# B&R Automation Studio project TD52 (part 39)

### module_CU.typ - Predefined package data types
```iecst
TYPE
	IN_Cust_Struct : 	STRUCT
		bEO_FreshOilPump_Dem : BOOL; (*Status: fresh oil pump (OUT_AG.tEO_FreshOilPump_Dem)*) (*OldName:new V4.14; Cycle:5*)
		bEO_WasteOilPump_Dem : BOOL; (*Status:waste oil pump(OUT_AG:tEO_WasteOilPump_Dem)*) (*OldName:new V4.14; Cycle:5*)
		bAux_OilValve_IsOpen : BOOL; (*valve status for fresh/waste oil in oil pan (without TOF), to be used for release of customized oil pump controls*) (*OldName:new V4.14; Cycle:5*)
		bFreshOilPump_RTC : BOOL; (*Status:fresh oil pump run time exceeded signal (OUT_AG.tFreshOilPump_RTC)*) (*OldName:new V4.14; Cycle:5*)
		tL_FreshOilTank : HALioAi_Type; (*Tank Level measurement input*) (*OldName: NewPv V4.14*)
		tL_WasteOilTank : HALioAi_Type; (*Tank Level measurement input*) (*OldName: NewPv V4.14*)
		tL_DayOilTank : HALioAi_Type; (*Tank Level measurement input*) (*OldName: NewPv V4.14*)
		bBlocDelay_ManStart : BOOL; (* = 		-	blocking of next manual start by delay	*) (*OldName: T26	; Cycle: 5;*)
		bCnt_Gas_NormM3 : BOOL; (*Normal cubic meter - Impulse*) (* OldName: NORM_M3; Cyclic: ; *)
		bCnt_Gas_OpM3 : BOOL; (*Operation cubic meter - Impulse*) (* OldName: BTRB_M3; Cyclic: ; *) (* Gridcode interfaces added *)
		bEG_BoVaOpened : BOOL; (* exhaust gas boiler valve opened *) (*OldName:M_KKAUF; Cycle:5*)
		bEG_ByVaOpened : BOOL; (* exhaust gas bypass valve opened *) (*OldName:M_BKAUF; Cycle:5*)
		bEng_Aux_Dem : BOOL; (* = 		-	demand auxiliaries	*) (*OldName: M_ANFHBT	; Cycle: 5;*)
		bEng_Aux_Dem_CDR : BOOL; (* SS445 Anforderung Hilfsbetriebe  *) (*OldName: ANFHBT	; Cycle: 5;*)
		bEng_Aux_Dem_TOF : BOOL; (* = Auxiliarys demand with TOF -  replacement for old T12 bReq_AuxMod_OfC - request auxiliary mode with off-carriage (Nachlauf)	*) (*OldName: T12	; Cycle: 5;*)
		bEng_Bloc : BOOL; (* = 		-	blocking engine	*) (*OldName: M_BLOCK	; Cycle: 5;*)
		bEng_CDR : BOOL; (* = 		-	manual stop	*) (*OldName: M_STOP	; Cycle: 5;*)
		bEng_Dem : BOOL; (* SS448 Modul ANGEFORDERT  *) (*OldName: M_AGFD	; Cycle: 5;*)
		bEng_Dem_Aut : BOOL; (* = 		-	demand automatic mode	*) (*OldName: M_ANF_A	; Cycle: 5;*)
		bEng_Dem_Bloc : BOOL; (* blocking release of engine	*) (*OldName: ANFBLO	; Cycle: 5;*)
		bEng_Dem_EPS : BOOL; (* = 		-	engine demand for emergency operation	*) (*OldName: M_NANF	; Cycle: 5;*)
		bEng_Dem_Man : BOOL; (* = 		-	demand manual mode	*) (*OldName: M_ANF_H	; Cycle: 5;*)
		bEng_Rdy_Aut : BOOL; (* ready for automatic mode	*) (*OldName: M_BERAUT	; Cycle: 5;*)
		bEng_Rdy_Aut_Exc : BOOL; (*engine ready for automatic operation information for the excitation system	*) (*OldName: BERAUT	; Cycle: 5;*)
		bEng_Rdy_Man : BOOL; (* = 		-	ready for manual mode	*) (*OldName: M_STBT_H	; Cycle: 5;*)
		bEng_Rel : BOOL; (* = 		-	release engine	*) (*OldName: M_FG_MOT	; Cycle: 5;*)
		bEng_Rel_SU : BOOL; (* = 		-	engine starting	*) (*OldName: M_MOST	; Cycle: 5;*)
		bEng_RPSDem : BOOL; (* = 		-	demand RPS	*) (*OldName: M_AGRPS	; Cycle: 5;*)
		bEng_RSBoc : BOOL; (* = 		-	cool down run	*) (*OldName: T10	; Cycle: 5;*)
		bEng_Start : BOOL; (* = 		-	engine start command	*) (*OldName: unkM_STRTnown	; Cycle: 5;*)
		bEng_Stop_Man : BOOL; (* = 		-	demand automatic for start up failure	*) (*OldName: BRI	; Cycle: 5;*)
		bEng_SU_Man : BOOL; (* = 		-	manual start	*) (*OldName: M_HSTART	; Cycle: 5;*)
		bFC_SOf_Bus : BOOL; (*Bus feedback signal: FC switched off*)
		bFC_SOn_Bus : BOOL; (*Bus feedback signal: FC switched on*)
		bILF_SOf_Bus : BOOL; (*Bus feedback signal: ILF switched off*)
		bILF_SOn_Bus : BOOL; (*Bus feedback signal: ILF switched on*)
		bGasTyp1_Act : BOOL; (* gas type 1 active	*) (*OldName: AN_GAS1	; Cycle: 5;*)
		bGasTyp2_Act : BOOL; (* = 		-	gas type 2 active	*) (*OldName: AN_GAS2	; Cycle: 5;*)
		bGasTyp3_Act : BOOL; (* = 		-	gas type 3 active	*) (*OldName: AN_GAS3	; Cycle: 5;*)
		bGasTyp4_Act : BOOL; (* = 		-	gas type 4 active	*) (*OldName: AN_GAS4	; Cycle: 5;*)
		bGasTypMix1_2_Act : BOOL; (* gas type mix 1-2 active	*) (*OldName: AN_GAS1_2 unknown	; Cycle: 5;*)
		bGCB_DemSy : BOOL; (*Demand synchronization generator circuit breaker *) (*OldName:ASYANW,gcb[1].dmnd_sy; Cycle:5;*)
		bGCB_On : BOOL; (* SS446 Generatorschalter EIN  *) (*OldName: MCB_ON	; Cycle: 5;*)
		bGV_Open_Opstate : BOOL; (* = 		-	gas valve open - from opstate module	*) (*OldName: ZM_GASV	; Cycle: 5;*)
		bGV_Rel : BOOL; (* = 		-	release gas valves - freigabe gasventile	*) (*OldName: ZUEND_WEG	; Cycle: 5;*)
		bIgn_Dem : BOOL; (* = 		-	demand ignition	*) (*OldName: ZUEND	; Cycle: 5;*)
		bImp_Start : BOOL; (*start counter impulse *) (*OldName: new PV; Cycle: 5;*)
		bLR_GasStop : BOOL; (*V04.02.00.00*)
		bMCB_DemSy : BOOL; (*Demand synchronization mains circuit breaker *) (*OldName:ARSYANW,mcb[1].dmnd_sy; Cycle:5;*)
		bMCB_On : BOOL; (* SS447 Netzschalter EIN  *) (*OldName: MCB_ON	; Cycle: 5;*)
		bMsg : ARRAY[0..9999]OF BOOL; (*V4.13 simplification: this array replaces all single boolean vars in IN_CU*)
		bOMSS_Aut : BOOL; (*SS427 Betriebswahlschalter AUTOMATIK *) (*OldName: AUTO	; Cycle: 5;*)
		bOMSS_Man : BOOL; (*SS426 Betriebswahlschalter HAND *) (*OldName: HAND; Cycle: 5;*)
		bOpAlm_Res01 : BOOL; (* Alarm Reserve failure 1 trip *) (*OldName: ;Cycle:5;*)
		bOpAlm_Res03 : BOOL; (* Alarm  Reserve failure 3 trip *) (*OldName: ;Cycle:5;*)
		bParaSetupOk : BOOL; (* 	parameter setup ok	*) (*OldName: FGDRPS	; Cycle: 5;*)
		bPr_ECW_Lo1 : BOOL; (*Limit reached pressure engine cooling water limit low 1*) (*OldName:AN_KDGW1; Cycle:5;*)
		bP_Red_Active : BOOL; (* = 		-	 power reduction active - any kind - Module Output and Visu	*) (*OldName: PredAkt	; Cycle: 5;*)
		bP_Rmp_Frz : BOOL; (* = 		-	freeze raising power ramp if control deviation of power exceeds 5% of nominal power	*) (*OldName: bPowerRampFreeze	; Cycle: 5;*)
		bP_Set_FC_Enable : BOOL; (*frequency control active *)
		bRel_Sync_Load : BOOL; (* = 		-	release engine load	*) (*OldName: SY_LFG	; Cycle: 5;*)
		bRPM_Count1_Act : BOOL; (* 	Handle for other modules to activate daily operation hour counter	*) (*OldName: RPMZ1	; Cycle: 5;*)
		bRPM_Count2_Act : BOOL; (* Handle for other modules to activate daily operation hour counter	*) (*OldName: RPMZ2	; Cycle: 5;*)
		bRPM_Count3_Act : BOOL; (* 	Handle for other modules to activate daily operation hour counter	*) (*OldName: RPMZ3	; Cycle: 5;*)
		bRPM_Count4_Act : BOOL; (* 	Handle for other modules to activate daily operation hour counter	*) (*OldName: RPMZ4	; Cycle: 5;*)
		bRPM_Count5_Act : BOOL; (* 	Handle for other modules to activate daily operation hour counter	*) (*OldName: RPMZ5	; Cycle: 5;*)
		bRPM_Count6_Act : BOOL; (* 	Handle for other modules to activate daily operation hour counter	*) (*OldName: RPMZ6	; Cycle: 5;*)
		bRPM_Count7_Act : BOOL; (* 	Handle for other modules to activate daily operation hour counter	*) (*OldName: RPMZ7	; Cycle: 5;*)
		bRPM_Count8_Act : BOOL; (*	Handle for other modules to activate daily operation hour counter	*) (*OldName: RPMZ8	; Cycle: 5;*)
		bRPM_Count9_Act : BOOL; (* 	Handle for other modules to activate daily operation hour counter	*) (*OldName: RPMZ9	; Cycle: 5;*)
		bRPM_Count10_Act : BOOL; (* Handle for other modules to activate daily operation hour counter	*) (*OldName: RPMZ10	; Cycle: 5;*)
		bRPM_Count11_Act : BOOL; (* Handle for other modules to activate daily operation hour counter	*) (*OldName: RPMZ11	; Cycle: 5;*)
		bRPM_Count12_Act : BOOL; (* Handle for other modules to activate daily operation hour counter	*) (*OldName: RPMZ12	; Cycle: 5;*)
		bRPM_Count13_Act : BOOL; (* Handle for other modules to activate daily operation hour counter	*) (*OldName: RPMZ13	; Cycle: 5;*)
		bRPM_Count14_Act : BOOL; (* Handle for other modules to activate daily operation hour counter	*) (*OldName: RPMZ14	; Cycle: 5;*)
		bRPM_Count15_Act : BOOL; (* Handle for other modules to activate daily operation hour counter	*) (*OldName: RPMZ15	; Cycle: 5;*)
		bRPM_Count16_Act : BOOL; (* 	Handle for other modules to activate daily operation hour counter	*) (*OldName: RPMZ16	; Cycle: 5;*)
		bScavFanCoOn : BOOL; (* Scavenging fan on *) (*OldName: unknown	; Cycle: 5;*)
		bSelGasTyp0 : BOOL; (* = 		-	Selection of gas type 0	*) (*OldName: GAS1_2_MAN	; Cycle: 5;*)
		bSelGasTyp1 : BOOL; (* = 		-	Selection of gas type 1	*) (*OldName: GAS1	; Cycle: 5;*)
		bSelGasTyp2 : BOOL; (* = 		-	Selection of gas type 2	*) (*OldName: GAS2	; Cycle: 5;*)
		bSelGasTyp3 : BOOL; (* = 		-	Selection of gas type 3	*) (*OldName: GAS3	; Cycle: 5;*)
		bSelGasTyp4 : BOOL; (* = 		-	Selection of gas type 4	*) (*OldName: GAS4	; Cycle: 5;*)
		bSelGasTypAut : BOOL; (* = 		-	Selection of automatic gas type switching	*) (*OldName: AUTGAS	; Cycle: 5;*)
		bSelGasTypMix : BOOL; (* = 		-	Selection of mixed gas 	*) (*OldName: GAS1_3_MAN	; Cycle: 5;*)
		bTC_CoolDownRun : BOOL; (* = Turbo charger CoolDownRun (from V4.2.x on)*)
		bUniDigSet : ARRAY[0..250]OF BOOL; (* *) (*OldName: bUniDigSet	; Cycle: 5;*)
		bWarn_AmbPress : BOOL; (* ?OLD-HANG LU? Warn: W1197 reserve, Ambient pressure deviation P2 to P2s *) (*OldName:new PV;Cycle:2;*)
		bWarn_TC_Speed_PRed : BOOL; (* ?OLD-HANG LU? Warn: W1198 reserve, Power reduction due to TC Speed *) (*OldName:new PV;Cycle:2;*)
		iCnt_OpHours : DINT; (*IF541 oper.hours count.high word	*) (* OldName:  	BTRB_high	; Cycle: 5;*)
		iCnt_Starts : DINT; (*IF543 start counter    high word	*) (* OldName:  	STRT_high	; Cycle: 5;*)
		iGM1_MStepActPos : DINT; (*gasmixer 1 - Actual position from SM1426-Module [Microsteps]*) (*OldName: slGM1_MStepActPos_TC1; Cycle: 5;*)
		iGM1_Status : UINT; (*gasmixer 1 - Status Word from SM1426-Module*) (*OldName: usGM1_Status_TC1; Cycle: 5;*)
		iGM2_MStepActPos : DINT; (*gasmixer 2 - Actual position from SM1426-Module [Microsteps]*) (*OldName: slGM2_MStepActPos_TC1; Cycle: 5;*)
		iGM2_Status : UINT; (*gasmixer 2 - Status Word from SM1426-Module*) (*OldName: usGM2_Status_TC1; Cycle: 5;*)
		iHeatPowerCount : DINT; (*Retired, not used anymore! old: STM - FXXX counter heating power engine heat water circuit*) (*OldName: Retired; Cycle: 5;*) (*STM*)
		iIdx_OMSS : INT; (* SS425 Betriebswahlschalter AUS *) (*OldName: BWS_HA; Cycle: 5;*)
		iIdx_ProcessStep : DINT; (*Optional step information to display on VIS*)
		iIdx_ProcessStep_AG : DINT; (*Optional step information to display on VIS from module AG*)
		iIdx_RSS : INT; (* = 		-	index of request selector switch	*) (*OldName: AWS_A	; Cycle: 5;*)
		iMsg : ARRAY[0..9999]OF USINT; (*provides data from all alarms - Version 2018, from CBM Version*) (*OldName:newPv; Cycle:2;*)
		InData1 : ARRAY[0..MAX_IN_DATA_ARRAY]OF INT; (*input data from master coupling 1*)
		InData2 : ARRAY[0..MAX_IN_DATA_ARRAY]OF INT; (*input data from master coupling 2*)
		iProcessStepTime : DINT; (*Optional step time  info to display on VIS*)
		iProcessStepTime_AG : DINT; (*Optional step time  info to display on VIS from module AG*)
		iSt_OpMode : UDINT; (* = 		-	engine operation mode	*) (*OldName: A_BWS_HA	; Cycle: 5;*)
		iSt_OpMode_Main : INT; (* = 		-	GeneratorControl.(iSt_OpMode / 65535) = 60	*) (*OldName: InselM	; Cycle: 5;*)
		rCA_IgnP_Set : REAL; (*Global ignition timing point*) (*OldName: ZZP_SOLL	; Cycle: 5;*)
		rScalBlock_X : ARRAY[0..30]OF REAL;
		rCustAnaIn : ARRAY[0..120]OF REAL; (*OLD_ DO NOT USE ANYMORE!  Prepared spare analog input = measured and scaled signal from hardcoded reserve channel			*) (*OldName: ANA_RAN; Cycle: ;*)
		rCustAnaIn_ErrMax : ARRAY[0..120]OF REAL;
		rCustAnaIn_ErrMin : ARRAY[0..120]OF REAL;
		rCustomizedAG : ARRAY[0..99]OF REAL; (*optional prepared customizable interface V4.5 - BETA PHASE, use only in coordination with TPSS*)
		rCustomizedCH : ARRAY[0..99]OF REAL; (*optional prepared customizable interface V4.5 - BETA PHASE, use only in coordination with TPSS*)
		rCustomizedCP : ARRAY[0..99]OF REAL; (*optional prepared customizable interface V4.5 - BETA PHASE, use only in coordination with TPSS*)
		rCustomizedEC : ARRAY[0..99]OF REAL; (*optional prepared customizable interface V4.5 - BETA PHASE, use only in coordination with TPSS*)
		rCustomizedHA : ARRAY[0..300]OF REAL; (*optional prepared customizable interface for HAL, V4.5 - BETA PHASE, use only in coordination with TPSS*)
		rCustomizedHC : ARRAY[0..99]OF REAL; (*optional prepared customizable interface V4.5 - BETA PHASE, use only in coordination with TPSS*)
		rCustomizedOP : ARRAY[0..99]OF REAL; (*optional prepared customizable interface V4.5 - BETA PHASE, use only in coordination with TPSS*)
		rEO_Level : REAL; (*IF630 oil level	*) (* OldName:  	ANA.OELST	; Cycle: 5;*)
		rF_MMD : ARRAY[0..2]OF REAL; (* frequency multi measure device *) (* OldName:ssFreq; Cycle: *)
		rGT_CH4 : REAL; (*CH4 content, 1.0 = 100% *) (* OldName: 	ANA_CH4	; Cyclic: ; *)
		rGT_CV : REAL; (*Calorific value *) (* OldName: 	ANA_CV	; Cyclic: ; *)
		rGT_O2 : REAL; (*O2 content *) (* OldName: 	ANA_O2	; Cyclic: ; *)
		rI_Avg : ARRAY[0..2]OF REAL; (* current average *) (* OldName:ssIAvg; Cycle: *)
		rI_L1 : ARRAY[0..2]OF REAL; (* current 1 *) (* OldName:ssIL1; Cycle: *)
		rI_L2 : ARRAY[0..2]OF REAL; (* current 2 *) (* OldName:ssIL2; Cycle: *)
		rI_L3 : ARRAY[0..2]OF REAL; (* current 3 *) (* OldName:ssIL3; Cycle: *)
		rI_N : ARRAY[0..2]OF REAL; (* current neutral *) (* OldName:ssIN; Cycle: *)
		rLam_Eng_LL_Set : REAL; (* Leanox Lambda set point *) (* OldName: ssPosGasmixerNominal; Cycle:2; *)
		rN_EngAct : REAL; (*IF611 speed	*) (* OldName:  	ANA.DREHZ	; Cycle: 5;*)
		rN_Set_Norm : REAL; (* = 		-	speed setpoint speed controller 	*) (*OldName: n_soll	; Cycle: 5;*)
		rPF_Act : ARRAY[0..2]OF REAL; (* power factor *) (* OldName:ssCosPhi; Cycle: *)
		rPos_Act_GM1_Norm : REAL; (*gasmixer 1 - normed actual position [%]*) (*OldName: bp_y; ANA.LLPOS; ANA.TJ_y; S_K_W[137]; S_K_W[142]; Cycle: 5;*)
		rPos_CBV : REAL; (* compressor bypass valve position *) (*OldName: rPos_CBV; Cycle: 2 *)
		rPos_ChC_Valve : REAL; (*IFXXX position control valve charge cooler circuit temperature*) (*OldName: newPV; Cycle: 5;*) (*STM*)
		rPos_CircLou1 : REAL; (*IFxxx position air circulation louver 1*) (*OldName: newPV; Cycle: 5;*) (*STM*)
		rPos_CircLou2 : REAL; (*IFxxx position air circulation louver 2*) (*OldName: newPV; Cycle: 5;*) (*STM*)
		rPos_GM_Set_Norm : REAL; (* set point for the gasmixer *) (*OldName: ssPosGasmixerNominal; Cycle:2; *)
		rPos_HW_EC_ReValve : REAL; (*IFXXX position control valve heat water return temperature after cooler*) (*OldName: newPV; Cycle: 5;*) (*STM*)
		rPos_HW_ReValve : REAL; (*IFXXX position control valve heat water return temperature*) (*OldName: newPV; Cycle: 5;*) (*STM*)
		rPos_InlLou1 : REAL; (*IFxxx position air inlet louver 1*) (*OldName: newPV; Cycle: 5;*) (*STM*)
		rPos_InlLou2 : REAL; (*IFxxx position air inlet louver 2*) (*OldName: newPV; Cycle: 5;*) (*STM*)
		rPos_OutlLou1 : REAL; (*IFxxx position air outlet louver 1*) (*OldName: newPV; Cycle: 5;*) (*STM*)
		rPos_OutlLou2 : REAL; (*IFxxx position air outlet louver 2*) (*OldName: newPV; Cycle: 5;*) (*STM*)
		rPos_TV : REAL; (* throttle valve position *) (*OldName: drkl_y; Cycle:2; *)
		rPrDiff_ER : REAL; (*IFxxx engine room difference pressure*) (*OldName: newPV; Cycle: 5;*) (*STM 2*)
		rPr_Baro_Internal : REAL; (*V04.02.00.00*)
		rPr_Ch_P2s_A : REAL; (*V04.02.00.00*)
		rPr_Ch_P2s_Avg : REAL; (*average charge pressure p2' (after throttle valve) [bar]*)
		rPr_Ch_P2s_B : REAL; (*V04.02.00.00*)
		rPr_ECW : REAL; (*IF502 jacket water pressure *) (* OldName:  	ANA.KWD		; Cycle: 5;*)
		rPr_EngLubOil : REAL; (*IF504 oil pressure *) (* OldName:  	ANA.ODR		; Cycle: 5;*)
		rPr_GT_Gas : REAL; (*Gas pressure *) (* OldName: 	ANA_GD	; Cyclic: ; *)
		rPr_GT_Suct : REAL; (*Gas suction pressure *) (* OldName: 	ANA_SD	; Cyclic: ; *)
		rPr_PCG : REAL; (*Pressure pre chamber gas compressor  *) (* OldName: 	ANA_VKGD	; Cyclic: ; *)
		rPr_PC_Diff : REAL; (*Prechamber differential pressure*) (* OldName: 	ANA_PDIFF	; Cyclic: ; *)
		rP_Act : ARRAY[0..2]OF REAL; (* IF500 active power (IF LIST FROM TASK snd_cst) ??normiert 0-1?? 	*) (*OldName: ANA.P_IST	; Cycle: 5;*)
		rP_Act_Norm_Filt : REAL; (* = 		-	actual power related to rP_Nom filtered T=1s	*) (*OldName: P_IST	; Cycle: 5;*)
		rP_FC_ContOutput : REAL; (*controller output FC*)
		rP_Heat : REAL; (*IFXXX heating power engine heat water circuit *) (*OldName: newPV; Cycle: 5;*) (*STM 2*)
		rP_Nom : REAL; (* = 		-	nominal power	*) (*OldName: PN_GASART	; Cycle: 5;*)
		rP_Red_Norm : REAL; (* = 		-	power reduction related to rP_Nom	*) (*OldName: RedPowerProm	; Cycle: 5;*)
		rP_Set : REAL; (*IF540 setpoint power control	*) (* OldName:  	ANA.SOLL_PREG ; Cycle: 5;*)
		rP_Set_ExtBus_Norm : REAL; (*external power setpoint via bus related to rP_Nom*)
		rP_Set_FC_Norm : REAL; (*generator power setpoint by frequency control*)
		rP_Set_Min : REAL; (*minimal power setpoint related to rP_nom*) (*OldName:p_min;Cycle:5;*)
		rP_Set_Min_Norm : REAL := 0.51; (*Fehlt Noch*)
		rP_Set_Norm : REAL; (* = 		-	power setpoint related to rP_Nom	*) (*OldName: p_soll	; Cycle: 5;*)
		rP_WorkAct : ARRAY[0..2]OF REAL; (*IF536 total act.  outp.high word OldName > iP_WorkAct?	*) (* OldName:  	ANA.WARBH	; Cycle: 5;*)
		rQ_Act : ARRAY[0..2]OF REAL; (* power reactive *) (* OldName:ssPReac; Cycle: *)
		rQ_WorkReac : ARRAY[0..2]OF REAL; (*IF538 total react.outp.high word  OldName > iQ_WorkReac?*) (* OldName:  	ANA.BARBH	; Cycle: 5;*)
		rQ_WorkReacRet : ARRAY[0..2]OF REAL; (* counter last received reactive engine work  *) (* OldName:slWorkReacRet; Cycle: *)
		rS_Act : ARRAY[0..2]OF REAL; (* power apperent *) (* OldName:ssPApper; Cycle: *)
		rT_AirER : REAL; (*vis air engine room temperature [degC]*) (*OldName:ANA_RTM; Cycle:5;*)
		rT_AirOutdoor : REAL; (*temperature air outdoor *) (*OldName:ANA_ULT; Cycle:5;*)
		rT_Cat : REAL; (*AI exhaust gas temperature catalyst general (before)*) (*OldName:ANA.KATP;Cycle:;*)
		rT_Ch_T1LP_Avg : REAL; (*average charge temperature before low-pressure turbocharger (= engine intake air) [degC]*) (*OldName:ssIATemp,ANA_ZLTP,rT_InAirER; Cycle:5;*) (* V04.04.00.00 *)
		rT_Ch_T2s_Avg : REAL; (*average charge temperature t2' (after throttle valve) [degC]*)
		rT_ECW : REAL; (*IF501 jacket water temperature	*) (* OldName:  	ANA.KWT		; Cycle: 5;*)
		rT_EGaCat : REAL; (*exhaust gas temperature after catalyst*) (*OldName:ANA.NKAT;Cycle:;*)
		rT_EGaHE : REAL; (*AI exhaust gas temperature after heat exchanger [degC]*) (*OldName:ANA.NABK;Cycle:5*)
		rT_EGaHE1 : REAL; (*exhaust gas temperature after heat exchanger 1*) (*OldName:NWTT1_WE;Cycle:5*)
		rT_EGaHE2 : REAL; (*exhaust gas temperature after heat exchanger 2*) (*OldName:NWTT2_WE;Cycle:5*)
		rT_EGaTC : REAL; (*AI exhaust gas temperature after turbo charger [degC]*) (*OldName:ANA.VABK;Cycle:5*)
		rT_EGbCat : REAL; (*exhaust gas temperature before catalyst*) (*OldName:ANA.VKAT;Cycle:;*)
		rT_EGbTC : REAL; (*AI exhaust gas temperature before turbo charger*) (*OldName:ANA.T3;Cycle:5*)
		rT_EG_Avg : REAL; (* cylinder temperature average [degC] *) (* OldName: t_zyl_mw; Cycle:5; *)
		rT_EO : REAL; (*IF503 oil temperature	*) (* OldName:  	ANA.OTP		; Cycle: 5;*)
		rT_EPU_EG : ARRAY[0..24]OF REAL; (*EngineController::  engine power unit exhaust gas temperatures *) (* OldName:  T_ZYL ; Cycle: 5;*)
		rT_Gen_Bear_A_Act : REAL; (*IF609 gen.bearing temp.(A)	*) (* OldName:  	ANA.LAG1	; Cycle: 5;*)
		rT_Gen_Bear_B_Act : REAL; (*IF610 gen.bearing temp.(B)	*) (* OldName:  	ANA.LAG2	; Cycle: 5;*)
		rT_Gen_Wind_Act : REAL; (* generator winding temperature signal *) (*OldName:ANA.WICK;Cycle:;*)
		rT_Gen_Wind_Act_L1 : REAL; (*IF606 gen.winding temp.L1	*) (* OldName:  	ANA.WICK1	; Cycle: 5;*)
		rT_Gen_Wind_Act_L2 : REAL; (*IF607 gen.winding temp.L2	*) (* OldName:  	ANA.WICK2	; Cycle: 5;*)
		rT_Gen_Wind_Act_L3 : REAL; (*IF608 gen.winding temp.L3	*) (* OldName:  	ANA.WICK3	; Cycle: 5;*)
		rT_GT : REAL; (*Gas temperature *) (* OldName: 	ANA_GT	; Cyclic: ; *)
		rT_HW_Re : REAL; (*IF509 return water temperature	*) (* OldName:  	ANA.RLTP	; Cycle: 5;*)
		rT_HW_ReAfEC : REAL; (*temperature heat water return after emergency cooler [degC]*) (*OldName:ANA.RLT_NK; Cycle:5;*)
		rT_HW_Su : REAL; (*IF510 supply water temperature	*) (* OldName:  	ANA.VLTP	; Cycle: 5;*)
		rT_PlateHE : REAL; (*AI exhaust gas temperature before heat exchanger*) (*OldName:ANA.ROHR;Cycle:5*)
		rT_PlateHE_Vis : REAL; (*IF507 plate temp.exh.gas heat exc.	*) (* OldName:  	ANA.ROHR	; Cycle: 5;*)
		rT_Re_PriCirc : REAL; (*IFXXX return water temperature high primary circuit*) (*OldName: newPV; Cycle: 5;*) (*STM*)
		rT_Re_SecCirc : REAL; (*IFXXX return water temperature high secondary circuit*) (*OldName: newPV; Cycle: 5;*) (*STM*)
		rT_Su_PriCirc : REAL; (*IFXXX supply water temperature high primary circui*) (*OldName: newPV; Cycle: 5;*) (*STM*)
		rT_Su_SecCirc : REAL; (*IFXXX supply water temperature high secondary circuit*) (*OldName: newPV; Cycle: 5;*) (*STM*)
		rUniAnaSet : ARRAY[0..151]OF REAL; (* *) (*OldName: rUniAnaSet	; Cycle: 5;*)
		rU_Avg : ARRAY[0..2]OF REAL; (* voltage average *) (* OldName:ssUAvg; Cycle: *)
		rU_Gen_Exc : REAL; (*IF605 gen.excitation voltage*) (*OldName: ANA.ERREG; Cycle:;*)
		rU_L1L2 : ARRAY[0..2]OF REAL; (* voltage 12 *) (* OldName:ssUL1L2; Cycle: *)
		rU_L1N : ARRAY[0..2]OF REAL; (* voltage 1 *) (* OldName:ssUL1N; Cycle: *)
		rU_L2L3 : ARRAY[0..2]OF REAL; (* voltage 23 *) (* OldName:ssUL2L3; Cycle: *)
		rU_L2N : ARRAY[0..2]OF REAL; (* voltage 2 *) (* OldName:ssUL2N; Cycle: *)
		rU_L3L1 : ARRAY[0..2]OF REAL; (* voltage 31 *) (* OldName:ssUL3L1; Cycle: *)
		rU_L3N : ARRAY[0..2]OF REAL; (* voltage 3 *) (* OldName:ssUL3N; Cycle: *)
		rVol_GT : REAL; (*Gas volume *) (* OldName: 	ANA_GM	; Cyclic: ; *)
		tAB2CU : AmmBase2MM; (* Caution: use apropriate structure member of local AMM- interfacestructure	*) (*OldName: QUITT_AB; Cycle: 5;*)
		tActFiltAlarm : HALioDi_Type; (*DIactivfilteralarm*)
		tActFiltWarn : HALioDi_Type; (*DIactivfilterwarning*)
		tActuator_Ok : HALioDi_Type; (*DI:Actuatorokay*)
		tActuator_Ok_CBV1 : HALioDi_Type; (*DI:Actuatorokaycompressorbypassvalve1*)
		tActuator_Ok_CBV2 : HALioDi_Type; (*DI:Actuatorokaycompressorbypassvalve2*)
		tActuator_Ok_CBV_A : HALioDi_Type; (* DI: Actuator okay compressor by pass valve 1A *) (* OldName: DI_F_ACT_TBV_A; Cycle:2; *)
		tActuator_Ok_CBV_B : HALioDi_Type; (* DI: Actuator okay compressor by pass valve 1B *) (* OldName: DI_F_ACT_TBV_B; Cycle:2; *)
		tActuator_Ok_TV1A : HALioDi_Type; (*DI:Actuatorokaythrottlevalve1A*)
		tActuator_Ok_TV1B : HALioDi_Type; (*DI:Actuatorokaythrottlevalve1B*)
		tActuator_Ok_TV2A : HALioDi_Type; (*DI:Actuatorokaythrottlevalve2A*)
		tActuator_Ok_TV2B : HALioDi_Type; (*DI:Actuatorokaythrottlevalve2B*)
		tAirER_FS : HALioDi_Type; (*DIengineroomVEflowswitch*)
		tAuxErrWarn : HALioDi_Type; (*DIauxiliarieserror*)
		tAuxFail : HALioDi_Type; (*DIauxilariesfailure*)
		tAuxOverVoltProt_Ok : HALioDi_Type; (*failureovervoltageprotectionauxiliariespowersupply*)
		tAuxV_Aux_ok : HALioDi_Type; (*DI: Auxiliaries voltage auxiliaries panel OK*)
		tAuxV_Eng_ok : HALioDi_Type; (*DIauxiliariesvoltageengineok*)
		tAuxV_ModIf_ok : HALioDi_Type; (*DI: Auxiliaries voltage module interface OK*)
		tAuxV_Supply_Ok : HALioDi_Type; (*DIauxiliaryvoltagesupplyok*)
		tBbBlower_FC_Rdy : HALioDi_Type; (*DI Blow-by Blower FC ready *)
		tBB_Alive : HALioDi_Type; (*DIbusbaralive*)
		tBB_Dead_MMD : ARRAY[0..2]OF HALioDi_Type; (*DIbusbardeadfromMMD*)
		tBHV_Op : HALioDi_Type; (*DI: Failure boiler house ventilation*)
		tCCWP_Op : HALioDi_Type; (*DIchargecoolingwaterpumpoperating*)
		tCDP_Op : HALioDi_Type; (*DI: Failure condensor pump*)
		tChC_Failure : HALioDi_Type; (*DIchargecoolerfailure*)
		tChC_FanRdy : HALioDi_Type; (*DIchargecoolerfanready*)
		tChUnit1_CB_On : HALioDi_Type; (*Circuit breaker tripped Charging unit 1*)
		tChUnit2_CB_On : HALioDi_Type; (*Circuit breaker tripped Charging unit 2*)
		tChUnit3_CB_On : HALioDi_Type; (*Circuit breaker tripped +ENGIA Charging unit 1*)
		tChUnit4_CB_On : HALioDi_Type; (*Circuit breaker tripped +ENGIA Charging unit 2*)
		tCnt_GasImp : HALioDi_Type; (*DIImpulsegascounter*)
		tCnt_N_AirStarter : HALioAi_INT_Type; (*AI air starter speed [rpm]*)
		tCnt_OilPulse : HALioDi_Type; (*DIoilcounter*)
		tCnt_Oil_DC2395 : HALioAi_INT_Type; (*AIoilcountercircularbuffer*)
		tCnt_Oil_NC150 : HALioAi_Type; (*AIoilcounter*)
		tCO2_Demand : HALioDi_Type; (*DICO2demand*)
		tCO2_DevFailure : HALioDi_Type; (*DICO2devicefailure*)
		tCO2_FanFailure : HALioDi_Type; (*DICO2fanfailure*)
		tCO2_VaClosed : HALioDi_Type; (*DICO2valveclosed*)
		tCO2_VaFailure : HALioDi_Type; (*DICO2valvefailure*)
		tCO2_VaLockout : HALioDi_Type; (*DIlockoutCO2valve*)
		tCO2_VaOpened : HALioDi_Type; (*DICO2valveopened*)
		tCodinox_Rdy : HALioDi_Type; (*DICODINOXreadyforoperation*)
		tCO_Alarm : HALioDi_Type; (*DICOalarm*)
		tCO_PreAlarm : HALioDi_Type; (*DICOprealarm*)
		tCP_CBTrip : HALioDi_Type; (*DImoduleand/orinterfacecontrolpanel-circuitbreakertripped*)
		tCtr_Mns_Anain_Setp_W_ext : HALioAi_Type; (*(Interace) Mains Ctrl*)
		tCustAnaIn : ARRAY[0..120]OF HALioAi_Type; (*Replacement for RAN_KANAL...*) (*OldName: ANA_RAN	; Cycle: 5;*)
		tCustDigIn : ARRAY[0..200]OF HALioDi_Type; (*Prepared Spare Inputs, reserved for project specific use*) (*OldName: new PV	; Cycle: 5;*)
		tCustDigIn_TC2 : ARRAY[0..200]OF HALioDi_Type; (*Prepared Spare Inputs, reserved for project specific use for fastc counter inputs in task class2  (V4.07)*) (*OldName: new PV	; Cycle: 5;*)
		tCV_Eng_Low : HALioDi_Type; (*Control voltage min*)
		tCV_MCP_Low : HALioDi_Type; (*control voltage low - module control panel*) (*OldName:DI_CV_MCP_low; Cycle:5;*)
		tCV_TCA_Low : HALioDi_Type; (*Control voltage min*)
		tC_CB_EDC : HALioDi_Type; (*DIcustomercircuitbreaker(engine*)
		tC_CB_ESL : HALioDi_Type; (*DIcustomercircuitbreaker(engine*)
		tC_CB_Off : HALioDi_Type; (*DIcustomercircuitbreakeropened*)
		tC_CB_On : HALioDi_Type; (*DIcustomercircuitbreakerclosed*)
		tDayOilTank_Leck : HALioDi_Type; (*DI: Leck day oil tank*)
		tDemEngOpExt : HALioDi_Type; (*externaldemandofengineoperation*)
		tDemFlair : HALioDi_Type; (*DIDemandgascompressorforflairoperationmode*)
		tDemnd_BHV : HALioDi_Type; (*DI: Demand boiler house ventilation*)
		tDem_Ctr_Mns : HALioDi_Type; (*Activation Customer Interface*)
		tDiffPrct : HALioDi_Type; (*DI:Differentialprotection*)
		tDI_Dem_EU_Block : HALioDi_Type; (*externalrequestfromutility(evu*)
		tDI_Dem_P_Red_EVU_Stage1 : HALioDi_Type; (*external request from utility (evu) ==>> lpower reduction stage 1*) (*OldName: DI_EVU_1; Cycle: 5;*)
		tDI_Dem_P_Red_EVU_Stage2 : HALioDi_Type; (*external request from utility (evu) ==>> power reduction stage 2*) (*OldName: DI_EVU_2; Cycle: 5;*)
		tDI_Dem_P_Red_EVU_Stage3 : HALioDi_Type; (*external request from utility (evu) ==>> power reduction stage 3*) (*OldName: DI_EVU_3; Cycle: 5;*)
		tDI_Dem_P_Red_EVU_Stage4 : HALioDi_Type; (*external request from utility (external, vintagestyled utilisation) ==>> power reduction stage 4*) (*OldName: DI_EVU_4; Cycle: 5;*)
		tDI_Dem_P_Red_EVU_Stage5 : HALioDi_Type; (*external request from utility (external, vintagestyled utilisation) ==>> power reduction stage 5*) (*OldName: DI_EVU_5; Cycle: 5;*)
		tDPr_AirFilt : HALioAi_Type; (*engineairinletfilterdifferencepressure[bar]*)
		tDPr_AirFilt_A : HALioAi_Type; (*engineairinletfilterdifferencepressureA[bar]*)
		tDPr_AirFilt_B : HALioAi_Type; (*engineairinletfilterdifferencepressureB[bar]*)
		tDPr_AirFilt_Hi : HALioDi_Type; (*engineairinletfilterdifferencepressureHIGH*)
		tDPr_OilSkid_FiltHP_DE_Hi : HALioDi_Type; (*DI OilSkid difference pressure - oil high pressure filter to DE bearing*)
		tDPr_OilSkid_FiltHP_NDE_Hi : HALioDi_Type; (*DI OilSkid fan - circuit breaker*)
		tDPr_OilSkid_FiltLP_Hi : HALioDi_Type; (*DI OilSkid difference pressure - oil low pressure filter*)
		tEarthCB_Off : HALioDi_Type; (*DIearthcircuitbreakeropened,francecountryspecific*)
		tECWPrehV_Opened : HALioDi_Type; (*DIenginecoolingwaterpreheatingvalveopened*)
		tECWP_FC_Rdy : HALioDi_Type; (*DIenginecoolingwaterpumpfrequencyconverterreadyforoperation*)
		tECWP_Op : HALioDi_Type; (*DIenginecoolingwaterpumpoperating*)
		tECWP_PreH_CB_On : HALioDi_Type; (*Failure Engine jacket water Preheating pump*)
		tECWP_PreH_Dem : HALioDo_Type; (*VORW  DO engine cooling water preheating pump demand*) (*OldName:A_VORW;Cycle:5*)
		tECWP_Service_CB_On : HALioDi_Type; (*Failure Service Pump Engine jacket water*)
		tECWP_Service_COn : HALioDi_Type; (*Demand Service Pump Engine jacket water*)
		tECWV_Fail : HALioDi_Type; (*Failure Flap Preheating Engine jacket water*)
		tECW_PreHV_Closed : HALioDi_Type; (*DIenginecoolingwaterpreheatingvalvestatusclosed*)
		tECW_PreHV_Opened : HALioDi_Type; (*DIenginecoolingwaterpreheatingvalvestatusopened*)
		tEC_Failure : HALioDi_Type; (*DIemergencycoolerfailure*)
		tEGScavStart_Ext : HALioDi_Type; (*DIexhaustgasscavengingstartfromexternal*)
		tEG_BoVaClosed : HALioDi_Type; (*DIexhaustgasboilervalveclosed*)
		tEG_BoVaClosedTo : HALioDi_Type; (*DIexhaustgasboilervalveclosedtorch*)
		tEG_BoVaFailure : HALioDi_Type; (*DIexhaustgasboilervalvefailure*)
		tEG_BoVaOpened : HALioDi_Type; (*DIexhaustgasboilervalveopened*)
		tEG_BypassDemand : HALioDi_Type; (*DIdemandexhaustgasbypass*)
		tEG_ByVaClosed : HALioDi_Type; (*DIexhaustgasbypassvalveclosed*)
		tEG_ByVaClosedTo : HALioDi_Type; (*DIexhaustgasbypassvalveclosedtorch*)
		tEG_ByVaFailure : HALioDi_Type; (*DIexhaustgasbypassvalvefailure*)
		tEG_ByVaOpened : HALioDi_Type; (*DIexhaustgasbypassvalveopened*)
		tEleStarter_Dem : HALioDo_Type; (*DO electric starter demand*) (*OldName:A_STRT;Cycle:5;*)
		tEmStop_CoolRun : HALioDi_Type; (*DI: Emergency stop with cool down run*)
		tEngDemIsland : HALioDi_Type; (*DIenginedemandforislandoperation*)
		tENGIA_CB_On : HALioDi_Type; (*power supply engine interface panel circuit breaker on*) (*OldName:DI_ENGIA_CB_On; Cycle:5;*)
		tENGIA_UPS_CB_On : HALioDi_Type; (*Circuit breaker tripped supply UPS +TCAI --> +ENGIA*)
		tEngStartFailure : HALioDi_Type; (*DIenginestartfailure*)
		tEngTurn : HALioDi_Type; (*DIengineturnequipmentactive*)
		tEngTurn2 : HALioDi_Type; (*Failure engine turning device*)
		tEng_Dem_EPS_Ext : HALioDi_Type; (*enginedemandemergencypowersupplyfromexternal*)
		tEng_Rdy_Rem : HALioDo_Type; (* Ready for Remote Operation *) (*OldName:BERZLT;Cycle:2;*)
		tEng_Run : HALioDo_Type; (* SS449 Betrieb EIN  *) (*OldName: M_BTRB	; Cycle: 5;*)
		tEng_SUExc_Rel : HALioDi_Type; (*start-upexcitationrelease*)
		tEOF_DiffMax : HALioDi_Type; (*DI:Oildifferencepressuremaximum*)
		tEOP1AC_CB_trip : HALioDi_Type; (*DIengineoilpump1ACcircuitbreakertrip*)
		tEOP_DemExt : HALioDi_Type; (*DIengineoilpumpdemandfromexternal*)
		tEOP_FC_Rdy : HALioDi_Type; (*DI:engineoilpumpfreq.converteroperation/ready*)
		tEOP_Op : HALioDi_Type; (*DIengineoilpumpoperating*)
		tEO_Level : HALioAi_Type; (*Engine Oil Pan Level*) (*OldName: unknown	; Cycle: 5;*)
		tEO_Level_Hi : HALioDi_Type; (*DIengineoillevelhighfromlevelswitch*)
		tEO_Level_Lo : HALioDi_Type; (*DIengineoillevellowfromlevelswitch*)
		tEO_Quality : HALioAi_Type; (*AI:Oilqualitysensor,QTOil1/AI_*)
		tEO_Refill : HALioDi_Type; (*DIengineoilrefillONfromlevelswitch*)
		tEO_Supply_Fail : HALioDi_Type; (*DI:Oilsupplyfailure*)
		tERV_InlAir_Op : HALioDi_Type; (*DIengineroomventilationinletairnoperating/airflowok*)
		tERV_Op : HALioDi_Type; (*DIengineroomventilationoperating/airflowok*)
		tERV_OutlAir_Op : HALioDi_Type; (*DIengineroomventilationoutletairnoperating/airflowok*)
		tER_DoorClosed : HALioDi_Type; (*DI engine room doors closed*)
		tER_Ext_Err : HALioDi_Type; (*DIengineroomVEfailure*)
		tER_InlAir_Ext_Err : HALioDi_Type; (*DIengineroomInlVEfailure*)
		tER_OutlAir_Ext_Err : HALioDi_Type; (*DIengineroomOutlVEfailure*)
		tEU_RM_BLOCK : HALioDo_Type;
		tEVU_PowerSet3Dem : HALioDi_Type; (*demandmoduleblockedbyutility*)
		tFastStartReq : HALioDi_Type; (* DI: Fast Start Required *) (* OldName: DI_FastStartReq; Cycle:2; *)
		tILF_SOf : HALioDo_Type; (*DO: feedback signal: ILF switched off*)
		tILF_SOn : HALioDo_Type; (*DO: feedback signal: ILF switched on*)
		tFC_SOf : HALioDo_Type; (*DO: feedback signal: FC switched off*)
		tFC_SOn : HALioDo_Type; (*DO: feedback signal: FC switched on*)
		tFireAlarm : HALioDi_Type; (*DIfirealarm*)
		tFlairRdy : HALioDi_Type; (*DIFlairready*)
		tFlow_Gen_Lube : HALioDi_Type; (*generatorlubricationfailure*)
		tFlow_HW_Lo : HALioDi_Type; (*DIheatwaterflowlow*)
		tFlow_OilSkid_DE : HALioAi_Type; (*AI OilSkid oil flow to DE bearing *)
		tFlow_OilSkid_NDE : HALioAi_Type; (*AI OilSkid oil flow to NDE bearing (G.03-FI-003)*)
		tFOP_Op : HALioDi_Type; (*DI: Fresh oil pump operation*)
		tFS_ECW : HALioDi_Type; (*DIflowswitchenginecoolingwater*)
		tF_GenBear_DE1 : HALioAi_Type; (*vibration generator bearing drive end 1*) (*Oldname:AI_v_GenBearDE1;Cycle:5;*)
		tF_GenBear_DE2 : HALioAi_Type; (*vibration generator bearing drive end 2*) (*Oldname:AI_v_GenBearDE2;Cycle:5;*)
		tF_GenBear_NDE1 : HALioAi_Type; (*vibration generator bearing non drive end 1*) (*Oldname:AI_v_GenBearNDE1;Cycle:5;*)
		tF_GenBear_NDE2 : HALioAi_Type; (*vibration generator bearing non drive end 2*) (*Oldname:AI_v_GenBearNDE2;Cycle:5;*)
		tF_MMD : ARRAY[0..2]OF HALioAi_Type; (*IF512 generator frequency	*) (* OldName:  	ANA.FREQ	; Cycle: 5;*)
		tF_MMD_BusBar : ARRAY[0..2]OF HALioAi_Type; (*Bus bar frequency*) (* OldName:  	ANA.FREQ	; Cycle: 5;*)
		tF_MMD_LimHi : ARRAY[0..2]OF HALioDi_Type; (*generatorfrequencytoohigh*)
		tF_MMD_LimLo : ARRAY[0..2]OF HALioDi_Type; (*generatorfrequencytoolow*)
		tF_MMD_Synch1 : ARRAY[0..2]OF HALioAi_Type; (* Frequency Sync-network 1 *)
		tF_MMD_Synch2 : ARRAY[0..2]OF HALioAi_Type; (* Frequency Sync-network 2 *)
		tF_N_DI_Dec : HALioDi_Type; (*synch.digitalindecreasespeed*)
		tF_N_DI_Inc : HALioDi_Type; (*synch.digitalinincreasespeed*)
		tGasAlarm : HALioDi_Type; (*DIgasalarm*)
		tGasPreAlarm : HALioDi_Type; (*DIgasprealarm*)
		tGCB_AGO : HALioDi_Type; (*DIallothergeneratorcircuitbreakeroff*)
		tGCB_DRM : HALioDi_Type; (*DIgeneratorcircuitbreakerdemandMCBclosingreturntomains*)
		tGCB_DSY : HALioDi_Type; (*DIgeneratorcircuitbreakerdemandsynchronization(synchline*)
		tGCB_DVM : HALioDi_Type; (*voltagematchingforsynchronization*)
		tGCB_Earth : HALioDi_Type; (*DIgeneratorcircuitbreakerpositionearth*)
		tGCB_MDL : HALioDi_Type; (*DIgeneratorcircuitbreakermasterdemandlock(forclosingotherGCBtodeadBB*)
		tGCB_MRC : HALioDi_Type; (*DIgeneratorcircuitbreakermasterreleaseclose(todeadbusbar*)
		tGCB_Off : HALioDi_Type; (*DIgeneratorcircuitbreakeropened*)
		tGCB_OGP : HALioDi_Type; (*DIgeneratorcircuitbreakerothergeneratorparallel*)
		tGCB_On : HALioDi_Type; (*DI generator circuit breaker closed*) (*OldName:GCB_ON;Cycle:5*)
		tGCB_OpF_Ext : HALioDi_Type; (*generator circuit breaker opening failure*) (*OldName:newPV; Cycle:5*)
		tGCB_Rac : HALioDi_Type; (*DIgeneratorcircuitbreakerrackedin*)
		tGCB_Rdy : HALioDi_Type; (*DIgeneratorcircuitbreakerready(forclose*)
		tGCB_RI : HALioDi_Type; (*DIgeneratorcircuitbreakerreelaseisland*)
		tGCB_SM1 : HALioDi_Type; (*DIgeneratorcircuitbreakeroutputsignalmonitoring1*)
		tGCB_SM2 : HALioDi_Type; (*DIgeneratorcircuitbreakercontactsignalmonitoring2*)
		tGenCtr_CktBkr_Trip : HALioDi_Type; (*generatorcicuitbreakeroff*)
		tGenHeat_CB_On : HALioDi_Type; (*Generator heater circuit breaker tripped*) (*Oldname:newPv;Cycle:5;*)
		tGenIF_CB_On : HALioDi_Type; (*Circuit breaker tripped supply +TCAI --> +GENI*)
		tGenLossExc_Ext : HALioDi_Type; (*Generator loss of excitation*) (* OldName: newPV; Cycle:2; *)
		tGenOverExc : HALioDi_Type; (*generator overexcitation*) (*OldName:newPV; Cycle:5*)
		tGenPrctTrip : HALioDi_Type; (*DI:Generatorprotectiontrip*)
		tGenRotorEarthFault : HALioDi_Type; (*rotor earth fault*) (*OldName:newPV; Cycle:5*)
		tGen_Exc_Off : HALioDi_Type; (*de-excitation*)
		tGen_LO_CoolingSys_Fail : HALioDi_Type; (*generatorlubeoilcoolingsystemfailure*)
		tGen_RVM : HALioDi_Type; (*DIgeneratorreleasevoltagematching(leroysomer*)
		tGen_T_In : HALioAi_Type; (*actualvaluegeneratorinlettemperature*)
		tGF_OilSystem : HALioDi_Type; (*DI general failure oil system*) (*OldName:newPV; Cycle:5*) (*STM*)
		tGndFailure : HALioDi_Type; (*DI:earthfailure*)
		tGT1_1_BackFireDev : HALioDi_Type; (*DIAntibackfiredevice1line1*)
		tGT1_1_SafeDevOK : HALioDi_Type; (*DIGassafetydevice1line1*)
		tGT1_2_BackFireDev : HALioDi_Type; (*DIAntibackfiredevice1line2*)
		tGT1_2_SafeDevOK : HALioDi_Type; (*DIGassafetydevice2line2*)
		tGT1_3_BackFireDev : HALioDi_Type; (*DIAntibackfiredevice1line3*)
		tGT1_3_SafeDevOK : HALioDi_Type; (*DIGassafetydevice3line3*)
		tGT1_4_BackFireDev : HALioDi_Type; (*DIAntibackfiredevice1line4*)
		tGT1_4_SafeDevOK : HALioDi_Type; (*DIGassafetydevice4line4*)
		tGT1_SafeDevOK : HALioDi_Type; (*DIGassafetydevice1*)
		tGT2_SafeDevOK : HALioDi_Type; (*DIGassafetydevice2*)
		tGT_AirSupply_LoLo : HALioDi_Type; (*DI FALSE = compressed air supply pressure for gas train too low - error*) (*Oldname : DI_GT_AirSupply_LoLo Cyclic: 2; *)
		tGT_BackFireDev : HALioDi_Type; (*DIAntibackfiredevice*)
		tGT_CalibrateActive : HALioDi_Type; (*DICalibrationGasanalysis*)
		tGT_CH4 : HALioAi_Type; (*IF653 CH4 content	*) (* OldName:  	ANA_CH4		; Cycle: 5;*)
		tGT_CV : HALioAi_Type; (*AICalorificvalue*)
		tGT_FlairFail : HALioDi_Type; (*DIFlarefailure*)
		tGT_Flap1_Closed : HALioDi_Type; (*DIGasflap1closed(Feedback*)
		tGT_Flap1_Opened : HALioDi_Type; (*DIGasflap1opened(Feedback*)
		tGT_Flap2_Closed : HALioDi_Type; (*DIGasflap2closed(Feedback*)
		tGT_Flap2_Opened : HALioDi_Type; (*DIGasflap2opened(Feedback*)
		tGT_FlareOpMod : HALioDi_Type; (*DIFlareinoperationalmode*)
		tGT_GC_Fail : HALioDi_Type; (*DIGascompressorfailure*)
		tGT_O2 : HALioAi_Type; (*IF656 O2 content	*) (* OldName:  	ANA_O2		; Cycle: 5;*)
		tGT_SelectRatioMix : HALioDi_Type; (*DI: Digital input to select gas mixing (1-3 or 1_2-3)*)
		tGT_TypSwitch : HALioDi_Type; (*DIGastypeswitchtosecondgas*)
		tHumidity_AirIn : HALioAi_Type;
		tHWF_Fail : HALioDi_Type; (*DI: Failure heat water flap*)
		tHWP_Op : HALioDi_Type; (*DIheatingwaterpumpoperating*)
		tIFCP_CBTrip : HALioDi_Type; (*DIinterfacecontrolpanel-circuitbreakertripped*)
		tIgn2_Run_Hal : HALioDi_Type; (*DI:Ignitionsystemdoublerunning*)
		tIgn_OverspeedRelay : HALioDi_Type; (*DI:Overspeedrelay*)
		tIgn_Run_Hal : HALioDi_Type; (*DI:Ignitionsystemrunning*)
		tImp_OpHour : HALioDo_Type; (*Operating hour impulse from Digital Output *) (*OldName: new PV; Cycle: 5;*)
		tInAirER_Lou1Opened : HALioDi_Type; (*DIintakeairengineroomlouver1open*)
		tInAirER_Lou2Opened : HALioDi_Type; (*DIintakeairengineroomlouver2open*)
		tIsoCB_Off : HALioDi_Type; (*DIdisconnectingcircuitbreakeropened,francecountryspecific*)
		tI_Avg : ARRAY[0..2]OF HALioAi_Type; (*IF513 gen.current average v.	*) (* OldName:  	ANA.IDURCH	; Cycle: 5;*)
		tI_Diff : HALioDi_Type; (*generatordifferentialprotectiontrip*)
		tI_GenAsy_Ext : HALioDi_Type; (*Current negative sequence*) (* OldName: newPV; Cycle:2; *)
		tI_L1 : ARRAY[0..2]OF HALioAi_Type; (*PhasecurrentgeneratorI1*)
		tI_L2 : ARRAY[0..2]OF HALioAi_Type; (*PhasecurrentgeneratorI2*)
		tI_L3 : ARRAY[0..2]OF HALioAi_Type; (*PhasecurrentgeneratorI3*)
		tI_MMD_Asy : ARRAY[0..2]OF HALioDi_Type; (*generatorcurrentnegativesequencetoohigh*)
		tI_MMD_LimHi : HALioDi_Type; (*MMD:overloadshortcircuit*)
		tI_MMD_Neutr_LimHi : ARRAY[0..2]OF HALioDi_Type; (*generatorneutralcurrenttoohigh*)
		tKLS90_1 : HALioAi_Type; (*AI:KLS90sensor1signal*)
		tKLS90_2 : HALioAi_Type; (*AI:KLS90sensor1signal*)
		tLam_Act : HALioAi_Type; (*actualLambdavalue*)
		tLeak_FreshOilPump : HALioDi_Type; (*DI leakage fresh oil pump*) (*OldName:newPV; Cycle:5*) (*STM*)
		tLeak_FreshOilTank : HALioDi_Type; (*DI leakage fresh oil tank*) (*OldName:newPV; Cycle:5*) (*STM*)
		tLeak_WasteOilPump : HALioDi_Type; (*DI leakage waste oil pump*) (*OldName:newPV; Cycle:5*) (*STM*)
		tLeak_WasteOilTank : HALioDi_Type; (*DI leakage waste oil tank*) (*OldName:newPV; Cycle:5*) (*STM*)
		tLev_OilSkid_Sump_Hi : HALioDi_Type; (*DI OilSkid oil in safety sump *)
		tLev_OilSkid_Tank : HALioAi_Type; (*AI OilSkid tank level*)
		tLineCB_On : HALioDi_Type; (*DIlinecircuitbreakerclosed*)
		tLSL_In : HALioAi_Type; (*AIloadsharingline*)
		tLSL_Out : HALioAo_Type; (* = 		-	AO load sharing line	*) (*OldName: LasttOut	; Cycle: 5;*)
		tL_DayOilSump_Hi : HALioDi_Type; (*DI: Day tank oil collector pan high*)
		tL_DayOilTank_Hi : HALioDi_Type; (*DI: Day oil tank high*)
		tL_DayOilTank_Lo : HALioDi_Type; (*DI Fresh oil day tank level low*)
		tL_DayOilTank_LoLo : HALioDi_Type; (*DI Fresh oil day tank level low (2nd level switch)*)
		tL_ECW_Lo : HALioDi_Type; (*DIenginecoolingwaterlevellow*)
		tL_ECW_LoLo : HALioDi_Type; (*DIenginecoolingwaterlevellowlow*)
		tL_FreshOilTank_Hi : HALioDi_Type; (*DI fresh oil tank level high*) (*OldName:newPV; Cycle:5*) (*STM*)
		tL_FreshOilTank_Lo : HALioDi_Type; (*DIfreshoiltanklevellow*)
		tL_FreshOilTank_LoLo : HALioDi_Type; (*DI Fresh oil tank level low (2nd level switch)*)
		tL_InMa_Hi : HALioDi_Type; (*DIwateringressintoinletmanifold*)
		tL_InMa_NotHi : HALioDi_Type; (*DIwateringressintoinletmanifoldnegated*)
		tL_OilSump2Hi : HALioDi_Type; (*DIleveloilsump2high*)
		tL_OilSump3Hi : HALioDi_Type; (*DIleveloilsump3high*)
		tL_OilSumpHi : HALioDi_Type; (*DIleveloilsumphigh*)
		tL_WasteOilDayTank_Hi : HALioDi_Type; (*DI Waste oil day tank level high*)
		tL_WasteOilTank_Hi : HALioDi_Type; (*DIwasteoiltanklevelhigh*)
		tMainsStartDevFail : HALioDi_Type; (*DImainsstartdevicefailure*)
		tMainsStartDevOk : HALioDi_Type; (*DImainsstartingdeviceOK*)
		tManAuxCtr : tManAuxCtr_typ; (*Manual operating auxiliaries control - Handbedienebene*) (*OldName: new PV; Cycle: 5;*)
		tMCB_DcpQu_SetEUCOf : HALioDi_Type; (* DI: reset decoupling quickly from EU (ERDF) *) (*OldName:DI_RFDemMCBoff PV;Cycle:2;*)
		tMCB_DcpQu_SetEUCOn : HALioDi_Type; (* DI: set decoupling quickly from EU (ERDF) *) (*OldName:DI_SFDemMCBoff PV;Cycle:2;*)
		tMCB_Dcp_SetEUCOf : HALioDi_Type; (* DI: rest requirement decoupling from EU(ERDF),DIs *) (*OldName:DI_RDemandMCBoff PV;Cycle:2;*)
		tMCB_Dcp_SetEUCOn : HALioDi_Type; (* DI: set requirement  decoupling from EU(ERDF),DIs *) (*OldName:DI_SDemandMCBoff PV;Cycle:2;*)
		tMCB_Off : HALioDi_Type; (*DImainscircuitbreakeropened*)
		tMCB_OL : HALioDi_Type; (*DImainscircuitbreakeroverload*)
		tMCB_On : HALioDi_Type; (*DI mains circuit breaker closed*) (*OldName:MCB_ON;Cycle:5*)
		tMCB_OpF_Ext : HALioDi_Type; (*generator circuit breaker opening failure*) (*OldName:newPV; Cycle:5*)
		tMCB_Rac : HALioDi_Type; (*DImainscircuitbreakerrackedin*)
		tMCB_Rdy : HALioDi_Type; (*DImainscircuitbreakerready(forclose*)
		tMCB_Rel_Sync : HALioDi_Type; (* DI: release synchronization from EU(ERDF) *) (*OldName:DI_ReleaseMCBon PV;Cycle:2;*)
		tMCB_Rem : HALioDi_Type; (*DImainscircuitbreakerremote(operatingmode*)
		tMCB_SM : HALioDi_Type; (*DImainscircuitbreakersignalmonitoring*)
		tMCP_CBTrip : HALioDi_Type; (*DImodulecontrolpanel-circuitbreakertripped*)
		tMMD_FW_Version : ARRAY[0..2]OF HALioAi_INT_Type; (* program version MMD firmware *)
		tMnsOk : HALioDi_Type; (*DImainsok*)
		tMnsOk_C13100 : HALioDi_Type; (*DImainsokC13.100monitoringdevice,francecountryspecific*)
		tMnsOk_ClosCond_Ok : HALioDi_Type; (*closing condition from external facility*) (* OldName: newPV; Cycle:2; *)
		tMnsOk_GTE : HALioDi_Type; (*DImainsokGTEmonitoringdevice,francecountryspecific*)
		tMnsOk_TGS : HALioDi_Type; (*DImainsokTGSmonitoringdevice,francecountryspecific*)
		tMns_MDF : HALioDi_Type; (*DImainsmonitoringdevicefailure*)
		tMO_PowerOverload : HALioDi_Type; (*DI:SAFIignitionpowermoduleoverload*)
		tMO_PwrReply : HALioDi_Type; (*DI:MORISIgnitionPowerModuleOn*)
		tMO_SaftyLoop : HALioDi_Type; (*DI:MORISSavetyloopclosed*)
		tN2_GV1_Closed : HALioDi_Type; (*DIN2gasvalve1closedstatus*)
		tN2_GV2_Closed : HALioDi_Type; (*DIN2gasvalve2closedstatus*)
		tN_Set_ExtAI_Norm : HALioAi_Type; (*External speed setpoint*) (*OldName: ; Cycle: 5;*)
		tN_TCHP : HALioAi_Type; (*highpressureturbochargerspeed[rpm]*)
		tN_TCHP_A : HALioAi_Type; (*highpressureturbochargerspeedA[rpm]*)
		tN_TCHP_B : HALioAi_Type; (*highpressureturbochargerspeedB[rpm]*)
		tN_TCLP : HALioAi_Type; (*lowpressureturbochargerspeed[rpm]*)
		tN_TCLP_A : HALioAi_Type; (*lowpressureturbochargerspeedA[rpm]*)
		tN_TCLP_B : HALioAi_Type; (*lowpressureturbochargerspeedB[rpm]*)
		tOF_DayOilTank : HALioDi_Type; (*DI Overfill prevention device fresh oil day tank*)
		tOF_FreshOilTank : HALioDi_Type; (*DI overfill prevention device fresh oil tank*) (*OldName:newPV; Cycle:5*) (*STM*)
		tOF_WasteOilDayTank : HALioDi_Type; (*DI Overfill prevention device waste oil day tank*)
		tOF_WasteOilTank : HALioDi_Type; (*DI overfill prevention device waste oil tank*) (*OldName:newPV; Cycle:5*) (*STM*)
		tOilSkid_AuxV_Ok : HALioDi_Type; (*DI OilSkid auxiliaries voltage not available*)
		tOilSkid_AuxV_Ok_UPS : HALioDi_Type; (*DI OilSkid auxiliaries voltage not available - UPS*)
		tOilSkid_Fan_CBOk : HALioDi_Type; (*DI OilSkid fan - circuit breaker*)
		tOilSkid_Heater_CBOk : HALioDi_Type; (*DI OilSkid heater - circuit breaker*)
		tOilSkid_MCB : HALioDi_Type; (*DI OilSkid main switch auxiliaries opened*)
		tOilSkid_PumpC_CBOk : HALioDi_Type; (*DI OilSkid circulation pump - circuit breaker*)
		tOilSkid_PumpHP_CBOk : HALioDi_Type; (*DI OilSkid high pressure pump - circuit breaker*)
		tOilSkid_PumpHP_CBOk_UPS : HALioDi_Type; (*DI OilSkid high pressure pump - circuit breaker UPS*)
		tOilSkid_PumpHP_DemOff : HALioDi_Type; (*DI OilSkid high pressure pump - demand OFF*)
		tOilSkid_PumpHP_DemOn : HALioDi_Type; (*DI OilSkid high pressure pump - demand ON*)
		tOilSkid_PumpLP_CBOk : HALioDi_Type; (*DI OilSkid low pressure pump - circuit breaker*)
		tOlShortCirc : HALioDi_Type; (*DI:Overload/shortcircuit*)
		tOnly_Island : HALioDi_Type; (*DIonlyislandoperation*)
		tOutAirER_LouOpened : HALioDi_Type; (*DIoutletairengineroomlouveropen*)
		tP0_BLOCK_DEIE : HALioDi_Type; (* DI : Installed 1/0 switch *) (*OldName:Cust_switch_erdf PV;Cycle:2;*)
		tPB2MM : ParaBase2MM_type; (*Data exchange structure to ParaBase*) (*OldName: new PV; Cycle: 5;*)
		tPCaComp_BackFireDev : HALioDi_Type; (*DIAntibackfire device prechamper after compressor*)
		tPCbComp_BackFireDev : HALioDi_Type; (*DIAntibackfire device prechamper before compressor*)
		tPCG_GC_Fail : HALioDi_Type; (*DIFailureprechambergascompressor*)
		tPCG_GC_Oil_Min : HALioDi_Type; (*DIprechambergascompressoroillevel*)
		tPFC_SetCOf : HALioDi_Type; (* DI:primary frequency control - off (deactivate) *) (* OldName: DI_GCP_PFC_R; Cycle:HALioDi_Type; *)
		tPFC_SetCOn : HALioDi_Type; (* DI:primary frequency control - on (activate) *) (* OldName: DI_GCP_PFC_S; Cycle:HALioDi_Type; *)
		tPFC_SOf : HALioDo_Type;
		tPFC_SOn : HALioDo_Type;
		tPFUC_GenC_SetEUCOf : HALioDi_Type; (* DI: setpoint reactive power characteristics COS(phi)=f(U) von EU -off (deactive) *) (* OldName: DI_GCQ_PFU_R; Cycle:HALioDi_Type; *)
		tPFUC_GenC_SetEUCOn : HALioDi_Type; (* DI: setpoint reactive power characteristics COS(phi)=f(U) von EU -on (active) *) (* OldName: DI_GCQ_PFU_S; Cycle:HALioDi_Type; *)
		tQP_GenC_SetEUCOf : HALioDi_Type; (* DI: setpoint reactive power characteristics Q=f(P) von EU -off (deactive) *) (* OldName: DI_GCQ_PFU_R; Cycle:HALioDi_Type; *)
		tQP_GenC_SetEUCOn : HALioDi_Type; (* DI: setpoint reactive power characteristics Q=f(P) von EU -on (active) *) (* OldName: DI_GCQ_PFU_S; Cycle:HALioDi_Type; *)
		tPFUC_GenC_SOf : HALioDo_Type;
		tPFUC_GenC_SOn : HALioDo_Type;
		tQP_GenC_SOn : HALioDo_Type; (*  reactive power characteristics Q=f(P) from EU is on  *)
		tQP_GenC_SOf : HALioDo_Type; (*  reactive power characteristics Q=f(P) from EU is off *)
		tPF_Act : ARRAY[0..2]OF HALioAi_Type; (*IF511 generator power factor	*) (* OldName:  	ANA.COSPHI	; Cycle: 5;*)
		tPF_GenC_Fix1SOn : HALioDo_Type;
		tPF_GenC_Fix2SOn : HALioDo_Type;
		tPF_GenC_Fix3SOn : HALioDo_Type;
		tPF_GenC_Fix4SOn : HALioDo_Type;
		tPF_GenC_Fix5SOn : HALioDo_Type;
		tPF_GenC_SetEU : HALioAi_Type; (* AI: setpoint  genetaror power factor (COS PHI) from EU *) (* OldName: AI_GCQ_PF; Cycle:HALioAi_Type; *)
		tPF_GenC_SetEUCOf : HALioDi_Type; (* DI: setpoint  genetaror power factor (COS PHI) from EVA - off (deactivate)  *) (* OldName: DI_GCQ_PF_R; Cycle:HALioDi_Type; *)
		tPF_GenC_SetEUCOn : HALioDi_Type; (* DI: setpoint  genetaror power factor (COS PHI) from EU - on (activate)  *) (* OldName: DI_GCQ_PF_S; Cycle:HALioDi_Type; *)
		tPF_GenC_SetFix1EU : HALioDi_Type; (* DI: setpoint  genetaror power factor (COS PHI) - Q-fixvalue 1 from EU *) (* OldName: DI_GCB_PF_FIX1; Cycle:HALioDi_Type; *)
		tPF_GenC_SetFix2EU : HALioDi_Type; (* DI: setpoint  genetaror power factor (COS PHI) - Q-fixvalue 2 from EU *) (* OldName: DI_GCB_PF_FIX2; Cycle:HALioDi_Type; *)
		tPF_GenC_SetFix3EU : HALioDi_Type; (* DI: setpoint  genetaror power factor (COS PHI) - Q-fixvalue 3 from EU *) (* OldName: DI_GCB_PF_FIX3; Cycle:HALioDi_Type; *)
		tPF_GenC_SetFix4EU : HALioDi_Type; (* DI: setpoint  genetaror power factor (COS PHI) - Q-fixvalue 4 from EU *) (* OldName: DI_GCB_PF_FIX4; Cycle:HALioDi_Type; *)
		tPF_GenC_SetFix5EU : HALioDi_Type; (* DI: setpoint  genetaror power factor (COS PHI) - Q-fixvalue 5 from EU *) (* OldName: DI_GCB_PF_FIX5; Cycle:HALioDi_Type; *)
		tPF_GenC_SOf : HALioDo_Type;
		tPF_GenC_SOn : HALioDo_Type;
		tPLim_GenC_Act : HALioDo_Type;
		tPLim_GenC_SetEU : HALioAi_Type; (*AI:setpointpowerlimitation(Plim*)
		tPLim_GenC_SetEUCOf : HALioDi_Type; (* DI: setpoint power limitation (Plim) from EU - off (deactivate) *) (* OldName: DI_GCP_Plim_R; Cycle:HALioDi_Type; *)
		tPLim_GenC_SetEUCOn : HALioDi_Type; (* DI: setpoint power limitation (Plim) from EU - on (activate) *) (* OldName: DI_GCP_Plim_S; Cycle:HALioDi_Type; *)
		tPLim_GenC_SetEUPFix1 : HALioDi_Type; (*DI:powerlimitationfixvalue1*)
		tPLim_GenC_SetEUPFix2 : HALioDi_Type; (*DI:powerlimitationfixvalue2*)
		tPLim_GenC_SetEUPFix3 : HALioDi_Type; (*DI:powerlimitationfixvalue3*)
		tPLim_GenC_SetEUPFix4 : HALioDi_Type; (*DI:powerlimitationfixvalue4*)
		tPLim_GenC_SetEUPFix5 : HALioDi_Type; (*DI:powerlimitationfixvalue5*)
		tPLim_GenC_SOf : HALioDo_Type;
		tPLim_GenC_SOn : HALioDo_Type;
		tPos_Act_CBV_A1 : HALioAi_Type; (*AI: compressor bypass valve position A1*)
		tPos_Act_CBV_A2 : HALioAi_Type; (*AI: compressor bypass valve position A2*)
		tPos_Act_CBV_B1 : HALioAi_Type; (*AI: compressor bypass valve position B1*)
		tPos_Act_CBV_B2 : HALioAi_Type; (*AI: compressor bypass valve position B2*)
		tPos_Act_GM1_Norm : HALioAi_Type; (*gasmixer1-normedactualpositionfrompotentiometer[%]*)
		tPos_Act_GM2_Norm : HALioAi_Type; (*gasmixer2-normedactualpositionfrompotentiometer[%]*)
		tPos_Act_TV : HALioAi_Type; (*AI: throttle valve bypass valve position*)
		tPos_Act_TV_A1 : HALioAi_Type; (*AI: throttle valve bypass valve position A1*)
		tPos_Act_TV_A2 : HALioAi_Type; (*AI: throttle valve bypass valve position A2*)
		tPos_Act_TV_B1 : HALioAi_Type; (*AI: throttle valve bypass valve position B1*)
		tPos_Act_TV_B2 : HALioAi_Type; (*AI: throttle valve bypass valve position B2*)
		tPos_Act_WG_A : HALioAi_Type; (*wastegatevalvepositionA*)
		tPos_Act_WG_B : HALioAi_Type; (*wastegatevalvepositionB*)
		tPos_ChC_Valve : HALioAi_Type; (*AI: position charge temperature regulation valve*) (*STM*)
		tPos_CircLou1 : HALioAi_Type; (*AI: position air circulation louver 1) (*STM*)
		tPos_CircLou2 : HALioAi_Type; (*AI: position air circulation louver 2 (*STM*)
		tPos_HW_EC_ReValve : HALioAi_Type; (*AI: position heating water return temperature after cooler regulation valve*) (*STM*)
		tPos_HW_ReValve : HALioAi_Type; (*AI: position heating water return temperature regulation valve*) (*STM*)
		tPos_InlLou1 : HALioAi_Type; (*AI: position air inlet louver 1*) (*STM*)
		tPos_InlLou2 : HALioAi_Type; (*AI: position air inlet louver 2*) (*STM*)
		tPos_OutlLou1 : HALioAi_Type; (*AI: position air outlet louver 1*) (*STM*)
		tPos_OutlLou2 : HALioAi_Type; (*AI: position air outlet louver 2*) (*STM*)
		tPos_SGM_Enc1 : HALioAi_INT_Type; (*SGM encoder position stepper 1 [1]*)
		tPos_SGM_Enc2 : HALioAi_INT_Type; (*SGM encoder position stepper 2 [1]*)
		tPos_SGM_Enc3 : HALioAi_INT_Type; (*SGM encoder position stepper 3 [1]*)
		tPos_ThR_Val_In1 : HALioDi_Type; (*DI1thermalreactorflapinpositionmovedin*)
		tPos_ThR_Val_In2 : HALioDi_Type; (*DI2thermalreactorflapinpositionmovedin*)
		tPos_ThR_Val_Mid : HALioDi_Type; (*DIthermalreactorflapinmiddleposition*)
		tPos_ThR_Val_Out1 : HALioDi_Type; (*DI1thermalreactorflapinpositionmovedout*)
		tPos_ThR_Val_Out2 : HALioDi_Type; (*DI2thermalreactorflapinpositionmovedout*)
		tPow_Heat : HALioAi_Type; (*IFXXX heating power engine heat water circuit*) (*OldName: newPV; Cycle: 5;*) (*STM*)
		tPrDiff_ER : HALioAi_Type; (*AI: engine room difference pressure*) (*STM 2*)
		tPr_AirStarter_Supply : HALioAi_Type; (*AI Air starter supply pressure [bar]*)
		tPr_AirStarter_Tank : HALioAi_Type; (*AI air starter tank pressure [bar]*)
		tPr_a_BbFilt : HALioAi_Type; (*AI Pressure after Blow-by filter *)
		tPr_a_BbFilt_A : HALioAi_Type; (*AI Pressure after Blow-by filter A*)
		tPr_a_BbFilt_B : HALioAi_Type; (*AI Pressure after Blow-by filter B*)
		tPr_Baro : HALioAi_Type; (*AIBarometricpressure*)
		tPr_CC : HALioAi_Type; (* AI pressure crank case [bar] *) (*OldName:AI_KGD; Cycle:5*)
		tPr_CCircuit_Lo : HALioDi_Type; (*DIwaterpressurecoolercircuitlow*)
		tPr_ChC_Lo : HALioDi_Type; (*DIchargecoolerwaterpressurelow*)
		tPr_Ch_P1HP : HALioAi_Type; (*chargepressurep1beforehighpressureTC[bar]*)
		tPr_Ch_P1HP_A : HALioAi_Type; (*chargepressurep1beforehighpressureTCA[bar]*)
		tPr_Ch_P1HP_B : HALioAi_Type; (*chargepressurep1beforehighpressureTCB[bar]*)
		tPr_Ch_P1LP_A : HALioAi_Type; (*Air pressure before low-pressure compressor A in exhaust gas turobcharger (P1 A)*)
		tPr_Ch_P1LP_B : HALioAi_Type; (*Air pressure before low-pressure compressor B in exhaust gas turobcharger (P1 B)*)
		tPr_Ch_P2 : HALioAi_Type; (*actualchargepressurebeforethrottlevalve*)
		tPr_Ch_P2s : HALioAi_Type; (*actualchargepressure  fuel mixture  - Input from HAL - !CONSIDER ALSO USING IN_CU.rPr_Ch_P2s_Avg! *)
		tPr_Ch_P2s_A : HALioAi_Type; (*chargepressurep2'afterthrottlevalveA[bar]*)
		tPr_Ch_P2s_B : HALioAi_Type; (*chargepressurep2'afterthrottlevalveB[bar]*)
		tPr_Ch_P2_A : HALioAi_Type; (*chargepressurep2beforethrottlevalveA[bar]*)
		tPr_Ch_P2_B : HALioAi_Type; (*chargepressurep2beforethrottlevalveB[bar]*)
		tPr_Diff_ExGCooler : HALioAi_Type; (*AI: Differential pressure exhaust gas cooler*)
		tPr_Diff_ExGFilter : HALioAi_Type; (*AI: Differential pressure exhaust gas filter*)
		tPr_ECW : HALioAi_Type; (*AIpressureenginecoolingwater*)
		tPr_ECWaEng : HALioAi_Type; (*Cooling water pressure downstream of the engine*)
		tPr_EGaHPTC_A : HALioAi_Type; (* AI: Exhaust gas pressure after high-pressure turbocharger A  (M.02-PI-153) *) (* OldName: AI_M_02_PI_153; Cyclic: 5; *)
		tPr_EGaHPTC_B : HALioAi_Type; (* AI: Exhaust gas pressure after high-pressure turbocharger B  (M.02-PI-253) *) (* OldName: AI_M_02_PI_253; Cyclic: 5; *)
		tPr_EGaLPTC_A : HALioAi_Type; (* AI: Exhaust gas pressure after low-pressure turbocharger A  (M.02-PI-154) *) (* OldName: AI_M_02_PI_154; Cyclic: 5; *)
		tPr_EGaLPTC_B : HALioAi_Type; (* AI: Exhaust gas pressure after low-pressure turbocharger B  (M.02-PI-254) *) (* OldName: AI_M_02_PI_254; Cyclic: 5; *)
		tPr_EGbHPTC_A : HALioAi_Type; (* AI: Exhaust gas pressure before high-pressure turbocharger A (M.02-PI-152) *) (* OldName: AI_M_02_PI_152; Cyclic: 5; *)
		tPr_EGbHPTC_B : HALioAi_Type; (* AI: Exhaust gas pressure before high-pressure turbocharger B (M.02-PI-252) *) (* OldName: AI_M_02_PI_252; Cyclic: 5; *)
		tPr_EG_Hi : HALioDi_Type; (*DIexhaustgasbackpressurehigh*)
		tPr_EngLubOil : HALioAi_Type; (*AIenginelubricatingoilpressure*)
		tPr_EOF_After : HALioAi_Type; (*AI:Engineoilpressureafteroilfilter,NUP57/AI_M_03_PI_057*)
		tPr_EOF_DiffMon : HALioAi_Type; (*AI:Oilpressurebeforeoilfilter*)
		tPr_EO_Gear_Min : HALioDi_Type; (*DI:Oilpressurelowtransmission*)
		tPr_EO_Mod_Out : HALioAi_Type; (*pressure engine oil module outlet M.03-PI-006*) (*V04.03.00.00*)
		tPr_f_BbFilt : HALioAi_Type; (*AI Pressure before Blow-by filter *)
		tPr_f_BbFilt_A : HALioAi_Type; (*AI Pressure before Blow-by filter A*)
		tPr_f_BbFilt_B : HALioAi_Type; (*AI Pressure before Blow-by filter B*)
		tPr_GR_I : HALioAi_Type; (*AI Gas Pressure in Gas Rail number 1 *) (* OldName: AIPressGasRail; Cyclic: 2; *)
		tPr_GR_II : HALioAi_Type; (*AI Gas Pressure in Gas Rail number 2*) (* OldName: AIPressGasRail_II; Cyclic: 2; *)
		tPr_GT1 : HALioAi_Type; (*AIGaspressuregastrain1afterfilter*)
		tPr_GT1_1_Max : HALioDi_Type; (*DIGaspressuremaximumgastrain1-line1*)
		tPr_GT1_1_Min : HALioDi_Type; (*DIGaspressurelowgastrain1-line1*)
		tPr_GT1_2_Max : HALioDi_Type; (*DIGaspressuremaximumgastrain1-line2*)
		tPr_GT1_2_Min : HALioDi_Type; (*DIGaspressurelowgastrain1-line2*)
		tPr_GT1_3_Max : HALioDi_Type; (*DIGaspressuremaximumgastrain1-line3*)
		tPr_GT1_3_Min : HALioDi_Type; (*DIGaspressurelowgastrain1-line3*)
		tPr_GT1_4_Max : HALioDi_Type; (*DIGaspressuremaximumgastrain1-line4*)
		tPr_GT1_4_Min : HALioDi_Type; (*DIGaspressurelowgastrain1-line4*)
		tPr_GT1_Max : HALioDi_Type; (*DIGaspressuremaximumgastrain1*)
		tPr_GT1_Min : HALioDi_Type; (*DIGaspressurelowgastrain1*)
		tPr_GT2_Max : HALioDi_Type; (*DIGaspressuremaximumgastrain2*)
		tPr_GT2_Min : HALioDi_Type; (*DIGaspressurelowgastrain2*)
		tPr_GT_Gas : HALioAi_Type; (*IF654 gas pressure	*) (* OldName:  	ANA_GD		; Cycle: 5;*)
		tPr_GT_MinBefCompr : HALioDi_Type; (*DIGaspressurelowbeforegascompressor*)
		tPr_GT_Suct : HALioAi_Type; (*IF655 suction pressure	*) (* OldName:  	ANA_SD		; Cycle: 5;*)
		tPr_HW_Hi : HALioDi_Type; (*DIheatwaterpressurehigh*)
		tPr_HW_Hi1 : HALioDi_Type; (*DIheatwaterpressurehigh*)
		tPr_HW_Lo : HALioDi_Type; (*DIheatwaterpressurelow*)
		tPr_HW_Re_HT : HALioAi_Type; (*pressure heat water return high temp.circuit M.06-PI-002*) (*V04.03.00.00*)
		tPr_HW_Re_LT : HALioAi_Type; (*pressure heat water return low temp.circuit M.07-PI-002*) (*V04.03.00.00*)
		tPr_HW_Re_PreH_ECW : HALioAi_Type; (*pressure heat water return preheating engine cooling water M.04-PI-005*) (*V04.03.00.00*)
		tPr_HW_Re_PreH_EO : HALioAi_Type; (*pressure heat water return preheating engine oil M.03-PI-005*) (*V04.03.00.00*)
		tPr_HW_Su_HT : HALioAi_Type; (*supply water pressure HT circuit*) (*OldName:AI_p_VL_HT; Cycle:5;*)
		tPr_HW_Su_LT : HALioAi_Type; (*supply water pressure LT circuit*) (*OldName:AI_p_VL_NT; Cycle:5;*)
		tPr_MGT_a_Filt : HALioAi_Type; (*AI main gas train pressure after filter [bar]*) (* OldName: AI_p_GT1; Cyclic: 2; *)
		tPr_N2_Hi : HALioDi_Type; (*DIpressureN2high*)
		tPr_N2_Lo : HALioDi_Type; (*DIpressureN2low*)
		tPr_OilSkid_HP_DE : HALioAi_Type; (*AI OilSkid oil pressure in high pressure circuit to DE bearing*)
		tPr_OilSkid_HP_NDE : HALioAi_Type; (*AI OilSkid oil pressure in high pressure circuit to NDE bearing *)
		tPr_Oil_LPTC_In_A : HALioAi_Type; (*oil pressure LP turbo charger A inlet*) (*OldName:P_OEL_ND_EintrittA; Cycle:5;*)
		tPr_Oil_LPTC_In_B : HALioAi_Type; (*oil pressure LP turbo charger B inlet*) (*OldName:P_OEL_ND_EintrittB; Cycle:5;*)
		tPr_PC : HALioAi_Type; (*AIPressureprechamber*)
		tPr_PCG : HALioAi_Type; (*IF650 pre chamber gas pressure	*) (* OldName:  	ANA_VKGD	; Cycle: 5;*)
		tPr_PCGBefComp_Lo : HALioDi_Type; (*DIsuctionpressureprechambergascompressorhigh*)
		tPr_PCGT : HALioAi_Type; (*AIGaspressureprechambergastrainafterfilter*)
		tPr_PCGT_a_Filt : HALioAi_Type; (*V04.02.00.00*)
		tPr_PCGT_Out : HALioAi_Type; (*AI Warning measuring signal failure - gas pressure after pre chamber gas pressure regulator*) (* OldName: AI_p_PCGT_Out; Cyclic: 2; *)
		tPr_PCG_Min : HALioDi_Type; (*DIPrechambergascompressorpressureminimum*)
		tPr_PC_Diff : HALioAi_Type; (*IFF	-	IF652 pre chamber diff.pressure	*) (* OldName:  	ANA_; Cycle: 5;*)
		tPr_TCOF_EOF_DiffMax : HALioDi_Type; (*DI:Differencepressureturbochargeroilfilterhigh*)
		tPr_TC_EOF_After : HALioAi_Type; (*AIoilpressureafterturbochargeroilfilter,NUP62/AI_M_03_PI_062*)
		tPr_TC_EOF_Before : HALioAi_Type; (*AI:Oilpressureinfrontofturbochargeroilfilter,NUP61/AI_M_03_PI_061*)
		tPr_ThR_AirLo : HALioDi_Type; (*DIthermalreactorcompressedairpressurelow*)
		tPS400V_ENGIA_CB_On : HALioDi_Type; (*Supply disconnecting device 400VAC +ENGIA on*)
		tPS_EI_CB_On : HALioDi_Type; (*power supply engine interface panel circuit breaker on*) (*OldName:PS_EI_CB_trip; Cycle:5;*)
		tPS_FreshOilPump_Hi : HALioDi_Type; (*DI Fresh oil pump oil pressure maximum*)
		tP_Act : ARRAY[0..2]OF HALioAi_Type; (*actualelectricpower[kW]*)
		tP_FC_RMC_neg : HALioAi_Type; (*AI: negative reserve power for FC [%/P_nom] *)
		tP_FC_RMC_pos : HALioAi_Type; (*AI: positive reserve power for FC [%/P_nom] *)
		tP_GenC_Fix0SOn : HALioDo_Type;
		tP_GenC_Fix1SOn : HALioDo_Type;
		tP_GenC_Fix2SOn : HALioDo_Type;
		tP_GenC_Fix3SOn : HALioDo_Type;
		tP_GenC_Fix4SOn : HALioDo_Type;
		tP_GenC_Fix5SOn : HALioDo_Type;
		tP_GenC_SetEU : HALioAi_Type; (*AI:requestpowervaluefromEU*)
		tP_GenC_SetEUCOf : HALioDi_Type; (* DI: request power value from EU - off (deactivate) *) (* OldName: DI_GCP_P_R; Cycle:HALioDi_Type; *)
		tP_GenC_SetEUCOn : HALioDi_Type; (* DI: request power value from EU - on (activate) *) (* OldName: DI_GCP_P_S; Cycle:HALioDi_Type; *)
		tP_GenC_SetFix1EU : HALioDi_Type; (*V04.03.00.00*)
		tP_GenC_SetFix2EU : HALioDi_Type; (*V04.03.00.00*)
		tP_GenC_SetFix3EU : HALioDi_Type; (*V04.03.00.00*)
		tP_GenC_SetFix4EU : HALioDi_Type; (*V04.03.00.00*)
		tP_GenC_SetFix5EU : HALioDi_Type; (*V04.03.00.00*)
		tP_GenC_SOf : HALioDo_Type;
		tP_GenC_SOn : HALioDo_Type;
		tP_GenRev_Ext : HALioDi_Type; (*Generator reverse power*) (* OldName: newPV; Cycle:2; *)
		tP_GT_Max_Backfire : HALioDi_Type; (*DIgaspressurehigh-backfire*)
		tP_Heat : HALioAi_Type; (*AI heating power engine heat water circuit [kW]*) (*STM 2*)
		tP_Heat_Imp : HALioDi_Type; (*heating power engine heat water circuit impulse (STM 2)*) (*STM*)
		tP_Mns_AnaIn : HALioAi_Type; (*(Interace) Mains Ctrl*)
		tP_Red_Active : HALioDo_Type; (* = 		-	power reduction active - any kind - HALIO DigitalOutput	*) (*OldName: PredAkt	; Cycle: 5;*)
		tP_Red_AI_Norm : HALioAi_Type; (*External power reduction	*) (*OldName: ; Cycle: 5;*)
		tP_Red_CH4Active : HALioDi_Type; (* Power limitation because of CH4 content active *) (*OldName: CH4RED_0; Cyclic:5*)
		tP_Red_GasPrActive : HALioDi_Type; (* Power limitation because OF gas pressure active*) (*OldName: GD_RED_0; Cyclic:5;*)
		tP_Red_Norm : HALioAo_Type; (* = 		-	power reduction	*) (*OldName: P_RED_WE	; Cycle: 5;*)
		tP_Red_SuctPrActive : HALioDi_Type; (* Power limitation because OF suction pressure active*) (*OldName: SD_RED_0; Cyclic:5;*)
		tP_Set_ExtAI_Norm : HALioAi_Type; (*External power setpoint	*) (*OldName:ssPowerSetAnalogWE; Cycle: 5;*)
		tP_Set_FC : HALioAi_Type; (*AI: generator power setpoint [%/P_nom]*)
		tQLim_GenC_Act : HALioDo_Type; (* DO: reactive power limitation (Plim) from EU is aktiv *) (* OldName: DO_GCQ_Qlim_ACT; Cycle: 5 *)
		tQLim_GenC_SetEU : HALioAi_Type; (*AI:setpointreactivepowerlimitation(Qlim*)
		tQLim_GenC_SetEUCOf : HALioDi_Type; (* DI: setpoint reactive power limitation (Qlim) from EU - off (deactivate) *) (* OldName: DI_GCQ_Qlim_R; Cycle:HALioDi_Type; *)
		tQLim_GenC_SetEUCOn : HALioDi_Type; (* DI: setpoint reactive power limitation (Qlim) from EU - on (activate) *) (* OldName: DI_GCQ_Qlim_S; Cycle:HALioDi_Type; *)
		tQLim_GenC_SOf : HALioDo_Type; (* DO: reactive power limiting (QLim)  is off *) (* OldName: DO_GCQ_Qlim_OFF; Cycle: 5 *)
		tQLim_GenC_SOn : HALioDo_Type; (* DO: reactive power limiting (QLim)  is on *) (* OldName: DO_GCQ_Qlim_ON; Cycle: 5 *)
		tQPC_GenC_SetEUCOf : HALioDi_Type; (* DI: setpoint reactive power characteristics COS(phi)=f(P) from EU - off (deactivate) *) (* OldName: DI_GCQ_PFP_R; Cycle:HALioDi_Type; *)
		tQPC_GenC_SetEUCOn : HALioDi_Type; (* DI: setpoint reactive power characteristics COS(phi)=f(P) from EU - on (activate) *) (* OldName: DI_GCQ_PFP_S; Cycle:HALioDi_Type; *)
		tQPC_GenC_SOf : HALioDo_Type;
		tQPC_GenC_SOn : HALioDo_Type;
		tQUC_GenC_SetEUCOf : HALioDi_Type; (* DI: setpoint reactive power characteristics Q=f(U) from EU -off (deactivate) *) (* OldName: DI_GCQ_QU_R; Cycle:HALioDi_Type; *)
		tQUC_GenC_SetEUCOn : HALioDi_Type; (* DI: setpoint reactive power characteristics Q=f(U) from EU -on (activate) *) (* OldName: DI_GCQ_QU_S; Cycle:HALioDi_Type; *)
		tQUC_GenC_SOf : HALioDo_Type;
		tQUC_GenC_SOn : HALioDo_Type;
		tQU_GenC_Set : HALioAi_Type; (*AI:setpointgeneratorvoltageforrectivepowercontrol[%]vorEU*)
		tQ_Act : ARRAY[0..2]OF HALioAi_Type; (*actualreactivepower[kVar]*)
		tQ_GenC_Fix1SOn : HALioDo_Type;
		tQ_GenC_Fix2SOn : HALioDo_Type;
		tQ_GenC_Fix3SOn : HALioDo_Type;
		tQ_GenC_Fix4SOn : HALioDo_Type;
		tQ_GenC_Fix5SOn : HALioDo_Type;
		tQ_GenC_SetEU : HALioAi_Type; (*AI:setpointreactivepowercharacteristic(Q*)
		tQ_GenC_SetEUCOf : HALioDi_Type; (* DI: setpoint reactive power characteristic (Q) from EU - off (deactivate) *) (* OldName: DI_GCQ_Q_R; Cycle:HALioDi_Type; *)
		tQ_GenC_SetEUCOn : HALioDi_Type; (* DI: setpoint reactive power characteristic (Q) from EU - on (activate) *) (* OldName: DI_GCQ_Q_S; Cycle:HALioDi_Type; *)
		tQ_GenC_SetFix1EU : HALioDi_Type; (*DI:reactivepower(Q*)
		tQ_GenC_SetFix2EU : HALioDi_Type; (*DI:reactivepower(Q*)
		tQ_GenC_SetFix3EU : HALioDi_Type; (*DI:reactivepower(Q*)
		tQ_GenC_SetFix4EU : HALioDi_Type; (*DI:reactivepower(Q*)
		tQ_GenC_SetFix5EU : HALioDi_Type; (*DI:reactivepower(Q*)
		tQ_GenC_SOf : HALioDo_Type;
		tQ_GenC_SOn : HALioDo_Type;
		tQ_GenUnderVoltProt : HALioDi_Type; (*reactive power/undervoltage protection (Q-U-protection)*) (*OldName:newPV; Cycle:5*)
		tRelAux : HALioDi_Type; (*DIreleaseengineoperationfromauxiliarieswithmonitoring*)
		tRelAuxNoMon : HALioDi_Type; (*DIreleaseengineoperationfromauxiliarieswithnomonitoring*)
		tRelEngOpFromGSy : HALioDi_Type; (*DIreleaseengineoperationfrom'gemeinsame'synchronization*)
		tRelGasPlant : HALioDi_Type; (*DIReleasefromgasplantmissing.FALSE=Missing*)
		tRelMainGVext : HALioDi_Type; (*DIreleasemaingasvalvefromexternal*)
		tRel_BS : HALioDi_Type; (*DIreleaseblackstart*)
		tRel_ER_PurgeCycle : HALioDi_Type; (*DIreleasepurgecycle*)
		tRel_I : HALioDi_Type; (*DIreleaseislandoperation*)
		tRel_LS : HALioDi_Type; (*DIreleaseloadshedding*)
		tRel_MasCtr : HALioDi_Type; (*releasefrommastercontrol*)
		tRel_U_Sel_LS_Gen : HALioDi_Type; (*ReleasevoltageselectionLS-Generator*)
		tReq_PeakLoad : HALioDi_Type; (*requestpeakload*)
		tReq_PowMod : HALioDi_Type; (*DIrequestpoweroperationmode*)
		tReq_Test : HALioDi_Type; (*requesttestmode*)
		tResetRemExt : HALioDi_Type; (*resetremoteexternal*)
		tResetRemoteExt : HALioDi_Type; (*resetremoteexternal*)
		tRMC_SetCOf : HALioDi_Type; (* DI:regulation margin control -off (deactivate) *) (* OldName: DI_GCP_RMC_R; Cycle:HALioDi_Type; *)
		tRMC_SetCOn : HALioDi_Type; (* DI:regulation margin control -on (activate) *) (* OldName: DI_GCP_RMC_S; Cycle:HALioDi_Type; *)
		tRMC_SOf : HALioDo_Type;
		tRMC_SOn : HALioDo_Type;
		tRSE_SetEUCOf : HALioDi_Type; (* DI: reset decoupling RSE from EU (ERDF) *) (*OldName:DI_RDEmRSE PV;Cycle:2;*)
		tRSE_SetEUCOn : HALioDi_Type; (* DI: set decoupling RSE from EU (ERDF) *) (*OldName:DI_SDEmRSE PV;Cycle:2;*)
		tSafetyLoop_EmStop : HALioDi_Type; (*safety loop emergency stop ok*) (*OldName:DI_SIS; Cycle:5*)
		tSafetyLoop_Eng : HALioDi_Type; (*safetyloopengine*)
		tSafetyLoop_Gas : HALioDi_Type; (*DIsafetyloopgasok*)
		tSafetyLoop_HWC : HALioDi_Type; (*safetyloopheatwatercircuitok*)
		tScavFanCB_trip : HALioDi_Type; (*DIexhaustgasscavengingfancircuitbreakertripped*)
		tScavFanFC_P_Lo : HALioDi_Type; (*DIexhaustgasscavengingfanfrequencyconverterpowerlow*)
		tScavFanFC_Rdy : HALioDi_Type; (*DIexhaustgasscavengingfanfrequencyconverterreadyforoperation*)
		tScavFanOp : HALioDi_Type; (*DIexhaustgasscavengingfanoperating*)
		tScavVaClosed : HALioDi_Type; (*DIscavengingvalveclosed*)
		tScavVaFailure : HALioDi_Type; (*DIscavengingvalvefailure*)
		tScavVaOpened : HALioDi_Type; (*DIscavengingvalveopened*)
		tSelGasTyp : HALioDi_Type; (*DI:Selectiongastype-general*)
		tSelGasTyp2 : HALioDi_Type; (*DI:Selectiongastype2*)
		tSelGasTyp3 : HALioDi_Type; (*DI:Selectiongastype3*)
		tSelGasTyp4 : HALioDi_Type; (*DI:Selectiongastype4*)
		tSet_ILF_COf : HALioDi_Type; (*DI: de-activation of local frequency integrator *)
		tSet_ILF_COn : HALioDi_Type; (*DI: activation of local frequency integrator *)
		tSet_FC_COf : HALioDi_Type; (*DI: de-activation of frequency control*)
		tSet_FC_COn : HALioDi_Type; (*DI: activation of frequency control*)
		tSTT_CB_On : HALioDi_Type; (*control voltage transformer circuit breaker on*) (*OldName:STT_CB_trip; Cycle:5;*)
		tSy_N_Down : HALioDi_Type; (*DIexternalspeedmatchingDOWN*)
		tSy_N_Up : HALioDi_Type; (*DIexternalspeedmatchingUP*)
		tS_Act : ARRAY[0..2]OF HALioAi_Type; (* appearent power [kV] *)
		tTBMode : HALioDi_Type; (*DItestbenchmode*)
		tTCOP_CB_On : HALioDi_Type; (*Failure Pump Turbocharger pressure*)
		tTCOP_Grid : HALioDi_Type; (*turbo charger oil pump mains voltage ok*)
		tTCOP_Op : HALioDi_Type; (*DIturbochargeroilpumpoperating*)
		tTCOP_UPS_CB_On : HALioDi_Type; (*Circuit breaker tripped Prelubrication oil pump / Cool down oilpump*)
		tTempMax_GenCB : HALioDi_Type; (*DI: Temperatur max Generatorschalter*)
		tThR_LampTest : HALioDi_Type; (*DIthermalreactorlamptest*)
		tThR_SL : HALioDi_Type; (*DIthermalreactorsafetyloop*)
		tThR_Swth_On : HALioDi_Type; (*DIthermalreactoroperationswitchon*)
		tTransformerTrip : HALioDi_Type; (*DItransformerfailure*)
		tTransformerWarning : HALioDi_Type; (*DItransformerfailure*)
		tT_AirER : HALioAi_Type; (*IF649 room temperature	*) (* OldName:  	ANA_RTM		; Cycle: 5;*)
		tT_AirER_Ext_Hi : HALioDi_Type; (*DIairengineroomtemperatureexternalhigh*)
		tT_AirER_Ext_Hi1 : HALioDi_Type; (*DIroomtemperaturelimit*)
		tT_AirER_Ext_Hi2 : HALioDi_Type; (*DIroomtemperaturelimit*)
		tT_AirER_Ext_Hi3 : HALioDi_Type; (*DIroomtemperaturelimit*)
		tT_AirIFCP_Hi : HALioDi_Type; (*DIairtemperatureinterfacecontrolpanelhigh*)
		tT_AirIn : HALioAi_Type;
		tT_AirOutdoor : HALioAi_Type; (*IF662 outdoor temperature	*) (* OldName:  	ANA_ULT		; Cycle: 5;*)
		tT_Cat : HALioAi_Type; (*AIcatalysttemperature*)
		tT_CBearing_Hi : HALioDi_Type; (*Warning Temperature conrod bearing*)
		tT_CBearing_HiHi : HALioDi_Type; (*Shut down Temperature conrod bearing*)
		tT_CD_Re : HALioAi_Type; (*AI: Return temperature condensor circuit*)
		tT_CD_Su : HALioAi_Type; (*AI: Supply temperature condensor circuit*)
		tT_ChCW_Hi : HALioDi_Type; (*DIchargecoolingwatertemperaturehigh*)
		tT_Ch_T1HP : HALioAi_Type; (*chargetemperaturebeforehighpressureTC[degC]*)
		tT_Ch_T1HP_A : HALioAi_Type; (*chargetemperaturebeforehighpressureTCA[degC]*)
		tT_Ch_T1HP_B : HALioAi_Type; (*chargetemperaturebeforehighpressureTCB[degC]*)
		tT_Ch_T2s : HALioAi_Type; (*AItemperaturechargeafterthrottlevalve IF601 fuel mixture temperature	- Input from HAL - !CONSIDER ALSO USING IN_CU.rT_Ch_T2s_Avg! 	(replaces old IN_CU.rT_Ch)*)
		tT_Ch_T2s_A : HALioAi_Type; (*chargetemperaturet2'afterthrottlevalveA[degC]*)
		tT_Ch_T2s_B : HALioAi_Type; (*chargetemperaturet2'afterthrottlevalveB[degC]*)
		tT_CO2_Hi : HALioDi_Type; (*DICO2temperaturereactorchamberhigh*)
		tT_ECW : HALioAi_Type; (*AItemperatureenginecoolingwater*)
		tT_ECWbEng : HALioAi_Type; (*Engine jacket water temperature befor Engine*)
		tT_ECW_AfEng : HALioAi_Type; (*AItemperatureenginecoolingwaterafterengine[degC]*)
		tT_ECW_Ext_Hi : HALioDi_Type; (*DItemperatureenginecoolingwaterhighexternal*)
		tT_ECW_Mod_In : HALioAi_Type; (*temperature engine cooling water, engine cooling water module inlet M.04-TI-003*) (*V04.03.00.00*)
		tT_ECW_Mod_Out : HALioAi_Type; (*temperature engine cooling water, engine cooling water module outlet M.04-TI-004*) (*V04.03.00.00*)
		tT_ECW_PreH_Hi : HALioDi_Type; (*DItemperatureenginecoolingwaterpreheatinghigh*)
		tT_ECW_PreH_HiHi : HALioDi_Type; (*DItemperatureenginecoolingwaterpreheatinghighhigh*)
		tT_EGaCat : HALioAi_Type; (*AIexhaustgastemperatureaftercatalyst*)
		tT_EGafHeEx1 : HALioAi_Type; (*IF660exh.gastemp.aft.heatexch.1*)
		tT_EGafHeEx2 : HALioAi_Type; (*IF661exh.gastemp.aft.heatexch.2*)
		tT_EGaHE : HALioAi_Type; (*AIexhaustgastemperatureafterheatexchanger*)
		tT_EGaHE1 : HALioAi_Type; (*AIexhaustgastemperatureafterheatexchanger1*)
		tT_EGaHE2 : HALioAi_Type; (*AIexhaustgastemperatureafterheatexchanger2*)
		tT_EGaHPTC_A : HALioAi_Type; (* AI: Exhaust gas temperatur after high-pressure turbocharger A  (M.02-TI-167) *) (* OldName: AI_M_02_TI_167; Cyclic: 5; *)
		tT_EGaHPTC_B : HALioAi_Type; (* AI: Exhaust gas temperatur after high-pressure turbocharger A  (M.02-TI-267) *) (* OldName: AI_M_02_TI_267; Cyclic: 5; *)
		tT_EGaLPTC_A : HALioAi_Type; (*AIexhaustgastemperatureafterlowpressureturbochargerA*)
		tT_EGaLPTC_B : HALioAi_Type; (*AIexhaustgastemperatureafterlowpressureturbochargerB*)
		tT_EGaTC : HALioAi_Type; (*AIexhaustgastemperatureafterturbocharger*)
		tT_EGbCat : HALioAi_Type; (*AIexhaustgastemperaturebeforecatalyst*)
		tT_EGbHPTC_A : HALioAi_Type; (* AI: Exhaust gas temperature before high-pressure turbocharger A  (M.02-TI-166) *) (* OldName: AI_M_02_TI_166; Cyclic: 5; *)
		tT_EGbHPTC_B : HALioAi_Type; (* AI: Exhaust gas temperature before high-pressure turbocharger B  (M.02-TI-266) *) (* OldName: AI_M_02_TI_266; Cyclic: 5; *)
		tT_EGbTC : HALioAi_Type; (*AIexhaustgastemperaturebeforeturbocharger*)
		tT_EG_Cyl : ARRAY[0..24]OF HALioAi_Type; (*AI cylinder exhaust gas temperatures*) (* OldName: t_zyl; Cycle:2*)
		tT_EO : HALioAi_Type; (*AItemperatureengineoil*)
		tT_EOP_After : HALioAi_Type; (*AI:Oiltemperatureafteroilpump,NUT71/AI_M_03_TI_071*)
		tT_EO_Gear_Max : HALioDi_Type; (*DI:Oiltemperaturehightransmission*)
		tT_EO_Mod_In : HALioAi_Type; (*temperature engine oil, oil module inlet M.03-TI-004*) (*V04.03.00.00*)
		tT_EO_Mod_Out : HALioAi_Type; (*temperature engine oil, oil module outlet M.03-TI-003*) (*V04.03.00.00*)
		tT_EO_Pan : HALioAi_Type; (*engine oil temperature oil pan, M.03-TI-002*) (*OldName:AI_t_OilPan; Cycle:5*)
		tT_EO_Preheating : HALioAi_Type; (*AI:Oiltemperaturepreheating,NUT78/AI_M_03_TI_078*)
		tT_EO_PreH_Hi : HALioDi_Type; (*Temperatur limit preheating EO warn*)
		tT_EO_PreH_HiHi : HALioDi_Type; (*Temperatur limit preheating EO alarm*)
		tT_GenAirOut : HALioAi_Type; (*Exhaust air Temperature*)
		tT_Gen_Bear_A_Act : HALioAi_Type; (*generatorbearingAtemperaturesignal*)
		tT_Gen_Bear_B_Act : HALioAi_Type; (*generatorbearingBtemperaturesignal*)
		tT_Gen_Wind : HALioAi_Type; (*actualgeneratorwindingtemperaturesignal*)
		tT_Gen_Wind_Act_L1 : HALioAi_Type; (*generatorwindingtemperaturesignal,windingphase1*)
		tT_Gen_Wind_Act_L2 : HALioAi_Type; (*generatorwindingtemperaturesignal,windingphase2*)
		tT_Gen_Wind_Act_L3 : HALioAi_Type; (*generatorwindingtemperaturesignal,windingphase3*)
		tT_GR : HALioAi_Type; (*AI Gas rail temperature*) (*OldName: AI_GRTP; Cyclic: 2; *)
		tT_GT : HALioAi_Type; (*IF657 gas temperature	*) (* OldName:  	ANA_GT		; Cycle: 5;*)
		tT_GT_Ok : HALioDi_Type; (*DIGastemperatureOK*)
		tT_HW_HC_Re : HALioAi_Type; (*AI: Heating circuit return temperature*)
		tT_HW_Hi : HALioDi_Type; (*DIheatwatertemperaturehigh*)
		tT_HW_Hi1 : HALioDi_Type; (*DIheatwatertemperaturehigh*)
		tT_HW_Re : HALioAi_Type; (*AItemperatureheatwaterreturn*)
		tT_HW_ReAfEC : HALioAi_Type; (*IF659 ret.wat.temp.after cooler	*) (* OldName:  	ANA.RLT_NK	; Cycle: 5;*)
		tT_HW_ReBeEng : HALioAi_Type; (*AItemperatureheatwaterreturnbeforeengine*)
		tT_HW_Re_LT : HALioAi_Type; (*AItemperatureheatwaterreturnlowtemp.circuit[degC]*)
		tT_HW_Re_PreH_ECW : HALioAi_Type; (*temperature heat water return preheating engine cooling water M.04-TI-006*) (*V04.03.00.00*)
		tT_HW_Re_PreH_EO : HALioAi_Type; (*temperature heat water return preheating engine oil M.03-TI-006*) (*V04.03.00.00*)
		tT_HW_Su : HALioAi_Type; (*AItemperatureheatwatersupply*)
		tT_HW_Su_LT : HALioAi_Type; (*AItemperatureheatwatersupplylowtemp.circuit[degC]*)
		tT_HW_Su_PreH_ECW : HALioAi_Type; (*temperature heat water supply preheating engine cooling water M.04-TI-005*) (*V04.03.00.00*)
		tT_HW_Su_PreH_EO : HALioAi_Type; (*temperature heat water supply preheating engine oil M.03-TI-005*) (*V04.03.00.00*)
		tT_OilSkid_Supply : HALioAi_Type; (*AI OilSkid supply temperature*)
		tT_OilSkid_Tank : HALioAi_Type; (*AI OilSkid tank temperature*)
		tT_PCGAfCo : HALioAi_Type; (*AItemperatureprechambergasaftercooler*)
		tT_PCGAfComp_Hi : HALioDi_Type; (*DItemperatureprechambergascompressoroutlethigh*)
		tT_PCGT : HALioAi_Type; (*AIPrechambergastemperature*)
		tT_PlateHE : HALioAi_Type; (*AIplatetemperatureheatexchanger*)
		tT_Re_PriCirc : HALioAi_Type; (*IFXXX return water temperature high primary circuit*) (*OldName: newPV; Cycle: 5;*) (*STM*)
		tT_Re_SecCirc : HALioAi_Type; (*IFXXX return water temperature high secondary circuit*) (*OldName: newPV; Cycle: 5;*) (*STM*)
		tT_Su_PriCirc : HALioAi_Type; (*IFXXX supply water temperature high primary circuit*) (*OldName: newPV; Cycle: 5;*) (*STM*)
		tT_Su_SecCirc : HALioAi_Type; (*IFXXX supply water temperature high secondary circuit*) (*OldName: newPV; Cycle: 5;*) (*STM*)
		tT_ThR_Chamber1_1 : HALioAi_Type; (*thermalreactorchambertemperature1_1*)
		tT_ThR_Chamber1_2 : HALioAi_Type; (*thermalreactorchambertemperature1_2*)
		tT_ThR_Chamber2_1 : HALioAi_Type; (*thermalreactorchambertemperature2_1*)
		tT_ThR_Chamber2_2 : HALioAi_Type; (*thermalreactorchambertemperature2_2*)
		tT_ThR_ChamberLo : HALioDi_Type; (*DIthermalreactorchambertemperaturelow*)
		tT_ThR_Comp : HALioAi_Type; (*thermalreactorcompensationtemperature*)
		tT_ThR_In : HALioAi_Type; (*thermalreactorinlettemperature*)
		tT_ThR_Out : HALioAi_Type; (*thermalreactoroutlettemperature*)
		tT_ThR_Swg_Hi : HALioDi_Type; (*DIthermalreactorswitchgeartemperaturehigh*)
		tUPS_CB_On : HALioDi_Type; (*Circuit breaker tripped supply UPS*)
		tUPS_Ok : HALioDi_Type; (*failureuninterruptedpowersupply*)
		tU_Adj_Minus : HALioDi_Type; (*VoltageadjustmentMinus*)
		tU_Adj_Plus : HALioDi_Type; (*VoltageadjustmentPlus*)
		tU_Avg : ARRAY[0..2]OF HALioAi_Type; (*IF514 gen.voltage average value	*) (* OldName:  	ANA.UDURCH	; Cycle: 5;*)
		tU_GenAsy_Ext : HALioDi_Type; (*Voltage negative sequence*) (* OldName: newPV; Cycle:2; *)
		tU_GenC_SetCUST : HALioAi_Type; (*costumiz:scalingvalueforgeneratorvoltageforreactivepowerfromEU*)
		tU_GenDiode_Fail : HALioDi_Type; (*generatordiodealarm*)
		tU_GenDiode_Trip : HALioDi_Type; (*generator diode trip*) (*OldName:DI_GEN_D_Tr ;Cycle:5*)
		tU_GenOverVolt : HALioDi_Type; (*failuregeneratorovervoltageprotection*)
		tU_Gen_Contr_Fail : HALioDi_Type; (*generatorvoltageregulatorfailure*)
		tU_Gen_Dec : HALioDi_Type; (*digitalinputforvoltageadjustmentbyMMU(decreasing*)
		tU_Gen_Exc : HALioAi_Type; (*actualexcitationvoltagesignal,filteredandscaled*)
		tU_Gen_Inc : HALioDi_Type; (*digitalinputforvoltageadjustmentbyMMU(increasing*)
		tU_Gen_LimHi : ARRAY[0..2]OF HALioDi_Type; (*generatorvoltagetoohigh*)
		tU_Gen_LimLo : ARRAY[0..2]OF HALioDi_Type; (*generatorvoltagetoolow*)
		tU_Gen_LimLo2 : ARRAY[0..2]OF HALioDi_Type; (*generatorvoltagetoolow2*)
		tU_L1L2 : ARRAY[0..2]OF HALioAi_Type; (* generator voltage phase 1_2 [V] *)
		tU_L1N : ARRAY[0..2]OF HALioAi_Type; (* generator voltage phase 1_N [V] *)
		tU_L2L3 : ARRAY[0..2]OF HALioAi_Type; (* generator voltage phase 2_3 [V] *)
		tU_L2N : ARRAY[0..2]OF HALioAi_Type; (* generator voltage phase 2_N [V] *)
		tU_L3L1 : ARRAY[0..2]OF HALioAi_Type; (* generator voltage phase 3_1 [V] *)
		tU_L3N : ARRAY[0..2]OF HALioAi_Type; (* generator voltage phase 3_N [V] *)
		tU_MMD_Asy : ARRAY[0..2]OF HALioDi_Type; (*generatorvoltagenegativesequencetoohigh*)
		tU_MMD_Synch1 : ARRAY[0..2]OF HALioAi_Type; (*synchronization voltage 1*)
		tU_MMD_Synch2 : ARRAY[0..2]OF HALioAi_Type; (*synchronization voltage 2*)
		tU_StarterBat_Lo : HALioDi_Type; (*DIvoltagestarterbatterylow*)
		tVol_GT : HALioAi_Type; (*IF658 gas quantity	*) (* OldName:  	ANA_GM		; Cycle: 5;*) (* ------------------ implemented for Coupling Module ---------------------------- -->> *)
		tSet_PU_COn : HALioDi_Type; (*DI: activation of P(U) on*)
		tSet_PU_COf : HALioDi_Type; (*DI: de-activation of P(U) off*)
		tPU_SOn : HALioDo_Type; (*DO: feedback signal: PU switched on*)
		tPU_SOf : HALioDo_Type; (*DO: feedback signal: PU switched off*)
		bReady4VeryFastStart : BOOL; (* Ready for very fast start *)
		bReady4FastStart : BOOL; (* Ready for fast start *)
		bVeryFastStart_Prep : BOOL; (* very fast start preperation running *)
		bFastStart_Prep : BOOL; (* fast start preperation running *)
		tU_SetExtAI_Norm : HALioAi_Type; (* External voltage set point [%Unom] *) (*OldName:tU_SetExt_Norm;Cycle:5*)
		tGR2CU : GRID2CUSTOM_Struct; (* Data exchange structure to Custom *)
		tHA2CU : HALIO2CUSTOM_Struct; (* Data exchange structure to HALIO *)
		rP_set_vis_Norm : REAL; (* setpoint value for power from visu [%Pnom] *)
		rDPr_OFU_Filt : REAL; (* Oilfilter difference pressure (oil filter unit) [bar] *)
		rGMU_Pr_DiffGas : ARRAY[0..4]OF REAL; (*Differential Pressure over device [mbar*10]*)
		rGMU_Pos_Valve_Prom : ARRAY[0..4]OF REAL; (*Valve Position [%o]*)
		rGMU_Pr_FuelGas : ARRAY[0..4]OF REAL; (*Fuel Gas Pressure at device inlet [mbar*10]*)
		rGMU_T_FuelGas : ARRAY[0..4]OF REAL; (*Fuel Gas Temperature at device inlet [degC *10]*)
		rGMU_Q_FuelGas : ARRAY[0..4]OF REAL; (*Fuel Gas Amount denormalized [l/s*1000]*)
		rCtr_Q_Set : REAL; (* Generator Q controller output *)
		rI_Dyn : ARRAY[0..2]OF REAL; (* current dynamic *) (* OldName:usIDyn; Cycle: *)
		rI_GenUnbalanced : ARRAY[0..2]OF REAL; (* unbalanced generator current [1/10 %]  *) (* OldName:ssIGenUnbalanced; Cycle: *)
		rU_MMD_Diff : ARRAY[0..2]OF REAL; (* votage deviation synchronization *) (* OldName:ssSynchVoltDeviation; Cycle: *)
		iIdx_MMD_SynchMode : ARRAY[0..2]OF INT; (* synchronization mode *) (* OldName:usVisSynchMode; Cycle: *)
		rU_Ign_Avg : REAL; (* *) (*OldName:AvgVolt; Cycle:;*)
		rU_Ign_Max : REAL; (* *) (*OldName:MaxVolt; Cycle:;*)
		rU_Ign_Min : REAL; (* *) (*OldName:MinVolt; Cycle:;*)
		rCA_Ign_Min : REAL; (*Actual min. cylinder ignition point*) (*OldName:ZZPMin; Cycle:;*)
		rCA_Ign_Max : REAL; (*Actual max. cylinder ignition point*) (*OldName:ZZPMax; Cycle:;*)
		iIdx_IgnSelfTest : INT; (*Number of shown picture regarding step of execution. 0 - 50 in steps of 10. Detailded description in every step where used.*) (*OldName:usP5xSelftestStep; Cycle:;*)
		bGen_DeExc_Rdy : BOOL; (* Generator Deexitation ready *)
		tCtrTR_Heater_Out : _tGeACtrOut; (* Heater Controller *) (*OldName: newPV; Cycle:5;*)
		rP_ThR_EH : REAL; (* thermal reactor electrical heating power *) (*OldName:y_HE_Prom; Cycle:5;*)
		tThR_Val_Air : HALioDo_Type; (* DO thermal reactor purge air valve *) (*OldName:DO_SPLU_STOP; Cycle:5;*)
		tThR_GT_COn1 : HALioDo_Type; (* DO1 thermal reactor gas injection command on *) (*OldName:DO_EIND_EIN1; Cycle:5;*)
		tThR_GT_COn2 : HALioDo_Type; (* DO2 thermal reactor gas injection command on *) (*OldName:DO_EIND_EIN2; Cycle:5;*)
		iSA_ERZuV : ARRAY[0..24]OF INT; (* Error Rate for spark delay  *) (* OldName:ucERZuV; Cycle: *)
		iSA_ERDurTol : ARRAY[0..24]OF INT; (* Error Rate for Duration Tolerance  *) (* OldName:ucERDurTol; Cycle: *)
		rPr_Leanox_Dev : REAL; (* leanox controller deviation [bar] *) (* OldName: ssPressLeanoxError; Cycle: 2 *)
		rMisf_Intgr : REAL; (* integrator electrical misfires [0..1] *) (* OldName: ssMisfInt; Cycle: 2 *)
		rP_Power_Dev : REAL; (* power controller deviation [kW] *) (* OldName: new PV; Cycle: 2 *)
		rN_Speed_Dev : REAL; (* speed controller deviation [rpm] *) (* OldName: new PV; Cycle: 2 *)
		tLL : _tLL_Struct; (* Leanox line for all gas types, including interpolation *)
		iPassLevel : INT; (*pass level actual*) (*OldName:ucPassLevel; Cycle:2;*)
		tExtCtrOk : HALioDi_Type; (* DI: External speed / voltage controller okay *) (*OldName: newPV; Cycle:5;*)
		iPanelSelection : INT; (*Controls lock of local operation for additional touch panels*)
		bMsg1041Set : BOOL; (*power signal missing*)
		bMsg1042Set : BOOL; (*power signal overload*)
		bMsg2801Set : BOOL; (*module blocked by grid connection conditions*)
		bMsg2934Set : BOOL; (*module blocked by grid connection conditions after mains failure*)
		bMsg1038Set : BOOL; (*Generator reverse power, Trip*)
		bMsg1109Set : BOOL; (*loss of excitation (trip)*)
		bMsg1110Set : BOOL; (*Generator frequency low, Trip*)
		bMsg1111Set : BOOL; (*Generator frequency high, Trip*)
		bMsg1112Set : BOOL; (*Neutral current high, Trip*)
		bMsg1126Set : BOOL; (*generator voltage low, Trip*)
		bMsg1127Set : BOOL; (*generator voltage high, Trip*)
		bMsg1143Set : BOOL; (*Voltage negative sequence (Voltage asymmetry), Trip*)
		bMsg1144Set : BOOL; (*Current negative sequnece (Current asymmetrt), Trip*)
		bMsg2277Set : BOOL; (*Generator voltage too low 2*)
		bMsg2316Set : BOOL; (*generator voltage high 2 (one phase)*)
		bMMD_BB_AlarmTestOn : BOOL; (*MMD_BB  alarm test On*)
		rP_Red_T_Oil_Norm : REAL; (*power reduction by oil temp. max related to rP_Nom*) (*OldName:RED_OLT; Cycle:5;*)
		tEOVal_DemOpen : HALioDo_Type; (*DO engine oil refill valve demand open *) (*OldName:OELV_AUF; Cycle:5*)
		rP_Red_Ch_T2HP_Norm : REAL; (*power reduction by charge temperatur T2 after high-pressure TC related to rP_Nom*) (*OldName:new PV;Cycle:5;*)
		rP_Red_Ch_T2LP_Norm : REAL; (*power reduction by charge temperatur T2 after low-pressure TC related to rP_Nom*) (*OldName:new PV;Cycle:5;*)
		rP_Red_Ch_T2s : REAL; (*	power reduction by mixture temperatiure [KW]	*) (*OldName:ssPowerRedGemisch;Cycle:5;*)
		rP_Red_Ch_T2s_Norm : REAL; (*power reduction by charge temperature T2'[%Pnom]*) (*OldName: ssPowerRedGemisch; Cycle: 5;*)
		rP_Red_TC_Norm : REAL; (*power reduction by turbo charger speed related to rP_Nom*) (*OldName:new PV;Cycle:5;*)
		bBus_Dem : BOOL; (*demand fieldbus*) (*OldName:BUS_ANF;Cycle:5;*)
		bBusPulse : BOOL; (*bus pulse signal from customer*) (*OldName:newPV; Cycle:5;*)
		bFastStartReq_Bus : BOOL; (* TRUE = Command: get ready for fast start *) (*OldName:newPV; Cycle:5;*)
		bVeryFastStartReq_Bus : BOOL; (* TRUE = Command: get ready for very fast start *) (*OldName:newPV; Cycle:5;*)
		rP_Red_ExtBus_Norm : REAL; (*power reduction by primary control related to rP_Nom [%]*) (*OldName: ssPowerRedZLT; Cyclic:5;*)
		rCA_Ign_Act : ARRAY[0..24]OF REAL; (*  actual cylinder ignition point  *) (* OldName: ActTiming / ZZPCyl; Cycle:5; *)
		rP_Red_EGT_Norm : REAL; (* power reduction by exhaust gas temp. *) (* OldName: abgas_dp; Cycle:5; *)
		rP_Red_Leanox_Norm : REAL; (*power reduction by leanox related to rP_Nom*) (*OldName:new PV;Cycle:5;*)
		rP_Red_Misf_Norm : REAL; (*power reduction by misfire related to rP_Nom*) (*OldName:new PV;Cycle:5;*)
		iIdx_Gtyp_Dem : INT; (* actual gassort 1..4 *) (*OldName:gasart;Cycle:5;*)
		rGT_QualMix_1_2 : REAL; (*Mixture ratio bet. gas 1 and 2 [%], e.g. value 0.75 =75%*) (* OldName: 	ssMisch1_2	; Cyclic:5; *)
		rGT_RatioMix : REAL; (*Gas mixture rate after ramp fub [%], e.g. 0.5 = 50%*) (* OldName: 	ssRatioMix	; Cyclic:5; *)
		rP_Red_Pr_PCGT_Norm : REAL; (*power redutcion by pre chamber gas pressure related to rP_Nom*) (*OldName:new PV;Cycle:5;*)
		tGV1_Open : HALioDo_Type; (*DO: open gas valve 1*) (*OldName: GASV1; Cycle: 5*)
		tGV2_Open : HALioDo_Type; (*DO: open gas valve 2*) (*OldName: GASV2; Cycle: 5*)
		bGCB_Off_CNS : BOOL; (* generator circuit breaker opened by curent negative sequence *) (*OldName:gcb_off_iasy; Cycle:5;*)
		bGCB_Off_RP : BOOL; (* generator circuit breaker opened by reverse power *) (*OldName:gcb_off_rlsg; Cycle:5;*)
		rP_Red_CosPCtr_F_Norm : REAL; (*Generator power reduction due to Frequency*) (*OldName:ssPowerRedGenFrq;Cycle:5;*)
		rP_Red_CosPCtr_T_Norm : REAL; (*Generator power reduction due to Temperature*) (*OldName:ssPowerRedGenTemp;Cycle:5;*)
		rP_Red_CosPCtr_U_Norm : REAL; (*Generator power reduction due to Voltage*) (*OldName:ssPowerRedGenSpg;Cycle:5;*)
		rP_Red_T_ECW_Norm : REAL; (*power reduction engine cooling water temperature high [% Pnom]*) (*OldName:ssPowerRedKWT; Cycle:5;*)
		rCA_Ign_Avg : REAL; (*Actual ignition point average*) (*OldName:ZZPAvg; Cycle:5;*)
		rU_Ign_Cyl : ARRAY[0..24]OF REAL; (*Ignition voltage for each cylinder *) (*OldName:V_Zyl; Cycle:5;*)
		iKls98_KnckValue_Avg : UINT; (* knocking value average *) (* OldName: Fenst1Avg ; Cycle: 5 *)
		iKls98_KnckValue_Max : UINT; (* maximum knocking value *) (* OldName: Fenst1Max ; Cycle: 5 *)
		iKls98_KnckValue_Min : UINT; (* minimum knocking value *) (* OldName: Fenst1Min ; Cycle: 5 *)
		iKls98_VNValue_Avg : UINT; (* valve noise average *) (* OldName: Fenst2Avg ; Cycle: 5 *)
		iKls98_VNValue_Max : UINT; (* maximum valve noise *) (* OldName: Fenst2Max ; Cycle: 5 *)
		iKls98_VNValue_Min : UINT; (* minimum valve noise *) (* OldName: Fenst2Min ; Cycle: 5 *)
		rKnck_Intgr : ARRAY[0..24]OF REAL; (* integrated cylinder knock values *) (* OldName: IntKlopf ; Cycle: 5 *)
		rKnck_Intgr_Avg : REAL; (* integrated knock value average  *) (* OldName: IntKlopfAv ; Cycle: 5 *)
		rKnck_Intgr_Max : REAL; (* maximum integrated knock value *) (* OldName: IntKlopfMx ; Cycle: 5 *)
		rKnck_Intgr_Min : REAL; (* minimum integrated knock value *) (* OldName: IntKlopfMn ; Cycle: 5 *)
		rKnck_Noise : ARRAY[0..24]OF REAL; (* cylinder value for knocking noise *) (* OldName: Fenst1; Cycle: 5 *)
		rKno_IP_Red : REAL; (* timing reduction by knocking *) (* OldName: klreg_dz ; Cycle: 5 *)
		rKno_T2s_Red : REAL; (* mixture temp. red. by knocking *) (* OldName: klreg_dt2 ; Cycle: 5 *)
		rP_Red_Knck_Norm : REAL; (* power reduction by knocking *) (* OldName: ssPowerRedKlopf ; Cycle: 5 *)
		rVNValue : ARRAY[0..24]OF REAL; (* cylinder values for valve noise *) (* OldName: Fenst2; Cycle: 5 *)
		bSel_DeExc : BOOL; (* DeExcitation selected *) (*OldName:newPV; Cycle:5;*)
		tGCB_RUC : HALioDo_Type; (* generator circuit breaker release undervoltage coil *) (*OldName:A_USP; Cycle:5;*)
		tN_EngStart : HALioDo_Type; (* DO engine startup speed exceeded*) (*OldName:A_DREHZ; Cycle:5;*)
		tP_Lo : HALioDo_Type; (* DO power low (for opening GCB) *) (*OldName:P_MIN; Cycle:5;*)
		rAng_MMD_Diff : ARRAY[0..2]OF REAL; (* angle deviation synchronization *) (* OldName:ssSynchAngleDeviation; Cycle: 5*)
		rT_ThR_Chamber : REAL; (* thermal reactor chamber temperature *) (*OldName:TK; Cycle:5;*)
		rT_ThR_Chamber1_1 : REAL; (* thermal reactor chamber temperature 1_1 *) (*OldName:TK1_1; Cycle:5;*)
		rT_ThR_Chamber1_2 : REAL; (* thermal reactor chamber temperature 1_2 *) (*OldName:TK1_2; Cycle:5;*)
		rT_ThR_Chamber2_1 : REAL; (* thermal reactor chamber temperature 2_1 *) (*OldName:TK2_1; Cycle:5;*)
		rT_ThR_Chamber2_2 : REAL; (* thermal reactor chamber temperature 2_2 *) (*OldName:TK2_2; Cycle:5;*)
		rT_ThR_Comp : REAL; (* thermal reactor compensation temperature *) (*OldName:Tvgl; Cycle:5;*)
		tPr_TCO : HALioAi_Type; (*pressure oil before turbo charger M.03-PI-063*) (*OldName: ; Cycle: 5;*)
		tPr_OFUbFilt : HALioAi_Type; (*pressure oil filter unit before filter M.03-PI-011*) (*Oldname:newPV;Cycle:5*)
		tPr_OFUaFilt : HALioAi_Type; (*pressure oil filter unit after filter M.03-PI-012*) (*Oldname:newPV;Cycle:5*)
		tECW_PreH_Dem : HALioDo_Type; (*DO engine cooling water preheating demand *) (*OldName:A_VORWH; Cycle:5*)
		tCtr_Q_Out : _tGeACtrOut; (* Controller to visulization out structure *) (*OldName:new pv;Cycle:5*)
		tP_Droop_Set : HALioAi_Type; (*Active power setpoint in frequency droop*)
		tQ_Droop_Set : HALioAi_Type; (* Reactive power Droop Offset Setpoint via AI *)
		tU_Bus_L3_1 : ARRAY[0..2]OF HALioAi_Type; (*Line voltage bus bar 3 1 [V] *) (*OldName:ssBusVoltPh3_1; Cycle:5*)
		tU_Bus_L2_3 : ARRAY[0..2]OF HALioAi_Type; (*Line voltage bus bar 2 3 [V] *) (*OldName:ssBusVoltPh2_3; Cycle:5*)
		tU_Bus_L1_2 : ARRAY[0..2]OF HALioAi_Type; (*Line voltage bus bar 1 2 [V] *) (*OldName:ssBusVoltPh1_2; Cycle:5*)
		tU_Bus_L1N : ARRAY[0..2]OF HALioAi_Type; (*bus bar voltage phase 1 [V] *) (*OldName:ssBusVoltPh1_2; Cycle:5*)
		tU_Bus_L2N : ARRAY[0..2]OF HALioAi_Type; (*bus bar voltage phase 2 [V] *) (*OldName:ssBusVoltPh1_2; Cycle:5*)
		tU_Bus_L3N : ARRAY[0..2]OF HALioAi_Type; (*bus bar voltage phase 3 [V] *) (*OldName:ssBusVoltPh1_2; Cycle:5*)
		tGT_RatioMix_Set : HALioAi_Type; (*AI Gas mixing ratio in percent. 1.0 = 100% *)
		bCust_EO_Level_Hi : BOOL; (*Bus signal for customer: Oil level max signal - oil overfill protection*) (*OldName:newPv; Cycle:5;*) (*V04.13.00.00*)
		bPFC_SOf_Bus : BOOL; (*Bus feedback signal: LFSM switched off*)
		bPFC_SOn_Bus : BOOL; (*Bus feedback signal: LFSM switched on*)
		rP_Set_PFC_Norm : REAL; (* Power Setpoint FSM/LFSM *)
		iIdx_Pset_Type : INT; (*power setpoint type*)
		tQ_GenC_CUST : HALioAi_Type; (*costumized scaling value for reactive power (Q) from EU *)
		bBus_failure : BOOL; (*Bus failure new w/v4.13*)
		rHum_Mixture_Abs : REAL; (* absolute humidity mixture [g/kg] *)
		tPlantCom_M2E_In_Cust100ms : ARRAY[0..4]OF tPlantComData_Cust100ms; (*PlantCom Customized Data M2E_In_100ms*)
		tPlantCom_E2E_In_Cust100ms : ARRAY[0..32]OF tPlantComData_Cust100ms; (*PlantCom Customized Data E2E_In_100ms*)
		tPlantCom_E2E_In_Cust10ms : ARRAY[0..32]OF tPlantComData_Cust10ms; (*PlantCom Customized Data E2E_In_10ms*)
		tPlantCom_M2E_In_Cust10ms : ARRAY[0..4]OF tPlantComData_Cust10ms; (*PlantCom Customized Data M2E_In_10ms*)
		bPlantComCfgOk : BOOL; (*PlantCom Config Status*)
	END_STRUCT;
	OUT_Cust_Struct : 	STRUCT
		bCust_Dem_FreshOilPump : BOOL; (*Customized demand for fresh oil pump*) (*OldName:new V4.14; Cycle:5*)
		bCust_Dem_WasteOilPump : BOOL; (*Customized demand for waste oil pump*) (*OldName:new V4.14; Cycle:5*)
		bCust_Dem_OilFillValve : BOOL; (*Customized demand for (fresh) oil valve*) (*OldName:new V4.14; Cycle:5*)
		bPr_GT1_Min_Cust : BOOL; (*Customized set for  1028*) (*OldName: bGasPressureLOW; Cycle: 5;*)
		bPr_GT1_Max_Cust : BOOL; (*Customized set for  1056*) (*OldName: bGasPressureHIGH; Cycle: 5;*)
		bAuxCust_Dem : ARRAY[0..70]OF BOOL; (* Demand reserve auxiliary #21	 * watch for HMI Extension*) (*OldName: B_SV[44] to B_SV[53]	; Cycle: 5;*)
		bBus_Dem : BOOL; (* demand over bus and no bus failure *)
		bChC_Rel : BOOL; (*release charge cooler from monitoring*) (*OldName:GK_frg; Cycle:5;*) (* Gridcode interfaces added  *)
		bCustAlarm_Tripped : ARRAY[0..116]OF BOOL; (* M_A1 to M_A16	-	stored state of reserve alarm	*) (*OldName: bCustAlarm_Tripped	; Cycle: 5;*)
		bCustDigIn : ARRAY[0..200]OF BOOL; (* *) (*OldName: bCustDigIn; Cycle: 5;*)
		bCustDigOut : ARRAY[0..150]OF BOOL; (* *) (*OldName: bCustDigOut; Cycle: 5;*)
		bCustWarn_Tripped : ARRAY[0..60]OF BOOL; (* M_W1 to M_W16	-	stored state of reserve warning	[0..60]*) (*OldName: bCustWarn_Tripped	; Cycle: 5;*)
		bECW_PreH_Dem_Customized : BOOL; (*Engine preheating demand from customer*) (*OldName: new PV; Cycle: 5;*)
		bEC_Rel : BOOL; (*release emergency cooler from monitoring*) (*OldName:K_frg; Cycle:5;*)
		bEGValCtr_HeatOutputDown : BOOL; (*  Interface to connect customized exhaust flap control 	*) (*OldName: unknown	; Cycle: 5;*)
		bEGValCtr_HeatOutputUp : BOOL; (*  Interface to connect customized exhaust flap control 	*) (*OldName: unknown	; Cycle: 5;*)
		bEngDemIsland_Customized : BOOL; (*Engine demind in island mode Customized*) (*OldName: new PV; Cycle: 5;*)
		bEngDSS_Mains : BOOL; (* activate task for engine demand from mains power control  	*) (*OldName: ANF_NB	; Cycle: 5;*)
		bEngDSS_Mains_Block : BOOL; (* Engine shutdown by exceeding allowed grid power	*) (*OldName: BLOCK_NB	; Cycle: 5;*)
		bEngDSS_Mains_Rel : BOOL; (* activate controller demand from mains power control  	*) (*OldName: FG_NB_REG	; Cycle: 5;*)
		bEng_Block_Customized : BOOL; (* = 	BLOCK_NB	-	Engine shutdown by customized module*) (*OldName: unknown	; Cycle: 5;*)
		bEng_Block_EVU : BOOL; (* = 	BLOCK_EVU Engine shutdown by external utility(evu)demand*) (*OldName: BLOCK_EVU; Cycle: 5;*)
		bERDF_Activ : BOOL; (*OLD!- just for compatibility*)
		bILF_SetCOf : BOOL; (* local frequency integrator set command off *)
		bILF_SetCOn : BOOL; (* local frequency integrator set command on *)
		bFC_SetCOf : BOOL; (* frequency control set command off *)
		bFC_SetCOn : BOOL; (* frequency control set command on *)
		bGenC_PBC_SetCOf : BOOL; (* bus: setpoint power P from EU -off (deactivate) *) (* OldName: BUS_GCP_P_R; Cycle:5; *)
		bGenC_PBC_SetCOn : BOOL; (* bus: setpoint power P from EU -on (activate) *) (* OldName: BUS_GCP_P_S; Cycle:5; *)
		bGenC_PFBC_Set : BOOL; (* bus: setpoint  genetaror power factor (COS PHI) from EU *) (* OldName: BUS_GCQ_PF; Cycle:5; *)
		bGenC_PFBC_SetCOf : BOOL; (* bus: setpoint  genetaror power factor (COS PHI) from EU - off (deactivate) *) (* OldName: BUS_GCQ_PF_R; Cycle:5; *)
		bGenC_PFBC_SetCOn : BOOL; (* bus: setpoint  genetaror power factor (COS PHI) from EU - on (activate) *) (* OldName: BUS_GCQ_PF_S; Cycle:5; *)
		bGenC_PFCBC_SetCOf : BOOL; (* bus: primary frequency control - off (deactivate) *) (* OldName: BUS_GCP_PFC_R; Cycle:5; *)
		bGenC_PFCBC_SetCOn : BOOL; (* bus: primary frequency control - on (activate) *) (* OldName: BUS_GCP_PFC_S; Cycle:5; *)
		bGenC_PFUCBC_SetCOf : BOOL; (* bus: setpoint reactive power characteristics COS(phi)=f(U) from EU -off (deactive) *) (* OldName: BUS_GCQ_PFU_R; Cycle:5; *)
		bGenC_PFUCBC_SetCOn : BOOL; (* bus: setpoint reactive power characteristics COS(phi)=f(U) from EU -on (active) *) (* OldName: BUS_GCQ_PFU_S; Cycle:5; *)
		bGenC_PLimBC_SetCOf : BOOL; (* bus: power limition from  EU - off (deactivate) *) (* OldName: BUS_GCP_Plim_R; Cycle:5; *)
		bGenC_PLimBC_SetCOn : BOOL; (* bus: power limition from  EU - on (activate) *) (* OldName: BUS_GCP_Plim_S; Cycle:5; *)
		bGenC_PUBC_SetCOf : BOOL; (*demand off P(U) over Bus*)
		bGenC_PUBC_SetCOn : BOOL; (*demand on P(U) over Bus*)
		bGenC_QBC_SetCOf : BOOL; (* bus: setpoint reactive power (Q) from EU - off (deactivate) *) (* OldName: BUS_GCQ_Q_R; Cycle:5; *)
		bGenC_QBC_SetCOn : BOOL; (* bus: setpoint reactive power (Q) from EU - on (activate) *) (* OldName: BUS_GCQ_Q_S; Cycle:5; *)
		bGenC_QCustBC_SetCOf : BOOL; (*bus: Customized Q setpoint - off (deactivate)*)
		bGenC_QCustBC_SetCOn : BOOL; (*bus: Customized Q setpoint - on (activate)*)
		bGenC_QLimBC_SetCOf : BOOL; (* bus: setpoint reactive power limitation (Qlim) from EU - off (deactivate) *) (* OldName: BUS_GCQ_Qlim_R; Cycle:5; *)
		bGenC_QLimBC_SetCOn : BOOL; (* bus: setpoint reactive power limitation (Qlim) from EU - on (activate) *) (* OldName: BUS_GCQ_Qlim_S; Cycle:5; *)
		bGenC_QLimSetErrBC : BOOL; (* bus: setpoint reactive power limitation from EU error - use backupvalue *)
		bGenC_QPBC_SetCOf : BOOL; (* Bus setpoint reactive power characteristics Q=f(P) from EU - off (deactivate) *)
		bGenC_QPBC_SetCOn : BOOL; (* Bus setpoint reactive power characteristics Q=f(P) from EU - on (activate) *)
		bGenC_QPCBC_SetCOf : BOOL; (* bus: setpoint reactive power characteristics COS(phi)=f(P) from - off (deactivate) *) (* OldName: BUS_GCQ_PFP_R; Cycle:5; *)
		bGenC_QPCBC_SetCOn : BOOL; (* bus: setpoint reactive power characteristics COS(phi)=f(P) from EU - on (activate) *) (* OldName: BUS_GCQ_PFP_S; Cycle:5; *)
		bGenC_QUCBC_SetCOf : BOOL; (* bus: setpoint reactive power characteristics Q=f(U) from EU -off (deactivate) *) (* OldName: BUS_GCQ_QU_R; Cycle:5; *)
		bGenC_QUCBC_SetCOn : BOOL; (* bus: setpoint reactive power characteristics Q=f(U) from EU -on (activate) *) (* OldName: BUS_GCQ_QU_S; Cycle:5; *)
		bGenC_RMCBC_SetCOf : BOOL; (* bus: regulation margin control -off (deactivate) *) (* OldName: BUS_GCP_RMC_R; Cycle:5; *)
		bGenC_RMCBC_SetCOn : BOOL; (* bus: regulation margin control -on (activate) *) (* OldName: BUS_GCP_RMC_S; Cycle:5; *)
		bGenC_UBC_SetCOf : BOOL; (*Bus: Voltage control for reactive power - off (deactivated)*)
		bGenC_UBC_SetCOn : BOOL; (*Bus: Voltage control for reactive power - on (activated)*)
		bGenC_UQBC_SetCOf : BOOL; (* bus: setpoint generator voltage for rective power - off (deactivate) *) (* OldName: BUS_GCQ_Uset_R; Cycle:5; *)
		bGenC_UQBC_SetCOn : BOOL; (* bus: setpoint generator voltage for rective power - on (activate) *) (* OldName: BUS_GCQ_Uset_S; Cycle:5; *)
		bMsg1001 : BOOL; (*reserve alarm message 1*)
		bMsg1002 : BOOL; (*reserve alarm message 2*)
		bMsg1003 : BOOL; (*reserve alarm message 3*)
		bMsg1004 : BOOL; (*reserve alarm message 4*)
		bMsg1005 : BOOL; (*reserve alarm message 5*)
		bMsg1006 : BOOL; (*reserve alarm message 6*)
		bMsg1007 : BOOL; (*reserve alarm message 7*)
		bMsg1008 : BOOL; (*reserve alarm message 8*)
		bMsg1009 : BOOL; (*reserve alarm message 9*)
		bMsg1010 : BOOL; (*reserve alarm message 10*)
		bMsg1011 : BOOL; (*reserve alarm message 11*)
		bMsg1012 : BOOL; (*reserve alarm message 12*)
		bMsg1013 : BOOL; (*reserve alarm message 13*)
		bMsg1014 : BOOL; (*reserve alarm message 14*)
		bMsg1015 : BOOL; (*reserve alarm message 15*)
		bMsg1016 : BOOL; (*reserve alarm message 16*)
		bMsg1177 : BOOL; (*Signal error Reserve Analog Input 1*)
		bMsg1178 : BOOL; (*Signal error Reserve Analog Input 2*)
		bMsg1179 : BOOL; (*Signal error Reserve Analog Input 3*)
		bMsg1180 : BOOL; (*Signal error Reserve Analog Input 4*)
		bMsg1181 : BOOL; (*Signal error Reserve Analog Input 5*)
		bMsg1182 : BOOL; (*Signal error Reserve Analog Input 6*)
		bMsg1183 : BOOL; (*Signal error Reserve Analog Input 7*)
		bMsg1184 : BOOL; (*Signal error Reserve Analog Input 8*)
		bMsg1193 : BOOL; (*reserve warning message 1*)
		bMsg1194 : BOOL; (*reserve warning message 2*)
		bMsg1195 : BOOL; (*reserve warning message 3*)
		bMsg1196 : BOOL; (*reserve warning message 4*)
		bMsg1197 : BOOL; (*reserve warning message 5*)
		bMsg1198 : BOOL; (*reserve warning message 6*)
		bMsg1199 : BOOL; (*reserve warning message 7*)
		bMsg1200 : BOOL; (*reserve warning message 8*)
		bMsg1201 : BOOL; (*reserve warning message 9*)
		bMsg1202 : BOOL; (*reserve warning message 10*)
		bMsg1203 : BOOL; (*reserve warning message 11*)
		bMsg1204 : BOOL; (*reserve warning message 12*)
		bMsg1205 : BOOL; (*reserve warning message 13*)
		bMsg1206 : BOOL; (*reserve warning message 14*)
		bMsg1207 : BOOL; (*reserve warning message 15*)
		bMsg1208 : BOOL; (*reserve warning message 16*)
		bMsg1601 : BOOL; (*reserve alarm message 17*)
		bMsg1602 : BOOL; (*reserve alarm message 18*)
		bMsg1603 : BOOL; (*reserve alarm message 19*)
		bMsg1604 : BOOL; (*reserve alarm message 20*)
		bMsg1605 : BOOL; (*reserve alarm message*)
		bMsg1606 : BOOL; (*reserve alarm message*)
		bMsg1607 : BOOL; (*reserve alarm message*)
		bMsg1608 : BOOL; (*reserve alarm message*)
		bMsg1609 : BOOL; (*reserve alarm message*)
		bMsg1610 : BOOL; (*reserve alarm message*)
		bMsg1611 : BOOL; (*reserve alarm message*)
		bMsg1612 : BOOL; (*reserve alarm message*)
		bMsg1613 : BOOL; (*reserve alarm message*)
		bMsg1614 : BOOL; (*reserve alarm message 30*)
		bMsg1615 : BOOL; (*reserve alarm message*)
		bMsg1616 : BOOL; (*reserve alarm message*)
		bMsg1617 : BOOL; (*reserve alarm message*)
		bMsg1618 : BOOL; (*reserve alarm message*)
		bMsg1619 : BOOL; (*reserve alarm message*)
		bMsg1620 : BOOL; (*reserve alarm message*)
		bMsg1621 : BOOL; (*reserve alarm message*)
		bMsg1622 : BOOL; (*reserve alarm message*)
		bMsg1623 : BOOL; (*reserve alarm message*)
		bMsg1624 : BOOL; (*reserve alarm message 40*)
		bMsg1625 : BOOL; (*reserve alarm message*)
		bMsg1626 : BOOL; (*reserve alarm message*)
		bMsg1627 : BOOL; (*reserve alarm message*)
		bMsg1628 : BOOL; (*reserve alarm message*)
		bMsg1629 : BOOL; (*reserve alarm message*)
		bMsg1630 : BOOL; (*reserve alarm message*)
		bMsg1631 : BOOL; (*reserve alarm message*)
		bMsg1632 : BOOL; (*reserve alarm message*)
		bMsg1633 : BOOL; (*reserve alarm message*)
		bMsg1634 : BOOL; (*reserve alarm message 50*)
		bMsg1635 : BOOL; (*reserve alarm message*)
		bMsg1636 : BOOL; (*reserve alarm message*)
		bMsg1637 : BOOL; (*reserve alarm message*)
		bMsg1638 : BOOL; (*reserve alarm message*)
		bMsg1639 : BOOL; (*reserve alarm message*)
		bMsg1640 : BOOL; (*reserve alarm message*)
		bMsg1641 : BOOL; (*reserve alarm message*)
		bMsg1642 : BOOL; (*reserve alarm message*)
		bMsg1643 : BOOL; (*reserve alarm message*)
		bMsg1644 : BOOL; (*reserve alarm message 60*)
		bMsg1645 : BOOL; (*reserve alarm message*)
		bMsg1646 : BOOL; (*reserve alarm message*)
		bMsg1647 : BOOL; (*reserve alarm message*)
		bMsg1648 : BOOL; (*reserve alarm message*)
		bMsg1649 : BOOL; (*reserve alarm message*)
		bMsg1650 : BOOL; (*reserve alarm message*)
		bMsg1651 : BOOL; (*reserve alarm message*)
		bMsg1652 : BOOL; (*reserve alarm message*)
		bMsg1653 : BOOL; (*reserve alarm message*)
		bMsg1654 : BOOL; (*reserve alarm message 70*)
		bMsg1655 : BOOL; (*reserve alarm message*)
		bMsg1656 : BOOL; (*reserve alarm message*)
		bMsg1657 : BOOL; (*reserve alarm message*)
		bMsg1658 : BOOL; (*reserve alarm message*)
		bMsg1659 : BOOL; (*reserve alarm message*)
		bMsg1660 : BOOL; (*reserve alarm message*)
		bMsg1661 : BOOL; (*reserve alarm message*)
		bMsg1662 : BOOL; (*reserve alarm message*)
		bMsg1663 : BOOL; (*reserve alarm message*)
		bMsg1664 : BOOL; (*reserve alarm message 80*)
		bMsg1665 : BOOL; (*reserve alarm message*)
		bMsg1666 : BOOL; (*reserve alarm message*)
		bMsg1667 : BOOL; (*reserve alarm message*)
		bMsg1668 : BOOL; (*reserve alarm message*)
		bMsg1669 : BOOL; (*reserve alarm message*)
		bMsg1670 : BOOL; (*reserve alarm message*)
		bMsg1671 : BOOL; (*reserve alarm message*)
		bMsg1672 : BOOL; (*reserve alarm message*)
		bMsg1673 : BOOL; (*reserve alarm message*)
		bMsg1674 : BOOL; (*reserve alarm message 90*)
		bMsg1675 : BOOL; (*reserve alarm message*)
		bMsg1676 : BOOL; (*reserve alarm message*)
		bMsg1677 : BOOL; (*reserve alarm message*)
		bMsg1678 : BOOL; (*reserve alarm message*)
		bMsg1679 : BOOL; (*reserve alarm message*)
		bMsg1680 : BOOL; (*reserve alarm message*)
		bMsg1681 : BOOL; (*reserve alarm message*)
		bMsg1682 : BOOL; (*reserve alarm message*)
		bMsg1683 : BOOL; (*reserve alarm message*)
		bMsg1684 : BOOL; (*reserve alarm message 100*)
		bMsg1685 : BOOL; (*reserve alarm message*)
		bMsg1686 : BOOL; (*reserve alarm message*)
		bMsg1687 : BOOL; (*reserve alarm message*)
		bMsg1688 : BOOL; (*reserve alarm message*)
		bMsg1689 : BOOL; (*reserve alarm message*)
		bMsg1690 : BOOL; (*reserve alarm message*)
		bMsg1691 : BOOL; (*reserve alarm message*)
		bMsg1692 : BOOL; (*reserve alarm message*)
		bMsg1693 : BOOL; (*reserve alarm message*)
		bMsg1694 : BOOL; (*reserve alarm message 110*)
		bMsg1695 : BOOL; (*reserve alarm message*)
		bMsg1696 : BOOL; (*reserve alarm message*)
		bMsg1697 : BOOL; (*reserve alarm message*)
		bMsg1698 : BOOL; (*reserve alarm message*)
		bMsg1699 : BOOL; (*reserve alarm message 115*)
		bMsg1700 : BOOL; (*reserve alarm message 116*)
		bMsg1701 : BOOL; (*reserve warning message 27*)
		bMsg1702 : BOOL; (*reserve warning message 28*)
		bMsg1703 : BOOL; (*reserve warning message 29*)
		bMsg1704 : BOOL; (*reserve warning message 30*)
		bMsg1705 : BOOL; (*reserve warning message 31*)
		bMsg1706 : BOOL; (*reserve warning message*)
		bMsg1707 : BOOL; (*reserve warning message*)
		bMsg1708 : BOOL; (*reserve warning message*)
		bMsg1709 : BOOL; (*reserve warning message*)
		bMsg1710 : BOOL; (*reserve warning message*)
		bMsg1711 : BOOL; (*reserve warning message*)
		bMsg1712 : BOOL; (*reserve warning message*)
		bMsg1713 : BOOL; (*reserve warning message*)
		bMsg1714 : BOOL; (*reserve warning message 40*)
		bMsg1715 : BOOL; (*reserve warning message 41*)
		bMsg1716 : BOOL; (*reserve warning message*)
		bMsg1717 : BOOL; (*reserve warning message*)
		bMsg1718 : BOOL; (*reserve warning message*)
		bMsg1719 : BOOL; (*reserve warning message*)
		bMsg1720 : BOOL; (*reserve warning message*)
		bMsg1721 : BOOL; (*reserve warning message*)
		bMsg1722 : BOOL; (*reserve warning message*)
		bMsg1723 : BOOL; (*reserve warning message*)
		bMsg1724 : BOOL; (*reserve warning message 50*)
		bMsg1725 : BOOL; (*reserve warning message*)
		bMsg1726 : BOOL; (*reserve warning message*)
		bMsg1727 : BOOL; (*reserve warning message*)
		bMsg1728 : BOOL; (*reserve warning message*)
		bMsg1729 : BOOL; (*reserve warning message*)
		bMsg1730 : BOOL; (*reserve warning message*)
		bMsg1731 : BOOL; (*reserve warning message*)
		bMsg1732 : BOOL; (*reserve warning message*)
		bMsg1733 : BOOL; (*reserve warning message*)
		bMsg1734 : BOOL; (*reserve warning message 60*)
		bMsg1735 : BOOL; (*reserve warning message*)
		bMsg1736 : BOOL; (*reserve warning message*)
		bMsg1737 : BOOL; (*reserve warning message*)
		bMsg1738 : BOOL; (*reserve warning message*)
		bMsg1739 : BOOL; (*reserve warning message*)
		bMsg1740 : BOOL; (*reserve warning message*)
		bMsg1741 : BOOL; (*reserve warning message*)
		bMsg1742 : BOOL; (*reserve warning message*)
		bMsg1743 : BOOL; (*reserve warning message*)
		bMsg1744 : BOOL; (*reserve warning message 70*)
		bMsg1745 : BOOL; (*reserve warning message*)
		bMsg1746 : BOOL; (*reserve warning message*)
		bMsg1747 : BOOL; (*reserve warning message*)
		bMsg1748 : BOOL; (*reserve warning message*)
		bMsg1749 : BOOL; (*reserve warning message*)
		bMsg1750 : BOOL; (*reserve warning message*)
		bMsg1751 : BOOL; (*reserve warning message*)
		bMsg1752 : BOOL; (*reserve warning message*)
		bMsg1753 : BOOL; (*reserve warning message*)
		bMsg1754 : BOOL; (*reserve warning message 80*)
		bMsg1755 : BOOL; (*reserve warning message*)
		bMsg1756 : BOOL; (*reserve warning message*)
		bMsg1757 : BOOL; (*reserve warning message*)
		bMsg1758 : BOOL; (*reserve warning message*)
		bMsg1759 : BOOL; (*reserve warning message*)
		bMsg1760 : BOOL; (*reserve warning message*)
		bMsg1761 : BOOL; (*reserve warning message*)
		bMsg1762 : BOOL; (*reserve warning message*)
		bMsg1763 : BOOL; (*reserve warning message*)
		bMsg1764 : BOOL; (*reserve warning message 90*)
		bMsg1765 : BOOL; (*reserve warning message*)
		bMsg1766 : BOOL; (*reserve warning message*)
		bMsg1767 : BOOL; (*reserve warning message*)
		bMsg1768 : BOOL; (*reserve warning message*)
		bMsg1769 : BOOL; (*reserve warning message*)
		bMsg1770 : BOOL; (*reserve warning message*)
		bMsg1771 : BOOL; (*reserve warning message*)
		bMsg1772 : BOOL; (*reserve warning message*)
		bMsg1773 : BOOL; (*reserve warning message*)
		bMsg1774 : BOOL; (*reserve warning message 100*)
		bMsg1775 : BOOL; (*reserve warning message*)
		bMsg1776 : BOOL; (*reserve warning message*)
		bMsg1777 : BOOL; (*reserve warning message*)
		bMsg1778 : BOOL; (*reserve warning message*)
		bMsg1779 : BOOL; (*reserve warning message*)
		bMsg1780 : BOOL; (*reserve warning message*)
		bMsg1781 : BOOL; (*reserve warning message*)
		bMsg1782 : BOOL; (*reserve warning message*)
		bMsg1783 : BOOL; (*reserve warning message*)
		bMsg1784 : BOOL; (*reserve warning message 110*)
		bMsg1785 : BOOL; (*reserve warning message*)
		bMsg1786 : BOOL; (*reserve warning message*)
		bMsg1787 : BOOL; (*reserve warning message*)
		bMsg1788 : BOOL; (*reserve warning message*)
		bMsg1789 : BOOL; (*reserve warning message*)
		bMsg1790 : BOOL; (*reserve warning message*)
		bMsg1791 : BOOL; (*reserve warning message*)
		bMsg1792 : BOOL; (*reserve warning message*)
		bMsg1793 : BOOL; (*reserve warning message*)
		bMsg1794 : BOOL; (*reserve warning message 120*)
		bMsg1795 : BOOL; (*reserve warning message 121*)
		bMsg1796 : BOOL; (*reserve warning message 122*)
		bMsg1797 : BOOL; (*reserve warning message 123*)
		bMsg1798 : BOOL; (*reserve warning message 124*)
		bMsg1799 : BOOL; (*reserve warning message 125*)
		bMsg1800 : BOOL; (*reserve warning message 126*)
		bMsg2032 : BOOL;
		bMsg2033 : BOOL;
		bMsg2034 : BOOL;
		bMsg2035 : BOOL;
		bMsg2036 : BOOL;
		bMsg2037 : BOOL;
		bMsg2050 : BOOL;
		bMsg2051 : BOOL;
		bMsg2087 : BOOL; (*reserve warning message 17*)
		bMsg2088 : BOOL; (*reserve warning message 18*)
		bMsg2089 : BOOL; (*reserve warning message 19*)
		bMsg2090 : BOOL; (*reserve warning message 20*)
		bMsg2091 : BOOL; (*reserve warning message 21*)
		bMsg2092 : BOOL; (*reserve warning message 22*)
		bMsg2093 : BOOL; (*reserve warning message 23*)
		bMsg2094 : BOOL; (*reserve warning message 24*)
		bMsg2095 : BOOL; (*reserve warning message 25*)
		bMsg2096 : BOOL; (*reserve warning message 26*)
		bMsg2302 : BOOL; (*alarm message mns import ctr*)
		bMsg2303 : BOOL; (*alarm message mns import ctr*)
		bMsg2415 : BOOL; (*warning message mns import ctr*)
		bMsg2416 : BOOL; (*warning message mns import ctr*)
		bMsg2417 : BOOL; (*warning message mns import ctr*)
		bMsg2418 : BOOL; (*warning message mns import ctr*)
		bMsg2419 : BOOL; (*operating message mns import ctr*)
		bMsg2420 : BOOL; (*operating message mns import ctr*)
		bMsg3232 : BOOL; (*reserve operating message 1*)
		bMsg3233 : BOOL; (*reserve operating message 2*)
		bMsg3234 : BOOL; (*reserve operating message 3*)
		bMsg3235 : BOOL; (*reserve operating message 4*)
		bMsg3236 : BOOL; (*reserve operating message 5*)
		bMsg3237 : BOOL; (*reserve operating message 6*)
		bMsg3250 : BOOL; (*reserve operating message 7*)
		bMsg3251 : BOOL; (*reserve operating message 8*)
		bMsg3565 : BOOL; (*Messignalstoerung Generator Leistungssollwert*)
		bMsg3566 : BOOL; (*Messignalstoerung Generator Leistungsfaktorsollwert*)
		bMsg3601 : BOOL; (*reserve operating message 9*)
		bMsg3602 : BOOL; (*reserve operating message 10*)
		bMsg3603 : BOOL; (*reserve operating message 11*)
		bMsg3604 : BOOL; (*reserve operating message 12*)
		bMsg3605 : BOOL; (*reserve operating message 13*)
		bMsg3606 : BOOL; (*reserve operating message 14*)
		bMsg3607 : BOOL; (*reserve operating message 15*)
		bMsg3608 : BOOL; (*reserve operating message 16*)
		bMsg3609 : BOOL; (*reserve operating message 17*)
		bMsg3610 : BOOL; (*reserve operating message 18*)
		bMsg3611 : BOOL; (*reserve operating message 19*)
		bMsg3612 : BOOL; (*reserve operating message 20*)
		bMsg3613 : BOOL; (*reserve operating message *)
		bMsg3614 : BOOL; (*reserve operating message *)
		bMsg3615 : BOOL; (*reserve operating message *)
		bMsg3616 : BOOL; (*reserve operating message *)
		bMsg3617 : BOOL; (*reserve operating message *)
		bMsg3618 : BOOL; (*reserve operating message *)
		bMsg3619 : BOOL; (*reserve operating message *)
		bMsg3620 : BOOL; (*reserve operating message *)
		bMsg3621 : BOOL; (*reserve operating message *)
		bMsg3622 : BOOL; (*reserve operating message 30*)
		bMsg3623 : BOOL; (*reserve operating message *)
		bMsg3624 : BOOL; (*reserve operating message *)
		bMsg3625 : BOOL; (*reserve operating message *)
		bMsg3626 : BOOL; (*reserve operating message *)
		bMsg3627 : BOOL; (*reserve operating message *)
		bMsg3628 : BOOL; (*reserve operating message *)
		bMsg3629 : BOOL; (*reserve operating message *)
		bMsg3630 : BOOL; (*reserve operating message *)
		bMsg3631 : BOOL; (*reserve operating message *)
		bMsg3632 : BOOL; (*reserve operating message 40*)
		bMsg3633 : BOOL; (*reserve operating message *)
		bMsg3634 : BOOL; (*reserve operating message *)
		bMsg3635 : BOOL; (*reserve operating message *)
		bMsg3636 : BOOL; (*reserve operating message *)
		bMsg3637 : BOOL; (*reserve operating message *)
		bMsg3638 : BOOL; (*reserve operating message *)
		bMsg3639 : BOOL; (*reserve operating message *)
		bMsg3640 : BOOL; (*reserve operating message *)
		bMsg3641 : BOOL; (*reserve operating message *)
		bMsg3642 : BOOL; (*reserve operating message 50*)
		bMsg3643 : BOOL; (*reserve operating message *)
		bMsg3644 : BOOL; (*reserve operating message *)
		bMsg3645 : BOOL; (*reserve operating message *)
		bMsg3646 : BOOL; (*reserve operating message *)
		bMsg3647 : BOOL; (*reserve operating message *)
		bMsg3648 : BOOL; (*reserve operating message *)
		bMsg3649 : BOOL; (*reserve operating message *)
		bMsg3650 : BOOL; (*reserve operating message *)
		bMsg3651 : BOOL; (*reserve operating message *)
		bMsg3652 : BOOL; (*reserve operating message 60*)
		bMsg3653 : BOOL; (*reserve operating message *)
		bMsg3654 : BOOL; (*reserve operating message *)
		bMsg3655 : BOOL; (*reserve operating message *)
		bMsg3656 : BOOL; (*reserve operating message *)
		bMsg3657 : BOOL; (*reserve operating message *)
		bMsg3658 : BOOL; (*reserve operating message *)
		bMsg3659 : BOOL; (*reserve operating message *)
		bMsg3660 : BOOL; (*reserve operating message *)
		bMsg3661 : BOOL; (*reserve operating message *)
		bMsg3662 : BOOL; (*reserve operating message 70*)
		bMsg3663 : BOOL; (*reserve operating message *)
		bMsg3664 : BOOL; (*reserve operating message *)
		bMsg3665 : BOOL; (*reserve operating message *)
		bMsg3666 : BOOL; (*reserve operating message *)
		bMsg3667 : BOOL; (*reserve operating message *)
		bMsg3668 : BOOL; (*reserve operating message *)
		bMsg3669 : BOOL; (*reserve operating message *)
		bMsg3670 : BOOL; (*reserve operating message *)
		bMsg3671 : BOOL; (*reserve operating message *)
		bMsg3672 : BOOL; (*reserve operating message 80*)
		bMsg3673 : BOOL; (*reserve operating message *)
		bMsg3674 : BOOL; (*reserve operating message *)
		bMsg3675 : BOOL; (*reserve operating message *)
		bMsg3676 : BOOL; (*reserve operating message *)
		bMsg3677 : BOOL; (*reserve operating message *)
		bMsg3678 : BOOL; (*reserve operating message *)
		bMsg3679 : BOOL; (*reserve operating message *)
		bMsg3680 : BOOL; (*reserve operating message *)
		bMsg3681 : BOOL; (*reserve operating message *)
		bMsg3682 : BOOL; (*reserve operating message 90*)
		bMsg3683 : BOOL; (*reserve operating message *)
		bMsg3684 : BOOL; (*reserve operating message *)
		bMsg3685 : BOOL; (*reserve operating message *)
		bMsg3686 : BOOL; (*reserve operating message *)
		bMsg3687 : BOOL; (*reserve operating message *)
		bMsg3688 : BOOL; (*reserve operating message *)
		bMsg3689 : BOOL; (*reserve operating message *)
		bMsg3690 : BOOL; (*reserve operating message *)
		bMsg3691 : BOOL; (*reserve operating message *)
		bMsg3692 : BOOL; (*reserve operating message 100*)
		bMsg3693 : BOOL; (*reserve operating message 101*)
		bMsg3694 : BOOL; (*reserve operating message 102*)
		bMsg3695 : BOOL; (*reserve operating message 103*)
		bMsg3696 : BOOL; (*reserve operating message 104*)
		bMsg3697 : BOOL; (*reserve operating message 105*)
		bMsg3698 : BOOL; (*reserve operating message 106*)
		bMsg3699 : BOOL; (*reserve operating message 107*)
		bMsg3700 : BOOL; (*reserve operating message 108*)
		bMsg3701 : BOOL; (*alarm message reserve analog input*)
		bMsg3702 : BOOL; (*alarm message reserve analog input*)
		bMsg3703 : BOOL; (*alarm message reserve analog input*)
		bMsg3704 : BOOL; (*alarm message reserve analog input*)
		bMsg3705 : BOOL; (*alarm message reserve analog input*)
		bMsg3706 : BOOL; (*alarm message reserve analog input*)
		bMsg3707 : BOOL; (*alarm message reserve analog input*)
		bMsg3708 : BOOL; (*alarm message reserve analog input*)
		bMsg3709 : BOOL; (*alarm message reserve analog input*)
		bMsg3710 : BOOL; (*alarm message reserve analog input*)
		bMsg3711 : BOOL; (*alarm message reserve analog input*)
		bMsg3712 : BOOL; (*alarm message reserve analog input*)
		bMsg3713 : BOOL; (*alarm message reserve analog input*)
		bMsg3714 : BOOL; (*alarm message reserve analog input*)
		bMsg3715 : BOOL; (*alarm message reserve analog input*)
		bMsg3716 : BOOL; (*alarm message reserve analog input*)
		bMsg3717 : BOOL; (*alarm message reserve analog input*)
		bMsg3718 : BOOL; (*alarm message reserve analog input*)
		bMsg3719 : BOOL; (*alarm message reserve analog input*)
		bMsg3720 : BOOL; (*alarm message reserve analog input*)
		bMsg3721 : BOOL; (*alarm message reserve analog input*)
		bMsg3722 : BOOL; (*alarm message reserve analog input*)
		bMsg3723 : BOOL; (*alarm message reserve analog input*)
		bMsg3724 : BOOL; (*alarm message reserve analog input*)
		bMsg3725 : BOOL; (*alarm message reserve analog input*)
		bMsg3726 : BOOL; (*alarm message reserve analog input*)
		bMsg3727 : BOOL; (*alarm message reserve analog input*)
		bMsg3728 : BOOL; (*alarm message reserve analog input*)
		bMsg3729 : BOOL; (*alarm message reserve analog input*)
		bMsg3730 : BOOL; (*alarm message reserve analog input*)
		bMsg3731 : BOOL; (*alarm message reserve analog input*)
		bMsg3732 : BOOL; (*alarm message reserve analog input*)
		bMsg3733 : BOOL; (*alarm message reserve analog input*)
		bMsg3734 : BOOL; (*alarm message reserve analog input*)
		bMsg3735 : BOOL; (*alarm message reserve analog input*)
		bMsg3736 : BOOL; (*alarm message reserve analog input*)
		bMsg3737 : BOOL; (*alarm message reserve analog input*)
		bMsg3738 : BOOL; (*alarm message reserve analog input*)
		bMsg3739 : BOOL; (*alarm message reserve analog input*)
		bMsg3740 : BOOL; (*alarm message reserve analog input*)
		bMsg3741 : BOOL; (*alarm message reserve analog input*)
		bMsg3742 : BOOL; (*alarm message reserve analog input*)
		bMsg3743 : BOOL; (*alarm message reserve analog input*)
		bMsg3744 : BOOL; (*alarm message reserve analog input*)
		bMsg3745 : BOOL; (*alarm message reserve analog input*)
		bMsg3746 : BOOL; (*alarm message reserve analog input*)
		bMsg3747 : BOOL; (*alarm message reserve analog input*)
		bMsg3748 : BOOL; (*alarm message reserve analog input*)
		bMsg3749 : BOOL; (*alarm message reserve analog input*)
		bMsg3750 : BOOL; (*alarm message reserve analog input*)
		bMsg3751 : BOOL; (*alarm message reserve analog input*)
		bMsg3752 : BOOL; (*alarm message reserve analog input*)
		bMsg3753 : BOOL; (*alarm message reserve analog input*)
		bMsg3754 : BOOL; (*alarm message reserve analog input*)
		bMsg3755 : BOOL; (*alarm message reserve analog input*)
		bMsg3756 : BOOL; (*alarm message reserve analog input*)
		bMsg3757 : BOOL; (*alarm message reserve analog input*)
		bMsg3758 : BOOL; (*alarm message reserve analog input*)
		bMsg3759 : BOOL; (*alarm message reserve analog input*)
		bMsg3760 : BOOL; (*alarm message reserve analog input*)
		bMsg3761 : BOOL; (*alarm message reserve analog input*)
		bMsg3762 : BOOL; (*alarm message reserve analog input*)
		bMsg3763 : BOOL; (*alarm message reserve analog input*)
		bMsg3764 : BOOL; (*alarm message reserve analog input*)
		bMsg3765 : BOOL; (*alarm message reserve analog input*)
		bMsg3766 : BOOL; (*alarm message reserve analog input*)
		bMsg3767 : BOOL; (*alarm message reserve analog input*)
		bMsg3768 : BOOL; (*alarm message reserve analog input*)
		bMsg3769 : BOOL; (*alarm message reserve analog input*)
		bMsg3770 : BOOL; (*alarm message reserve analog input*)
		bMsg3771 : BOOL; (*alarm message reserve analog input*)
		bMsg3772 : BOOL; (*alarm message reserve analog input*)
		bMsg3773 : BOOL; (*alarm message reserve analog input*)
		bMsg3774 : BOOL; (*alarm message reserve analog input*)
		bMsg3775 : BOOL; (*alarm message reserve analog input*)
		bMsg3776 : BOOL; (*alarm message reserve analog input*)
		bMsg3777 : BOOL; (*alarm message reserve analog input*)
		bMsg3778 : BOOL; (*alarm message reserve analog input*)
		bMsg3779 : BOOL; (*alarm message reserve analog input*)
		bMsg3780 : BOOL; (*alarm message reserve analog input*)
		bMsg3781 : BOOL; (*alarm message reserve analog input*)
		bMsg3782 : BOOL; (*alarm message reserve analog input*)
		bMsg3783 : BOOL; (*alarm message reserve analog input*)
		bMsg3784 : BOOL; (*alarm message reserve analog input*)
		bMsg3785 : BOOL; (*alarm message reserve analog input*)
		bMsg3786 : BOOL; (*alarm message reserve analog input*)
		bMsg3787 : BOOL; (*alarm message reserve analog input*)
		bMsg3788 : BOOL; (*alarm message reserve analog input*)
		bMsg3789 : BOOL; (*alarm message reserve analog input*)
		bMsg3790 : BOOL; (*alarm message reserve analog input*)
		bMsg6701 : BOOL; (*reserve operating message 109*) (*import HMI Extension*)
		bMsg6702 : BOOL; (*reserve operating message 110*) (*import HMI Extension*)
		bMsg6703 : BOOL; (*reserve operating message 111*) (*import HMI Extension*)
		bMsg6704 : BOOL; (*reserve operating message 112*) (*import HMI Extension*)
		bMsg6705 : BOOL; (*reserve operating message 113*) (*import HMI Extension*)
		bMsg6706 : BOOL; (*reserve operating message 114*) (*import HMI Extension*)
		bMsg6707 : BOOL; (*reserve operating message 115*) (*import HMI Extension*)
		bMsg6708 : BOOL; (*reserve operating message 116*) (*import HMI Extension*)
		bMsg6709 : BOOL; (*reserve operating message 117*) (*import HMI Extension*)
		bMsg6710 : BOOL; (*reserve operating message 118*) (*import HMI Extension*)
		bMsg6711 : BOOL; (*reserve operating message 119*) (*import HMI Extension*)
		bMsg6712 : BOOL; (*reserve operating message 120*) (*import HMI Extension*)
		bMsg6713 : BOOL; (*reserve operating message 121*) (*import HMI Extension*)
		bMsg6714 : BOOL; (*reserve operating message 122*) (*import HMI Extension*)
		bMsg6715 : BOOL; (*reserve operating message 123*) (*import HMI Extension*)
		bMsg6716 : BOOL; (*reserve operating message 124*) (*import HMI Extension*)
		bMsg6717 : BOOL; (*reserve operating message 125*) (*import HMI Extension*)
		bMsg6718 : BOOL; (*reserve operating message 126*) (*import HMI Extension*)
		bMsg6719 : BOOL; (*reserve operating message 127*) (*import HMI Extension*)
		bMsg6720 : BOOL; (*reserve operating message 128*) (*import HMI Extension*)
		bMsg6721 : BOOL; (*reserve operating message 129*) (*import HMI Extension*)
		bMsg6722 : BOOL; (*reserve operating message 130*) (*import HMI Extension*)
		bMsg6723 : BOOL; (*reserve operating message 131*) (*import HMI Extension*)
		bMsg6724 : BOOL; (*reserve operating message 132*) (*import HMI Extension*)
		bMsg6725 : BOOL; (*reserve operating message 133*) (*import HMI Extension*)
		bMsg6726 : BOOL; (*reserve operating message 134*) (*import HMI Extension*)
		bMsg6727 : BOOL; (*reserve operating message 135*) (*import HMI Extension*)
		bMsg6728 : BOOL; (*reserve operating message 136*) (*import HMI Extension*)
		bMsg6729 : BOOL; (*reserve operating message 137*) (*import HMI Extension*)
		bMsg6730 : BOOL; (*reserve operating message 138*) (*import HMI Extension*)
		bMsg6731 : BOOL; (*reserve operating message 139*) (*import HMI Extension*)
		bMsg6732 : BOOL; (*reserve operating message 140*) (*import HMI Extension*)
		bMsg6733 : BOOL; (*reserve operating message 141*) (*import HMI Extension*)
		bMsg6734 : BOOL; (*reserve operating message 142*) (*import HMI Extension*)
		bMsg6735 : BOOL; (*reserve operating message 143*) (*import HMI Extension*)
		bMsg6736 : BOOL; (*reserve operating message 144*) (*import HMI Extension*)
		bMsg6737 : BOOL; (*reserve operating message 145*) (*import HMI Extension*)
		bMsg6738 : BOOL; (*reserve operating message 146*) (*import HMI Extension*)
		bMsg6739 : BOOL; (*reserve operating message 147*) (*import HMI Extension*)
		bMsg6740 : BOOL; (*reserve operating message 148*) (*import HMI Extension*)
		bMsg6741 : BOOL; (*reserve operating message 149*) (*import HMI Extension*)
		bMsg6742 : BOOL; (*reserve operating message 150*) (*import HMI Extension*)
		bMsg6743 : BOOL; (*reserve operating message 151*) (*import HMI Extension*)
		bMsg6744 : BOOL; (*reserve operating message 152*) (*import HMI Extension*)
		bMsg6745 : BOOL; (*reserve operating message 153*) (*import HMI Extension*)
		bMsg6746 : BOOL; (*reserve operating message 154*) (*import HMI Extension*)
		bMsg6747 : BOOL; (*reserve operating message 155*) (*import HMI Extension*)
		bMsg6748 : BOOL; (*reserve operating message 156*) (*import HMI Extension*)
		bMsg6749 : BOOL; (*reserve operating message 157*) (*import HMI Extension*)
		bMsg6750 : BOOL; (*reserve operating message 158*) (*import HMI Extension*)
		bMsg6751 : BOOL; (*reserve operating message 159*) (*import HMI Extension*)
		bMsg6752 : BOOL; (*reserve operating message 160*) (*import HMI Extension*)
		bMsg6753 : BOOL; (*reserve operating message 161*) (*import HMI Extension*)
		bMsg6754 : BOOL; (*reserve operating message 162*) (*import HMI Extension*)
		bMsg6755 : BOOL; (*reserve operating message 163*) (*import HMI Extension*)
		bMsg6756 : BOOL; (*reserve operating message 164*) (*import HMI Extension*)
		bMsg6757 : BOOL; (*reserve operating message 165*) (*import HMI Extension*)
		bMsg6758 : BOOL; (*reserve operating message 166*) (*import HMI Extension*)
		bMsg6759 : BOOL; (*reserve operating message 167*) (*import HMI Extension*)
		bMsg6760 : BOOL; (*reserve operating message 168*) (*import HMI Extension*)
		bMsg6761 : BOOL; (*reserve operating message 169*) (*import HMI Extension*)
		bMsg6762 : BOOL; (*reserve operating message 170*) (*import HMI Extension*)
		bMsg6763 : BOOL; (*reserve operating message 171*) (*import HMI Extension*)
		bMsg6764 : BOOL; (*reserve operating message 172*) (*import HMI Extension*)
		bMsg6765 : BOOL; (*reserve operating message 173*) (*import HMI Extension*)
		bMsg6766 : BOOL; (*reserve operating message 174*) (*import HMI Extension*)
		bMsg6767 : BOOL; (*reserve operating message 175*) (*import HMI Extension*)
		bMsg6768 : BOOL; (*reserve operating message 176*) (*import HMI Extension*)
		bMsg6769 : BOOL; (*reserve operating message 177*) (*import HMI Extension*)
		bMsg6770 : BOOL; (*reserve operating message 178*) (*import HMI Extension*)
		bMsg6771 : BOOL; (*reserve operating message 179*) (*import HMI Extension*)
		bMsg6772 : BOOL; (*reserve operating message 180*) (*import HMI Extension*)
		bMsg6773 : BOOL; (*reserve operating message 181*) (*import HMI Extension*)
		bMsg6774 : BOOL; (*reserve operating message 182*) (*import HMI Extension*)
		bMsg6775 : BOOL; (*reserve operating message 183*) (*import HMI Extension*)
		bMsg6776 : BOOL; (*reserve operating message 184*) (*import HMI Extension*)
		bMsg6777 : BOOL; (*reserve operating message 185*) (*import HMI Extension*)
		bMsg6778 : BOOL; (*reserve operating message 186*) (*import HMI Extension*)
		bMsg6779 : BOOL; (*reserve operating message 187*) (*import HMI Extension*)
		bMsg6780 : BOOL; (*reserve operating message 188*) (*import HMI Extension*)
		bMsg6781 : BOOL; (*reserve operating message 189*) (*import HMI Extension*)
		bMsg6782 : BOOL; (*reserve operating message 190*) (*import HMI Extension*)
		bMsg6783 : BOOL; (*reserve operating message 191*) (*import HMI Extension*)
		bMsg6784 : BOOL; (*reserve operating message 192*) (*import HMI Extension*)
		bMsg6785 : BOOL; (*reserve operating message 193*) (*import HMI Extension*)
		bMsg6786 : BOOL; (*reserve operating message 194*) (*import HMI Extension*)
		bMsg6787 : BOOL; (*reserve operating message 195*) (*import HMI Extension*)
		bMsg6788 : BOOL; (*reserve operating message 196*) (*import HMI Extension*)
		bMsg6789 : BOOL; (*reserve operating message 197*) (*import HMI Extension*)
		bMsg6790 : BOOL; (*reserve operating message 198*) (*import HMI Extension*)
		bMsg6791 : BOOL; (*reserve operating message 199*) (*import HMI Extension*)
		bMsg6792 : BOOL; (*reserve operating message 200*) (*import HMI Extension*)
		bMsg6793 : BOOL; (*reserve operating message 201*) (*import HMI Extension*)
		bMsg6794 : BOOL; (*reserve operating message 202*) (*import HMI Extension*)
		bMsg6795 : BOOL; (*reserve operating message 203*) (*import HMI Extension*)
		bMsg6796 : BOOL; (*reserve operating message 204*) (*import HMI Extension*)
		bMsg6797 : BOOL; (*reserve operating message 205*) (*import HMI Extension*)
		bMsg6798 : BOOL; (*reserve operating message 206*) (*import HMI Extension*)
		bMsg6799 : BOOL; (*reserve operating message 207*) (*import HMI Extension*)
		bMsg6800 : BOOL; (*reserve operating message 208*) (*import HMI Extension*)
		bMsg6801 : BOOL; (*reserve operating message 209*) (*import HMI Extension*)
		bMsg6802 : BOOL; (*reserve operating message 210*) (*import HMI Extension*)
		bMsg6803 : BOOL; (*reserve operating message 211*) (*import HMI Extension*)
		bMsg6804 : BOOL; (*reserve operating message 212*) (*import HMI Extension*)
		bMsg6805 : BOOL; (*reserve operating message 213*) (*import HMI Extension*)
		bMsg6806 : BOOL; (*reserve operating message 214*) (*import HMI Extension*)
		bMsg6807 : BOOL; (*reserve operating message 215*) (*import HMI Extension*)
		bMsg6808 : BOOL; (*reserve operating message 216*) (*import HMI Extension*)
		bMsg6809 : BOOL; (*reserve operating message 217*) (*import HMI Extension*)
		bMsg6810 : BOOL; (*reserve operating message 218*) (*import HMI Extension*)
		bMsg6811 : BOOL; (*reserve operating message 219*) (*import HMI Extension*)
		bMsg6812 : BOOL; (*reserve operating message 220*) (*import HMI Extension*)
		bMsg6813 : BOOL; (*reserve operating message 221*) (*import HMI Extension*)
		bMsg6814 : BOOL; (*reserve operating message 222*) (*import HMI Extension*)
		bMsg6815 : BOOL; (*reserve operating message 223*) (*import HMI Extension*)
		bMsg6816 : BOOL; (*reserve operating message 224*) (*import HMI Extension*)
		bMsg6817 : BOOL; (*reserve operating message 225*) (*import HMI Extension*)
		bMsg6818 : BOOL; (*reserve operating message 226*) (*import HMI Extension*)
		bMsg6819 : BOOL; (*reserve operating message 227*) (*import HMI Extension*)
		bMsg6820 : BOOL; (*reserve operating message 228*) (*import HMI Extension*)
		bMsg6821 : BOOL; (*reserve operating message 229*) (*import HMI Extension*)
		bMsg6822 : BOOL; (*reserve operating message 230*) (*import HMI Extension*)
		bMsg6823 : BOOL; (*reserve operating message 231*) (*import HMI Extension*)
		bMsg6824 : BOOL; (*reserve operating message 232*) (*import HMI Extension*)
		bMsg6825 : BOOL; (*reserve operating message 233*) (*import HMI Extension*)
		bMsg6826 : BOOL; (*reserve operating message 234*) (*import HMI Extension*)
		bMsg6827 : BOOL; (*reserve operating message 235*) (*import HMI Extension*)
		bMsg6828 : BOOL; (*reserve operating message 236*) (*import HMI Extension*)
		bMsg6829 : BOOL; (*reserve operating message 237*) (*import HMI Extension*)
		bMsg6830 : BOOL; (*reserve operating message 238*) (*import HMI Extension*)
		bMsg6831 : BOOL; (*reserve operating message 239*) (*import HMI Extension*)
		bMsg6832 : BOOL; (*reserve operating message 240*) (*import HMI Extension*)
		bMsg6833 : BOOL; (*reserve operating message 241*) (*import HMI Extension*)
		bMsg6834 : BOOL; (*reserve operating message 242*) (*import HMI Extension*)
		bMsg6835 : BOOL; (*reserve operating message 243*) (*import HMI Extension*)
		bMsg6836 : BOOL; (*reserve operating message 244*) (*import HMI Extension*)
		bMsg6837 : BOOL; (*reserve operating message 245*) (*import HMI Extension*)
		bMsg6838 : BOOL; (*reserve operating message 246*) (*import HMI Extension*)
		bMsg6839 : BOOL; (*reserve operating message 247*) (*import HMI Extension*)
		bMsg6840 : BOOL; (*reserve operating message 248*) (*import HMI Extension*)
		bMsg6841 : BOOL; (*reserve operating message 249*) (*import HMI Extension*)
		bMsg6842 : BOOL; (*reserve operating message 250*) (*import HMI Extension*)
		bMsg6843 : BOOL; (*reserve operating message 251*) (*import HMI Extension*)
		bMsg6844 : BOOL; (*reserve operating message 252*) (*import HMI Extension*)
		bMsg6845 : BOOL; (*reserve operating message 253*) (*import HMI Extension*)
		bMsg6846 : BOOL; (*reserve operating message 254*) (*import HMI Extension*)
		bMsg6847 : BOOL; (*reserve operating message 255*) (*import HMI Extension*)
		bMsg6848 : BOOL; (*reserve operating message 256*) (*import HMI Extension*)
		bMsg6849 : BOOL; (*reserve operating message 257*) (*import HMI Extension*)
		bMsg6850 : BOOL; (*reserve operating message 258*) (*import HMI Extension*)
		bMsg6851 : BOOL; (*reserve operating message 259*) (*import HMI Extension*)
		bMsg6852 : BOOL; (*reserve operating message 260*) (*import HMI Extension*)
		bMsg6853 : BOOL; (*reserve operating message 261*) (*import HMI Extension*)
		bMsg6854 : BOOL; (*reserve operating message 262*) (*import HMI Extension*)
		bMsg6855 : BOOL; (*reserve operating message 263*) (*import HMI Extension*)
		bMsg6856 : BOOL; (*reserve operating message 264*) (*import HMI Extension*)
		bMsg6857 : BOOL; (*reserve operating message 265*) (*import HMI Extension*)
		bMsg6858 : BOOL; (*reserve operating message 266*) (*import HMI Extension*)
		bMsg6859 : BOOL; (*reserve operating message 267*) (*import HMI Extension*)
		bMsg6860 : BOOL; (*reserve operating message 268*) (*import HMI Extension*)
		bMsg6861 : BOOL; (*reserve operating message 269*) (*import HMI Extension*)
		bMsg6862 : BOOL; (*reserve operating message 270*) (*import HMI Extension*)
		bMsg6863 : BOOL; (*reserve operating message 271*) (*import HMI Extension*)
		bMsg6864 : BOOL; (*reserve operating message 272*) (*import HMI Extension*)
		bMsg6865 : BOOL; (*reserve operating message 273*) (*import HMI Extension*)
		bMsg6866 : BOOL; (*reserve operating message 274*) (*import HMI Extension*)
		bMsg6867 : BOOL; (*reserve operating message 275*) (*import HMI Extension*)
		bMsg6868 : BOOL; (*reserve operating message 276*) (*import HMI Extension*)
		bMsg6869 : BOOL; (*reserve operating message 277*) (*import HMI Extension*)
		bMsg6870 : BOOL; (*reserve operating message 278*) (*import HMI Extension*)
		bMsg6871 : BOOL; (*reserve operating message 279*) (*import HMI Extension*)
		bMsg6872 : BOOL; (*reserve operating message 280*) (*import HMI Extension*)
		bMsg6873 : BOOL; (*reserve operating message 281*) (*import HMI Extension*)
		bMsg6874 : BOOL; (*reserve operating message 282*) (*import HMI Extension*)
		bMsg6875 : BOOL; (*reserve operating message 283*) (*import HMI Extension*)
		bMsg6876 : BOOL; (*reserve operating message 284*) (*import HMI Extension*)
		bMsg6877 : BOOL; (*reserve operating message 285*) (*import HMI Extension*)
		bMsg6878 : BOOL; (*reserve operating message 286*) (*import HMI Extension*)
		bMsg6879 : BOOL; (*reserve operating message 287*) (*import HMI Extension*)
		bMsg6880 : BOOL; (*reserve operating message 288*) (*import HMI Extension*)
		bMsg6881 : BOOL; (*reserve operating message 289*) (*import HMI Extension*)
		bMsg6882 : BOOL; (*reserve operating message 290*) (*import HMI Extension*)
		bMsg6883 : BOOL; (*reserve operating message 291*) (*import HMI Extension*)
		bMsg6884 : BOOL; (*reserve operating message 292*) (*import HMI Extension*)
		bMsg6885 : BOOL; (*reserve operating message 293*) (*import HMI Extension*)
		bMsg6886 : BOOL; (*reserve operating message 294*) (*import HMI Extension*)
		bMsg6887 : BOOL; (*reserve operating message 295*) (*import HMI Extension*)
		bMsg6888 : BOOL; (*reserve operating message 296*) (*import HMI Extension*)
		bMsg6889 : BOOL; (*reserve operating message 297*) (*import HMI Extension*)
		bMsg6890 : BOOL; (*reserve operating message 298*) (*import HMI Extension*)
		bMsg6891 : BOOL; (*reserve operating message 299*) (*import HMI Extension*)
		bMsg6892 : BOOL; (*reserve operating message 300*) (*import HMI Extension*)
		bMsg6893 : BOOL; (*reserve operating message 301*) (*import HMI Extension*)
		bMsg6894 : BOOL; (*reserve operating message 302*) (*import HMI Extension*)
		bMsg6895 : BOOL; (*reserve operating message 303*) (*import HMI Extension*)
		bMsg6896 : BOOL; (*reserve operating message 304*) (*import HMI Extension*)
		bMsg6897 : BOOL; (*reserve operating message 305*) (*import HMI Extension*)
		bMsg6898 : BOOL; (*reserve operating message 306*) (*import HMI Extension*)
		bMsg6899 : BOOL; (*reserve operating message 307*) (*import HMI Extension*)
		bMsg6700 : BOOL; (* DO NOT USE 308! reserve operating message 308 DO NOT USE LINE!*) (*import HMI Extension*)
		bMsg8701 : BOOL; (*reserve warning message 127*) (*import HMI Extension*)
		bMsg8702 : BOOL; (*reserve warning message 128*) (*import HMI Extension*)
		bMsg8703 : BOOL; (*reserve warning message 129*) (*import HMI Extension*)
		bMsg8704 : BOOL; (*reserve warning message 130*) (*import HMI Extension*)
		bMsg8705 : BOOL; (*reserve warning message 131*) (*import HMI Extension*)
		bMsg8706 : BOOL; (*reserve warning message 132*) (*import HMI Extension*)
		bMsg8707 : BOOL; (*reserve warning message 133*) (*import HMI Extension*)
		bMsg8708 : BOOL; (*reserve warning message 134*) (*import HMI Extension*)
		bMsg8709 : BOOL; (*reserve warning message 135*) (*import HMI Extension*)
		bMsg8710 : BOOL; (*reserve warning message 136*) (*import HMI Extension*)
		bMsg8711 : BOOL; (*reserve warning message 137*) (*import HMI Extension*)
		bMsg8712 : BOOL; (*reserve warning message 138*) (*import HMI Extension*)
		bMsg8713 : BOOL; (*reserve warning message 139*) (*import HMI Extension*)
		bMsg8714 : BOOL; (*reserve warning message 140*) (*import HMI Extension*)
		bMsg8715 : BOOL; (*reserve warning message 141*) (*import HMI Extension*)
		bMsg8716 : BOOL; (*reserve warning message 142*) (*import HMI Extension*)
		bMsg8717 : BOOL; (*reserve warning message 143*) (*import HMI Extension*)
		bMsg8718 : BOOL; (*reserve warning message 144*) (*import HMI Extension*)
		bMsg8719 : BOOL; (*reserve warning message 145*) (*import HMI Extension*)
		bMsg8720 : BOOL; (*reserve warning message 146*) (*import HMI Extension*)
		bMsg8721 : BOOL; (*reserve warning message 147*) (*import HMI Extension*)
		bMsg8722 : BOOL; (*reserve warning message 148*) (*import HMI Extension*)
		bMsg8723 : BOOL; (*reserve warning message 149*) (*import HMI Extension*)
		bMsg8724 : BOOL; (*reserve warning message 150*) (*import HMI Extension*)
		bMsg8725 : BOOL; (*reserve warning message 151*) (*import HMI Extension*)
		bMsg8726 : BOOL; (*reserve warning message 152*) (*import HMI Extension*)
		bMsg8727 : BOOL; (*reserve warning message 153*) (*import HMI Extension*)
		bMsg8728 : BOOL; (*reserve warning message 154*) (*import HMI Extension*)
		bMsg8729 : BOOL; (*reserve warning message 155*) (*import HMI Extension*)
		bMsg8730 : BOOL; (*reserve warning message 156*) (*import HMI Extension*)
		bMsg8731 : BOOL; (*reserve warning message 157*) (*import HMI Extension*)
		bMsg8732 : BOOL; (*reserve warning message 158*) (*import HMI Extension*)
		bMsg8733 : BOOL; (*reserve warning message 159*) (*import HMI Extension*)
		bMsg8734 : BOOL; (*reserve warning message 160*) (*import HMI Extension*)
		bMsg8735 : BOOL; (*reserve warning message 161*) (*import HMI Extension*)
		bMsg8736 : BOOL; (*reserve warning message 162*) (*import HMI Extension*)
		bMsg8737 : BOOL; (*reserve warning message 163*) (*import HMI Extension*)
		bMsg8738 : BOOL; (*reserve warning message 164*) (*import HMI Extension*)
		bMsg8739 : BOOL; (*reserve warning message 165*) (*import HMI Extension*)
		bMsg8740 : BOOL; (*reserve warning message 166*) (*import HMI Extension*)
		bMsg8741 : BOOL; (*reserve warning message 167*) (*import HMI Extension*)
		bMsg8742 : BOOL; (*reserve warning message 168*) (*import HMI Extension*)
		bMsg8743 : BOOL; (*reserve warning message 169*) (*import HMI Extension*)
		bMsg8744 : BOOL; (*reserve warning message 170*) (*import HMI Extension*)
		bMsg8745 : BOOL; (*reserve warning message 171*) (*import HMI Extension*)
		bMsg8746 : BOOL; (*reserve warning message 172*) (*import HMI Extension*)
		bMsg8747 : BOOL; (*reserve warning message 173*) (*import HMI Extension*)
		bMsg8748 : BOOL; (*reserve warning message 174*) (*import HMI Extension*)
		bMsg8749 : BOOL; (*reserve warning message 175*) (*import HMI Extension*)
		bMsg8750 : BOOL; (*reserve warning message 176*) (*import HMI Extension*)
		bMsg8751 : BOOL; (*reserve warning message 177*) (*import HMI Extension*)
		bMsg8752 : BOOL; (*reserve warning message 178*) (*import HMI Extension*)
		bMsg8753 : BOOL; (*reserve warning message 179*) (*import HMI Extension*)
		bMsg8754 : BOOL; (*reserve warning message 180*) (*import HMI Extension*)
		bMsg8755 : BOOL; (*reserve warning message 181*) (*import HMI Extension*)
		bMsg8756 : BOOL; (*reserve warning message 182*) (*import HMI Extension*)
		bMsg8757 : BOOL; (*reserve warning message 183*) (*import HMI Extension*)
		bMsg8758 : BOOL; (*reserve warning message 184*) (*import HMI Extension*)
		bMsg8759 : BOOL; (*reserve warning message 185*) (*import HMI Extension*)
		bMsg8760 : BOOL; (*reserve warning message 186*) (*import HMI Extension*)
		bMsg8761 : BOOL; (*reserve warning message 187*) (*import HMI Extension*)
		bMsg8762 : BOOL; (*reserve warning message 188*) (*import HMI Extension*)
		bMsg8763 : BOOL; (*reserve warning message 189*) (*import HMI Extension*)
		bMsg8764 : BOOL; (*reserve warning message 190*) (*import HMI Extension*)
		bMsg8765 : BOOL; (*reserve warning message 191*) (*import HMI Extension*)
		bMsg8766 : BOOL; (*reserve warning message 192*) (*import HMI Extension*)
		bMsg8767 : BOOL; (*reserve warning message 193*) (*import HMI Extension*)
		bMsg8768 : BOOL; (*reserve warning message 194*) (*import HMI Extension*)
		bMsg8769 : BOOL; (*reserve warning message 195*) (*import HMI Extension*)
		bMsg8770 : BOOL; (*reserve warning message 196*) (*import HMI Extension*)
		bMsg8771 : BOOL; (*reserve warning message 197*) (*import HMI Extension*)
		bMsg8772 : BOOL; (*reserve warning message 198*) (*import HMI Extension*)
		bMsg8773 : BOOL; (*reserve warning message 199*) (*import HMI Extension*)
		bMsg8774 : BOOL; (*reserve warning message 200*) (*import HMI Extension*)
		bMsg8775 : BOOL; (*reserve warning message 201*) (*import HMI Extension*)
		bMsg8776 : BOOL; (*reserve warning message 202*) (*import HMI Extension*)
		bMsg8777 : BOOL; (*reserve warning message 203*) (*import HMI Extension*)
		bMsg8778 : BOOL; (*reserve warning message 204*) (*import HMI Extension*)
		bMsg8779 : BOOL; (*reserve warning message 205*) (*import HMI Extension*)
		bMsg8780 : BOOL; (*reserve warning message 206*) (*import HMI Extension*)
		bMsg8781 : BOOL; (*reserve warning message 207*) (*import HMI Extension*)
		bMsg8782 : BOOL; (*reserve warning message 208*) (*import HMI Extension*)
		bMsg8783 : BOOL; (*reserve warning message 209*) (*import HMI Extension*)
		bMsg8784 : BOOL; (*reserve warning message 210*) (*import HMI Extension*)
		bMsg8785 : BOOL; (*reserve warning message 211*) (*import HMI Extension*)
		bMsg8786 : BOOL; (*reserve warning message 212*) (*import HMI Extension*)
		bMsg8787 : BOOL; (*reserve warning message 213*) (*import HMI Extension*)
		bMsg8788 : BOOL; (*reserve warning message 214*) (*import HMI Extension*)
		bMsg8789 : BOOL; (*reserve warning message 215*) (*import HMI Extension*)
		bMsg8790 : BOOL; (*reserve warning message 216*) (*import HMI Extension*)
		bMsg8791 : BOOL; (*reserve warning message 217*) (*import HMI Extension*)
		bMsg8792 : BOOL; (*reserve warning message 218*) (*import HMI Extension*)
		bMsg8793 : BOOL; (*reserve warning message 219*) (*import HMI Extension*)
		bMsg8794 : BOOL; (*reserve warning message 220*) (*import HMI Extension*)
		bMsg8795 : BOOL; (*reserve warning message 221*) (*import HMI Extension*)
		bMsg8796 : BOOL; (*reserve warning message 222*) (*import HMI Extension*)
		bMsg8797 : BOOL; (*reserve warning message 223*) (*import HMI Extension*)
		bMsg8798 : BOOL; (*reserve warning message 224*) (*import HMI Extension*)
		bMsg8799 : BOOL; (*reserve warning message 225*) (*import HMI Extension*) (*		bMsg4300 : BOOL; (xxx do not use this 226 *reserve warning message 226*)
		bMsg7966 : BOOL; (*reserve analog in 1 limit warning message*)
		bMsg7967 : BOOL; (*reserve analog in 2 limit warning message*)
		bMsg7968 : BOOL; (*reserve analog in 3 limit warning message*)
		bMsg7969 : BOOL; (*reserve analog in 4 limit warning message*)
		bMsg7970 : BOOL; (*reserve analog in 5 limit warning message*)
		bMsg7971 : BOOL; (*reserve analog in 6 limit warning message*)
		bMsg7972 : BOOL; (*reserve analog in 7 limit warning message*)
		bMsg7973 : BOOL; (*reserve analog in 8 limit warning message*)
		bMsg7974 : BOOL; (*reserve analog in 9 limit warning message*)
		bMsg7975 : BOOL; (*reserve analog in 10 limit warning message*)
		bMsg7976 : BOOL; (*reserve analog in 11 limit warning message*)
		bMsg7977 : BOOL; (*reserve analog in 12 limit warning message*)
		bMsg7978 : BOOL; (*reserve analog in 13 limit warning message*)
		bMsg7979 : BOOL; (*reserve analog in 14 limit warning message*)
		bMsg7980 : BOOL; (*reserve analog in 15 limit warning message*)
		bMsg7981 : BOOL; (*reserve analog in 16 limit warning message*)
		bMsg7982 : BOOL; (*reserve analog in 17 limit warning message*)
		bMsg7983 : BOOL; (*reserve analog in 18 limit warning message*)
		bMsg7984 : BOOL; (*reserve analog in 19 limit warning message*)
		bMsg7985 : BOOL; (*reserve analog in 20 limit warning message*)
		bMsg7986 : BOOL; (*reserve analog in 21 limit warning message*)
		bMsg7987 : BOOL; (*reserve analog in 22 limit warning message*)
		bMsg7988 : BOOL; (*reserve analog in 23 limit warning message*)
		bMsg7989 : BOOL; (*reserve analog in 24 limit warning message*)
		bMsg7990 : BOOL; (*reserve analog in 25 limit warning message*)
		bMsg7991 : BOOL; (*reserve analog in 26 limit warning message*)
		bMsg7992 : BOOL; (*reserve analog in 27 limit warning message*)
		bMsg7993 : BOOL; (*reserve analog in 28 limit warning message*)
		bMsg7994 : BOOL; (*reserve analog in 29 limit warning message*)
		bMsg7995 : BOOL; (*reserve analog in 30 limit warning message*)
		bMsg7996 : BOOL; (*reserve analog in 31 limit warning message*)
		bMsg7997 : BOOL; (*reserve analog in 32 limit warning message*)
		bMsg8966 : BOOL; (*reserve analog in 1 limit alarm message*)
		bMsg8967 : BOOL; (*reserve analog in 2 limit alarm message*)
		bMsg8968 : BOOL; (*reserve analog in 3 limit alarm message*)
		bMsg8969 : BOOL; (*reserve analog in 4 limit alarm message*)
		bMsg8970 : BOOL; (*reserve analog in 5 limit alarm message*)
		bMsg8971 : BOOL; (*reserve analog in 6 limit alarm message*)
		bMsg8972 : BOOL; (*reserve analog in 7 limit alarm message*)
		bMsg8973 : BOOL; (*reserve analog in 8 limit alarm message*)
		bMsg8974 : BOOL; (*reserve analog in 9 limit alarm message*)
		bMsg8975 : BOOL; (*reserve analog in 10 limit alarm message*)
		bMsg8976 : BOOL; (*reserve analog in 11 limit alarm message*)
		bMsg8977 : BOOL; (*reserve analog in 12 limit alarm message*)
		bMsg8978 : BOOL; (*reserve analog in 13 limit alarm message*)
		bMsg8979 : BOOL; (*reserve analog in 14 limit alarm message*)
		bMsg8980 : BOOL; (*reserve analog in 15 limit alarm message*)
		bMsg8981 : BOOL; (*reserve analog in 16 limit alarm message*)
		bMsg8982 : BOOL; (*reserve analog in 17 limit alarm message*)
		bMsg8983 : BOOL; (*reserve analog in 18 limit alarm message*)
		bMsg8984 : BOOL; (*reserve analog in 19 limit alarm message*)
		bMsg8985 : BOOL; (*reserve analog in 20 limit alarm message*)
		bMsg8986 : BOOL; (*reserve analog in 21 limit alarm message*)
		bMsg8987 : BOOL; (*reserve analog in 22 limit alarm message*)
		bMsg8988 : BOOL; (*reserve analog in 23 limit alarm message*)
		bMsg8989 : BOOL; (*reserve analog in 24 limit alarm message*)
		bMsg8990 : BOOL; (*reserve analog in 25 limit alarm message*)
		bMsg8991 : BOOL; (*reserve analog in 26 limit alarm message*)
		bMsg8992 : BOOL; (*reserve analog in 27 limit alarm message*)
		bMsg8993 : BOOL; (*reserve analog in 28 limit alarm message*)
		bMsg8994 : BOOL; (*reserve analog in 29 limit alarm message*)
		bMsg8995 : BOOL; (*reserve analog in 30 limit alarm message*)
		bMsg8996 : BOOL; (*reserve analog in 31 limit alarm message*)
		bMsg8997 : BOOL; (*reserve analog in 32 limit alarm message*)
		bMsg8998 : BOOL; (*reserve analog in 32 limit alarm message*)
		bMsg8999 : BOOL; (*reserve analog in 32 limit alarm message*)
		bN_Set_ExtAI_Enable : BOOL; (* *) (*OldName: AW_EXDSH; Cycle: 5;*)
		bOptGT_RatioMix_Set : BOOL; (*activation bit for custom gasmixing ratio setpoint - new V4.5*)
		bParaSetupOk : BOOL; (* = 	FGDRPS	-	parameter setup ok - release RPS operation (bAllModulesOk)	*) (*OldName: unknown	; Cycle: 5;*)
		bPFBC_GenC_SetErrBC : BOOL; (* bus: setpoint generator power factor (COS PHI) from EU error - use backupvalue *) (* OldName: bMSST_BUS_GCQ_PF; Cycle:5; *)
		bPFC_SetCOf : BOOL; (* primary frequency control - off (deactivate) *) (* OldName: DI_GCP_PFC_R; Cycle:HALioDi_Type; *)
		bPFC_SetCOn : BOOL; (* primary frequency control - on (activate) *) (* OldName: DI_GCP_PFC_S; Cycle:HALioDi_Type; *)
		bPFUC_GenC_SetEUCOf : BOOL; (* setpoint reactive power characteristics COS(phi)=f(U) von EU -off (deactive) *) (* OldName: DI_GCQ_PFU_R; Cycle:HALioDi_Type; *)
		bPFUC_GenC_SetEUCOn : BOOL; (* setpoint reactive power characteristics COS(phi)=f(U) von EU -on (active) *) (* OldName: DI_GCQ_PFU_S; Cycle:HALioDi_Type; *)
		bPF_GenC_SetEUCOf : BOOL; (* setpoint  genetaror power factor (COS PHI) from EVA - off (deactivate)  *) (* OldName: DI_GCQ_PF_R; Cycle:HALioDi_Type; *)
		bPF_GenC_SetEUCOn : BOOL; (* setpoint  genetaror power factor (COS PHI) from EU - on (activate)  *) (* OldName: DI_GCQ_PF_S; Cycle:HALioDi_Type; *)
		bPLim_GenC_SetEUCOf : BOOL; (* setpoint power limitation (Plim) from EU - off (deactivate) *) (* OldName: DI_GCP_Plim_R; Cycle:HALioDi_Type; *)
		bPLim_GenC_SetEUCOn : BOOL; (* setpoint power limitation (Plim) from EU - on (activate) *) (* OldName: DI_GCP_Plim_S; Cycle:HALioDi_Type; *)
		bPU_SetCOf : BOOL; (*demand off  P(U) over DIs*)
		bPU_SetCOn : BOOL; (*demand on P(U) over DIs*)
		bP_GenC_SetErr : BOOL; (* Generator power setpoint measuring signal failure *) (* OldName: bMSST_BUS_GCP_P; Cycle:5; *)
		bP_GenC_SetErrPlim : BOOL; (* Leistungslimitierung BUS EU gestoert - Backupwert verwenden *) (* OldName: bMSST_BUS_GCP_Plim; Cycle:5; *)
		bP_GenC_SetEUCOf : BOOL; (* request power value from EU - off (deactivate) *) (* OldName: DI_GCP_P_R; Cycle:HALioDi_Type; *)
		bP_GenC_SetEUCOn : BOOL; (* request power value from EU - on (activate) *) (* OldName: DI_GCP_P_S; Cycle:HALioDi_Type; *)
		bP_Red_AI_Enable : BOOL; (* *) (*OldName: RED_EVU_Aktiv; Cycle: 5;*)
		bP_Red_EVU_Enable : BOOL; (* *) (*OldName: RED_EVU_Aktiv; Cycle: 5;*)
		bP_Red_Sp_Lim1Act : BOOL; (* power setpoint limit 1 activ *) (*OldName: bPowerSetpointLimit1; Cycle: 5;*)
		bP_Red_Sp_Lim2Act : BOOL; (* power setpoint limit 2 activ *) (*OldName: bPowerSetpointLimit2; Cycle: 5;*)
		bP_Red_Sp_Lim3Act : BOOL; (* power setpoint limit 3 activ *) (*OldName: bPowerSetpointLimit3; Cycle: 5;*)
		bP_Set_Ctr_Mns_Enable : BOOL; (*! new V4.5 2017 !  (Mains Power Controller)*)
		bP_Set_ExtAI_Enable : BOOL; (* *) (*OldName: ssNominalPowerAnalog		; Cycle: 5;*)
		bP_Set_ExtDI_Enable : BOOL; (* *) (*OldName: AW_EXPSH_DI; Cycle: 5;*)
		bQLim_GenC_SetEUCOf : BOOL; (* setpoint reactive power limitation (Qlim) from EU - off (deactivate) *) (* OldName: DI_GCQ_Qlim_R; Cycle:HALioDi_Type; *)
		bQLim_GenC_SetEUCOn : BOOL; (* setpoint reactive power limitation (Qlim) from EU - on (activate) *) (* OldName: DI_GCQ_Qlim_S; Cycle:HALioDi_Type; *)
		bQPC_GenC_SetEUCOf : BOOL; (* setpoint reactive power characteristics COS(phi)=f(P) from EU - off (deactivate) *) (* OldName: DI_GCQ_PFP_R; Cycle:HALioDi_Type; *)
		bQPC_GenC_SetEUCOn : BOOL; (* setpoint reactive power characteristics COS(phi)=f(P) from EU - on (activate) *) (* OldName: DI_GCQ_PFP_S; Cycle:HALioDi_Type; *)
		bQP_GenC_SetEUCOf : BOOL; (* DI setpoint reactive power characteristics Q=f(P) from EU - off (deactivate) *)
		bQP_GenC_SetEUCOn : BOOL; (* DI setpoint reactive power characteristics Q=f(P) from EU - on (activate) *)
		bQUC_GenC_SetEUCOf : BOOL; (* setpoint reactive power characteristics Q=f(U) from EU -off (deactivate) *) (* OldName: DI_GCQ_QU_R; Cycle:HALioDi_Type; *)
		bQUC_GenC_SetEUCOn : BOOL; (* setpoint reactive power characteristics Q=f(U) from EU -on (activate) *) (* OldName: DI_GCQ_QU_S; Cycle:HALioDi_Type; *)
		bQ_GenC_SetErrBC : BOOL; (* W3594 - Q setpoint BUS EU error - use Backupvalue *) (* OldName: bMSST_BUS_GCQ_Q; Cycle:5; *)
		bQ_GenC_SetErrQlim : BOOL; (* W3595 - reactive power limitation meassur signal error *) (* OldName: bMSST_BUS_GCQ_Qlim; Cycle:5; *)
		bQ_GenC_SetEUCOf : BOOL; (* setpoint reactive power characteristic (Q) from EU - off (deactivate) *) (* OldName: DI_GCQ_Q_R; Cycle:HALioDi_Type; *)
		bQ_GenC_SetEUCOn : BOOL; (* setpoint reactive power characteristic (Q) from EU - on (activate) *) (* OldName: DI_GCQ_Q_S; Cycle:HALioDi_Type; *)
		bRelSy_Customized : BOOL; (*Freigabe Syncronisierungl vo Customized Modul*)
		bReqMaintenance : BOOL; (* =    maintenance counter has run out *) (*OldName: WART; Cycle: 5;*)
		bResetRemBus : BOOL; (* remote reset from fieldbus *)
		bRMC_SetCOf : BOOL; (* regulation margin control -off (deactivate) *) (* OldName: DI_GCP_RMC_R; Cycle:HALioDi_Type; *)
		bRMC_SetCOn : BOOL; (* regulation margin control -on (activate) *) (* OldName: DI_GCP_RMC_S; Cycle:HALioDi_Type; *)
		bRPM_Count1 : BOOL; (* = 		-	Report of daily operation hour counter	*) (*OldName: RPMZ1; Cycle: 5;*)
		bRPM_Count2 : BOOL; (* = 		-	Report of daily operation hour counter	*) (*OldName: RPMZ2; Cycle: 5;*)
		bRPM_Count3 : BOOL; (* = 		-	Report of daily operation hour counter	*) (*OldName: RPMZ3; Cycle: 5;*)
		bRPM_Count4 : BOOL; (* = 		-	Report of daily operation hour counter	*) (*OldName: RPMZ4; Cycle: 5;*)
		bRPM_Count5 : BOOL; (* = 		-	Report of daily operation hour counter	*) (*OldName: RPMZ5; Cycle: 5;*)
		bRPM_Count6 : BOOL; (* = 		-	Report of daily operation hour counter	*) (*OldName: RPMZ6; Cycle: 5;*)
		bRPM_Count7 : BOOL; (* = 		-	Report of daily operation hour counter	*) (*OldName: RPMZ7; Cycle: 5;*)
		bRPM_Count8 : BOOL; (* = 		-	Report of daily operation hour counter	*) (*OldName: RPMZ8; Cycle: 5;*)
		bRPM_Count9 : BOOL; (* = 		-	Report of daily operation hour counter	*) (*OldName: RPMZ9; Cycle: 5;*)
		bRPM_Count10 : BOOL; (* = 		-	Report of daily operation hour counter	*) (*OldName: RPMZ10; Cycle: 5;*)
		bRPM_Count11 : BOOL; (* = 		-	Report of daily operation hour counter	*) (*OldName: RPMZ11; Cycle: 5;*)
		bRPM_Count12 : BOOL; (* = 		-	Report of daily operation hour counter	*) (*OldName: RPMZ12; Cycle: 5;*)
		bRPM_Count13 : BOOL; (* = 		-	Report of daily operation hour counter	*) (*OldName: RPMZ13; Cycle: 5;*)
		bRPM_Count14 : BOOL; (* = 		-	Report of daily operation hour counter	*) (*OldName: RPMZ14; Cycle: 5;*)
		bRPM_Count15 : BOOL; (* = 		-	Report of daily operation hour counter	*) (*OldName: RPMZ15; Cycle: 5;*)
		bRPM_Count16 : BOOL; (* = 		-	Report of daily operation hour counter	*) (*OldName: RPMZ16; Cycle: 5;*)
		bSet_ILF_COf_Bus : BOOL; (* Bus: local frequency integrator set command off *)
		bSet_ILF_COn_Bus : BOOL; (* Bus: local frequency integrator set command on*)
		bSet_FC_COf_Bus : BOOL; (* Bus: frequency control set command off *)
		bSet_FC_COn_Bus : BOOL; (* Bus: frequency control set command on*)
		bT_ChC_Ctr_Wex_Enable_Cust : BOOL;
		bUist_max : BOOL; (*TRUE = Uist for Q(U) & cosphi(U) max. generator voltage Ph-Ph, FALSE = average generator voltage Ph-Ph*)
		bUniDig : ARRAY[0..125]OF BOOL; (* ARRAY of processed digita channel  values from UniversalIO system bUniDig[1]  to bUniDig[255]*) (*OldName: bUniDig; Cycle: 5;*)
		bUseCtrCust2_4HumidityCtr : BOOL; (*! new V4.5 2017 !  Option to use CtrCust2 as LLTP controller with humidity function *)
		bU_GenC_SetErrBC : BOOL; (* bus: setpoint voltage from EU error - use backupvalue *)
		bU_GenC_SetEUCOf : BOOL; (*DI: Voltage control for reactive power - off (deactivated)*)
		bU_GenC_SetEUCOn : BOOL; (*DI: Voltage control for reactive power - on (activated)*)
		iCount1 : DINT; (* = OutDisplay Customized Counter*) (*OldName: ZAEHL_1; Cycle: 5;*)
		iCount2 : DINT; (* = OutDisplay Customized Counter*) (*OldName: ZAEHL_2; Cycle: 5;*)
		iCount3 : DINT; (* = OutDisplay Customized Counter*) (*OldName: ZAEHL_3; Cycle: 5;*)
		iCount4 : DINT; (* = OutDisplay Customized Counter*) (*OldName: ZAEHL_4; Cycle: 5;*)
		iCount5 : DINT; (* = OutDisplay Customized Counter*) (*OldName: new PV; Cycle: 5;*)
		iCount6 : DINT; (* = OutDisplay Customized Counter*) (*OldName: new PV; Cycle: 5;*)
		iCount7 : DINT; (* = OutDisplay Customized Counter*) (*OldName: new PV; Cycle: 5;*)
		iCount8 : DINT; (* = OutDisplay Customized Counter*) (*OldName: new PV; Cycle: 5;*)
		iCount9 : DINT; (* = OutDisplay Customized Counter*) (*OldName: new PV; Cycle: 5;*)
		iCount10 : DINT; (* = OutDisplay Customized Counter*) (*OldName: new PV; Cycle: 5;*)
		iCount11 : DINT; (* = OutDisplay Customized Counter*) (*OldName: new PV; Cycle: 5;*)
		iCount12 : DINT; (* = OutDisplay Customized Counter*) (*OldName: new PV; Cycle: 5;*)
		iCount13 : DINT; (* = OutDisplay Customized Counter*) (*OldName: new PV; Cycle: 5;*)
		iCount14 : DINT; (* = OutDisplay Customized Counter*) (*OldName: new PV; Cycle: 5;*)
		iCount15 : DINT; (* = OutDisplay Customized Counter*) (*OldName: new PV; Cycle: 5;*)
		iCount16 : DINT; (* = OutDisplay Customized Counter*) (*OldName: new PV; Cycle: 5;*)
		iCount17 : DINT; (* = OutDisplay Customized Counter*) (*OldName: new PV; Cycle: 5;*)
		iCount18 : DINT; (* = OutDisplay Customized Counter*) (*OldName: new PV; Cycle: 5;*)
		iCount19 : DINT; (* = OutDisplay Customized Counter*) (*OldName: new PV; Cycle: 5;*)
		iCount20 : DINT; (* = OutDisplay Customized Counter*) (*OldName: new PV; Cycle: 5;*)
		iGenC_PLimBC : INT; (* bus: setpoint power limitation (Plim) from EU - on (activate) *) (* OldName: BUS_GCP_Plim; Cycle:5; *)
		iGenC_PrioPF : USINT; (* Prioritet  genetaror power factor (COS(phi)) - fixvalue *) (* OldName: usPrio_PFset; Cycle:5; *)
		iGenC_PrioPFPC : USINT; (* Prioritet  reactive power characteristic COS(phi)=f(P) *) (* OldName: usPrio_PF_P; Cycle:5; *)
		iGenC_PrioPFUC : USINT; (* Prioritet  reactive power characteristic COS(phi)=f(U) *) (* OldName: usPrio_PF_U; Cycle:5; *)
		iGenC_PrioQ : USINT; (* Prioritet  reactive power (Q) - fixvalue *) (* OldName: usPrio_Qset; Cycle:5; *)
		iGenC_PrioQCustSet : USINT; (* Prioritet  reactive power Q customized 	*)
		iGenC_PrioQP : USINT; (* Prioritet  reactive power characteristic Q=f(P)  *)
		iGenC_PrioQUC : USINT; (* Prioritet  reactive power characteristic Q=f(U) *) (* OldName: usPrio_Q_U; Cycle:5; *)
		iGenC_PrioQUset : USINT; (* Prioritet  reactive power U control(Q) -    *)
		iIdx_ProcessStep_CU : DINT; (*Step Time Display*) (*new with V4.4, 2016*)
		iMaintenanceCount1 : DINT; (* = OutDisplay Maintenance Counter*) (*OldName: wart_z1; Cycle: 5;*)
		iMaintenanceCount2 : DINT; (* = OutDisplay Maintenance Counter*) (*OldName: wart_z2; Cycle: 5;*)
		iMaintenanceCount3 : DINT; (* = OutDisplay Maintenance Counter*) (*OldName: wart_z3; Cycle: 5;*)
		iMaintenanceCount4 : DINT; (* = OutDisplay Maintenance Counter*) (*OldName: wart_z4; Cycle: 5;*)
		iMaintenanceCount5 : DINT; (* = OutDisplay Maintenance Counter*) (*OldName: new PV; Cycle: 5;*)
		iMaintenanceCount6 : DINT; (* = OutDisplay Maintenance Counter*) (*OldName: new PV; Cycle: 5;*)
		iMaintenanceCount7 : DINT; (* = OutDisplay Maintenance Counter*) (*OldName: new PV; Cycle: 5;*)
		iMaintenanceCount8 : DINT; (* = OutDisplay Maintenance Counter*) (*OldName: new PV; Cycle: 5;*)
		iMsg69xxErrInfo : ARRAY[0..100]OF INT;
		iMsg79xxErrInfo : ARRAY[0..100]OF INT;
		iMsg89xxErrInfo : ARRAY[0..100]OF INT;
		iProcessStepTime_CU : DINT; (*Step Time Display*) (*new with V4.4, 2016*)
		iP_FC_RMC_neg : INT; (* Bus: negative reserve power for frequency control [kW]*)
		iP_FC_RMC_pos : INT; (* Bus: positive reserve power for frequency control [kW]*)
		iRPS_Day : DINT; (* = 	Time			*)
		iRPS_h : DINT; (* = 	Time			*)
		iRPS_m : DINT; (* = 	Time			*)
		iRPS_Month : DINT; (* = 	Time			*)
		iRPS_s : DINT; (* = 	Time			*)
		PF_GenC_SetFix1 : BOOL; (* setpoint  genetaror power factor (COS PHI) - Fixvalue 1 from EU *)
		PF_GenC_SetFix2 : BOOL; (* setpoint  genetaror power factor (COS PHI) - Fixvalue 2 from EU *)
		PF_GenC_SetFix3 : BOOL; (* setpoint  genetaror power factor (COS PHI) - Fixvalue 3 from EU *)
		PF_GenC_SetFix4 : BOOL; (* setpoint  genetaror power factor (COS PHI) - Fixvalue 4 from EU *)
		PF_GenC_SetFix5 : BOOL; (* setpoint  genetaror power factor (COS PHI) - Fixvalue 5 from EU *)
		PLim_GenC_SetEUPFix1 : BOOL; (*power limitation fixvalue 1 *)
		PLim_GenC_SetEUPFix2 : BOOL; (*power limitation fixvalue 2*)
		PLim_GenC_SetEUPFix3 : BOOL; (*power limitation fixvalue 3*)
		PLim_GenC_SetEUPFix4 : BOOL; (*power limitation fixvalue 4*)
		PLim_GenC_SetEUPFix5 : BOOL; (*power limitation fixvalue 5*)
		Pt_RAN1 : BOOL := 0; (* Pt100 *) (*OldName: unknown	; Cycle: 5;*)
		P_GenC_SetFix1 : BOOL;
		P_GenC_SetFix2 : BOOL;
		P_GenC_SetFix3 : BOOL;
		P_GenC_SetFix4 : BOOL;
		P_GenC_SetFix5 : BOOL;
		Q_GenC_SetFix1 : BOOL; (* reactive power (Q) - Q-fixvalue 1 from EU *)
		Q_GenC_SetFix2 : BOOL; (* reactive power (Q) - Q-fixvalue 2 from EU *)
		Q_GenC_SetFix3 : BOOL; (* reactive power (Q) - Q-fixvalue 3 from EU *)
		Q_GenC_SetFix4 : BOOL; (* reactive power (Q) - Q-fixvalue 4 from EU *)
		Q_GenC_SetFix5 : BOOL; (* reactive power (Q) - Q-fixvalue 5 from EU *)
		rCA_IgnP_CylOffset : ARRAY[0..24]OF REAL; (*ZZP Offset Vorgabe*)
		rCA_PI_Dur_COffset : ARRAY[0..24]OF REAL; (* custom PI duration offset *) (* OldName: ssTestBenchOffset; Cycle:2; *)
		rCtr_Cust2_W_set : REAL; (*! new V4.5 2017 !  Setpoint Ctr Cust 2 for Japan Option for humidity function *)
		rScalBlock_Y : ARRAY[0..30]OF REAL; (*Y form scaling blocks*)
		bScalBlock_Err : ARRAY[0..30]OF BOOL; (*Error flag from scaling blocks*)
		rCustAnaIn : ARRAY[0..120]OF REAL; (* =ANA.RAN1 to ANA.RAN44(16)	-measured and scaled signal from reserve channel, copied for reuse in other modules*) (*OldName: ANA.RAN1, ANA.RAN2, ANA.RAN3, ANA.RAN16	; Cycle: 5;*)
		rCustAnaIn_SM_TrigMax : ARRAY[0..120]OF REAL; (* *) (*OldName: unknown	; Cycle: 5;*)
		rCustAnaIn_SM_TrigMin : ARRAY[0..120]OF REAL; (* *) (*OldName: unknown	; Cycle: 5;*)
		rCustomizedAG : ARRAY[0..99]OF REAL; (*optional prepared customizable interface V4.5 - BETA PHASE, use only in coordination with TPSS*)
		rCustomizedCH : ARRAY[0..99]OF REAL; (*optional prepared customizable interface V4.5 - BETA PHASE, use only in coordination with TPSS*)
		rCustomizedCP : ARRAY[0..99]OF REAL; (*optional prepared customizable interface V4.5 - BETA PHASE, use only in coordination with TPSS*)
		rCustomizedEC : ARRAY[0..99]OF REAL; (*optional prepared customizable interface V4.5 - BETA PHASE, use only in coordination with TPSS*)
		rCustomizedHA : ARRAY[0..300]OF REAL; (*optional prepared customizable interface for HAL, V4.5 - BETA PHASE, use only in coordination with TPSS*)
		rCustomizedHC : ARRAY[0..99]OF REAL; (*New customizable interface 2017  - BETA PHASE, use only in coordination with TPSS*)
		rCustomizedOP : ARRAY[0..99]OF REAL; (*optional prepared customizable interface V4.5 - BETA PHASE, use only in coordination with TPSS*)
		rCustomizedSpare : ARRAY[0..99]OF REAL; (*optional prepared customizable spare out interface V4.5 - BETA PHASE, use only in coordination with TPSS*)
		rCust_IF : ARRAY[740..756]OF REAL; (*INPUT VALUES, read from Customer bus coupling, -> See Para.rCustFactor_IF[] also*)
		rCust_SparePara : ARRAY[0..200]OF REAL; (*WATCH FOR POSSIBLE HMI Extension [201..500] NOT FORWARDED TO OTHER MODULES!*) (*OldName: SPS_REZP1, SPS_REZP2, SPS_REZP3, SPS_REZP16 ; Cycle: 5;*)
		rDroop_FC_neg : REAL; (*negative droop for frequency control*)
		rDroop_FC_pos : REAL; (*positive droop for frequency control*)
		rF_Act : REAL; (* actual frequency [Hz]*)
		rF_MMD_FC : REAL; (* actual frequency *)
		rF_Ref : REAL; (* frequency setpoint [Hz]*)
		rGenC_PBC : REAL; (* bus: scaling value for power P from EU [kW]*) (* OldName: rBUS_GCP_P; Cycle:5; *)
		rGenC_PFBC : REAL; (* bus: scaling value genetaror power factor (COS PHI) from EU [-] 1.00 = 1.00*) (* OldName: rBUS_GCQ_PF; Cycle:5; *)
		rGenC_PLimBC : REAL; (* bus: scaling value power limitation from EU [kW]*) (* OldName: rBUS_GCP_Plim; Cycle:5; *)
		rGenC_QBC : REAL; (* bus: scaling value reactive power (Q) from EU [kVAr]*) (* OldName: rBUS_GCQ_Q; Cycle:5; *)
		rGenC_QLimBC : REAL; (* bus: scaling value for reactive power limitation for EVA BUS[kVAr] *) (* OldName: rBUS_GCQ_Qlim; Cycle:5; *)
		rGenC_UQBC : REAL; (* bus: scaling value generator voltage for reactive power (Q) [1.00] = 100% from nominal Value for Setpoint (Parameter 11696)*) (* OldName: rBUS_GCQ_Uset; Cycle:5; *)
		rGT_RatioMix_Set : REAL; (*custom gasmixing ratio setpoint - new V4.5*)
		rLam_Eng_LL_ManSet_Cust : REAL; (*new 2016*)
		rLeanox_Man_Cust : REAL; (*new 2016*)
		rN_Set_ExtAI_Norm : REAL; (* *) (*OldName: Dig_N_SOLL; Cycle: 5;*)
		rPF_CosPCtr_Bus : REAL; (*CosPhi setpoint via bus. Range: -0.9 to -0.99, 0.7 to 1.0*) (*OldName:newPV; Cycle: 5;*)
		rPF_POC_Act_Cust : REAL; (*power factor actual from customer(point of connection)*) (*OldName:newPV;Cycle:5*)
		rP_MainsImport : REAL; (*+=grid to plant power value in [KW], -=plant to grid power*)
		rP_POC_Act_Cust : REAL; (*active power actual  from customer(point of connection)[kW]*) (*OldName:newPV;Cycle:5*)
		rP_POR_Act_Cust : REAL; (*actual active power used as point of reference [kW]*)
		rP_Red_AI_Norm : REAL; (* power reduction by analog input *) (*OldName: ssPowerRedAnalog; Cycle: 5;*)
		rP_Red_EVU_Norm : REAL; (* power reduction by utility *) (*OldName: RED_EVU; Cycle: 5;*)
		rP_Red_Sp_Lim1_Norm : REAL; (* power setpoint limit 1  related to rP_Nom *) (*OldName: ssPowerSetpointLimit1; Cycle: 5;*)
		rP_Red_Sp_Lim2_Norm : REAL; (* power setpoint limit 2  related to rP_Nom] *) (*OldName: ssPowerSetpointLimit2; Cycle: 5;*)
		rP_Red_Sp_Lim3_Norm : REAL; (* power setpoint limit 3  related to rP_Nom *) (*OldName: ssPowerSetpointLimit3; Cycle: 5;*)
		rP_RMC_FC_neg : REAL; (*negative reserve power for frequency control [kW]*)
		rP_RMC_FC_pos : REAL; (*positive reserve power for frequency control [kW]*)
		rP_Set_Ctr_Mns_Norm : REAL; (*! new V4.5 2017 !  (Mains Power Controller)*)
		rP_Set_ExtAI_Norm : REAL; (* *) (*OldName: AW_EXPSH_AI; Cycle: 5;*)
		rP_Set_ExtDI_Cust_Norm : REAL; (* external power setpoint via digital input related to rP_Nom V04.03.00.00 NEW (function moved from GRID Module to  Customized, replaces rP_Set_ExtDI_Norm)*) (*OldName:Dig_P_SOLL;Cycle:5;*)
		rP_Set_FC : REAL; (* generator power setpoint by frequency control [kW]*)
		rP_Set_Mns_Norm : REAL; (*Mains Ctrl engine setpoint power Solleistung*)
		rPr_Leanox_ManSet_Cust : REAL; (*new 2016*)
		rQ_Cust : REAL; (*Customized Q setpoint [kVAr]*)
		rQ_POC_Act_Cust : REAL; (*reactive power actual from customer(point of connection)[kVAr]*) (*OldName:newPV;Cycle:5*)
		rRatioAdd1_Set_Customized : REAL; (* = customized gas mixture setpoint  for TB*) (*OldName: new PV; Cycle: 5;*)
		rRatioAdd_Set_Customized : REAL; (* = customized gas mixture setpoint for TB*) (*OldName: new PV; Cycle: 5;*)
		rRatioMix1_Set_Customized : REAL; (* = customized gas mixture setpoint for TB*) (*OldName: new PV; Cycle: 5;*)
		rRatioMixS_Set_Customized : REAL; (* = customized gas mixture setpoint for TB*) (*OldName: new PV; Cycle: 5;*)
		rRatioMix_Set_Customized : REAL; (* = customized gas mixture setpoint*) (*OldName: new PV; Cycle: 5;*)
		rS_POC_Act_Cust : REAL; (*apparent power actual from customer(point of connection)[kVA]*) (*OldName:newPV;Cycle:5*)
		rT_AirER_Customized : REAL; (* = customized adopted room temperature *) (*OldName: new PV; Cycle: 5;*)
		rT_ChC_Ctr_Wex_Cust : REAL; (*new out interface prepared in V4.5*)
		rUniAna : ARRAY[0..250]OF REAL; (*ARRAY of scaled value from UniversalIO system	rUniAna[1] to rUniAna[250]*) (*OldName: rUniAna; Cycle: 5;*)
		rU_POR_Act_Cust : REAL; (*actual voltage used as point of reference [V]*)
		ssUniAi : ARRAY[0..251]OF INT; (*OBSOLETE, for compatibility only, converted input values [unit depends on configuration]*) (*OldName: ssUniAi	; Cycle: 5;*)
		szUniAiOutState : ARRAY[0..250]OF STRING[16]; (*status message text output*) (*OldName: szUniAiOutState	; Cycle: 5;*)
		szUniDigOutState : ARRAY[0..250]OF STRING[16]; (*textinfo with details to channel state*) (*OldName: szUniDigOutState	; Cycle: 5;*)
		tAO_UniAo : ARRAY[0..250]OF HALioAo_Type; (*CustomerIO HAL- connector*) (*OldName: tAO_UniAo	; Cycle: 5;*)
		tCtr_Cust1_In : _tGeACtrIn; (*  customizable controllers inputs are available for other modules and therefor here in OUT declared 	*) (*OldName: new PV; Cycle: 5;*)
		tCtr_Cust1_Out : _tGeACtrOut; (*  customizable controllers without predefined purpose	*) (*OldName: REG1.y, usw PV; Cycle: 5;*)
		tCtr_Cust2_In : _tGeACtrIn; (*  customizable controllers inputs are available for other modules and therefor here in OUT declared 	*) (*OldName: new PV; Cycle: 5;*)
		tCtr_Cust2_Out : _tGeACtrOut; (*  customizable controllers without predefined purpose	*) (*OldName: REG2.y, usw PV; Cycle: 5;*)
		tCtr_Cust3_In : _tGeACtrIn; (*  customizable controllers inputs are available for other modules and therefor here in OUT declared 	*) (*OldName: new PV; Cycle: 5;*)
		tCtr_Cust3_Out : _tGeACtrOut; (*  customizable controllers without predefined purpose	*) (*OldName: REG3.y, usw PV; Cycle: 5;*)
		tCtr_Cust4_In : _tGeACtrIn; (*  customizable controllers inputs are available for other modules and therefor here in OUT declared 	*) (*OldName: new PV; Cycle: 5;*)
		tCtr_Cust4_Out : _tGeACtrOut; (*  customizable controllers without predefined purpose	*) (*OldName: REG4.y, usw PV; Cycle: 5;*)
		tCtr_Cust5_In : _tGeACtrIn; (*  customizable controllers inputs are available for other modules and therefor here in OUT declared 	*) (*OldName: new PV; Cycle: 5;*)
		tCtr_Cust5_Out : _tGeACtrOut; (*  customizable controllers without predefined purpose	*) (*OldName: REG5.y, usw PV; Cycle: 5;*)
		tCtr_Cust6_In : _tGeACtrIn; (*  customizable controllers inputs are available for other modules and therefor here in OUT declared 	*) (*OldName: new PV; Cycle: 5;*)
		tCtr_Cust6_Out : _tGeACtrOut; (*  customizable controllers without predefined purpose	*) (*OldName: REG6.y, usw PV; Cycle: 5;*)
		tCtr_Cust7_In : _tGeACtrIn; (*  customizable controllers inputs are available for other modules and therefor here in OUT declared 	*) (*OldName: new PV; Cycle: 5;*)
		tCtr_Cust7_Out : _tGeACtrOut; (*  customizable controllers without predefined purpose	*) (*OldName: REG7.y, usw PV; Cycle: 5;*)
		tCtr_Cust8_In : _tGeACtrIn; (*  customizable controllers inputs are available for other modules and therefor here in OUT declared 	*) (*OldName: new PV; Cycle: 5;*)
		tCtr_Cust8_Out : _tGeACtrOut; (*  customizable controllers without predefined purpose	*) (*OldName: REG8.y, usw PV; Cycle: 5;*)
		tCtr_Cust41_In : _tGeACtrIn; (*  customizable controllers inputs are available for other modules and therefor here in OUT declared 	*) (*OldName: new PV; Cycle: 5;*)
		tCtr_Cust41_Out : _tGeACtrOut; (*  customizable controllers without predefined purpose	*) (*OldName: new PV; Cycle: 5;*)
		tCtr_Cust42_In : _tGeACtrIn; (*  customizable controllers inputs are available for other modules and therefor here in OUT declared 	*) (*OldName: new PV; Cycle: 5;*)
		tCtr_Cust42_Out : _tGeACtrOut; (*  customizable controllers without predefined purpose	*) (*OldName: new PV; Cycle: 5;*)
		tCtr_Cust43_In : _tGeACtrIn; (*  customizable controllers inputs are available for other modules and therefor here in OUT declared 	*) (*OldName: new PV; Cycle: 5;*)
		tCtr_Cust43_Out : _tGeACtrOut; (*  customizable controllers without predefined purpose	*) (*OldName: new PV; Cycle: 5;*)
		tCtr_Cust44_In : _tGeACtrIn; (*  customizable controllers inputs are available for other modules and therefor here in OUT declared 	*) (*OldName: new PV; Cycle: 5;*)
		tCtr_Cust44_Out : _tGeACtrOut; (*  customizable controllers without predefined purpose	*) (*OldName: new PV; Cycle: 5;*)
		tCtr_Cust45_In : _tGeACtrIn; (*  customizable controllers inputs are available for other modules and therefor here in OUT declared 	*) (*OldName: new PV; Cycle: 5;*)
		tCtr_Cust45_Out : _tGeACtrOut; (*  customizable controllers without predefined purpose	*) (*OldName: new PV; Cycle: 5;*)
		tCtr_CustOut : ARRAY[0..45]OF HALioAo_Type; (*new output channel for direct usage of customized controllers on HAL*) (*OldName: new PV	; Cycle: 5;*)
		tCtr_Mns_In : _tGeACtrIn; (*MnsCtrl*)
		tCtr_Mns_Out : _tGeACtrOut; (*MnsCtrl*)
		tCU2AB : MM2AmmBase; (* Data exchange structure to AlarmBase*) (*OldName: new PV; Cycle: 5;*)
		tCU2CP_OutData : ARRAY[0..MAX_OUT_DATA_ARRAY]OF INT; (*output data to Coupling Module*)
		tCU2PB : MM2ParaBase_type; (* Data exchange structure TO ParaBase*) (*OldName: new PV; Cycle: 5;*)
		tCustAnaOut : ARRAY[0..iNoOf_AnaOut]OF HALioAo_Type; (*watch for HMI Extension   [0..60]*) (*OldName: new PV	; Cycle: 5;*)
		tCustDigOut : ARRAY[0..150]OF HALioDo_Type; (*Connection to HAL*) (*OldName: tCustDigOut; Cycle: 5;*)
		tDO_Eng_Block_EVU : HALioDo_Type; (*acknowlege request from utility (evu) ==>> lockout module *) (*OldName: DO_RM_EVU_BLOCK; Cycle: 5;*)
		tDO_P_Red_EVU_Stage0 : HALioDo_Type; (*acknowlege request from utility (evu) ==>> no power reduction from evu*) (*OldName: DO_RM_EVU_0; Cycle: 5;*)
		tDO_P_Red_EVU_Stage1 : HALioDo_Type; (*acknowlege request from utility (evu) ==>> power reduction stage 1*) (*OldName: DO_RM_EVU_1; Cycle: 5;*)
		tDO_P_Red_EVU_Stage2 : HALioDo_Type; (*acknowlege request from utility (evu) ==>> power reduction stage 2*) (*OldName: DO_RM_EVU_2; Cycle: 5;*)
		tDO_P_Red_EVU_Stage3 : HALioDo_Type; (*acknowlege request from utility (evu) ==>> power reduction stage 3*) (*OldName: DO_RM_EVU_3; Cycle: 5;*)
		tDO_P_Red_EVU_Stage4 : HALioDo_Type; (*acknowlege request from utility (external, vintagestyled utilisationfeedback) ==>> power reduction stage 4*) (*OldName: DO_RM_EVU_4; Cycle: 5;*)
		tDO_P_Red_EVU_Stage5 : HALioDo_Type; (*acknowlege request from utility (external, vintagestyled utilisationfeedback) ==>> power reduction stage 5*) (*OldName: DO_RM_EVU_5; Cycle: 5;*)
		tDO_UniDo : ARRAY[0..250]OF HALioDo_Type; (*CustomerIO HAL- connector*) (*OldName: tDO_UniDo	; Cycle: 5;*)
		tF_Act_FC : HALioAo_Type; (* AO: actual frequency *)
		tF_Set_FC : HALioAo_Type; (* AO: nominal frequency *)
		tGen_DVM : HALioDo_Type; (*Generator voltage matching output (Leroy Somer)*) (*OldName: unknown; Cycle: 5;*)
		tProtectionTest : ARRAY[0..3]OF HALioDo_Type; (*protection test - grid code logic*) (*OldName:newPV;Cycle:5;*)
		tP_Act_FC : HALioAo_Type; (* AO: actual power *)
		tP_PRLCont_FC : HALioAo_Type; (* AO: power output of FC controller *)
		tUniAnaErrors : ARRAY[0..251]OF tAnaInErrors_typ; (* *) (*OldName: tUniAnaErrors	; Cycle: 5;*)
		tUniDigErrors : ARRAY[0..64]OF tDigInErrors_typ; (* *) (*OldName: tUniDigErrors	; Cycle: 5;*)
		bChC2_Rel : BOOL; (*release charge cooler 2 from monitoring*) (*OldName:newPV; Cycle:5;*) (* Gridcode interfaces added  *)
		rCust_AG : ARRAY[0..99]OF REAL; (*New customizable interface 2017 - BETA PHASE, use only in coordination with TPSS*)
		rCust_CH : ARRAY[0..99]OF REAL; (*New customizable interface 2017 - BETA PHASE, use only in coordination with TPSS*)
		rCust_CP : ARRAY[0..99]OF REAL; (*New customizable interface 2017 - BETA PHASE, use only in coordination with TPSS*)
		rCust_EC : ARRAY[0..99]OF REAL; (*prepared- not active! customizable interface 2017 - BETA PHASE, use only in coordination with TPSS*)
		rCust_HA : ARRAY[0..300]OF REAL; (*New customizable HAL interface 2017 - BETA PHASE, use only in coordination with TPSS*)
		rCust_OP : ARRAY[0..99]OF REAL; (*prepared-not active! customizable interface 2017 - BETA PHASE, use only in coordination with TPSS*)
		rCust_Spare : ARRAY[0..99]OF REAL; (*New customizable interface 2017 - BETA PHASE, use only in coordination with TPSS*)
		rU_Set_Norm_Cust : REAL; (* External voltage set point from CU module [%Unom] *) (*OldName:new PV V4.07;Cycle:5*)
		tCU2GT : CUSTOM2GASTRAIN_Struct; (*Data exchange structure to Custom - new V4.07*)
		tCU2GR : CUSTOM2GRID_Struct; (* Data exchange structure to Custom *)
		bCust_Dem : BOOL; (* Remote Engine demand from CU module *)
		rN_Offs_Cust : REAL; (* Speed offset setpoint from CU module [rpm] *)
		rP_Droop_Set_Bus_Norm : REAL; (* Droop Offset Setpoint via Bus [%Pnom] *)
		bP_Droop_Set_Bus : BOOL; (* Enable Droop Offset Setpoint via Bus *)
		rCH4_Bus : REAL; (* CH4 content via Bus, 1.0 = 100% *)
		bCH4_Bus_Active : BOOL; (* CH4 content measuring via Bus active *)
		bH2_Bus_Active : BOOL; (* Bus - H2 content signal via bus *)
		rH2_Bus : REAL; (* Bus - H2 content in percent. 1.0 = 100% *)
		bH2_Bus_MSF : BOOL; (*Bus - Measurement signal failure. FALSE = Failure *)
		bDem_I_Bus : BOOL; (* Demand Island Operation by Bus *)
		bRel_I_Bus : BOOL; (* Release Island Operation by Bus *)
		bDem_Sy_Bus : BOOL; (* Demand synchronization by Bus *)
		bDem_RSy_Bus : BOOL; (* Demand re-synchronization by Bus *)
		bDem_BS_GCBOn_Bus : BOOL; (* Demand blouck-out start with GCB closed by Bus *)
		bDem_BS_DeExc_Bus : BOOL; (* Demand blouck-out start with deexcitation by Bus *)
		bGCB_by_Customer : BOOL; (* GCB controled by Customer *)
		bMsg9286 : BOOL; (* W9286 Measuring signal failure external speed offset *)
		bMsg9287 : BOOL; (* W9287 Failure external speed / voltage controller *)
		bBloc_SY_ProtTest : BOOL; (*blocking synchr./load release by protection test*)
		iPanelSelection_Cust : INT; (*Controls lock of local operation for additional touch panels - Customized*)
		bPanelSelection_Cust : BOOL; (*Controls lock of local operation for additional touch panels - Customized*)
		bBloc_SY_Rel_Cust : BOOL; (* Remote Synchronization / load release from CU module *) (*OldName:newPV; Cycle:5;*)
		bRel_P_Red_I_Bus : BOOL; (*IF720: Release automatic power reduction in island operation*) (*OldName:newPV; Cycle:5;*)
		bN_U_Set_Ext_On : BOOL; (*External speed and voltage control ON*) (*OldName:newPV; Cycle:5;*)
		bReq_PowMod_Ext : BOOL; (*External power mode selection*) (*OldName:newPV; Cycle:5;*)
		bCust_Dem_Sy : BOOL; (* Demand synchronization from CU module *) (*OldName:ssBusVoltPh1_2; Cycle:5*)
		bCust_Dem_RSy : BOOL; (* Demand re-synchronization from CU module *) (*OldName:ssBusVoltPh1_2; Cycle:5*)
		b_FilterScav_Active : BOOL; (* Activation signal of FGQC from customer *)
		bP_Droop_Set_AI : BOOL; (* Enable Droop power setpoint by Analog input *)
		iIdx_Droop_SetDefaultCase : USINT; (*Droop fallback mode,  0: default Para, 1: freeze last value*)
		rP_Set_Default_Norm : REAL; (* normalized Droop set default Para value [-]*)
		rP_Droop_Set_AI_Norm : REAL; (* Normalized Droop Offset Setpoint via AI [-] *)
		iSource_F_N_OffsSet : INT; (* F/N Setpoint: 0= no setpoint, 1= Droop, 2= External, 3= LSL *)
		tF_FSM_Simulated : HALioAo_Type; (*simulated test frequency in FSM/LFSM test mode[Hz]*)
		sLocIdent_CtrlBatMon : ARRAY[1..iNum_CtrlBatMon]OF STRING[10]; (*Control battery test set location*)
		bAuxV_ok_CtrlBatMon : ARRAY[1..iNum_CtrlBatMon]OF BOOL; (*Control battery test set status AuxV supply*)
		iSource_U_OffsSet : INT; (* Voltage offset set point in island mode: 0= no setpoint, 1= Droop, 2= External *)
		rQ_Droop_Set_Bus_Norm : REAL; (* Normalized reactive power Droop offset set point via Bus [PercentQnom] *)
		bQ_Droop_Set_Bus : BOOL; (* Enable reactive power Droop offset set point via Bus *)
		rQ_Droop_Set_AI_Norm : REAL; (* Normalized reactive power Droop offset set point via AI [PercentQnom] *)
		bQ_Droop_Set_AI : BOOL; (* Enable reactive power Droop offset set point via AI *)
		rQ_Set_Default_Norm : REAL; (* Normalized reactive power Droop set default value *)
		rQset_Droop_Bus : REAL; (*Reactive power setpoint for droop mode via Bus*) (* V04.04.00.00 *)
		rUset_Isl_Bus : REAL; (*Generator voltage setpoint via Bus*) (* V04.04.00.00 *)
		bExtCtrOk : BOOL; (*External voltage/speed control released*)
		bGT_CalibrateActive_Bus : BOOL; (* Bus - Calibration Gas analysis *)
		bCV_Bus_Active : BOOL; (* Bus - CV content measuring active *)
		rCV_Bus : REAL; (* Bus - CV content [kWh/Nm3] *)
		bRelGasPlant_Bus_Active : BOOL; (* Bus - Release from gas plant missing active *)
		bRelGasPlant_Bus : BOOL; (*Bus - Release from gas plant missing. FALSE = Missing *)
		bLeanox_Man_Cust : BOOL; (*DO NOT TOUCH!*)
		iAggrekoEngineVersion : INT; (* engine Version for Agrekko calibration 1 = B, 2 = C, 3 = E *)
		iAggrekoTCConfig : INT; (* engine TA configuration for Agrekko calibration 1 = TA40, 2 = TA45, 3 = TA65, 4 = TA70 *)
		bSCR_CemsExtCatOut_Rdy : BOOL; (*Validity of external customer CEMS signal at catalyst output*) (*OldName: new PV; Cycle:5*) (*V04.05.00.00*)
		rCO_SCR_CemsExtCatOut : REAL; (*CO measured by external customer CEMS at catalyst output (ppm dry)*) (*OldName: new PV; Cycle:5*) (*V04.05.00.00*)
		rHum_SCR_CemsExtCatOut : REAL; (*Exhaust water content measured by external customer CEMS at catalyst output [%]*) (*OldName: new PV; Cycle:5*) (*V04.05.00.00*)
		rNH3_SCR_CemsExtCatOut : REAL; (*NH3 measured by external customer CEMS at catalyst output (ppm dry)*) (*OldName: new PV; Cycle:5*) (*V04.05.00.00*)
		rNO2_SCR_CemsExtCatOut : REAL; (*NO2 measured by external customer CEMS at catalyst output (ppm dry)*) (*OldName: new PV; Cycle:5*) (*V04.05.00.00*)
		rNO_SCR_CemsExtCatOut : REAL; (*NO measured by external customer CEMS at catalyst output (ppm dry)*) (*OldName: new PV; Cycle:5*) (*V04.05.00.00*)
		rO2_SCR_CemsExtCatOut : REAL; (*O2 measured by external customer CEMS at catalyst output [Vol-%]*) (*OldName: new PV; Cycle:5*) (*V04.05.00.00*)
		rHum_GasIn_Abs : REAL; (* absolute humidity gas via customer BUS [g H2O/kg dry gas] *)
		bBypassMCB_deadBB : BOOL; (*bypass MCB status information from the standard dead_bb check*)
		bSoftEnergDem : BOOL; (*demand transformer soft energisation*)
		bBypassMCB_SoftStart : BOOL; (*bypass MCB status information from the standard soft energisation logic*)
		bBypassMCB_LoadShed : BOOL; (*bypass MCB status information from the standard load shedding logic*)
		bReq_PowMod : BOOL; (*request power mode - over-written in customization*)
		bBypassMCB_FSM : BOOL; (*bypass MCB status information from the standard dead_bb check*)
		bDroopDB_Active : BOOL; (*The droop deadband remote and local/HMI setpoint data*)
		rDB_FSM_LFSM : REAL; (*Dead band setpoint to be used*)
		bBypassMCB_CosPhi : BOOL; (*bypass MCB status information from the standard CosPhi Ctrl check*)
		bExtendedOpRangeRel : BOOL; (*release extended operation power range*)
		rP_Set_Min_Norm_Ext : REAL; (*minimum power set limitation in p.u. for exteded range*)
		bOtherGeneratorsInLSL : BOOL; (*LSL: FALSE if there are no other other generators in parallel with this generator that are actively participating in the LSL*)
		bSet_LFSM_Test_COn : BOOL; (*LFSM Test command on external (DI or Bus)*)
		bLFSM_Test_Enabled : BOOL; (*FSM/LFSM test enabled external*)
		rF_Act_FSM_Test_Ext : REAL; (*Actual frequency for FSM test via external signal*)
		bBus_Active : BOOL; (*Bus communication active*)
		bOM_Bus : BOOL; (*Operation mode via Bus*)
		bSetIslandMode : BOOL; (*Set Island mode event based via Bus*)
		bSetFixedPwrMode : BOOL; (*Set fixed power mode event based via Bus*)
		bPara_MainsParallel : BOOL; (*mains parallel mode with active mains monitoring*)
		bCust_Dem_EPS_Sy : BOOL; (*Custom demand EPS SY modul*)
		bEng_Dem_EPS_Bus : BOOL; (*Custom engine demand EPS via BUS in OP modul*)
		bSmoothDischarge_CU : BOOL; (*Smooth engine discharge in Island mode*)
		bGCB_OGP_Bus : BOOL; (*Other generator parallel via BUS*)
		bSetGCB2Close : BOOL; (*Set GCB state to close - event based*)
		bSetGCB2Open : BOOL; (*Set GCB state to open - event based*)
		bSetManControlMode : BOOL; (*Set Manual control mode - event based*)
		bSetAutControlMode : BOOL; (*Set Auto control mode - event based*)
		bCust_Rel_I : BOOL; (*Custom release island bit to SY modul*)
		bCust_RelI_BB : BOOL; (*Custom Release Island operation busbar to SY modul*)
		bUseEventBased_P_Set : BOOL; (* Use event based power setpoint from CU module *)
		bEvent_Change : BOOL; (*Trigger bit for event change in case of power set point via bus*)
		rP_Set_Norm_EventBased : REAL; (* Event based external power setpoint via bus related to rP_Nom *)
		rSetPointPW : REAL; (* External power setpoint in AUTO/ON *)
		bDem_EU_Block2_Bus : BOOL; (*IF727 	Module blocked from grid operator - shutdown*)
		bDem_EU_Block3_Bus : BOOL; (*IF727 	Module blocked from grid operator - request off*)
		bBus_Dem_OpcUa : BOOL; (*Demand via OPC UA*) (*OldName:BUS_ANF; Cycle:5;*)
		bBusPulse_OpcUa : BOOL; (*Pulse signal from customer via OPC UA*) (*OldName:newPV; Cycle:5;*)
		rP_Set_OpcUa : REAL; (*Power setpoint from OPC UA [%]*)
		tPlantCom_E2E_Out_Cust100ms : tPlantComData_Cust100ms; (*PlantCom Customized Data E2E_Out_100ms*)
		tPlantCom_E2M_Out_Cust100ms : ARRAY[0..4]OF tPlantComData_Cust100ms; (*PlantCom Customized Data E2M_Out_100ms*)
		tPlantCom_E2E_Out_Cust10ms : tPlantComData_Cust10ms; (*PlantCom Customized Data E2E_Out_10ms*)
		tPlantCom_E2M_Out_Cust10ms : ARRAY[0..4]OF tPlantComData_Cust10ms; (*PlantCom Customized Data E2M_Out_10ms*)
	END_STRUCT;
	MM2Vis_Struct : 	STRUCT
		bAuxCust : ARRAY[0..70]OF BOOL; (*Status display of customized aux * watch for HMI Extension*)
		bCustAlarm_Tripped : ARRAY[0..16]OF BOOL; (* = 	stored state of reserve alarm			*)
		bCustDigIn : ARRAY[0..200]OF BOOL; (*Prepared spare digital input*)
		bCustDigOut : ARRAY[0..150]OF BOOL; (*Prepared spare digital output*)
		bCustOPC : ARRAY[0..32]OF BOOL; (*Prepared spare digital values to customer OPC		*) (*OldName: newPV; Cycle: 5;*)
		bCustVis : ARRAY[0..50]OF BOOL; (*Prepared spare digital input to VISU		*) (*OldName: newPV; Cycle: 5;*)
		bCustWarn_Tripped : ARRAY[0..16]OF BOOL; (* = 	stored state of reserve warning			*)
		bEGValCtr_HeatOutputDown : BOOL; (* = 	New Interface to connect customized exhaust flap control 			*)
		bEGValCtr_HeatOutputUp : BOOL; (* = 	New Interface to connect customized exhaust flap control 			*)
		bEngDSS_Mains : BOOL; (*mains import power controller*) (*OldName: newPV; Cycle: 5;*)
		bFC_SOn : BOOL; (*feedback signal: FC switched on*)
		bMsg1001 : BOOL; (* = 	Alarmbit to visu			*)
		bMsg1002 : BOOL; (* = 	Alarmbit to visu			*)
		bMsg1003 : BOOL; (* = 	Alarmbit to visu			*)
		bMsg1004 : BOOL; (* = 	Alarmbit to visu			*)
		bMsg1005 : BOOL; (* = 	Alarmbit to visu			*)
		bMsg1006 : BOOL; (* = 	Alarmbit to visu			*)
		bMsg1007 : BOOL; (* = 	Alarmbit to visu			*)
		bMsg1008 : BOOL; (* = 	Alarmbit to visu			*)
		bMsg1009 : BOOL; (* = 	Alarmbit to visu			*)
		bMsg1010 : BOOL; (* = 	Alarmbit to visu			*)
		bMsg1011 : BOOL; (* = 	Alarmbit to visu			*)
		bMsg1012 : BOOL; (* = 	Alarmbit to visu			*)
		bMsg1013 : BOOL; (* = 	Alarmbit to visu			*)
		bMsg1014 : BOOL; (* = 	Alarmbit to visu			*)
		bMsg1015 : BOOL; (* = 	Alarmbit to visu			*)
		bMsg1016 : BOOL; (* = 	Alarmbit to visu			*)
		bMsg1177 : BOOL; (* = 	Alarmbit to visu			*)
		bMsg1178 : BOOL; (* = 	Alarmbit to visu			*)
		bMsg1179 : BOOL; (* = 	Alarmbit to visu			*)
		bMsg1180 : BOOL; (* = 	Alarmbit to visu			*)
		bMsg1181 : BOOL; (* = 	Alarmbit to visu			*)
		bMsg1182 : BOOL; (* = 	Alarmbit to visu			*)
		bMsg1183 : BOOL; (* = 	Alarmbit to visu			*)
		bMsg1184 : BOOL; (* = 	Alarmbit to visu			*)
		bMsg1193 : BOOL; (* = 	Alarmbit to visu			*)
		bMsg1194 : BOOL; (* = 	Alarmbit to visu			*)
		bMsg1195 : BOOL; (* = 	Alarmbit to visu			*)
		bMsg1196 : BOOL; (* = 	Alarmbit to visu			*)
		bMsg1197 : BOOL; (* = 	Alarmbit to visu			*)
		bMsg1198 : BOOL; (* = 	Alarmbit to visu			*)
		bMsg1199 : BOOL; (* = 	Alarmbit to visu			*)
		bMsg1200 : BOOL; (* = 	Alarmbit to visu			*)
		bMsg1201 : BOOL; (* = 	Alarmbit to visu			*)
		bMsg1202 : BOOL; (* = 	Alarmbit to visu			*)
		bMsg1203 : BOOL; (* = 	Alarmbit to visu			*)
		bMsg1204 : BOOL; (* = 	Alarmbit to visu			*)
		bMsg1205 : BOOL; (* = 	Alarmbit to visu			*)
		bMsg1206 : BOOL; (* = 	Alarmbit to visu			*)
		bMsg1207 : BOOL; (* = 	Alarmbit to visu			*)
		bMsg1208 : BOOL; (* = 	Alarmbit to visu			*)
		bMsg1300 : BOOL; (* = 	Alarmbit to visu ReserveAi1 Lo	*)
		bMsg1301 : BOOL; (* = 	Alarmbit to visu ReserveAi1 Hi	*)
		bMsg1302 : BOOL; (* = 	Alarmbit to visu ReserveAi1  SigErr	*)
		bMsg1303 : BOOL; (* = 	Alarmbit to visu			*)
		bMsg1304 : BOOL; (* = 	Alarmbit to visu			*)
		bMsg1305 : BOOL; (* = 	Alarmbit to visu			*)
		bMsg1306 : BOOL; (* = 	Alarmbit to visu			*)
		bMsg1307 : BOOL; (* = 	Alarmbit to visu			*)
		bMsg1308 : BOOL; (* = 	Alarmbit to visu			*)
		bMsg1309 : BOOL; (* = 	Alarmbit to visu			*)
		bMsg1310 : BOOL; (* = 	Alarmbit to visu			*)
		bMsg1311 : BOOL; (* = 	Alarmbit to visu			*)
		bMsg1312 : BOOL; (* = 	Alarmbit to visu			*)
		bMsg1313 : BOOL; (* = 	Alarmbit to visu			*)
		bMsg1314 : BOOL; (* = 	Alarmbit to visu			*)
		bMsg1315 : BOOL; (* = 	Alarmbit to visu			*)
		bMsg1316 : BOOL; (* = 	Alarmbit to visu			*)
		bMsg1317 : BOOL; (* = 	Alarmbit to visu			*)
		bMsg1318 : BOOL; (* = 	Alarmbit to visu			*)
		bMsg1319 : BOOL; (* = 	Alarmbit to visu			*)
		bMsg1320 : BOOL; (* = 	Alarmbit to visu			*)
		bMsg1321 : BOOL; (* = 	Alarmbit to visu			*)
		bMsg1322 : BOOL; (* = 	Alarmbit to visu			*)
		bMsg1323 : BOOL; (* = 	Alarmbit to visu			*)
		bMsg1324 : BOOL; (* = 	Alarmbit to visu			*)
		bMsg1325 : BOOL; (* = 	Alarmbit to visu			*)
		bMsg1326 : BOOL; (* = 	Alarmbit to visu			*)
		bMsg1327 : BOOL; (* = 	Alarmbit to visu			*)
		bMsg1328 : BOOL; (* = 	Alarmbit to visu			*)
		bMsg1329 : BOOL; (* = 	Alarmbit to visu			*)
		bMsg1330 : BOOL; (* = 	Alarmbit to visu			*)
		bMsg1331 : BOOL; (* = 	Alarmbit to visu			*)
		bMsg1332 : BOOL; (* = 	Alarmbit to visu			*)
		bMsg1333 : BOOL; (* = 	Alarmbit to visu			*)
		bMsg1334 : BOOL; (* = 	Alarmbit to visu			*)
		bMsg1335 : BOOL; (* = 	Alarmbit to visu			*)
		bMsg1336 : BOOL; (* = 	Alarmbit to visu			*)
		bMsg1337 : BOOL; (* = 	Alarmbit to visu			*)
		bMsg1338 : BOOL; (* = 	Alarmbit to visu			*)
		bMsg1339 : BOOL; (* = 	Alarmbit to visu			*)
		bMsg1340 : BOOL; (* = 	Alarmbit to visu			*)
		bMsg1341 : BOOL; (* = 	Alarmbit to visu			*)
		bMsg1342 : BOOL; (* = 	Alarmbit to visu			*)
		bMsg1343 : BOOL; (* = 	Alarmbit to visu			*)
		bMsg1344 : BOOL; (* = 	Alarmbit to visu			*)
		bMsg1345 : BOOL; (* = 	Alarmbit to visu			*)
		bMsg1346 : BOOL; (* = 	Alarmbit to visu			*)
		bMsg1347 : BOOL; (* = 	Alarmbit to visu			*)
		bMsg1348 : BOOL; (* = 	Alarmbit to visu			*)
		bMsg1349 : BOOL; (* = 	Alarmbit to visu			*)
		bMsg1350 : BOOL; (* = 	Alarmbit to visu			*)
		bMsg1351 : BOOL; (* = 	Alarmbit to visu			*)
		bMsg1352 : BOOL; (* = 	Alarmbit to visu			*)
		bMsg1353 : BOOL; (* = 	Alarmbit to visu			*)
		bMsg1354 : BOOL; (* = 	Alarmbit to visu			*)
		bMsg1355 : BOOL; (* = 	Alarmbit to visu			*)
		bMsg1356 : BOOL; (* = 	Alarmbit to visu			*)
		bMsg1357 : BOOL; (* = 	Alarmbit to visu			*)
		bMsg1358 : BOOL; (* = 	Alarmbit to visu			*)
		bMsg1359 : BOOL; (* = 	Alarmbit to visu			*)
		bMsg1360 : BOOL; (* = 	Alarmbit to visu			*)
		bMsg1361 : BOOL; (* = 	Alarmbit to visu			*)
		bMsg1362 : BOOL; (* = 	Alarmbit to visu			*)
		bMsg1363 : BOOL; (* = 	Alarmbit to visu			*)
		bMsg1364 : BOOL; (* = 	Alarmbit to visu			*)
		bMsg1365 : BOOL; (* = 	Alarmbit to visu			*)
		bMsg1366 : BOOL; (* = 	Alarmbit to visu			*)
		bMsg1367 : BOOL; (* = 	Alarmbit to visu			*)
		bMsg1368 : BOOL; (* = 	Alarmbit to visu			*)
		bMsg1369 : BOOL; (* = 	Alarmbit to visu			*)
		bMsg1370 : BOOL; (* = 	Alarmbit to visu			*)
		bMsg1371 : BOOL; (* = 	Alarmbit to visu			*)
		bMsg1372 : BOOL; (* = 	Alarmbit to visu			*)
		bMsg1373 : BOOL; (* = 	Alarmbit to visu			*)
		bMsg1374 : BOOL; (* = 	Alarmbit to visu			*)
		bMsg1375 : BOOL; (* = 	Alarmbit to visu			*)
		bMsg1376 : BOOL; (* = 	Alarmbit to visu			*)
		bMsg1377 : BOOL; (* = 	Alarmbit to visu			*)
		bMsg1378 : BOOL; (* = 	Alarmbit to visu			*)
		bMsg1379 : BOOL; (* = 	Alarmbit to visu			*)
		bMsg1380 : BOOL; (* = 	Alarmbit to visu			*)
		bMsg1381 : BOOL; (* = 	Alarmbit to visu			*)
		bMsg1382 : BOOL; (* = 	Alarmbit to visu			*)
		bMsg1383 : BOOL; (* = 	Alarmbit to visu			*)
		bMsg1384 : BOOL; (* = 	Alarmbit to visu			*)
		bMsg1385 : BOOL; (* = 	Alarmbit to visu			*)
		bMsg1386 : BOOL; (* = 	Alarmbit to visu			*)
		bMsg1387 : BOOL; (* = 	Alarmbit to visu			*)
		bMsg1388 : BOOL; (* = 	Alarmbit to visu			*)
		bMsg1389 : BOOL; (* = 	Alarmbit to visu			*)
		bMsg1390 : BOOL; (* = 	Alarmbit to visu			*)
		bMsg1391 : BOOL; (* = 	Alarmbit to visu			*)
		bMsg1392 : BOOL; (* = 	Alarmbit to visu			*)
		bMsg1393 : BOOL; (* = 	Alarmbit to visu			*)
		bMsg1394 : BOOL; (* = 	Alarmbit to visu			*)
		bMsg1395 : BOOL; (* = 	Alarmbit to visu			*)
		bMsg1396 : BOOL; (* = 	Alarmbit to visu			*)
		bMsg1397 : BOOL; (* = 	Alarmbit to visu			*)
		bMsg1398 : BOOL; (* = 	Alarmbit to visu			*)
		bMsg1399 : BOOL; (* = 	Alarmbit to visu			*)
		bMsg1400 : BOOL; (*= additional alarmbit to visu*)
		bMsg1401 : BOOL; (*= additional alarmbit to visu*)
		bMsg1402 : BOOL; (*= additional alarmbit to visu*)
		bMsg1403 : BOOL; (*= additional alarmbit to visu*)
		bMsg1404 : BOOL; (*= additional alarmbit to visu*)
		bMsg1405 : BOOL; (*= additional alarmbit to visu*)
		bMsg1406 : BOOL; (*= additional alarmbit to visu*)
		bMsg1407 : BOOL; (*= additional alarmbit to visu*)
		bMsg1408 : BOOL; (*= additional alarmbit to visu*)
		bMsg1409 : BOOL; (*= additional alarmbit to visu*)
		bMsg1410 : BOOL; (*= additional alarmbit to visu*)
		bMsg1411 : BOOL; (*= additional alarmbit to visu*)
		bMsg1412 : BOOL; (*= additional alarmbit to visu*)
		bMsg1413 : BOOL; (*= additional alarmbit to visu*)
		bMsg1414 : BOOL; (*= additional alarmbit to visu*)
		bMsg1415 : BOOL; (*= additional alarmbit to visu*)
		bMsg1416 : BOOL; (*= additional alarmbit to visu*)
		bMsg1417 : BOOL; (*= additional alarmbit to visu*)
		bMsg1418 : BOOL; (*= additional alarmbit to visu*)
		bMsg1419 : BOOL; (*= additional alarmbit to visu*)
		bMsg1420 : BOOL; (*= additional alarmbit to visu*)
		bMsg1421 : BOOL; (*= additional alarmbit to visu*)
		bMsg1422 : BOOL; (*= additional alarmbit to visu*)
		bMsg1423 : BOOL; (*= additional alarmbit to visu*)
		bMsg1424 : BOOL; (*= additional alarmbit to visu*)
		bMsg1425 : BOOL; (*= additional alarmbit to visu*)
		bMsg1426 : BOOL; (*= additional alarmbit to visu*)
		bMsg1427 : BOOL; (*= additional alarmbit to visu*)
		bMsg1428 : BOOL; (*= additional alarmbit to visu*)
		bMsg1429 : BOOL; (*= additional alarmbit to visu*)
		bMsg1430 : BOOL; (*= additional alarmbit to visu*)
		bMsg1431 : BOOL; (*= additional alarmbit to visu*)
		bMsg1432 : BOOL; (*= additional alarmbit to visu*)
		bMsg1433 : BOOL; (*= additional alarmbit to visu*)
		bMsg1434 : BOOL; (*= additional alarmbit to visu*)
		bMsg1435 : BOOL; (*= additional alarmbit to visu*)
		bMsg1436 : BOOL; (*= additional alarmbit to visu*)
		bMsg1437 : BOOL; (*= additional alarmbit to visu*)
		bMsg1438 : BOOL; (*= additional alarmbit to visu*)
		bMsg1439 : BOOL; (*= additional alarmbit to visu*)
		bMsg1440 : BOOL; (*= additional alarmbit to visu*)
		bMsg1441 : BOOL; (*= additional alarmbit to visu*)
		bMsg1442 : BOOL; (*= additional alarmbit to visu*)
		bMsg1443 : BOOL; (*= additional alarmbit to visu*)
		bMsg1444 : BOOL; (*= additional alarmbit to visu*)
		bMsg1445 : BOOL; (*= additional alarmbit to visu*)
		bMsg1446 : BOOL; (*= additional alarmbit to visu*)
		bMsg1447 : BOOL; (*= additional alarmbit to visu*)
		bMsg1448 : BOOL; (*= additional alarmbit to visu*)
		bMsg1449 : BOOL; (*= additional alarmbit to visu*)
		bMsg1450 : BOOL; (*= additional alarmbit to visu*)
		bMsg1451 : BOOL; (*= additional alarmbit to visu*)
		bMsg1452 : BOOL; (*= additional alarmbit to visu*)
		bMsg1453 : BOOL; (*= additional alarmbit to visu*)
		bMsg1454 : BOOL; (*= additional alarmbit to visu*)
		bMsg1455 : BOOL; (*= additional alarmbit to visu*)
		bMsg1456 : BOOL; (*= additional alarmbit to visu*)
		bMsg1457 : BOOL; (*= additional alarmbit to visu*)
		bMsg1458 : BOOL; (*= additional alarmbit to visu*)
		bMsg1459 : BOOL; (*= additional alarmbit to visu*)
		bMsg1460 : BOOL; (*= additional alarmbit to visu*)
		bMsg1461 : BOOL; (*= additional alarmbit to visu*)
		bMsg1462 : BOOL; (*= additional alarmbit to visu*)
		bMsg1463 : BOOL; (*= additional alarmbit to visu*)
		bMsg1464 : BOOL; (*= additional alarmbit to visu*)
		bMsg1465 : BOOL; (*= additional alarmbit to visu*)
		bMsg1466 : BOOL; (*= additional alarmbit to visu*)
		bMsg1467 : BOOL; (*= additional alarmbit to visu*)
		bMsg1468 : BOOL; (*= additional alarmbit to visu*)
		bMsg1469 : BOOL; (*= additional alarmbit to visu*)
		bMsg1470 : BOOL; (*= additional alarmbit to visu*)
		bMsg1471 : BOOL; (*= additional alarmbit to visu*)
		bMsg1472 : BOOL; (*= additional alarmbit to visu*)
		bMsg1473 : BOOL; (*= additional alarmbit to visu*)
		bMsg1474 : BOOL; (*= additional alarmbit to visu*)
		bMsg1475 : BOOL; (*= additional alarmbit to visu*)
		bMsg1476 : BOOL; (*= additional alarmbit to visu*)
		bMsg1477 : BOOL; (*= additional alarmbit to visu*)
		bMsg1478 : BOOL; (*= additional alarmbit to visu*)
		bMsg1479 : BOOL; (*= additional alarmbit to visu*)
		bMsg1480 : BOOL; (*= additional alarmbit to visu*)
		bMsg1481 : BOOL; (*= additional alarmbit to visu*)
		bMsg1482 : BOOL; (*= additional alarmbit to visu*)
		bMsg1483 : BOOL; (*= additional alarmbit to visu*)
		bMsg1484 : BOOL; (*= additional alarmbit to visu*)
		bMsg1485 : BOOL; (*= additional alarmbit to visu*)
		bMsg1486 : BOOL; (*= additional alarmbit to visu*)
		bMsg1487 : BOOL; (*= additional alarmbit to visu*)
		bMsg1488 : BOOL; (*= additional alarmbit to visu*)
		bMsg1489 : BOOL; (*= additional alarmbit to visu*)
		bMsg1490 : BOOL; (*= additional alarmbit to visu*)
		bMsg1491 : BOOL; (*= additional alarmbit to visu*)
		bMsg1492 : BOOL; (*= additional alarmbit to visu*)
		bMsg1493 : BOOL; (*= additional alarmbit to visu*)
		bMsg1494 : BOOL; (*= additional alarmbit to visu*)
		bMsg1495 : BOOL; (*= additional alarmbit to visu*)
		bMsg1496 : BOOL; (*= additional alarmbit to visu*)
		bMsg1497 : BOOL; (*= additional alarmbit to visu*)
		bMsg1498 : BOOL; (*= additional alarmbit to visu*)
		bMsg1499 : BOOL; (*= additional alarmbit to visu*)
		bMsg1500 : BOOL; (*= additional alarmbit to visu*)
		bMsg1601 : BOOL; (*reserve alarm message 17*)
		bMsg1602 : BOOL; (*reserve alarm message 18*)
		bMsg1603 : BOOL; (*reserve alarm message 19*)
		bMsg1604 : BOOL; (*reserve alarm message 20*)
		bMsg1605 : BOOL; (*reserve alarm message*)
		bMsg1606 : BOOL; (*reserve alarm message*)
		bMsg1607 : BOOL; (*reserve alarm message*)
		bMsg1608 : BOOL; (*reserve alarm message*)
		bMsg1609 : BOOL; (*reserve alarm message*)
		bMsg1610 : BOOL; (*reserve alarm message*)
		bMsg1611 : BOOL; (*reserve alarm message*)
		bMsg1612 : BOOL; (*reserve alarm message*)
		bMsg1613 : BOOL; (*reserve alarm message*)
		bMsg1614 : BOOL; (*reserve alarm message 30*)
		bMsg1615 : BOOL; (*reserve alarm message*)
		bMsg1616 : BOOL; (*reserve alarm message*)
		bMsg1617 : BOOL; (*reserve alarm message*)
		bMsg1618 : BOOL; (*reserve alarm message*)
		bMsg1619 : BOOL; (*reserve alarm message*)
		bMsg1620 : BOOL; (*reserve alarm message*)
		bMsg1621 : BOOL; (*reserve alarm message*)
		bMsg1622 : BOOL; (*reserve alarm message*)
		bMsg1623 : BOOL; (*reserve alarm message*)
		bMsg1624 : BOOL; (*reserve alarm message 40*)
		bMsg1625 : BOOL; (*reserve alarm message*)
		bMsg1626 : BOOL; (*reserve alarm message*)
		bMsg1627 : BOOL; (*reserve alarm message*)
		bMsg1628 : BOOL; (*reserve alarm message*)
		bMsg1629 : BOOL; (*reserve alarm message*)
		bMsg1630 : BOOL; (*reserve alarm message*)
		bMsg1631 : BOOL; (*reserve alarm message*)
		bMsg1632 : BOOL; (*reserve alarm message*)
		bMsg1633 : BOOL; (*reserve alarm message*)
		bMsg1634 : BOOL; (*reserve alarm message 50*)
		bMsg1635 : BOOL; (*reserve alarm message*)
		bMsg1636 : BOOL; (*reserve alarm message*)
		bMsg1637 : BOOL; (*reserve alarm message*)
		bMsg1638 : BOOL; (*reserve alarm message*)
		bMsg1639 : BOOL; (*reserve alarm message*)
		bMsg1640 : BOOL; (*reserve alarm message*)
		bMsg1641 : BOOL; (*reserve alarm message*)
		bMsg1642 : BOOL; (*reserve alarm message*)
		bMsg1643 : BOOL; (*reserve alarm message*)
		bMsg1644 : BOOL; (*reserve alarm message 60*)
		bMsg1645 : BOOL; (*reserve alarm message*)
		bMsg1646 : BOOL; (*reserve alarm message*)
		bMsg1647 : BOOL; (*reserve alarm message*)
		bMsg1648 : BOOL; (*reserve alarm message*)
		bMsg1649 : BOOL; (*reserve alarm message*)
		bMsg1650 : BOOL; (*reserve alarm message*)
		bMsg1651 : BOOL; (*reserve alarm message*)
		bMsg1652 : BOOL; (*reserve alarm message*)
		bMsg1653 : BOOL; (*reserve alarm message*)
		bMsg1654 : BOOL; (*reserve alarm message 70*)
		bMsg1655 : BOOL; (*reserve alarm message*)
		bMsg1656 : BOOL; (*reserve alarm message*)
		bMsg1657 : BOOL; (*reserve alarm message*)
		bMsg1658 : BOOL; (*reserve alarm message*)
		bMsg1659 : BOOL; (*reserve alarm message*)
		bMsg1660 : BOOL; (*reserve alarm message*)
		bMsg1661 : BOOL; (*reserve alarm message*)
		bMsg1662 : BOOL; (*reserve alarm message*)
		bMsg1663 : BOOL; (*reserve alarm message*)
		bMsg1664 : BOOL; (*reserve alarm message 80*)
		bMsg1665 : BOOL; (*reserve alarm message*)
		bMsg1666 : BOOL; (*reserve alarm message*)
		bMsg1667 : BOOL; (*reserve alarm message*)
		bMsg1668 : BOOL; (*reserve alarm message*)
		bMsg1669 : BOOL; (*reserve alarm message*)
		bMsg1670 : BOOL; (*reserve alarm message*)
		bMsg1671 : BOOL; (*reserve alarm message*)
		bMsg1672 : BOOL; (*reserve alarm message*)
		bMsg1673 : BOOL; (*reserve alarm message*)
		bMsg1674 : BOOL; (*reserve alarm message 90*)
		bMsg1675 : BOOL; (*reserve alarm message*)
		bMsg1676 : BOOL; (*reserve alarm message*)
		bMsg1677 : BOOL; (*reserve alarm message*)
		bMsg1678 : BOOL; (*reserve alarm message*)
		bMsg1679 : BOOL; (*reserve alarm message*)
		bMsg1680 : BOOL; (*reserve alarm message*)
		bMsg1681 : BOOL; (*reserve alarm message*)
		bMsg1682 : BOOL; (*reserve alarm message*)
		bMsg1683 : BOOL; (*reserve alarm message*)
		bMsg1684 : BOOL; (*reserve alarm message 100*)
		bMsg1685 : BOOL; (*reserve alarm message*)
		bMsg1686 : BOOL; (*reserve alarm message*)
		bMsg1687 : BOOL; (*reserve alarm message*)
		bMsg1688 : BOOL; (*reserve alarm message*)
		bMsg1689 : BOOL; (*reserve alarm message*)
		bMsg1690 : BOOL; (*reserve alarm message*)
		bMsg1691 : BOOL; (*reserve alarm message*)
		bMsg1692 : BOOL; (*reserve alarm message*)
		bMsg1693 : BOOL; (*reserve alarm message*)
		bMsg1694 : BOOL; (*reserve alarm message 110*)
		bMsg1695 : BOOL; (*reserve alarm message*)
		bMsg1696 : BOOL; (*reserve alarm message*)
		bMsg1697 : BOOL; (*reserve alarm message*)
		bMsg1698 : BOOL; (*reserve alarm message*)
		bMsg1699 : BOOL; (*reserve alarm message 115*)
		bMsg1700 : BOOL; (*reserve alarm message 116*)
		bMsg1701 : BOOL; (*reserve warning message 27*)
		bMsg1702 : BOOL; (*reserve warning message 28*)
		bMsg1703 : BOOL; (*reserve warning message 29*)
		bMsg1704 : BOOL; (*reserve warning message 30*)
		bMsg1705 : BOOL; (*reserve warning message 31*)
		bMsg1706 : BOOL; (*reserve warning message*)
		bMsg1707 : BOOL; (*reserve warning message*)
		bMsg1708 : BOOL; (*reserve warning message*)
		bMsg1709 : BOOL; (*reserve warning message*)
		bMsg1710 : BOOL; (*reserve warning message*)
		bMsg1711 : BOOL; (*reserve warning message*)
		bMsg1712 : BOOL; (*reserve warning message*)
		bMsg1713 : BOOL; (*reserve warning message*)
		bMsg1714 : BOOL; (*reserve warning message 40*)
		bMsg1715 : BOOL; (*reserve warning message 41*)
		bMsg1716 : BOOL; (*reserve warning message*)
		bMsg1717 : BOOL; (*reserve warning message*)
		bMsg1718 : BOOL; (*reserve warning message*)
		bMsg1719 : BOOL; (*reserve warning message*)
		bMsg1720 : BOOL; (*reserve warning message*)
		bMsg1721 : BOOL; (*reserve warning message*)
		bMsg1722 : BOOL; (*reserve warning message*)
		bMsg1723 : BOOL; (*reserve warning message*)
		bMsg1724 : BOOL; (*reserve warning message 50*)
		bMsg1725 : BOOL; (*reserve warning message*)
		bMsg1726 : BOOL; (*reserve warning message*)
		bMsg1727 : BOOL; (*reserve warning message*)
		bMsg1728 : BOOL; (*reserve warning message*)
		bMsg1729 : BOOL; (*reserve warning message*)
		bMsg1730 : BOOL; (*reserve warning message*)
		bMsg1731 : BOOL; (*reserve warning message*)
		bMsg1732 : BOOL; (*reserve warning message*)
		bMsg1733 : BOOL; (*reserve warning message*)
		bMsg1734 : BOOL; (*reserve warning message 60*)
		bMsg1735 : BOOL; (*reserve warning message*)
		bMsg1736 : BOOL; (*reserve warning message*)
		bMsg1737 : BOOL; (*reserve warning message*)
		bMsg1738 : BOOL; (*reserve warning message*)
		bMsg1739 : BOOL; (*reserve warning message*)
		bMsg1740 : BOOL; (*reserve warning message*)
		bMsg1741 : BOOL; (*reserve warning message*)
		bMsg1742 : BOOL; (*reserve warning message*)
		bMsg1743 : BOOL; (*reserve warning message*)
		bMsg1744 : BOOL; (*reserve warning message 70*)
		bMsg1745 : BOOL; (*reserve warning message*)
		bMsg1746 : BOOL; (*reserve warning message*)
		bMsg1747 : BOOL; (*reserve warning message*)
		bMsg1748 : BOOL; (*reserve warning message*)
		bMsg1749 : BOOL; (*reserve warning message*)
		bMsg1750 : BOOL; (*reserve warning message*)
		bMsg1751 : BOOL; (*reserve warning message*)
		bMsg1752 : BOOL; (*reserve warning message*)
		bMsg1753 : BOOL; (*reserve warning message*)
		bMsg1754 : BOOL; (*reserve warning message 80*)
		bMsg1755 : BOOL; (*reserve warning message*)
		bMsg1756 : BOOL; (*reserve warning message*)
		bMsg1757 : BOOL; (*reserve warning message*)
		bMsg1758 : BOOL; (*reserve warning message*)
		bMsg1759 : BOOL; (*reserve warning message*)
		bMsg1760 : BOOL; (*reserve warning message*)
		bMsg1761 : BOOL; (*reserve warning message*)
		bMsg1762 : BOOL; (*reserve warning message*)
		bMsg1763 : BOOL; (*reserve warning message*)
		bMsg1764 : BOOL; (*reserve warning message 90*)
		bMsg1765 : BOOL; (*reserve warning message*)
		bMsg1766 : BOOL; (*reserve warning message*)
		bMsg1767 : BOOL; (*reserve warning message*)
		bMsg1768 : BOOL; (*reserve warning message*)
		bMsg1769 : BOOL; (*reserve warning message*)
		bMsg1770 : BOOL; (*reserve warning message*)
		bMsg1771 : BOOL; (*reserve warning message*)
		bMsg1772 : BOOL; (*reserve warning message*)
		bMsg1773 : BOOL; (*reserve warning message*)
		bMsg1774 : BOOL; (*reserve warning message 100*)
		bMsg1775 : BOOL; (*reserve warning message*)
		bMsg1776 : BOOL; (*reserve warning message*)
		bMsg1777 : BOOL; (*reserve warning message*)
		bMsg1778 : BOOL; (*reserve warning message*)
		bMsg1779 : BOOL; (*reserve warning message*)
		bMsg1780 : BOOL; (*reserve warning message*)
		bMsg1781 : BOOL; (*reserve warning message*)
		bMsg1782 : BOOL; (*reserve warning message*)
		bMsg1783 : BOOL; (*reserve warning message*)
		bMsg1784 : BOOL; (*reserve warning message 110*)
		bMsg1785 : BOOL; (*reserve warning message*)
		bMsg1786 : BOOL; (*reserve warning message*)
		bMsg1787 : BOOL; (*reserve warning message*)
		bMsg1788 : BOOL; (*reserve warning message*)
		bMsg1789 : BOOL; (*reserve warning message*)
		bMsg1790 : BOOL; (*reserve warning message*)
		bMsg1791 : BOOL; (*reserve warning message*)
		bMsg1792 : BOOL; (*reserve warning message*)
		bMsg1793 : BOOL; (*reserve warning message*)
		bMsg1794 : BOOL; (*reserve warning message 120*)
		bMsg1795 : BOOL; (*reserve warning message 121*)
		bMsg1796 : BOOL; (*reserve warning message 122*)
		bMsg1797 : BOOL; (*reserve warning message 123*)
		bMsg1798 : BOOL; (*reserve warning message 124*)
		bMsg1799 : BOOL; (*reserve warning message 125*)
		bMsg1800 : BOOL; (*reserve warning message 126*)
		bMsg2032 : BOOL; (* = 	Alarmbit to visu			*)
		bMsg2033 : BOOL; (* = 	Alarmbit to visu			*)
		bMsg2034 : BOOL; (* = 	Alarmbit to visu			*)
		bMsg2035 : BOOL; (* = 	Alarmbit to visu			*)
		bMsg2036 : BOOL; (* = 	Alarmbit to visu			*)
		bMsg2037 : BOOL; (* = 	Alarmbit to visu			*)
		bMsg2050 : BOOL; (* = 	Alarmbit to visu			*)
		bMsg2051 : BOOL; (* = 	Alarmbit to visu			*)
		bMsg2087 : BOOL; (*reserve warning message 17*)
		bMsg2088 : BOOL; (*reserve warning message 18*)
		bMsg2089 : BOOL; (*reserve warning message 19*)
		bMsg2090 : BOOL; (*reserve warning message 20*)
		bMsg2091 : BOOL; (*reserve warning message 21*)
		bMsg2092 : BOOL; (*reserve warning message 22*)
		bMsg2093 : BOOL; (*reserve warning message 23*)
		bMsg2094 : BOOL; (*reserve warning message 24*)
		bMsg2095 : BOOL; (*reserve warning message 25*)
		bMsg2096 : BOOL; (*reserve warning message 26*)
		bMsg2302 : BOOL; (*alarm message mns import ctr*)
		bMsg2303 : BOOL; (*alarm message mns import ctr*)
		bMsg2415 : BOOL; (*warning message mns import ctr*)
		bMsg2416 : BOOL; (*warning message mns import ctr*)
		bMsg2417 : BOOL; (*warning message mns import ctr*)
		bMsg2418 : BOOL; (*warning message mns import ctr*)
		bMsg2419 : BOOL; (*operating message mns import ctr*)
		bMsg2420 : BOOL; (*operating message mns import ctr*)
		bMsg2811 : BOOL; (*operating message EVU reduction*)
		bMsg2812 : BOOL; (*operating message EVU reduction*)
		bMsg3232 : BOOL; (*reserve operating message 1*)
		bMsg3233 : BOOL; (*reserve operating message 2*)
		bMsg3234 : BOOL; (*reserve operating message 3*)
		bMsg3235 : BOOL; (*reserve operating message 4*)
		bMsg3236 : BOOL; (*reserve operating message 5*)
		bMsg3237 : BOOL; (*reserve operating message 6*)
		bMsg3250 : BOOL; (*reserve operating message 7*)
		bMsg3251 : BOOL; (*reserve operating message 8*)
		bMsg3565 : BOOL; (*Messignalstoerung Generator Leistungssollwert*)
		bMsg3566 : BOOL; (*Messignalstoerung Generator Leistungsfaktorsollwert*)
		bMsg3601 : BOOL; (*reserve operating message 9*)
		bMsg3602 : BOOL; (*reserve operating message 10*)
		bMsg3603 : BOOL; (*reserve operating message 11*)
		bMsg3604 : BOOL; (*reserve operating message 12*)
		bMsg3605 : BOOL; (*reserve operating message 13*)
		bMsg3606 : BOOL; (*reserve operating message 14*)
		bMsg3607 : BOOL; (*reserve operating message 15*)
		bMsg3608 : BOOL; (*reserve operating message 16*)
		bMsg3609 : BOOL; (*reserve operating message 17*)
		bMsg3610 : BOOL; (*reserve operating message 18*)
		bMsg3611 : BOOL; (*reserve operating message 19*)
		bMsg3612 : BOOL; (*reserve operating message 20*)
		bMsg3613 : BOOL; (*reserve operating message *)
		bMsg3614 : BOOL; (*reserve operating message *)
		bMsg3615 : BOOL; (*reserve operating message *)
		bMsg3616 : BOOL; (*reserve operating message *)
		bMsg3617 : BOOL; (*reserve operating message *)
		bMsg3618 : BOOL; (*reserve operating message *)
		bMsg3619 : BOOL; (*reserve operating message *)
		bMsg3620 : BOOL; (*reserve operating message *)
		bMsg3621 : BOOL; (*reserve operating message *)
		bMsg3622 : BOOL; (*reserve operating message 30*)
		bMsg3623 : BOOL; (*reserve operating message *)
		bMsg3624 : BOOL; (*reserve operating message *)
		bMsg3625 : BOOL; (*reserve operating message *)
		bMsg3626 : BOOL; (*reserve operating message *)
		bMsg3627 : BOOL; (*reserve operating message *)
		bMsg3628 : BOOL; (*reserve operating message *)
		bMsg3629 : BOOL; (*reserve operating message *)
		bMsg3630 : BOOL; (*reserve operating message *)
		bMsg3631 : BOOL; (*reserve operating message *)
		bMsg3632 : BOOL; (*reserve operating message 40*)
		bMsg3633 : BOOL; (*reserve operating message *)
		bMsg3634 : BOOL; (*reserve operating message *)
		bMsg3635 : BOOL; (*reserve operating message *)
		bMsg3636 : BOOL; (*reserve operating message *)
		bMsg3637 : BOOL; (*reserve operating message *)
		bMsg3638 : BOOL; (*reserve operating message *)
		bMsg3639 : BOOL; (*reserve operating message *)
		bMsg3640 : BOOL; (*reserve operating message *)
		bMsg3641 : BOOL; (*reserve operating message *)
		bMsg3642 : BOOL; (*reserve operating message 50*)
		bMsg3643 : BOOL; (*reserve operating message *)
		bMsg3644 : BOOL; (*reserve operating message *)
		bMsg3645 : BOOL; (*reserve operating message *)
		bMsg3646 : BOOL; (*reserve operating message *)
		bMsg3647 : BOOL; (*reserve operating message *)
		bMsg3648 : BOOL; (*reserve operating message *)
		bMsg3649 : BOOL; (*reserve operating message *)
		bMsg3650 : BOOL; (*reserve operating message *)
		bMsg3651 : BOOL; (*reserve operating message *)
		bMsg3652 : BOOL; (*reserve operating message 60*)
		bMsg3653 : BOOL; (*reserve operating message *)
		bMsg3654 : BOOL; (*reserve operating message *)
		bMsg3655 : BOOL; (*reserve operating message *)
		bMsg3656 : BOOL; (*reserve operating message *)
		bMsg3657 : BOOL; (*reserve operating message *)
		bMsg3658 : BOOL; (*reserve operating message *)
		bMsg3659 : BOOL; (*reserve operating message *)
		bMsg3660 : BOOL; (*reserve operating message *)
		bMsg3661 : BOOL; (*reserve operating message *)
		bMsg3662 : BOOL; (*reserve operating message 70*)
		bMsg3663 : BOOL; (*reserve operating message *)
		bMsg3664 : BOOL; (*reserve operating message *)
		bMsg3665 : BOOL; (*reserve operating message *)
		bMsg3666 : BOOL; (*reserve operating message *)
		bMsg3667 : BOOL; (*reserve operating message *)
		bMsg3668 : BOOL; (*reserve operating message *)
		bMsg3669 : BOOL; (*reserve operating message *)
		bMsg3670 : BOOL; (*reserve operating message *)
		bMsg3671 : BOOL; (*reserve operating message *)
		bMsg3672 : BOOL; (*reserve operating message 80*)
		bMsg3673 : BOOL; (*reserve operating message *)
		bMsg3674 : BOOL; (*reserve operating message *)
		bMsg3675 : BOOL; (*reserve operating message *)
		bMsg3676 : BOOL; (*reserve operating message *)
		bMsg3677 : BOOL; (*reserve operating message *)
		bMsg3678 : BOOL; (*reserve operating message *)
		bMsg3679 : BOOL; (*reserve operating message *)
		bMsg3680 : BOOL; (*reserve operating message *)
		bMsg3681 : BOOL; (*reserve operating message *)
		bMsg3682 : BOOL; (*reserve operating message 90*)
		bMsg3683 : BOOL; (*reserve operating message *)
		bMsg3684 : BOOL; (*reserve operating message *)
		bMsg3685 : BOOL; (*reserve operating message *)
		bMsg3686 : BOOL; (*reserve operating message *)
		bMsg3687 : BOOL; (*reserve operating message *)
		bMsg3688 : BOOL; (*reserve operating message *)
		bMsg3689 : BOOL; (*reserve operating message *)
		bMsg3690 : BOOL; (*reserve operating message *)
		bMsg3691 : BOOL; (*reserve operating message *)
		bMsg3692 : BOOL; (*reserve operating message 100*)
		bMsg3693 : BOOL; (*reserve operating message 101*)
		bMsg3694 : BOOL; (*reserve operating message 102*)
		bMsg3695 : BOOL; (*reserve operating message 103*)
		bMsg3696 : BOOL; (*reserve operating message 104*)
		bMsg3697 : BOOL; (*reserve operating message 105*)
		bMsg3698 : BOOL; (*reserve operating message 106*)
		bMsg3699 : BOOL; (*reserve operating message 107*)
		bMsg3700 : BOOL; (*reserve operating message 108*)
		bMsg3701 : BOOL; (* = Alarmbit to visu *)
		bMsg3702 : BOOL; (* = Alarmbit to visu *)
		bMsg3703 : BOOL; (* = Alarmbit to visu *)
		bMsg3704 : BOOL; (* = Alarmbit to visu *)
		bMsg3705 : BOOL; (* = Alarmbit to visu *)
		bMsg3706 : BOOL; (* = Alarmbit to visu *)
		bMsg3707 : BOOL; (* = Alarmbit to visu *)
		bMsg3708 : BOOL; (* = Alarmbit to visu *)
		bMsg3709 : BOOL; (* = Alarmbit to visu *)
		bMsg3710 : BOOL; (* = Alarmbit to visu *)
		bMsg3711 : BOOL; (* = Alarmbit to visu *)
		bMsg3712 : BOOL; (* = Alarmbit to visu *)
		bMsg3713 : BOOL; (* = Alarmbit to visu *)
		bMsg3714 : BOOL; (* = Alarmbit to visu *)
		bMsg3715 : BOOL; (* = Alarmbit to visu *)
		bMsg3716 : BOOL; (* = Alarmbit to visu *)
		bMsg3717 : BOOL; (* = Alarmbit to visu *)
		bMsg3718 : BOOL; (* = Alarmbit to visu *)
		bMsg3719 : BOOL; (* = Alarmbit to visu *)
		bMsg3720 : BOOL; (* = Alarmbit to visu *)
		bMsg3721 : BOOL; (* = Alarmbit to visu *)
		bMsg3722 : BOOL; (* = Alarmbit to visu *)
		bMsg3723 : BOOL; (* = Alarmbit to visu *)
		bMsg3724 : BOOL; (* = Alarmbit to visu *)
		bMsg3725 : BOOL; (* = Alarmbit to visu *)
		bMsg3726 : BOOL; (* = Alarmbit to visu *)
		bMsg3727 : BOOL; (* = Alarmbit to visu *)
		bMsg3728 : BOOL; (* = Alarmbit to visu *)
		bMsg3729 : BOOL; (* = Alarmbit to visu *)
		bMsg3730 : BOOL; (* = Alarmbit to visu *)
		bMsg3731 : BOOL; (* = Alarmbit to visu *)
		bMsg3732 : BOOL; (* = Alarmbit to visu *)
		bMsg3733 : BOOL; (* = Alarmbit to visu *)
		bMsg3734 : BOOL; (* = Alarmbit to visu *)
		bMsg3735 : BOOL; (* = Alarmbit to visu *)
		bMsg3736 : BOOL; (* = Alarmbit to visu *)
		bMsg3737 : BOOL; (* = Alarmbit to visu *)
		bMsg3738 : BOOL; (* = Alarmbit to visu *)
		bMsg3739 : BOOL; (* = Alarmbit to visu *)
		bMsg3740 : BOOL; (* = Alarmbit to visu *)
		bMsg3741 : BOOL; (* = Alarmbit to visu *)
		bMsg3742 : BOOL; (* = Alarmbit to visu *)
		bMsg3743 : BOOL; (* = Alarmbit to visu *)
		bMsg3744 : BOOL; (* = Alarmbit to visu *)
		bMsg3745 : BOOL; (* = Alarmbit to visu *)
		bMsg3746 : BOOL; (* = Alarmbit to visu *)
		bMsg3747 : BOOL; (* = Alarmbit to visu *)
		bMsg3748 : BOOL; (* = Alarmbit to visu *)
		bMsg3749 : BOOL; (* = Alarmbit to visu *)
		bMsg3750 : BOOL; (* = Alarmbit to visu *)
		bMsg3751 : BOOL; (* = Alarmbit to visu *)
		bMsg3752 : BOOL; (* = Alarmbit to visu *)
		bMsg3753 : BOOL; (* = Alarmbit to visu *)
		bMsg3754 : BOOL; (* = Alarmbit to visu *)
		bMsg3755 : BOOL; (* = Alarmbit to visu *)
		bMsg3756 : BOOL; (* = Alarmbit to visu *)
		bMsg3757 : BOOL; (* = Alarmbit to visu *)
		bMsg3758 : BOOL; (* = Alarmbit to visu *)
		bMsg3759 : BOOL; (* = Alarmbit to visu *)
		bMsg3760 : BOOL; (* = Alarmbit to visu *)
		bMsg3761 : BOOL; (* = Alarmbit to visu *)
		bMsg3762 : BOOL; (* = Alarmbit to visu *)
		bMsg3763 : BOOL; (* = Alarmbit to visu *)
		bMsg3764 : BOOL; (* = Alarmbit to visu *)
		bMsg3765 : BOOL; (* = Alarmbit to visu *)
		bMsg3766 : BOOL; (* = Alarmbit to visu *)
		bMsg3767 : BOOL; (* = Alarmbit to visu *)
		bMsg3768 : BOOL; (* = Alarmbit to visu *)
		bMsg3769 : BOOL; (* = Alarmbit to visu *)
		bMsg3770 : BOOL; (* = Alarmbit to visu *)
		bMsg3771 : BOOL; (* = Alarmbit to visu *)
		bMsg3772 : BOOL; (* = Alarmbit to visu *)
		bMsg3773 : BOOL; (* = Alarmbit to visu *)
		bMsg3774 : BOOL; (* = Alarmbit to visu *)
		bMsg3775 : BOOL; (* = Alarmbit to visu *)
		bMsg3776 : BOOL; (* = Alarmbit to visu *)
		bMsg3777 : BOOL; (* = Alarmbit to visu *)
		bMsg3778 : BOOL; (* = Alarmbit to visu *)
		bMsg3779 : BOOL; (* = Alarmbit to visu *)
		bMsg3780 : BOOL; (* = Alarmbit to visu *)
		bMsg3781 : BOOL; (* = Alarmbit to visu *)
		bMsg3782 : BOOL; (* = Alarmbit to visu *)
		bMsg3783 : BOOL; (* = Alarmbit to visu *)
		bMsg3784 : BOOL; (* = Alarmbit to visu *)
		bMsg3785 : BOOL; (* = Alarmbit to visu *)
		bMsg3786 : BOOL; (* = Alarmbit to visu *)
		bMsg3787 : BOOL; (* = Alarmbit to visu *)
		bMsg3788 : BOOL; (* = Alarmbit to visu *)
		bMsg3789 : BOOL; (* = Alarmbit to visu *)
		bMsg3790 : BOOL; (* = Alarmbit to visu *)
		bMsg3801 : BOOL; (* = Alarmbit to visu *)
		bMsg3802 : BOOL; (* = Alarmbit to visu *)
		bMsg3803 : BOOL; (* = Alarmbit to visu *)
		bMsg3804 : BOOL; (* = Alarmbit to visu *)
		bMsg3805 : BOOL; (* = Alarmbit to visu *)
		bMsg3806 : BOOL; (* = Alarmbit to visu *)
		bMsg3807 : BOOL; (* = Alarmbit to visu *)
		bMsg3808 : BOOL; (* = Alarmbit to visu *)
		bMsg3809 : BOOL; (* = Alarmbit to visu *)
		bMsg3810 : BOOL; (* = Alarmbit to visu *)
		bMsg3811 : BOOL; (* = Alarmbit to visu *)
		bMsg3812 : BOOL; (* = Alarmbit to visu *)
		bMsg3813 : BOOL; (* = Alarmbit to visu *)
		bMsg3814 : BOOL; (* = Alarmbit to visu *)
		bMsg3815 : BOOL; (* = Alarmbit to visu *)
		bMsg3816 : BOOL; (* = Alarmbit to visu *)
		bMsg3817 : BOOL; (* = Alarmbit to visu *)
		bMsg3818 : BOOL; (* = Alarmbit to visu *)
		bMsg3819 : BOOL; (* = Alarmbit to visu *)
		bMsg3820 : BOOL; (* = Alarmbit to visu *)
		bMsg3821 : BOOL; (* = Alarmbit to visu *)
		bMsg3822 : BOOL; (* = Alarmbit to visu *)
		bMsg3823 : BOOL; (* = Alarmbit to visu *)
		bMsg3824 : BOOL; (* = Alarmbit to visu *)
		bMsg3825 : BOOL; (* = Alarmbit to visu *)
		bMsg3826 : BOOL; (* = Alarmbit to visu *)
		bMsg3827 : BOOL; (* = Alarmbit to visu *)
		bMsg3828 : BOOL; (* = Alarmbit to visu *)
		bMsg3829 : BOOL; (* = Alarmbit to visu *)
		bMsg3830 : BOOL; (* = Alarmbit to visu *)
		bMsg3831 : BOOL; (* = Alarmbit to visu *)
		bMsg3832 : BOOL; (* = Alarmbit to visu *)
		bMsg3833 : BOOL; (* = Alarmbit to visu *)
		bMsg3834 : BOOL; (* = Alarmbit to visu *)
		bMsg3835 : BOOL; (* = Alarmbit to visu *)
		bMsg3836 : BOOL; (* = Alarmbit to visu *)
		bMsg3837 : BOOL; (* = Alarmbit to visu *)
		bMsg3838 : BOOL; (* = Alarmbit to visu *)
		bMsg3839 : BOOL; (* = Alarmbit to visu *)
		bMsg3840 : BOOL; (* = Alarmbit to visu *)
		bMsg3841 : BOOL; (* = Alarmbit to visu *)
		bMsg3842 : BOOL; (* = Alarmbit to visu *)
		bMsg3843 : BOOL; (* = Alarmbit to visu *)
		bMsg3844 : BOOL; (* = Alarmbit to visu *)
		bMsg3845 : BOOL; (* = Alarmbit to visu *)
		bMsg3846 : BOOL; (* = Alarmbit to visu *)
		bMsg3847 : BOOL; (* = Alarmbit to visu *)
		bMsg3848 : BOOL; (* = Alarmbit to visu *)
		bMsg3849 : BOOL; (* = Alarmbit to visu *)
		bMsg3850 : BOOL; (* = Alarmbit to visu *)
		bMsg3851 : BOOL; (* = Alarmbit to visu *)
		bMsg3852 : BOOL; (* = Alarmbit to visu *)
		bMsg3853 : BOOL; (* = Alarmbit to visu *)
		bMsg3854 : BOOL; (* = Alarmbit to visu *)
		bMsg3855 : BOOL; (* = Alarmbit to visu *)
		bMsg3856 : BOOL; (* = Alarmbit to visu *)
		bMsg3857 : BOOL; (* = Alarmbit to visu *)
		bMsg3858 : BOOL; (* = Alarmbit to visu *)
		bMsg3859 : BOOL; (* = Alarmbit to visu *)
		bMsg3860 : BOOL; (* = Alarmbit to visu *)
		bMsg3861 : BOOL; (* = Alarmbit to visu *)
		bMsg3862 : BOOL; (* = Alarmbit to visu *)
		bMsg3863 : BOOL; (* = Alarmbit to visu *)
		bMsg3864 : BOOL; (* = Alarmbit to visu *)
		bMsg3865 : BOOL; (* = Alarmbit to visu *)
		bMsg3866 : BOOL; (* = Alarmbit to visu *)
		bMsg3867 : BOOL; (* = Alarmbit to visu *)
		bMsg3868 : BOOL; (* = Alarmbit to visu *)
		bMsg3869 : BOOL; (* = Alarmbit to visu *)
		bMsg3870 : BOOL; (* = Alarmbit to visu *)
		bMsg3871 : BOOL; (* = Alarmbit to visu *)
		bMsg3872 : BOOL; (* = Alarmbit to visu *)
		bMsg3873 : BOOL; (* = Alarmbit to visu *)
		bMsg3874 : BOOL; (* = Alarmbit to visu *)
		bMsg3875 : BOOL; (* = Alarmbit to visu *)
		bMsg3876 : BOOL; (* = Alarmbit to visu *)
		bMsg3877 : BOOL; (* = Alarmbit to visu *)
		bMsg3878 : BOOL; (* = Alarmbit to visu *)
		bMsg3879 : BOOL; (* = Alarmbit to visu *)
		bMsg3880 : BOOL; (* = Alarmbit to visu *)
		bMsg3881 : BOOL; (* = Alarmbit to visu *)
		bMsg3882 : BOOL; (* = Alarmbit to visu *)
		bMsg3883 : BOOL; (* = Alarmbit to visu *)
		bMsg3884 : BOOL; (* = Alarmbit to visu *)
		bMsg3885 : BOOL; (* = Alarmbit to visu *)
		bMsg3886 : BOOL; (* = Alarmbit to visu *)
		bMsg3887 : BOOL; (* = Alarmbit to visu *)
		bMsg3888 : BOOL; (* = Alarmbit to visu *)
		bMsg3889 : BOOL; (* = Alarmbit to visu *)
		bMsg3890 : BOOL; (* = Alarmbit to visu *)
		bMsg3891 : BOOL; (* = Alarmbit to visu *)
		bMsg3892 : BOOL; (* = Alarmbit to visu *)
		bMsg3893 : BOOL; (* = Alarmbit to visu *)
		bMsg3894 : BOOL; (* = Alarmbit to visu *)
		bMsg3895 : BOOL; (* = Alarmbit to visu *)
		bMsg3896 : BOOL; (* = Alarmbit to visu *)
		bMsg3897 : BOOL; (* = Alarmbit to visu *)
		bMsg3898 : BOOL; (* = Alarmbit to visu *)
		bMsg3899 : BOOL; (* = Alarmbit to visu *)
		bMsg3900 : BOOL; (* = Alarmbit to visu *)
		bMsg3901 : BOOL; (* = Alarmbit to visu *)
		bMsg3902 : BOOL; (* = Alarmbit to visu *)
		bMsg3903 : BOOL; (* = Alarmbit to visu *)
		bMsg3904 : BOOL; (* = Alarmbit to visu *)
		bMsg3905 : BOOL; (* = Alarmbit to visu *)
		bMsg3906 : BOOL; (* = Alarmbit to visu *)
		bMsg3907 : BOOL; (* = Alarmbit to visu *)
		bMsg3908 : BOOL; (* = Alarmbit to visu *)
		bMsg3909 : BOOL; (* = Alarmbit to visu *)
		bMsg3910 : BOOL; (* = Alarmbit to visu *)
		bMsg3911 : BOOL; (* = Alarmbit to visu *)
		bMsg3912 : BOOL; (* = Alarmbit to visu *)
		bMsg3913 : BOOL; (* = Alarmbit to visu *)
		bMsg3914 : BOOL; (* = Alarmbit to visu *)
		bMsg3915 : BOOL; (* = Alarmbit to visu *)
		bMsg3916 : BOOL; (* = Alarmbit to visu *)
		bMsg3917 : BOOL; (* = Alarmbit to visu *)
		bMsg3918 : BOOL; (* = Alarmbit to visu *)
		bMsg3919 : BOOL; (* = Alarmbit to visu *)
		bMsg3920 : BOOL; (* = Alarmbit to visu *)
		bMsg3921 : BOOL; (* = Alarmbit to visu *)
		bMsg3922 : BOOL; (* = Alarmbit to visu *)
		bMsg3923 : BOOL; (* = Alarmbit to visu *)
		bMsg3924 : BOOL; (* = Alarmbit to visu *)
		bMsg3925 : BOOL; (* = Alarmbit to visu *)
		bMsg3926 : BOOL; (* = Alarmbit to visu *)
		bMsg3927 : BOOL; (* = Alarmbit to visu *)
		bMsg3928 : BOOL; (* = Alarmbit to visu *)
		bMsg3929 : BOOL; (* = Alarmbit to visu *)
		bMsg3930 : BOOL; (* = Alarmbit to visu *)
		bMsg3931 : BOOL; (* = Alarmbit to visu *)
		bMsg3932 : BOOL; (* = Alarmbit to visu *)
		bMsg3933 : BOOL; (* = Alarmbit to visu *)
		bMsg3934 : BOOL; (* = Alarmbit to visu *)
		bMsg3935 : BOOL; (* = Alarmbit to visu *)
		bMsg3936 : BOOL; (* = Alarmbit to visu *)
		bMsg3937 : BOOL; (* = Alarmbit to visu *)
		bMsg3938 : BOOL; (* = Alarmbit to visu *)
		bMsg3939 : BOOL; (* = Alarmbit to visu *)
		bMsg3940 : BOOL; (* = Alarmbit to visu *)
		bMsg3941 : BOOL; (* = Alarmbit to visu *)
		bMsg3942 : BOOL; (* = Alarmbit to visu *)
		bMsg3943 : BOOL; (* = Alarmbit to visu *)
		bMsg3944 : BOOL; (* = Alarmbit to visu *)
		bMsg3945 : BOOL; (* = Alarmbit to visu *)
		bMsg3946 : BOOL; (* = Alarmbit to visu *)
		bMsg3947 : BOOL; (* = Alarmbit to visu *)
		bMsg3948 : BOOL; (* = Alarmbit to visu *)
		bMsg3949 : BOOL; (* = Alarmbit to visu *)
		bMsg3950 : BOOL; (* = Alarmbit to visu *)
		bMsg3951 : BOOL; (* = Alarmbit to visu *)
		bMsg3952 : BOOL; (* = Alarmbit to visu *)
		bMsg3953 : BOOL; (* = Alarmbit to visu *)
		bMsg3954 : BOOL; (* = Alarmbit to visu *)
		bMsg3955 : BOOL; (* = Alarmbit to visu *)
		bMsg3956 : BOOL; (* = Alarmbit to visu *)
		bMsg3957 : BOOL; (* = Alarmbit to visu *)
		bMsg3958 : BOOL; (* = Alarmbit to visu *)
		bMsg3959 : BOOL; (* = Alarmbit to visu *)
		bMsg3960 : BOOL; (* = Alarmbit to visu *)
		bMsg6701 : BOOL; (*reserve operating message 109*) (*import HMI Extension*)
		bMsg6702 : BOOL; (*reserve operating message 110*) (*import HMI Extension*)
		bMsg6703 : BOOL; (*reserve operating message 111*) (*import HMI Extension*)
		bMsg6704 : BOOL; (*reserve operating message 112*) (*import HMI Extension*)
		bMsg6705 : BOOL; (*reserve operating message 113*) (*import HMI Extension*)
		bMsg6706 : BOOL; (*reserve operating message 114*) (*import HMI Extension*)
		bMsg6707 : BOOL; (*reserve operating message 115*) (*import HMI Extension*)
		bMsg6708 : BOOL; (*reserve operating message 116*) (*import HMI Extension*)
		bMsg6709 : BOOL; (*reserve operating message 117*) (*import HMI Extension*)
		bMsg6710 : BOOL; (*reserve operating message 118*) (*import HMI Extension*)
		bMsg6711 : BOOL; (*reserve operating message 119*) (*import HMI Extension*)
		bMsg6712 : BOOL; (*reserve operating message 120*) (*import HMI Extension*)
		bMsg6713 : BOOL; (*reserve operating message 121*) (*import HMI Extension*)
		bMsg6714 : BOOL; (*reserve operating message 122*) (*import HMI Extension*)
		bMsg6715 : BOOL; (*reserve operating message 123*) (*import HMI Extension*)
		bMsg6716 : BOOL; (*reserve operating message 124*) (*import HMI Extension*)
		bMsg6717 : BOOL; (*reserve operating message 125*) (*import HMI Extension*)
		bMsg6718 : BOOL; (*reserve operating message 126*) (*import HMI Extension*)
		bMsg6719 : BOOL; (*reserve operating message 127*) (*import HMI Extension*)
		bMsg6720 : BOOL; (*reserve operating message 128*) (*import HMI Extension*)
		bMsg6721 : BOOL; (*reserve operating message 129*) (*import HMI Extension*)
		bMsg6722 : BOOL; (*reserve operating message 130*) (*import HMI Extension*)
		bMsg6723 : BOOL; (*reserve operating message 131*) (*import HMI Extension*)
		bMsg6724 : BOOL; (*reserve operating message 132*) (*import HMI Extension*)
		bMsg6725 : BOOL; (*reserve operating message 133*) (*import HMI Extension*)
		bMsg6726 : BOOL; (*reserve operating message 134*) (*import HMI Extension*)
		bMsg6727 : BOOL; (*reserve operating message 135*) (*import HMI Extension*)
		bMsg6728 : BOOL; (*reserve operating message 136*) (*import HMI Extension*)
		bMsg6729 : BOOL; (*reserve operating message 137*) (*import HMI Extension*)
		bMsg6730 : BOOL; (*reserve operating message 138*) (*import HMI Extension*)
		bMsg6731 : BOOL; (*reserve operating message 139*) (*import HMI Extension*)
		bMsg6732 : BOOL; (*reserve operating message 140*) (*import HMI Extension*)
		bMsg6733 : BOOL; (*reserve operating message 141*) (*import HMI Extension*)
		bMsg6734 : BOOL; (*reserve operating message 142*) (*import HMI Extension*)
		bMsg6735 : BOOL; (*reserve operating message 143*) (*import HMI Extension*)
		bMsg6736 : BOOL; (*reserve operating message 144*) (*import HMI Extension*)
		bMsg6737 : BOOL; (*reserve operating message 145*) (*import HMI Extension*)
		bMsg6738 : BOOL; (*reserve operating message 146*) (*import HMI Extension*)
		bMsg6739 : BOOL; (*reserve operating message 147*) (*import HMI Extension*)
		bMsg6740 : BOOL; (*reserve operating message 148*) (*import HMI Extension*)
		bMsg6741 : BOOL; (*reserve operating message 149*) (*import HMI Extension*)
		bMsg6742 : BOOL; (*reserve operating message 150*) (*import HMI Extension*)
		bMsg6743 : BOOL; (*reserve operating message 151*) (*import HMI Extension*)
		bMsg6744 : BOOL; (*reserve operating message 152*) (*import HMI Extension*)
		bMsg6745 : BOOL; (*reserve operating message 153*) (*import HMI Extension*)
		bMsg6746 : BOOL; (*reserve operating message 154*) (*import HMI Extension*)
		bMsg6747 : BOOL; (*reserve operating message 155*) (*import HMI Extension*)
		bMsg6748 : BOOL; (*reserve operating message 156*) (*import HMI Extension*)
		bMsg6749 : BOOL; (*reserve operating message 157*) (*import HMI Extension*)
		bMsg6750 : BOOL; (*reserve operating message 158*) (*import HMI Extension*)
		bMsg6751 : BOOL; (*reserve operating message 159*) (*import HMI Extension*)
		bMsg6752 : BOOL; (*reserve operating message 160*) (*import HMI Extension*)
		bMsg6753 : BOOL; (*reserve operating message 161*) (*import HMI Extension*)
		bMsg6754 : BOOL; (*reserve operating message 162*) (*import HMI Extension*)
		bMsg6755 : BOOL; (*reserve operating message 163*) (*import HMI Extension*)
		bMsg6756 : BOOL; (*reserve operating message 164*) (*import HMI Extension*)
		bMsg6757 : BOOL; (*reserve operating message 165*) (*import HMI Extension*)
		bMsg6758 : BOOL; (*reserve operating message 166*) (*import HMI Extension*)
		bMsg6759 : BOOL; (*reserve operating message 167*) (*import HMI Extension*)
		bMsg6760 : BOOL; (*reserve operating message 168*) (*import HMI Extension*)
		bMsg6761 : BOOL; (*reserve operating message 169*) (*import HMI Extension*)
		bMsg6762 : BOOL; (*reserve operating message 170*) (*import HMI Extension*)
		bMsg6763 : BOOL; (*reserve operating message 171*) (*import HMI Extension*)
		bMsg6764 : BOOL; (*reserve operating message 172*) (*import HMI Extension*)
		bMsg6765 : BOOL; (*reserve operating message 173*) (*import HMI Extension*)
		bMsg6766 : BOOL; (*reserve operating message 174*) (*import HMI Extension*)
		bMsg6767 : BOOL; (*reserve operating message 175*) (*import HMI Extension*)
		bMsg6768 : BOOL; (*reserve operating message 176*) (*import HMI Extension*)
		bMsg6769 : BOOL; (*reserve operating message 177*) (*import HMI Extension*)
		bMsg6770 : BOOL; (*reserve operating message 178*) (*import HMI Extension*)
		bMsg6771 : BOOL; (*reserve operating message 179*) (*import HMI Extension*)
		bMsg6772 : BOOL; (*reserve operating message 180*) (*import HMI Extension*)
		bMsg6773 : BOOL; (*reserve operating message 181*) (*import HMI Extension*)
		bMsg6774 : BOOL; (*reserve operating message 182*) (*import HMI Extension*)
		bMsg6775 : BOOL; (*reserve operating message 183*) (*import HMI Extension*)
		bMsg6776 : BOOL; (*reserve operating message 184*) (*import HMI Extension*)
		bMsg6777 : BOOL; (*reserve operating message 185*) (*import HMI Extension*)
		bMsg6778 : BOOL; (*reserve operating message 186*) (*import HMI Extension*)
		bMsg6779 : BOOL; (*reserve operating message 187*) (*import HMI Extension*)
		bMsg6780 : BOOL; (*reserve operating message 188*) (*import HMI Extension*)
		bMsg6781 : BOOL; (*reserve operating message 189*) (*import HMI Extension*)
		bMsg6782 : BOOL; (*reserve operating message 190*) (*import HMI Extension*)
		bMsg6783 : BOOL; (*reserve operating message 191*) (*import HMI Extension*)
		bMsg6784 : BOOL; (*reserve operating message 192*) (*import HMI Extension*)
		bMsg6785 : BOOL; (*reserve operating message 193*) (*import HMI Extension*)
		bMsg6786 : BOOL; (*reserve operating message 194*) (*import HMI Extension*)
		bMsg6787 : BOOL; (*reserve operating message 195*) (*import HMI Extension*)
		bMsg6788 : BOOL; (*reserve operating message 196*) (*import HMI Extension*)
		bMsg6789 : BOOL; (*reserve operating message 197*) (*import HMI Extension*)
		bMsg6790 : BOOL; (*reserve operating message 198*) (*import HMI Extension*)
		bMsg6791 : BOOL; (*reserve operating message 199*) (*import HMI Extension*)
		bMsg6792 : BOOL; (*reserve operating message 200*) (*import HMI Extension*)
		bMsg6793 : BOOL; (*reserve operating message 201*) (*import HMI Extension*)
		bMsg6794 : BOOL; (*reserve operating message 202*) (*import HMI Extension*)
		bMsg6795 : BOOL; (*reserve operating message 203*) (*import HMI Extension*)
		bMsg6796 : BOOL; (*reserve operating message 204*) (*import HMI Extension*)
		bMsg6797 : BOOL; (*reserve operating message 205*) (*import HMI Extension*)
		bMsg6798 : BOOL; (*reserve operating message 206*) (*import HMI Extension*)
		bMsg6799 : BOOL; (*reserve operating message 207*) (*import HMI Extension*)
		bMsg6800 : BOOL; (*reserve operating message 208*) (*import HMI Extension*)
		bMsg6801 : BOOL; (*reserve operating message 209*) (*import HMI Extension*)
		bMsg6802 : BOOL; (*reserve operating message 210*) (*import HMI Extension*)
		bMsg6803 : BOOL; (*reserve operating message 211*) (*import HMI Extension*)
		bMsg6804 : BOOL; (*reserve operating message 212*) (*import HMI Extension*)
		bMsg6805 : BOOL; (*reserve operating message 213*) (*import HMI Extension*)
		bMsg6806 : BOOL; (*reserve operating message 214*) (*import HMI Extension*)
		bMsg6807 : BOOL; (*reserve operating message 215*) (*import HMI Extension*)
		bMsg6808 : BOOL; (*reserve operating message 216*) (*import HMI Extension*)
		bMsg6809 : BOOL; (*reserve operating message 217*) (*import HMI Extension*)
		bMsg6810 : BOOL; (*reserve operating message 218*) (*import HMI Extension*)
		bMsg6811 : BOOL; (*reserve operating message 219*) (*import HMI Extension*)
		bMsg6812 : BOOL; (*reserve operating message 220*) (*import HMI Extension*)
		bMsg6813 : BOOL; (*reserve operating message 221*) (*import HMI Extension*)
		bMsg6814 : BOOL; (*reserve operating message 222*) (*import HMI Extension*)
		bMsg6815 : BOOL; (*reserve operating message 223*) (*import HMI Extension*)
		bMsg6816 : BOOL; (*reserve operating message 224*) (*import HMI Extension*)
		bMsg6817 : BOOL; (*reserve operating message 225*) (*import HMI Extension*)
		bMsg6818 : BOOL; (*reserve operating message 226*) (*import HMI Extension*)
		bMsg6819 : BOOL; (*reserve operating message 227*) (*import HMI Extension*)
		bMsg6820 : BOOL; (*reserve operating message 228*) (*import HMI Extension*)
		bMsg6821 : BOOL; (*reserve operating message 229*) (*import HMI Extension*)
		bMsg6822 : BOOL; (*reserve operating message 230*) (*import HMI Extension*)
		bMsg6823 : BOOL; (*reserve operating message 231*) (*import HMI Extension*)
		bMsg6824 : BOOL; (*reserve operating message 232*) (*import HMI Extension*)
		bMsg6825 : BOOL; (*reserve operating message 233*) (*import HMI Extension*)
		bMsg6826 : BOOL; (*reserve operating message 234*) (*import HMI Extension*)
		bMsg6827 : BOOL; (*reserve operating message 235*) (*import HMI Extension*)
		bMsg6828 : BOOL; (*reserve operating message 236*) (*import HMI Extension*)
		bMsg6829 : BOOL; (*reserve operating message 237*) (*import HMI Extension*)
		bMsg6830 : BOOL; (*reserve operating message 238*) (*import HMI Extension*)
		bMsg6831 : BOOL; (*reserve operating message 239*) (*import HMI Extension*)
		bMsg6832 : BOOL; (*reserve operating message 240*) (*import HMI Extension*)
		bMsg6833 : BOOL; (*reserve operating message 241*) (*import HMI Extension*)
		bMsg6834 : BOOL; (*reserve operating message 242*) (*import HMI Extension*)
		bMsg6835 : BOOL; (*reserve operating message 243*) (*import HMI Extension*)
		bMsg6836 : BOOL; (*reserve operating message 244*) (*import HMI Extension*)
		bMsg6837 : BOOL; (*reserve operating message 245*) (*import HMI Extension*)
		bMsg6838 : BOOL; (*reserve operating message 246*) (*import HMI Extension*)
		bMsg6839 : BOOL; (*reserve operating message 247*) (*import HMI Extension*)
		bMsg6840 : BOOL; (*reserve operating message 248*) (*import HMI Extension*)
		bMsg6841 : BOOL; (*reserve operating message 249*) (*import HMI Extension*)
		bMsg6842 : BOOL; (*reserve operating message 250*) (*import HMI Extension*)
		bMsg6843 : BOOL; (*reserve operating message 251*) (*import HMI Extension*)
		bMsg6844 : BOOL; (*reserve operating message 252*) (*import HMI Extension*)
		bMsg6845 : BOOL; (*reserve operating message 253*) (*import HMI Extension*)
		bMsg6846 : BOOL; (*reserve operating message 254*) (*import HMI Extension*)
		bMsg6847 : BOOL; (*reserve operating message 255*) (*import HMI Extension*)
		bMsg6848 : BOOL; (*reserve operating message 256*) (*import HMI Extension*)
		bMsg6849 : BOOL; (*reserve operating message 257*) (*import HMI Extension*)
		bMsg6850 : BOOL; (*reserve operating message 258*) (*import HMI Extension*)
		bMsg6851 : BOOL; (*reserve operating message 259*) (*import HMI Extension*)
		bMsg6852 : BOOL; (*reserve operating message 260*) (*import HMI Extension*)
		bMsg6853 : BOOL; (*reserve operating message 261*) (*import HMI Extension*)
		bMsg6854 : BOOL; (*reserve operating message 262*) (*import HMI Extension*)
		bMsg6855 : BOOL; (*reserve operating message 263*) (*import HMI Extension*)
		bMsg6856 : BOOL; (*reserve operating message 264*) (*import HMI Extension*)
		bMsg6857 : BOOL; (*reserve operating message 265*) (*import HMI Extension*)
		bMsg6858 : BOOL; (*reserve operating message 266*) (*import HMI Extension*)
		bMsg6859 : BOOL; (*reserve operating message 267*) (*import HMI Extension*)
		bMsg6860 : BOOL; (*reserve operating message 268*) (*import HMI Extension*)
		bMsg6861 : BOOL; (*reserve operating message 269*) (*import HMI Extension*)
		bMsg6862 : BOOL; (*reserve operating message 270*) (*import HMI Extension*)
		bMsg6863 : BOOL; (*reserve operating message 271*) (*import HMI Extension*)
		bMsg6864 : BOOL; (*reserve operating message 272*) (*import HMI Extension*)
		bMsg6865 : BOOL; (*reserve operating message 273*) (*import HMI Extension*)
		bMsg6866 : BOOL; (*reserve operating message 274*) (*import HMI Extension*)
		bMsg6867 : BOOL; (*reserve operating message 275*) (*import HMI Extension*)
		bMsg6868 : BOOL; (*reserve operating message 276*) (*import HMI Extension*)
		bMsg6869 : BOOL; (*reserve operating message 277*) (*import HMI Extension*)
		bMsg6870 : BOOL; (*reserve operating message 278*) (*import HMI Extension*)
		bMsg6871 : BOOL; (*reserve operating message 279*) (*import HMI Extension*)
		bMsg6872 : BOOL; (*reserve operating message 280*) (*import HMI Extension*)
		bMsg6873 : BOOL; (*reserve operating message 281*) (*import HMI Extension*)
		bMsg6874 : BOOL; (*reserve operating message 282*) (*import HMI Extension*)
		bMsg6875 : BOOL; (*reserve operating message 283*) (*import HMI Extension*)
		bMsg6876 : BOOL; (*reserve operating message 284*) (*import HMI Extension*)
		bMsg6877 : BOOL; (*reserve operating message 285*) (*import HMI Extension*)
		bMsg6878 : BOOL; (*reserve operating message 286*) (*import HMI Extension*)
		bMsg6879 : BOOL; (*reserve operating message 287*) (*import HMI Extension*)
		bMsg6880 : BOOL; (*reserve operating message 288*) (*import HMI Extension*)
		bMsg6881 : BOOL; (*reserve operating message 289*) (*import HMI Extension*)
		bMsg6882 : BOOL; (*reserve operating message 290*) (*import HMI Extension*)
		bMsg6883 : BOOL; (*reserve operating message 291*) (*import HMI Extension*)
		bMsg6884 : BOOL; (*reserve operating message 292*) (*import HMI Extension*)
		bMsg6885 : BOOL; (*reserve operating message 293*) (*import HMI Extension*)
		bMsg6886 : BOOL; (*reserve operating message 294*) (*import HMI Extension*)
		bMsg6887 : BOOL; (*reserve operating message 295*) (*import HMI Extension*)
		bMsg6888 : BOOL; (*reserve operating message 296*) (*import HMI Extension*)
		bMsg6889 : BOOL; (*reserve operating message 297*) (*import HMI Extension*)
		bMsg6890 : BOOL; (*reserve operating message 298*) (*import HMI Extension*)
		bMsg6891 : BOOL; (*reserve operating message 299*) (*import HMI Extension*)
		bMsg6892 : BOOL; (*reserve operating message 300*) (*import HMI Extension*)
		bMsg6893 : BOOL; (*reserve operating message 301*) (*import HMI Extension*)
		bMsg6894 : BOOL; (*reserve operating message 302*) (*import HMI Extension*)
		bMsg6895 : BOOL; (*reserve operating message 303*) (*import HMI Extension*)
		bMsg6896 : BOOL; (*reserve operating message 304*) (*import HMI Extension*)
		bMsg6897 : BOOL; (*reserve operating message 305*) (*import HMI Extension*)
		bMsg6898 : BOOL; (*reserve operating message 306*) (*import HMI Extension*)
		bMsg6899 : BOOL; (*reserve operating message 307*) (*import HMI Extension*)
		bMsg6900 : BOOL; (* DO NOT USE ANYMORE reserve operating message 308xxx*) (*import HMI Extension*)
		bMsg8701 : BOOL; (*reserve warning message 127*) (*import HMI Extension*)
		bMsg8702 : BOOL; (*reserve warning message 128*) (*import HMI Extension*)
		bMsg8703 : BOOL; (*reserve warning message 129*) (*import HMI Extension*)
		bMsg8704 : BOOL; (*reserve warning message 130*) (*import HMI Extension*)
		bMsg8705 : BOOL; (*reserve warning message 131*) (*import HMI Extension*)
		bMsg8706 : BOOL; (*reserve warning message 132*) (*import HMI Extension*)
		bMsg8707 : BOOL; (*reserve warning message 133*) (*import HMI Extension*)
		bMsg8708 : BOOL; (*reserve warning message 134*) (*import HMI Extension*)
		bMsg8709 : BOOL; (*reserve warning message 135*) (*import HMI Extension*)
		bMsg8710 : BOOL; (*reserve warning message 136*) (*import HMI Extension*)
		bMsg8711 : BOOL; (*reserve warning message 137*) (*import HMI Extension*)
		bMsg8712 : BOOL; (*reserve warning message 138*) (*import HMI Extension*)
		bMsg8713 : BOOL; (*reserve warning message 139*) (*import HMI Extension*)
		bMsg8714 : BOOL; (*reserve warning message 140*) (*import HMI Extension*)
		bMsg8715 : BOOL; (*reserve warning message 141*) (*import HMI Extension*)
		bMsg8716 : BOOL; (*reserve warning message 142*) (*import HMI Extension*)
		bMsg8717 : BOOL; (*reserve warning message 143*) (*import HMI Extension*)
		bMsg8718 : BOOL; (*reserve warning message 144*) (*import HMI Extension*)
		bMsg8719 : BOOL; (*reserve warning message 145*) (*import HMI Extension*)
		bMsg8720 : BOOL; (*reserve warning message 146*) (*import HMI Extension*)
		bMsg8721 : BOOL; (*reserve warning message 147*) (*import HMI Extension*)
		bMsg8722 : BOOL; (*reserve warning message 148*) (*import HMI Extension*)
		bMsg8723 : BOOL; (*reserve warning message 149*) (*import HMI Extension*)
		bMsg8724 : BOOL; (*reserve warning message 150*) (*import HMI Extension*)
		bMsg8725 : BOOL; (*reserve warning message 151*) (*import HMI Extension*)
		bMsg8726 : BOOL; (*reserve warning message 152*) (*import HMI Extension*)
		bMsg8727 : BOOL; (*reserve warning message 153*) (*import HMI Extension*)
		bMsg8728 : BOOL; (*reserve warning message 154*) (*import HMI Extension*)
		bMsg8729 : BOOL; (*reserve warning message 155*) (*import HMI Extension*)
		bMsg8730 : BOOL; (*reserve warning message 156*) (*import HMI Extension*)
		bMsg8731 : BOOL; (*reserve warning message 157*) (*import HMI Extension*)
		bMsg8732 : BOOL; (*reserve warning message 158*) (*import HMI Extension*)
		bMsg8733 : BOOL; (*reserve warning message 159*) (*import HMI Extension*)
		bMsg8734 : BOOL; (*reserve warning message 160*) (*import HMI Extension*)
		bMsg8735 : BOOL; (*reserve warning message 161*) (*import HMI Extension*)
		bMsg8736 : BOOL; (*reserve warning message 162*) (*import HMI Extension*)
		bMsg8737 : BOOL; (*reserve warning message 163*) (*import HMI Extension*)
		bMsg8738 : BOOL; (*reserve warning message 164*) (*import HMI Extension*)
		bMsg8739 : BOOL; (*reserve warning message 165*) (*import HMI Extension*)
		bMsg8740 : BOOL; (*reserve warning message 166*) (*import HMI Extension*)
		bMsg8741 : BOOL; (*reserve warning message 167*) (*import HMI Extension*)
		bMsg8742 : BOOL; (*reserve warning message 168*) (*import HMI Extension*)
		bMsg8743 : BOOL; (*reserve warning message 169*) (*import HMI Extension*)
		bMsg8744 : BOOL; (*reserve warning message 170*) (*import HMI Extension*)
		bMsg8745 : BOOL; (*reserve warning message 171*) (*import HMI Extension*)
		bMsg8746 : BOOL; (*reserve warning message 172*) (*import HMI Extension*)
		bMsg8747 : BOOL; (*reserve warning message 173*) (*import HMI Extension*)
		bMsg8748 : BOOL; (*reserve warning message 174*) (*import HMI Extension*)
		bMsg8749 : BOOL; (*reserve warning message 175*) (*import HMI Extension*)
		bMsg8750 : BOOL; (*reserve warning message 176*) (*import HMI Extension*)
		bMsg8751 : BOOL; (*reserve warning message 177*) (*import HMI Extension*)
		bMsg8752 : BOOL; (*reserve warning message 178*) (*import HMI Extension*)
		bMsg8753 : BOOL; (*reserve warning message 179*) (*import HMI Extension*)
		bMsg8754 : BOOL; (*reserve warning message 180*) (*import HMI Extension*)
		bMsg8755 : BOOL; (*reserve warning message 181*) (*import HMI Extension*)
		bMsg8756 : BOOL; (*reserve warning message 182*) (*import HMI Extension*)
		bMsg8757 : BOOL; (*reserve warning message 183*) (*import HMI Extension*)
		bMsg8758 : BOOL; (*reserve warning message 184*) (*import HMI Extension*)
		bMsg8759 : BOOL; (*reserve warning message 185*) (*import HMI Extension*)
		bMsg8760 : BOOL; (*reserve warning message 186*) (*import HMI Extension*)
		bMsg8761 : BOOL; (*reserve warning message 187*) (*import HMI Extension*)
		bMsg8762 : BOOL; (*reserve warning message 188*) (*import HMI Extension*)
		bMsg8763 : BOOL; (*reserve warning message 189*) (*import HMI Extension*)
		bMsg8764 : BOOL; (*reserve warning message 190*) (*import HMI Extension*)
		bMsg8765 : BOOL; (*reserve warning message 191*) (*import HMI Extension*)
		bMsg8766 : BOOL; (*reserve warning message 192*) (*import HMI Extension*)
		bMsg8767 : BOOL; (*reserve warning message 193*) (*import HMI Extension*)
		bMsg8768 : BOOL; (*reserve warning message 194*) (*import HMI Extension*)
		bMsg8769 : BOOL; (*reserve warning message 195*) (*import HMI Extension*)
		bMsg8770 : BOOL; (*reserve warning message 196*) (*import HMI Extension*)
		bMsg8771 : BOOL; (*reserve warning message 197*) (*import HMI Extension*)
		bMsg8772 : BOOL; (*reserve warning message 198*) (*import HMI Extension*)
		bMsg8773 : BOOL; (*reserve warning message 199*) (*import HMI Extension*)
		bMsg8774 : BOOL; (*reserve warning message 200*) (*import HMI Extension*)
		bMsg8775 : BOOL; (*reserve warning message 201*) (*import HMI Extension*)
		bMsg8776 : BOOL; (*reserve warning message 202*) (*import HMI Extension*)
		bMsg8777 : BOOL; (*reserve warning message 203*) (*import HMI Extension*)
		bMsg8778 : BOOL; (*reserve warning message 204*) (*import HMI Extension*)
		bMsg8779 : BOOL; (*reserve warning message 205*) (*import HMI Extension*)
		bMsg8780 : BOOL; (*reserve warning message 206*) (*import HMI Extension*)
		bMsg8781 : BOOL; (*reserve warning message 207*) (*import HMI Extension*)
		bMsg8782 : BOOL; (*reserve warning message 208*) (*import HMI Extension*)
		bMsg8783 : BOOL; (*reserve warning message 209*) (*import HMI Extension*)
		bMsg8784 : BOOL; (*reserve warning message 210*) (*import HMI Extension*)
		bMsg8785 : BOOL; (*reserve warning message 211*) (*import HMI Extension*)
		bMsg8786 : BOOL; (*reserve warning message 212*) (*import HMI Extension*)
		bMsg8787 : BOOL; (*reserve warning message 213*) (*import HMI Extension*)
		bMsg8788 : BOOL; (*reserve warning message 214*) (*import HMI Extension*)
		bMsg8789 : BOOL; (*reserve warning message 215*) (*import HMI Extension*)
		bMsg8790 : BOOL; (*reserve warning message 216*) (*import HMI Extension*)
		bMsg8791 : BOOL; (*reserve warning message 217*) (*import HMI Extension*)
		bMsg8792 : BOOL; (*reserve warning message 218*) (*import HMI Extension*)
		bMsg8793 : BOOL; (*reserve warning message 219*) (*import HMI Extension*)
		bMsg8794 : BOOL; (*reserve warning message 220*) (*import HMI Extension*)
		bMsg8795 : BOOL; (*reserve warning message 221*) (*import HMI Extension*)
		bMsg8796 : BOOL; (*reserve warning message 222*) (*import HMI Extension*)
		bMsg8797 : BOOL; (*reserve warning message 223*) (*import HMI Extension*)
		bMsg8798 : BOOL; (*reserve warning message 224*) (*import HMI Extension*)
		bMsg8799 : BOOL; (*reserve warning message 225*) (*import HMI Extension*)
		bMsg8800 : BOOL; (*DO NOT USE ANYMORE! - reserve warning message 226*) (*import HMI Extension*)
		bMsg6901 : BOOL; (* = 	Alarmbit to visu			*)
		bMsg6902 : BOOL; (* = 	Alarmbit to visu			*)
		bMsg6903 : BOOL; (* = 	Alarmbit to visu			*)
		bMsg6904 : BOOL; (* = 	Alarmbit to visu			*)
		bMsg6905 : BOOL; (* = 	Alarmbit to visu			*)
		bMsg6906 : BOOL; (* = 	Alarmbit to visu			*)
		bMsg6907 : BOOL; (* = 	Alarmbit to visu			*)
		bMsg6908 : BOOL; (* = 	Alarmbit to visu			*)
		bMsg6909 : BOOL; (* = 	Alarmbit to visu			*)
		bMsg6910 : BOOL; (* = 	Alarmbit to visu			*)
		bMsg6911 : BOOL; (* = 	Alarmbit to visu			*)
		bMsg6912 : BOOL; (* = 	Alarmbit to visu			*)
		bMsg6913 : BOOL; (* = 	Alarmbit to visu			*)
		bMsg6914 : BOOL; (* = 	Alarmbit to visu			*)
		bMsg6915 : BOOL; (* = 	Alarmbit to visu			*)
		bMsg6916 : BOOL; (* = 	Alarmbit to visu			*)
		bMsg6917 : BOOL; (* = 	Alarmbit to visu			*)
		bMsg6918 : BOOL; (* = 	Alarmbit to visu			*)
		bMsg6919 : BOOL; (* = 	Alarmbit to visu			*)
		bMsg6920 : BOOL; (* = 	Alarmbit to visu			*)
		bMsg6921 : BOOL; (* = 	Alarmbit to visu			*)
		bMsg6922 : BOOL; (* = 	Alarmbit to visu			*)
		bMsg6923 : BOOL; (* = 	Alarmbit to visu			*)
		bMsg6924 : BOOL; (* = 	Alarmbit to visu			*)
		bMsg6925 : BOOL; (* = 	Alarmbit to visu			*)
		bMsg6926 : BOOL; (* = 	Alarmbit to visu			*)
		bMsg6927 : BOOL; (* = 	Alarmbit to visu			*)
		bMsg6928 : BOOL; (* = 	Alarmbit to visu			*)
		bMsg6929 : BOOL; (* = 	Alarmbit to visu			*)
		bMsg6930 : BOOL; (* = 	Alarmbit to visu			*)
		bMsg6931 : BOOL; (* = 	Alarmbit to visu			*)
		bMsg6932 : BOOL; (* = 	Alarmbit to visu			*)
		bMsg6933 : BOOL; (* = 	Alarmbit to visu			*)
		bMsg6934 : BOOL; (* = 	Alarmbit to visu			*)
		bMsg6935 : BOOL; (* = 	Alarmbit to visu			*)
		bMsg6936 : BOOL; (* = 	Alarmbit to visu			*)
		bMsg6937 : BOOL; (* = 	Alarmbit to visu			*)
		bMsg6938 : BOOL; (* = 	Alarmbit to visu			*)
		bMsg6939 : BOOL; (* = 	Alarmbit to visu			*)
		bMsg6940 : BOOL; (* = 	Alarmbit to visu			*)
		bMsg6941 : BOOL; (* = 	Alarmbit to visu			*)
		bMsg6942 : BOOL; (* = 	Alarmbit to visu			*)
		bMsg6943 : BOOL; (* = 	Alarmbit to visu			*)
		bMsg6944 : BOOL; (* = 	Alarmbit to visu			*)
		bMsg6945 : BOOL; (* = 	Alarmbit to visu			*)
		bMsg6946 : BOOL; (* = 	Alarmbit to visu			*)
		bMsg6947 : BOOL; (* = 	Alarmbit to visu			*)
		bMsg6948 : BOOL; (* = 	Alarmbit to visu			*)
		bMsg6949 : BOOL; (* = 	Alarmbit to visu			*)
		bMsg6950 : BOOL; (* = 	Alarmbit to visu			*)
		bMsg6951 : BOOL; (* = 	Alarmbit to visu			*)
		bMsg6952 : BOOL; (* = 	Alarmbit to visu			*)
		bMsg6953 : BOOL; (* = 	Alarmbit to visu			*)
		bMsg6954 : BOOL; (* = 	Alarmbit to visu			*)
		bMsg6955 : BOOL; (* = 	Alarmbit to visu			*)
		bMsg6956 : BOOL; (* = 	Alarmbit to visu			*)
		bMsg6957 : BOOL; (* = 	Alarmbit to visu			*)
		bMsg6958 : BOOL; (* = 	Alarmbit to visu			*)
		bMsg6959 : BOOL; (* = 	Alarmbit to visu			*)
		bMsg6960 : BOOL; (* = 	Alarmbit to visu			*)
		bMsg6961 : BOOL; (* = 	Alarmbit to visu			*)
		bMsg6962 : BOOL; (* = 	Alarmbit to visu			*)
		bMsg6963 : BOOL; (* = 	Alarmbit to visu			*)
		bMsg6964 : BOOL; (* = 	Alarmbit to visu			*)
		bMsg6965 : BOOL; (* = 	Alarmbit to visu			*)
		bMsg6966 : BOOL; (* = 	Alarmbit to visu			*)
		bMsg6967 : BOOL; (* = 	Alarmbit to visu			*)
		bMsg6968 : BOOL; (* = 	Alarmbit to visu			*)
		bMsg6969 : BOOL; (* = 	Alarmbit to visu			*)
		bMsg6970 : BOOL; (* = 	Alarmbit to visu			*)
		bMsg6971 : BOOL; (* = 	Alarmbit to visu			*)
		bMsg6972 : BOOL; (* = 	Alarmbit to visu			*)
		bMsg6973 : BOOL; (* = 	Alarmbit to visu			*)
		bMsg6974 : BOOL; (* = 	Alarmbit to visu			*)
		bMsg6975 : BOOL; (* = 	Alarmbit to visu			*)
		bMsg6976 : BOOL; (* = 	Alarmbit to visu			*)
		bMsg6977 : BOOL; (* = 	Alarmbit to visu			*)
		bMsg6978 : BOOL; (* = 	Alarmbit to visu			*)
		bMsg6979 : BOOL; (* = 	Alarmbit to visu			*)
		bMsg6980 : BOOL; (* = 	Alarmbit to visu			*)
		bMsg6981 : BOOL; (* = 	Alarmbit to visu			*)
		bMsg6982 : BOOL; (* = 	Alarmbit to visu			*)
		bMsg6983 : BOOL; (* = 	Alarmbit to visu			*)
		bMsg6984 : BOOL; (* = 	Alarmbit to visu			*)
		bMsg6985 : BOOL; (* = 	Alarmbit to visu			*)
		bMsg6986 : BOOL; (* = 	Alarmbit to visu			*)
		bMsg6987 : BOOL; (* = 	Alarmbit to visu			*)
		bMsg6988 : BOOL; (* = 	Alarmbit to visu			*)
		bMsg6989 : BOOL; (* = 	Alarmbit to visu			*)
		bMsg6990 : BOOL; (* = 	Alarmbit to visu			*)
		bMsg6991 : BOOL; (* = 	Alarmbit to visu			*)
		bMsg6992 : BOOL; (* = 	Alarmbit to visu			*)
		bMsg6993 : BOOL; (* = 	Alarmbit to visu			*)
		bMsg6994 : BOOL; (* = 	Alarmbit to visu			*)
		bMsg6995 : BOOL; (* = 	Alarmbit to visu			*)
		bMsg6996 : BOOL; (* = 	Alarmbit to visu			*)
		bMsg6997 : BOOL; (* = 	Alarmbit to visu			*)
		bMsg6998 : BOOL; (* = 	Alarmbit to visu			*)
		bMsg6999 : BOOL; (* = 	Alarmbit to visu			*)
		bMsg7901 : BOOL; (* = 	Alarmbit to visu			*)
		bMsg7902 : BOOL; (* = 	Alarmbit to visu			*)
		bMsg7903 : BOOL; (* = 	Alarmbit to visu			*)
		bMsg7904 : BOOL; (* = 	Alarmbit to visu			*)
		bMsg7905 : BOOL; (* = 	Alarmbit to visu			*)
		bMsg7906 : BOOL; (* = 	Alarmbit to visu			*)
		bMsg7907 : BOOL; (* = 	Alarmbit to visu			*)
		bMsg7908 : BOOL; (* = 	Alarmbit to visu			*)
		bMsg7909 : BOOL; (* = 	Alarmbit to visu			*)
		bMsg7910 : BOOL; (* = 	Alarmbit to visu			*)
		bMsg7911 : BOOL; (* = 	Alarmbit to visu			*)
		bMsg7912 : BOOL; (* = 	Alarmbit to visu			*)
		bMsg7913 : BOOL; (* = 	Alarmbit to visu			*)
		bMsg7914 : BOOL; (* = 	Alarmbit to visu			*)
		bMsg7915 : BOOL; (* = 	Alarmbit to visu			*)
		bMsg7916 : BOOL; (* = 	Alarmbit to visu			*)
		bMsg7917 : BOOL; (* = 	Alarmbit to visu			*)
		bMsg7918 : BOOL; (* = 	Alarmbit to visu			*)
		bMsg7919 : BOOL; (* = 	Alarmbit to visu			*)
		bMsg7920 : BOOL; (* = 	Alarmbit to visu			*)
		bMsg7921 : BOOL; (* = 	Alarmbit to visu			*)
		bMsg7922 : BOOL; (* = 	Alarmbit to visu			*)
		bMsg7923 : BOOL; (* = 	Alarmbit to visu			*)
		bMsg7924 : BOOL; (* = 	Alarmbit to visu			*)
		bMsg7925 : BOOL; (* = 	Alarmbit to visu			*)
		bMsg7926 : BOOL; (* = 	Alarmbit to visu			*)
		bMsg7927 : BOOL; (* = 	Alarmbit to visu			*)
		bMsg7928 : BOOL; (* = 	Alarmbit to visu			*)
		bMsg7929 : BOOL; (* = 	Alarmbit to visu			*)
		bMsg7930 : BOOL; (* = 	Alarmbit to visu			*)
		bMsg7931 : BOOL; (* = 	Alarmbit to visu			*)
		bMsg7932 : BOOL; (* = 	Alarmbit to visu			*)
		bMsg7933 : BOOL; (* = 	Alarmbit to visu			*)
		bMsg7934 : BOOL; (* = 	Alarmbit to visu			*)
		bMsg7935 : BOOL; (* = 	Alarmbit to visu			*)
		bMsg7936 : BOOL; (* = 	Alarmbit to visu			*)
		bMsg7937 : BOOL; (* = 	Alarmbit to visu			*)
		bMsg7938 : BOOL; (* = 	Alarmbit to visu			*)
		bMsg7939 : BOOL; (* = 	Alarmbit to visu			*)
		bMsg7940 : BOOL; (* = 	Alarmbit to visu			*)
		bMsg7941 : BOOL; (* = 	Alarmbit to visu			*)
		bMsg7942 : BOOL; (* = 	Alarmbit to visu			*)
		bMsg7943 : BOOL; (* = 	Alarmbit to visu			*)
		bMsg7944 : BOOL; (* = 	Alarmbit to visu			*)
		bMsg7945 : BOOL; (* = 	Alarmbit to visu			*)
		bMsg7946 : BOOL; (* = 	Alarmbit to visu			*)
		bMsg7947 : BOOL; (* = 	Alarmbit to visu			*)
		bMsg7948 : BOOL; (* = 	Alarmbit to visu			*)
		bMsg7949 : BOOL; (* = 	Alarmbit to visu			*)
		bMsg7950 : BOOL; (* = 	Alarmbit to visu			*)
		bMsg7951 : BOOL; (* = 	Alarmbit to visu			*)
		bMsg7952 : BOOL; (* = 	Alarmbit to visu			*)
		bMsg7953 : BOOL; (* = 	Alarmbit to visu			*)
		bMsg7954 : BOOL; (* = 	Alarmbit to visu			*)
		bMsg7955 : BOOL; (* = 	Alarmbit to visu			*)
		bMsg7956 : BOOL; (* = 	Alarmbit to visu			*)
		bMsg7957 : BOOL; (* = 	Alarmbit to visu			*)
		bMsg7958 : BOOL; (* = 	Alarmbit to visu			*)
		bMsg7959 : BOOL; (* = 	Alarmbit to visu			*)
		bMsg7960 : BOOL; (* = 	Alarmbit to visu			*)
		bMsg7961 : BOOL; (* = 	Alarmbit to visu			*)
		bMsg7962 : BOOL; (* = 	Alarmbit to visu			*)
		bMsg7963 : BOOL; (* = 	Alarmbit to visu			*)
		bMsg7964 : BOOL; (* = 	Alarmbit to visu			*)
		bMsg7965 : BOOL; (* = 	Alarmbit to visu			*)
		bMsg7966 : BOOL; (* = 	Alarmbit to visu			*)
		bMsg7967 : BOOL; (* = 	Alarmbit to visu			*)
		bMsg7968 : BOOL; (* = 	Alarmbit to visu			*)
		bMsg7969 : BOOL; (* = 	Alarmbit to visu			*)
		bMsg7970 : BOOL; (* = 	Alarmbit to visu			*)
		bMsg7971 : BOOL; (* = 	Alarmbit to visu			*)
		bMsg7972 : BOOL; (* = 	Alarmbit to visu			*)
		bMsg7973 : BOOL; (* = 	Alarmbit to visu			*)
		bMsg7974 : BOOL; (* = 	Alarmbit to visu			*)
		bMsg7975 : BOOL; (* = 	Alarmbit to visu			*)
		bMsg7976 : BOOL; (* = 	Alarmbit to visu			*)
		bMsg7977 : BOOL; (* = 	Alarmbit to visu			*)
		bMsg7978 : BOOL; (* = 	Alarmbit to visu			*)
		bMsg7979 : BOOL; (* = 	Alarmbit to visu			*)
		bMsg7980 : BOOL; (* = 	Alarmbit to visu			*)
		bMsg7981 : BOOL; (* = 	Alarmbit to visu			*)
		bMsg7982 : BOOL; (* = 	Alarmbit to visu			*)
		bMsg7983 : BOOL; (* = 	Alarmbit to visu			*)
		bMsg7984 : BOOL; (* = 	Alarmbit to visu			*)
		bMsg7985 : BOOL; (* = 	Alarmbit to visu			*)
		bMsg7986 : BOOL; (* = 	Alarmbit to visu			*)
		bMsg7987 : BOOL; (* = 	Alarmbit to visu			*)
		bMsg7988 : BOOL; (* = 	Alarmbit to visu			*)
		bMsg7989 : BOOL; (* = 	Alarmbit to visu			*)
		bMsg7990 : BOOL; (* = 	Alarmbit to visu			*)
		bMsg7991 : BOOL; (* = 	Alarmbit to visu			*)
		bMsg7992 : BOOL; (* = 	Alarmbit to visu			*)
		bMsg7993 : BOOL; (* = 	Alarmbit to visu			*)
		bMsg7994 : BOOL; (* = 	Alarmbit to visu			*)
		bMsg7995 : BOOL; (* = 	Alarmbit to visu			*)
		bMsg7996 : BOOL; (* = 	Alarmbit to visu			*)
		bMsg7997 : BOOL; (* = 	Alarmbit to visu			*)
		bMsg7998 : BOOL; (* = 	Alarmbit to visu			*)
		bMsg7999 : BOOL; (* = 	Alarmbit to visu			*)
		bMsg8900 : BOOL; (* = 	Alarmbit to visu			*)
		bMsg8901 : BOOL; (* = 	Alarmbit to visu			*)
		bMsg8902 : BOOL; (* = 	Alarmbit to visu			*)
		bMsg8903 : BOOL; (* = 	Alarmbit to visu			*)
		bMsg8904 : BOOL; (* = 	Alarmbit to visu			*)
		bMsg8905 : BOOL; (* = 	Alarmbit to visu			*)
		bMsg8906 : BOOL; (* = 	Alarmbit to visu			*)
		bMsg8907 : BOOL; (* = 	Alarmbit to visu			*)
		bMsg8908 : BOOL; (* = 	Alarmbit to visu			*)
		bMsg8909 : BOOL; (* = 	Alarmbit to visu			*)
		bMsg8910 : BOOL; (* = 	Alarmbit to visu			*)
		bMsg8911 : BOOL; (* = 	Alarmbit to visu			*)
		bMsg8912 : BOOL; (* = 	Alarmbit to visu			*)
		bMsg8913 : BOOL; (* = 	Alarmbit to visu			*)
		bMsg8914 : BOOL; (* = 	Alarmbit to visu			*)
		bMsg8915 : BOOL; (* = 	Alarmbit to visu			*)
		bMsg8916 : BOOL; (* = 	Alarmbit to visu			*)
		bMsg8917 : BOOL; (* = 	Alarmbit to visu			*)
		bMsg8918 : BOOL; (* = 	Alarmbit to visu			*)
		bMsg8919 : BOOL; (* = 	Alarmbit to visu			*)
		bMsg8920 : BOOL; (* = 	Alarmbit to visu			*)
		bMsg8921 : BOOL; (* = 	Alarmbit to visu			*)
		bMsg8922 : BOOL; (* = 	Alarmbit to visu			*)
		bMsg8923 : BOOL; (* = 	Alarmbit to visu			*)
		bMsg8924 : BOOL; (* = 	Alarmbit to visu			*)
		bMsg8925 : BOOL; (* = 	Alarmbit to visu			*)
		bMsg8926 : BOOL; (* = 	Alarmbit to visu			*)
		bMsg8927 : BOOL; (* = 	Alarmbit to visu			*)
		bMsg8928 : BOOL; (* = 	Alarmbit to visu			*)
		bMsg8929 : BOOL; (* = 	Alarmbit to visu			*)
		bMsg8930 : BOOL; (* = 	Alarmbit to visu			*)
		bMsg8931 : BOOL; (* = 	Alarmbit to visu			*)
		bMsg8932 : BOOL; (* = 	Alarmbit to visu			*)
		bMsg8933 : BOOL; (* = 	Alarmbit to visu			*)
		bMsg8934 : BOOL; (* = 	Alarmbit to visu			*)
		bMsg8935 : BOOL; (* = 	Alarmbit to visu			*)
		bMsg8936 : BOOL; (* = 	Alarmbit to visu			*)
		bMsg8937 : BOOL; (* = 	Alarmbit to visu			*)
		bMsg8938 : BOOL; (* = 	Alarmbit to visu			*)
		bMsg8939 : BOOL; (* = 	Alarmbit to visu			*)
		bMsg8940 : BOOL; (* = 	Alarmbit to visu			*)
		bMsg8941 : BOOL; (* = 	Alarmbit to visu			*)
		bMsg8942 : BOOL; (* = 	Alarmbit to visu			*)
		bMsg8943 : BOOL; (* = 	Alarmbit to visu			*)
		bMsg8944 : BOOL; (* = 	Alarmbit to visu			*)
		bMsg8945 : BOOL; (* = 	Alarmbit to visu			*)
		bMsg8946 : BOOL; (* = 	Alarmbit to visu			*)
		bMsg8947 : BOOL; (* = 	Alarmbit to visu			*)
		bMsg8948 : BOOL; (* = 	Alarmbit to visu			*)
		bMsg8949 : BOOL; (* = 	Alarmbit to visu			*)
		bMsg8950 : BOOL; (* = 	Alarmbit to visu			*)
		bMsg8951 : BOOL; (* = 	Alarmbit to visu			*)
		bMsg8952 : BOOL; (* = 	Alarmbit to visu			*)
		bMsg8953 : BOOL; (* = 	Alarmbit to visu			*)
		bMsg8954 : BOOL; (* = 	Alarmbit to visu			*)
		bMsg8955 : BOOL; (* = 	Alarmbit to visu			*)
		bMsg8956 : BOOL; (* = 	Alarmbit to visu			*)
		bMsg8957 : BOOL; (* = 	Alarmbit to visu			*)
		bMsg8958 : BOOL; (* = 	Alarmbit to visu			*)
		bMsg8959 : BOOL; (* = 	Alarmbit to visu			*)
		bMsg8960 : BOOL; (* = 	Alarmbit to visu			*)
		bMsg8961 : BOOL; (* = 	Alarmbit to visu			*)
		bMsg8962 : BOOL; (* = 	Alarmbit to visu			*)
		bMsg8963 : BOOL; (* = 	Alarmbit to visu			*)
		bMsg8964 : BOOL; (* = 	Alarmbit to visu			*)
		bMsg8965 : BOOL; (* = 	Alarmbit to visu			*)
		bMsg8966 : BOOL; (* = 	Alarmbit to visu			*)
		bMsg8967 : BOOL; (* = 	Alarmbit to visu			*)
		bMsg8968 : BOOL; (* = 	Alarmbit to visu			*)
		bMsg8969 : BOOL; (* = 	Alarmbit to visu			*)
		bMsg8970 : BOOL; (* = 	Alarmbit to visu			*)
		bMsg8971 : BOOL; (* = 	Alarmbit to visu			*)
		bMsg8972 : BOOL; (* = 	Alarmbit to visu			*)
		bMsg8973 : BOOL; (* = 	Alarmbit to visu			*)
		bMsg8974 : BOOL; (* = 	Alarmbit to visu			*)
		bMsg8975 : BOOL; (* = 	Alarmbit to visu			*)
		bMsg8976 : BOOL; (* = 	Alarmbit to visu			*)
		bMsg8977 : BOOL; (* = 	Alarmbit to visu			*)
		bMsg8978 : BOOL; (* = 	Alarmbit to visu			*)
		bMsg8979 : BOOL; (* = 	Alarmbit to visu			*)
		bMsg8980 : BOOL; (* = 	Alarmbit to visu			*)
		bMsg8981 : BOOL; (* = 	Alarmbit to visu			*)
		bMsg8982 : BOOL; (* = 	Alarmbit to visu			*)
		bMsg8983 : BOOL; (* = 	Alarmbit to visu			*)
		bMsg8984 : BOOL; (* = 	Alarmbit to visu			*)
		bMsg8985 : BOOL; (* = 	Alarmbit to visu			*)
		bMsg8986 : BOOL; (* = 	Alarmbit to visu			*)
		bMsg8987 : BOOL; (* = 	Alarmbit to visu			*)
		bMsg8988 : BOOL; (* = 	Alarmbit to visu			*)
		bMsg8989 : BOOL; (* = 	Alarmbit to visu			*)
		bMsg8990 : BOOL; (* = 	Alarmbit to visu			*)
		bMsg8991 : BOOL; (* = 	Alarmbit to visu			*)
		bMsg8992 : BOOL; (* = 	Alarmbit to visu			*)
		bMsg8993 : BOOL; (* = 	Alarmbit to visu			*)
		bMsg8994 : BOOL; (* = 	Alarmbit to visu			*)
		bMsg8995 : BOOL; (* = 	Alarmbit to visu			*)
		bMsg8996 : BOOL; (* = 	Alarmbit to visu			*)
		bMsg8997 : BOOL; (* = 	Alarmbit to visu			*)
		bMsg8998 : BOOL; (* = 	Alarmbit to visu			*)
		bMsg8999 : BOOL; (* = 	Alarmbit to visu			*)
		bParaSetupOk : BOOL; (* = 	parameter setup ok - release RPS operation (bAllModulesOk)			*)
		bUniDig : ARRAY[0..125]OF BOOL; (* = 	ARRAY of processed digita channel  values from UniversalIO system			*)
		iCount1 : DINT; (* = 	Customized Counter			*)
		iCount2 : DINT; (* = 	Customized Counter			*)
		iCount3 : DINT; (* = 	Customized Counter			*)
		iCount4 : DINT; (* = 	Customized Counter			*)
		iCount5 : DINT; (* = 	Customized Counter			*)
		iCount6 : DINT; (* = 	Customized Counter			*)
		iCount7 : DINT; (* = 	Customized Counter			*)
		iCount8 : DINT; (* = 	Customized Counter			*)
		iCount9 : DINT; (* = 	Customized Counter			*)
		iCount10 : DINT; (* = 	Customized Counter			*)
		iCount11 : DINT; (* = 	Customized Counter			*)
		iCount12 : DINT; (* = 	Customized Counter			*)
		iCount13 : DINT; (* = 	Customized Counter			*)
		iCount14 : DINT; (* = 	Customized Counter			*)
		iCount15 : DINT; (* = 	Customized Counter			*)
		iCount16 : DINT; (* = 	Customized Counter			*)
		iCount17 : DINT; (* = 	Customized Counter			*)
		iCount18 : DINT; (* = 	Customized Counter			*)
		iCount19 : DINT; (* = 	Customized Counter			*)
		iCount20 : DINT; (* = 	Customized Counter			*)
		iHeatCount : DINT; (*counter heating power engine heat water circuit*)
		iIdx_ProcessStep : DINT; (*Display step information on VIS*)
		iMaintenanceCount1 : DINT; (* = 	Maintenance Counter			*)
		iMaintenanceCount2 : DINT; (* = 	Maintenance Counter			*)
		iMaintenanceCount3 : DINT; (* = 	Maintenance Counter			*)
		iMaintenanceCount4 : DINT; (* = 	Maintenance Counter			*)
		iMaintenanceCount5 : DINT; (* = 	Maintenance Counter			*)
		iMaintenanceCount6 : DINT; (* = 	Maintenance Counter			*)
		iMaintenanceCount7 : DINT; (* = 	Maintenance Counter			*)
		iMaintenanceCount8 : DINT; (* = 	Maintenance Counter			*)
		iProcessStepTime : DINT; (*Display step time  info on VIS*)
		iRPS_Day : DINT; (* = 	Time			*)
		iRPS_h : DINT; (* = 	Time			*)
		iRPS_m : DINT; (* = 	Time			*)
		iRPS_Month : DINT; (* = 	Time			*)
		iRPS_s : DINT; (* = 	Time			*)
		i_FC_Test_var : INT; (*Testvariante	[0=kein Test / 1=AUTO Hoecker ueber FrequenzSollwert / 2=MAN ueber FrequenzSollwert / 3=AUTO Hoecker ueber FrequenzIstwert / 4=MAN ueber FrequenzIstwert]*)
		rCustAnaIn : ARRAY[0..120]OF REAL; (*Prepared spare analog input = measured and scaled signal from hardcoded reserve channel			*)
		rCustAnaOut : ARRAY[0..iNoOf_AnaOut]OF REAL; (*Prepared spare analog output for VIS service display    REAL[0..60]		 (OLD:   rCustAnaOut_Norm )*)
		rCustOPC : ARRAY[0..32]OF REAL; (*Prepared spare analog values to customer OPC		*) (*OldName: newPV; Cycle: 5;*)
		rCustVis : ARRAY[0..50]OF REAL; (*Prepared spare analog input to VISU		*) (*OldName: newPV; Cycle: 5;*)
		rCustScalingBlock_X : ARRAY[0..30]OF REAL; (*Scaling Block X Value - import HMI Extension*)
		rCustScalingBlock_Y : ARRAY[0..30]OF REAL; (*Scaling Block Y Value - import HMI Extension*)
		rF_FC_Deadband_neg : REAL; (*negative deathband for frequency control [Hz]*)
		rF_FC_Deadband_pos : REAL; (*positive deathband for frequency control [Hz]*)
		rF_FC_Delta : REAL; (*frequency deviation for frequency control*)
		rF_FC_Dlt_neg : REAL; (*negative range of frequency control [Hz]*)
		rF_FC_Dlt_pos : REAL; (*positive range of frequency control [Hz]*)
		rF_MMD_FC : REAL; (*actual frequency for frequency control [Hz]*)
		rF_Ref : REAL; (*nominal frequency [Hz] *)
		rPcsm_act : REAL; (*mains import power controller*) (*OldName: rP_Consumption; Cycle: 5;*)
		rPmns_act : REAL; (*mains import power controller*) (*OldName: rP_MainsImport; Cycle: 5;*)
		rPmns_DemGenerate : REAL; (*new V4.5 beta*)
		rPmns_DemGenerate_Lim_Off : REAL; (*new V4.5 beta*)
		rPmns_DemGenerate_Lim_On : REAL; (*new V4.5 beta*)
		rPmns_setpoint : REAL; (*mains import power controller*) (*OldName: newPV; Cycle: 5;*)
		rP_Act_Filt : REAL; (*actual power [kW]*)
		rP_DemGenerate : REAL; (*= New Generator Setpoint from mains import controller*)
		rP_FC_ContOutput : REAL; (*controller output FC [kW]*)
		rP_RMC_FC_neg : REAL; (*negative reserve power for frequency control [kW]*)
		rP_RMC_FC_pos : REAL; (*positive reserve power for frequency control [kW]*)
		rP_Set_FC : REAL; (*power setpoint [kW]*)
		rTime_Dem_On_CntDn : REAL; (*mains import power controller*) (*OldName: newPV; Cycle: 5;*)
		rUniAna : ARRAY[0..151]OF REAL; (* = 	ARRAY of scaled value from UniversalIO system			*)
		tBaseProg_Vers : Revision_type; (*Vis display of software origin (base) version; UNCHANGED, not affected by SW updates*) (* OldName:newPV	; Cycle: 5;*)
		tCtr_Cust1_Out : _tGeACtrOut; (* = 	New customizable controllers without predefined purpose			*)
		tCtr_Cust2_Out : _tGeACtrOut; (* = 	New customizable controllers without predefined purpose			*)
		tCtr_Cust3_Out : _tGeACtrOut; (* = 	New customizable controllers without predefined purpose			*)
		tCtr_Cust4_Out : _tGeACtrOut; (* = 	New customizable controllers without predefined purpose			*)
		tCtr_Cust5_Out : _tGeACtrOut; (* = 	New customizable controllers without predefined purpose			*)
		tCtr_Cust6_Out : _tGeACtrOut; (* = 	New customizable controllers without predefined purpose			*)
		tCtr_Cust7_Out : _tGeACtrOut; (* = 	New customizable controllers without predefined purpose			*)
		tCtr_Cust8_Out : _tGeACtrOut; (* = 	New customizable controllers without predefined purpose			*)
		tCtr_Cust41_Out : _tGeACtrOut; (* = 	New customizable controllers without predefined purpose			*)
		tCtr_Cust42_Out : _tGeACtrOut; (* = 	New customizable controllers without predefined purpose			*)
		tCtr_Cust43_Out : _tGeACtrOut; (* = 	New customizable controllers without predefined purpose			*)
		tCtr_Cust44_Out : _tGeACtrOut; (* = 	New customizable controllers without predefined purpose			*)
		tCtr_Cust45_Out : _tGeACtrOut; (* = 	New customizable controllers without predefined purpose			*)
		tCtr_Mns_Out : _tGeACtrOut; (* = 	New mains power controller *)
		tRPM_Count1 : _rpm_count; (*conditional daily runtime counter *)
		tRPM_Count2 : _rpm_count; (*conditional daily runtime counter *)
		tRPM_Count3 : _rpm_count; (*conditional daily runtime counter *)
		tRPM_Count4 : _rpm_count; (*conditional daily runtime counter *)
		tRPM_Count5 : _rpm_count; (*conditional daily runtime counter *)
		tRPM_Count6 : _rpm_count; (*conditional daily runtime counter *)
		tRPM_Count7 : _rpm_count; (*conditional daily runtime counter *)
		tRPM_Count8 : _rpm_count; (*conditional daily runtime counter *)
		tRPM_Count9 : _rpm_count; (*conditional daily runtime counter *)
		tRPM_Count10 : _rpm_count; (*conditional daily runtime counter *)
		tRPM_Count11 : _rpm_count; (*conditional daily runtime counter *)
		tRPM_Count12 : _rpm_count; (*conditional daily runtime counter *)
		tRPM_Count13 : _rpm_count; (*conditional daily runtime counter *)
		tRPM_Count14 : _rpm_count; (*conditional daily runtime counter *)
		tRPM_Count15 : _rpm_count; (*conditional daily runtime counter *)
		tRPM_Count16 : _rpm_count; (*conditional daily runtime counter *)
		rCust_AG : ARRAY[0..99]OF REAL; (*New customizable interface 2017 - BETA PHASE, use only in coordination with TPSS*)
		rCust_CH : ARRAY[0..99]OF REAL; (*New customizable interface 2017 - BETA PHASE, use only in coordination with TPSS*)
		rCust_CP : ARRAY[0..99]OF REAL; (*New customizable interface 2017 - BETA PHASE, use only in coordination with TPSS*)
		rCust_EC : ARRAY[0..99]OF REAL; (*prepared- not active! customizable interface 2017 - BETA PHASE, use only in coordination with TPSS*)
		rCust_HA : ARRAY[0..300]OF REAL; (*New customizable HAL interface 2017 - BETA PHASE, use only in coordination with TPSS*)
		rCust_OP : ARRAY[0..99]OF REAL; (*prepared- not active! customizable interface 2017 - BETA PHASE, use only in coordination with TPSS*)
		bMsg9285 : BOOL; (* Measuring signal failure external voltage setpoint *)
		bMsg9286 : BOOL; (* Measuring signal failure external speed setpoint *)
		bMsg9287 : BOOL; (* W9287 Failure external speed / voltage controller *)
		iSource_F_N_OffsSet : INT; (* F/N Setpoint: 0= no setpoint, 1= Droop, 2= External, 3= LSL *)
	END_STRUCT;
	Vis2MM_Struct : 	STRUCT
		bCustOPC : ARRAY[0..32]OF BOOL; (*Prepared spare digital values from customer OPC*) (*OldName: OPC_BIN1,OPC_BIN2,OPC_BIN3,OPC_BIN4,OPC_BIN5,OPC_BIN6; Cycle: 5;*)
		bCustVis : ARRAY[0..50]OF BOOL; (*Prepared spare digital input from VISU		*) (*OldName: newPV; Cycle: 5;*)
		bTime_Dem_On_delay_Reset : BOOL; (*mains power controller*) (*OldName: NewPV; Cycle: 5;*)
		iCount1 : DINT; (* Input field to Customized Counter*) (*OldName: ZAEHL_1; Cycle: 5;*)
		iCount2 : DINT; (* Input field to  Customized Counter*) (*OldName: ZAEHL_2; Cycle: 5;*)
		iCount3 : DINT; (* Input field to  Customized Counter*) (*OldName: ZAEHL_3; Cycle: 5;*)
		iCount4 : DINT; (* Input field to  Customized Counter*) (*OldName: ZAEHL_4; Cycle: 5;*)
		iCount5 : DINT; (* Input field to  Customized Counter new*) (*OldName: new PV; Cycle: 5;*)
		iCount6 : DINT; (* Input field to  Customized Counter new*) (*OldName: new PV; Cycle: 5;*)
		iCount7 : DINT; (* Input field to  Customized Counter new*) (*OldName: new PV; Cycle: 5;*)
		iCount8 : DINT; (* Input field to  Customized Counter new*) (*OldName: new PV; Cycle: 5;*)
		iCount9 : DINT; (* Input field to  Customized Counter new*) (*OldName: new PV; Cycle: 5;*)
		iCount10 : DINT; (* Input field to  Customized Counter new*) (*OldName: new PV; Cycle: 5;*)
		iCount11 : DINT; (* Input field to  Customized Counter new*) (*OldName: new PV; Cycle: 5;*)
		iCount12 : DINT; (* Input field to  Customized Counter new*) (*OldName: new PV; Cycle: 5;*)
		iCount13 : DINT; (* Input field to  Customized Counter new*) (*OldName: new PV; Cycle: 5;*)
		iCount14 : DINT; (* Input field to  Customized Counter new*) (*OldName: new PV; Cycle: 5;*)
		iCount15 : DINT; (* Input field to  Customized Counter new*) (*OldName: new PV; Cycle: 5;*)
		iCount16 : DINT; (* Input field to  Customized Counter new*) (*OldName: new PV; Cycle: 5;*)
		iCount17 : DINT; (* Input field to  Customized Counter new*) (*OldName: new PV; Cycle: 5;*)
		iCount18 : DINT; (* Input field to  Customized Counter new*) (*OldName: new PV; Cycle: 5;*)
		iCount19 : DINT; (* Input field to  Customized Counter new*) (*OldName: new PV; Cycle: 5;*)
		iCount20 : DINT; (* Input field to  Customized Counter new*) (*OldName: new PV; Cycle: 5;*)
		iMaintenanceCount1 : DINT; (* Input field to Maintenance Counter*) (*OldName: wart_z1; Cycle: 5;*)
		iMaintenanceCount2 : DINT; (* Input field to Maintenance Counter*) (*OldName: wart_z2; Cycle: 5;*)
		iMaintenanceCount3 : DINT; (* Input field to Maintenance Counter*) (*OldName: wart_z3; Cycle: 5;*)
		iMaintenanceCount4 : DINT; (* Input field to Maintenance Counter*) (*OldName: wart_z4; Cycle: 5;*)
		iMaintenanceCount5 : DINT; (* Input field to Maintenance Counter*) (*OldName: new PV; Cycle: 5;*)
		iMaintenanceCount6 : DINT; (* Input field to Maintenance Counter*) (*OldName: new PV; Cycle: 5;*)
		iMaintenanceCount7 : DINT; (* Input field to Maintenance Counter*) (*OldName: new PV; Cycle: 5;*)
		iMaintenanceCount8 : DINT; (* Input field to Maintenance Counter*) (*OldName: new PV; Cycle: 5;*)
		rCustOPC : ARRAY[0..32]OF REAL; (*Prepared spare analog values from customer OPC*) (*OldName: OPC_ANA1 - OPC_ANA16; Cycle: 5;*)
		rCustVis : ARRAY[0..50]OF REAL; (*Prepared spare analog input from VISU		*) (*OldName: newPV; Cycle: 5;*)
		tCtr_Cust1_In : _tGeACtrIn; (* = 	New customizable controllers without predefined purpose	*) (*OldName: REG1.x, REG1.w_ext, usw; Cycle: 5;*)
		tCtr_Cust2_In : _tGeACtrIn; (* = 	New customizable controllers without predefined purpose	*) (*OldName: REG2.x, REG2.w_ext, usw; Cycle: 5;*)
		tCtr_Cust3_In : _tGeACtrIn; (* = 	New customizable controllers without predefined purpose	*) (*OldName: REG3.x, REG3.w_ext, usw; Cycle: 5;*)
		tCtr_Cust4_In : _tGeACtrIn; (* = 	New customizable controllers without predefined purpose	*) (*OldName: REG4.x, REG4.w_ext, usw; Cycle: 5;*)
		tCtr_Cust5_In : _tGeACtrIn; (* = 	New customizable controllers without predefined purpose	*) (*OldName: REG5.x, REG5.w_ext, usw; Cycle: 5;*)
		tCtr_Cust6_In : _tGeACtrIn; (* = 	New customizable controllers without predefined purpose	*) (*OldName: REG6.x, REG6.w_ext, usw; Cycle: 5;*)
		tCtr_Cust7_In : _tGeACtrIn; (* = 	New customizable controllers without predefined purpose	*) (*OldName: REG7.x, REG7.w_ext, usw; Cycle: 5;*)
		tCtr_Cust8_In : _tGeACtrIn; (* = 	New customizable controllers without predefined purpose	*) (*OldName: REG8.x, REG8.w_ext, usw; Cycle: 5;*)
		tCtr_Cust41_In : _tGeACtrIn; (* = 	New customizable controllers without predefined purpose	*) (*OldName: REG41.x, REG41.w_ext, usw; Cycle: 5;*)
		tCtr_Cust42_In : _tGeACtrIn; (* = 	New customizable controllers without predefined purpose	*) (*OldName: REG42.x, REG42.w_ext, usw; Cycle: 5;*)
		tCtr_Cust43_In : _tGeACtrIn; (* = 	New customizable controllers without predefined purpose	*) (*OldName: REG43.x, REG43.w_ext, usw; Cycle: 5;*)
		tCtr_Cust44_In : _tGeACtrIn; (* = 	New customizable controllers without predefined purpose	*) (*OldName: REG44.x, REG44.w_ext, usw; Cycle: 5;*)
		tCtr_Cust45_In : _tGeACtrIn; (* = 	New customizable controllers without predefined purpose	*) (*OldName: REG45.x, REG45.w_ext, usw; Cycle: 5;*)
		tCtr_Mns_In : _tGeACtrIn; (* = 	New mains power controller*) (*OldName: P_ctrl_from_plant_control_system ; Cycle: 5;*)
		rCust_AG : ARRAY[0..99]OF REAL; (*New customizable interface 2017 - BETA PHASE, use only in coordination with TPSS*)
		rCust_CH : ARRAY[0..99]OF REAL; (*New customizable interface 2017 - BETA PHASE, use only in coordination with TPSS*)
		rCust_CP : ARRAY[0..99]OF REAL; (*New customizable interface 2017 - BETA PHASE, use only in coordination with TPSS*)
		rCust_EC : ARRAY[0..99]OF REAL; (*prepared- not active! customizable interface 2017 - BETA PHASE, use only in coordination with TPSS*)
		rCust_HA : ARRAY[0..300]OF REAL; (*New customizable HAL interface 2017 - BETA PHASE, use only in coordination with TPSS*)
		rCust_OP : ARRAY[0..99]OF REAL; (*Newprepared- not active! customizable interface 2017 - BETA PHASE, use only in coordination with TPSS*)
		rCustomizedSpare : ARRAY[0..99]OF REAL; (*New customizable Spare OUT interface 2017 - BETA PHASE, use only in coordination with TPSS*)
		rFNom_FSM_ManualTest : REAL;
		rFAct_FSM_ManualTest : REAL;
		iSet_FSM_Testmode : INT; (* Frequency Control Testmode [1= AUTO Hoecker ueber Frequenzsollwert, 2 = MAN ueber FrequenzSollwert, 3 = AUTO Hoecker ueber FrequenzIstwert, 4 = MAN ueber FreuqenzIstwert]*)
		bLFSM_TestStart : BOOL;
		bLFSM_TestStop : BOOL;
		bLFSM_TestFRamp_Active : BOOL;
		rLFSM_TestFRampRate : REAL;
	END_STRUCT;
	_tLinear : 	STRUCT
		x1 : INT;
		y1 : INT;
		x2 : INT;
		y2 : INT;
	END_STRUCT;
	_rpm_count : 	STRUCT
		count : DINT;
		h : INT;
		m : INT;
		s : INT;
	END_STRUCT;
	_tMeasurePoint : 	STRUCT
		P : INT;
		t : INT;
		w : INT;
		n : INT;
	END_STRUCT;
	_tPIDpar : 	STRUCT
		tast : UINT;
		kp : INT;
		ki : INT;
		kd : INT;
		y_min : INT;
		y_max : INT;
		soll : INT;
		ist : INT;
	END_STRUCT;
	_tMonicLimit : 	STRUCT
		limit : USINT;
		kind : USINT;
		delay : USINT;
	END_STRUCT;
	rtctime_typ : 	STRUCT
		year : UINT;
		month : USINT;
		day : USINT;
		reserve : USINT;
		hour : USINT;
		minute : USINT;
		second : USINT;
		millisec : UINT;
		microsec : UINT;
	END_STRUCT;
	alarmP : 	STRUCT
		ENABLE : BOOL;
		SET : BOOL;
		PTON : TIME;
		RESET : BOOL;
		PRIO : INT;
		TEST : BOOL;
		Q : BOOL;
	END_STRUCT;
	tManAuxCtr_typ : 	STRUCT
		bGnl_Rel : BOOL; (*General release. Safety conditions (gas alarm, fire alarm, safety loop, ..) are OK.*) (*OldName: new PV; Cycle: 5;*)
		bECWP_PreH_COf_Man : BOOL; (*engine cooling water pump preheating demand off*) (*OldName: new PV; Cycle: 5;*)
		bECW_PreH_COf_Man : BOOL; (*engine cooling water preheating demand off*) (*OldName: new PV; Cycle: 5;*)
		bInAirER_Lou2DemOpen_Man : BOOL; (*demand open air inlet louver 2*) (*OldName: new PV; Cycle:5;*)
		bInAirER_Lou1DemOpen_Man : BOOL; (*demand open air inlet louver 1*) (*OldName: new PV; Cycle:5;*)
		bOutAirER_LouDemOpen_Man : BOOL; (*open air outlet louver *) (*OldName: new PV; Cycle:5;*)
		bInAirER_Fan1DemOn_Man : BOOL; (*demand air inlet ventilator 1*) (*OldName: new PV; Cycle:5;*)
		bInAirER_Fan2DemOn_Man : BOOL; (*demand air inlet ventilator 2*) (*OldName: new PV; Cycle:5;*)
		bER_FC_Set_Man : BOOL; (*demand engine room frequency converter setpoint*) (*OldName: new PV; Cycle:5;*)
		rER_FC_Set_Man : REAL; (*engine room frequency converter setpoint [%]*) (*OldName: new PV; Cycle:5;*)
		bER_OutlV_FC_Set_Man : BOOL; (*demand engine room air outlet ventilation frequency converter setpoint*) (*OldName: new PV; Cycle:5;*)
		rER_OutlV_FC_Set_Man : REAL; (*engine room air outlet ventilation frequency converter setpoint [%]*) (*OldName: new PV; Cycle:5;*)
		bEC_DemPump_Man : BOOL; (*emergency cooler demand pump*) (*OldName: new PV; Cycle:5;*)
		bEC_DemFan_Man : BOOL; (*emergency cooler demand fan 1 - 16*) (*OldName: new PV; Cycle:5;*)
		bChC_DemPump_Man : BOOL; (*charge cooler demand pump*) (*OldName: new PV; Cycle:5;*)
		bChC_DemFan_Man : BOOL; (*charge cooler demand fan 1 - 16*) (*OldName: new PV; Cycle:5;*)
		bEG_BoVaCoOpen_Man : BOOL; (*exhaust gas boiler valve command open*) (*OldName: new PV; Cycle:5;*)
		bEG_BoVaCoClose_Man : BOOL; (*exhaust gas boiler valve command close*) (*OldName: new PV; Cycle:5;*)
		bEG_ByVaCoOpen_Man : BOOL; (*exhaust gas bypass valve command open*) (*OldName: new PV; Cycle:5;*)
		bEG_ByVaCoClose_Man : BOOL; (*exhaust gas bypass valve command close*) (*OldName: new PV; Cycle:5;*)
		bAuxCust_Man : ARRAY[0..40]OF BOOL; (*reserve customer auxiliaries*) (*OldName: new PV; Cycle:5;*)
		bCDP_Dem_Man : BOOL; (*demand condensor pump*) (*OldName: new PV; Cycle:5;*)
		bBHV_Dem_Man : BOOL; (*demand boiler house ventilation*) (*OldName: newPv; Cycle:5;*)
		bHWF_Dem_Man : BOOL; (*demand heating circuit flap*) (*OldName:newPv; Cycle:5;*)
		bChC_Heating_Man : BOOL; (*charge cooler pre heating*) (*OldName:newPv; Cycle:5;*)
		bCO2_DemCodinox_Man : BOOL; (*CO2 demand CODINOX*) (*OldName:newPv; Cycle:5;*)
		bECWP_PreH_COf : BOOL; (*engine cooling water pump preheating demand off*) (*OldName: new PV; Cycle: 5;*)
		bECW_PreH_COf : BOOL; (*engine cooling water preheating demand off*) (*OldName: new PV; Cycle: 5;*)
		bInAirER_Lou2DemOpen : BOOL; (*demand open air inlet louver 2*) (*OldName: new PV; Cycle:5;*)
		bInAirER_Lou1DemOpen : BOOL; (*demand open air inlet louver 1*) (*OldName: new PV; Cycle:5;*)
		bOutAirER_LouDemOpen : BOOL; (*open air outlet louver *) (*OldName: new PV; Cycle:5;*)
		bInAirER_Fan1DemOn : BOOL; (*demand air inlet ventilator 1*) (*OldName: new PV; Cycle:5;*)
		bInAirER_Fan2DemOn : BOOL; (*demand air inlet ventilator 2*) (*OldName: new PV; Cycle:5;*)
		bER_OutlV_FC_Set : BOOL; (*demand engine room air outlet ventilation frequency converter setpoint*) (*OldName: new PV; Cycle:5;*)
		rER_OutlV_FC_Set : REAL; (*engine room air outlet ventilation frequency converter setpoint [%]*) (*OldName: new PV; Cycle:5;*)
		bER_FC_Set : BOOL; (*demand engine room frequency converter setpoint*) (*OldName: new PV; Cycle:5;*)
		rER_FC_Set : REAL; (*engine room frequency converter setpoint [%]*) (*OldName: new PV; Cycle:5;*)
		bEC_DemPump : BOOL; (*emergency cooler demand pump*) (*OldName: new PV; Cycle:5;*)
		bEC_DemFan : BOOL; (*emergency cooler demand fan 1 - 16*) (*OldName: new PV; Cycle:5;*)
		bChC_DemPump : BOOL; (*charge cooler demand pump*) (*OldName: new PV; Cycle:5;*)
		bChC_DemFan : BOOL; (*charge cooler demand fan 1 - 16*) (*OldName: new PV; Cycle:5;*)
		bEG_BoVaCoOpen : BOOL; (*exhaust gas boiler valve command open*) (*OldName: new PV; Cycle:5;*)
		bEG_BoVaCoClose : BOOL; (*exhaust gas boiler valve command close*) (*OldName: new PV; Cycle:5;*)
		bEG_ByVaCoOpen : BOOL; (*exhaust gas bypass valve command open*) (*OldName: new PV; Cycle:5;*)
		bEG_ByVaCoClose : BOOL; (*exhaust gas bypass valve command close*) (*OldName: new PV; Cycle:5;*)
		bAuxCust : ARRAY[0..70]OF BOOL; (*reserve customer auxiliaries*) (*OldName: new PV; Cycle:5;*) (*watch for HMI Extension*)
		bCDP_Dem : BOOL; (*demand condensor pump*) (*OldName: new PV; Cycle:5;*)
		bBHV_Dem : BOOL; (*demand boiler house ventilation*) (*OldName: newPv; Cycle:5;*)
		bHWF_Dem : BOOL; (*demand heating circuit flap*) (*OldName:newPv; Cycle:5;*)
		bChC_Heating : BOOL; (*charge cooler pre heating*) (*OldName:newPv; Cycle:5;*)
		bCO2_DemCodinox : BOOL; (*CO2 demand CODINOX*) (*OldName:newPv; Cycle:5;*)
		bChC2_DemPump : BOOL; (*charge cooler 2 demand pump*) (*OldName: new PV; Cycle:5;*)
		bChC2_DemPump_Man : BOOL; (*charge cooler 2 demand pump*) (*OldName: new PV; Cycle:5;*)
		bChC2_DemFan : BOOL; (*charge cooler 2 demand fan 1 - 16*) (*OldName: new PV; Cycle:5;*)
		bChC2_DemFan_Man : BOOL; (*charge cooler 2 demand fan 1 - 16*) (*OldName: new PV; Cycle:5;*)
		bChC2_Heating : BOOL; (*charge cooler 2 pre heating*) (*OldName:newPv; Cycle:5;*)
		bChC2_Heating_Man : BOOL; (*charge cooler 2 pre heating*) (*OldName:newPv; Cycle:5;*)
		bECW_HydrPreH_COf : BOOL; (*engine cooling water hydraulic preheating demand off*) (*OldName: new PV; Cycle: 5;*)
		bECW_HydrPreH_COf_Man : BOOL; (*engine cooling water hydraulic preheating demand off*) (*OldName: new PV; Cycle: 5;*)
		bEOP_DemPump : BOOL; (*engine prelubrication pump manual demand*) (*OldName: new PV; Cycle: 5;*)
		bEOP_DemPump_Man : BOOL; (*engine prelubrication pump manual demand*) (*OldName: new PV; Cycle: 5;*)
	END_STRUCT;
	BAD_INTERFACES : 	STRUCT
		bMsg1045 : BOOL; (* canceled for implementation of OXIcat V4.05; Msg: catalyst temperature high*) (*OldName:AMM_A10xx;Cycle:5*)
		bMsg1069 : BOOL; (* canceled for implementation of OXIcat V4.05; Msg: catalyst temperature signal failure*) (*OldName:AMM_A10xx;Cycle:5*)
		bMsg1161 : BOOL; (* canceled for implementation of OXIcat V4.05; Msg: exhaust gas temperature before catalyst signal failure*) (*OldName:AMM_W11xx;Cycle:5*)
		bMsg1162 : BOOL; (* canceled for implementation of OXIcat V4.05; Msg: exhaust gas temperature after catalyst signal failure*) (*OldName:AMM_W11xx;Cycle:5*)
		bMsg1169 : BOOL; (* canceled for implementation of OXIcat V4.05; Msg: exhaust gas temperature before catalyst high*) (*OldName:AMM_W11xx;Cycle:5*)
		bMsg1170 : BOOL; (* canceled for implementation of OXIcat V4.05; Msg: exhaust gas temperature after catalyst high*) (*OldName:AMM_W11xx;Cycle:5*)
		bMsg1174 : BOOL; (* canceled for implementation of OXIcat V4.05; Msg: catalyst temperature high high*) (*OldName:AMM_W11xx;Cycle:5*)
		bMsg2112 : BOOL; (* canceled for implementation of OXIcat V4.05; Msg: catalyst temperature signal failure*) (*OldName:AMM_W21xx;Cycle:5*)
		bReq_AuxMod_OfC : BOOL; (* = WRONG INTERFACE VARIABLE, DO NOT  USE!  -> bEng_Aux_Dem_TOF*) (*OldName: T12	; Cycle: 5;*)
		bStart_Imp : BOOL; (* = WRONG INTERFACE VARIABLE, DO NOT  USE!  ->   Startzaehlerimpuls  (Replacement IN_CU.bImp_Start) *) (*OldName: T25, M_STRTIMP	; Cycle: 5;*)
		rT_Cat_Vis : REAL; (* = WRONG INTERFACE VARIABLE, DO NOT  USE!  ->  IF603 exh.gas temp.after  cat.	*) (* OldName:  	ANA.NKAT	; Cycle: 5;*)
		rT_Ch : REAL; (* = WRONG INTERFACE VARIABLE, DO NOT USE!  -> IF601 fuel mixture temperature	*) (* OldName:  	ANA.LLTP	; Cycle: 5;*)
		rT_EGafHeEx1 : HALioAi_Type; (* = WRONG INTERFACE VARIABLE, DO NOT  USE!  ->  IF660 exh.gas temp.aft.heat exch.1*) (* OldName:  	ANA_NWTT1	; Cycle: 5;*)
		rT_EGafHeEx2 : HALioAi_Type; (* = WRONG INTERFACE VARIABLE, DO NOT  USE!  ->     IF661 exh.gas temp.aft.heat exch.2*) (* OldName:  	ANA_NWTT2	; Cycle: 5;*)
		rT_EGaHE_Vis : REAL; (* = WRONG INTERFACE VARIABLE, DO NOT  USE!  ->  IF506 exh.gas temp.aft.heat exch. 	*) (* OldName:  	ANA.NABK	; Cycle: 5;*)
		rT_EGaTC_Vis : REAL; (* = WRONG INTERFACE VARIABLE, DO NOT  USE!  ->  IF505 exh.gas temp.after engine (RENAMED FROM IN_CU.rT_EG(bHE)_Vis)*) (* OldName:  	ANA.VABK	; Cycle: 5;*)
		rT_EGbCat_Vis : REAL; (* = WRONG INTERFACE VARIABLE, DO NOT  USE!  ->  IF602 exh.gas temp.before cat.	*) (* OldName:  	ANA.VKAT	; Cycle: 5;*)
	END_STRUCT;
	GRID2CUSTOM_Struct : 	STRUCT
		rDroop_GrC_FSMU : REAL; (*FSMU Droop reference [Hz]*)
		rDroop_GrC_FSMO : REAL; (*FSMO Droop reference [Hz]*)
		rFSMU_GRC_DB : REAL; (*FSMU Deadband reference [Hz]*)
		rFSMO_GRC_DB : REAL; (*FSMO Deadband reference [Hz]*)
		bSet_GrC_ILF : BOOL; (*ILF function active*)
		bSet_GrC_FSM : BOOL; (*FSM function active*)
		rFNom_LFSM_Ref : REAL; (*Frequency reference for FSM/LFSM [Hz]*)
		bLFSM_Test_On : BOOL; (* Test FC active *)
		iSet_FC_Testmode : INT; (* Testmode [0 = testmode off / 1 = AUTO square wave nominal frequency / 2 = MAN nominal frequency  / 3 = AUTO square wave current frequency / 4 = MAN current frequency] *)
		rFNom_FSM_ManualTest : REAL; (* MAN test - Adjustable nominal frequency [Hz] *)
		rFAct_FSM_ManualTest : REAL; (* MAN test - Adjustable current frequency [Hz] *)
		rMarg_GrC_FSM_Pos : REAL; (* Power margin FSM positiv *)
		rMarg_GrC_FSM_Neg : REAL; (* Power margin FSM negativ *)
		bCheck_GR2CU : BOOL; (* Controlbit for Grid to Custom structure *)
	END_STRUCT;
	CUSTOM2GRID_Struct : 	STRUCT
		bLFSMO_DB_AI_COn : BOOL; (* AI:LFSMO Deadband set command on *)
		bLFSMO_DB_AI_COf : BOOL; (* AI:LFSMO Deadband set command off *)
		bLFSMO_DB_BC_COn : BOOL; (* Bus:LFSMO Deadband set command on *)
		bLFSMO_DB_BC_COf : BOOL; (* Bus:LFSMO Deadband set command off *)
		rF_LFSMO_DB_BC : REAL; (* Bus: Scaling value LFSMO Deadband from EU [Hz] *)
		bLFSMO_DB_BC_SetErr : BOOL; (* Bus: LFSMO Deadband measuring signal failure *)
		bLFSMU_DB_AI_COn : BOOL; (* AI:LFSMU Deadband set command on *)
		bLFSMU_DB_AI_COf : BOOL; (* AI:LFSMU Deadband set command off *)
		bLFSMU_DB_BC_COn : BOOL; (* Bus:LFSMU Deadband set command on *)
		bLFSMU_DB_BC_COf : BOOL; (* Bus:LFSMU Deadband set command off *)
		rF_LFSMU_DB_BC : REAL; (* Bus: Scaling value LFSMU Deadband from EU [Hz] *)
		bLFSMU_DB_BC_SetErr : BOOL; (* Bus: LFSMU Deadband measuring signal failure *)
		bLFSMO_Droop_AI_COn : BOOL; (* AI:LFSMO Droop set command on *)
		bLFSMO_Droop_AI_COf : BOOL; (* AI:LFSMO Droop set command off *)
		bLFSMO_Droop_BC_COn : BOOL; (* Bus:LFSMO Droop set command on *)
		bLFSMO_Droop_BC_COf : BOOL; (* Bus:LFSMO Droop set command off *)
		rP_LFSMO_Droop_BC : REAL; (* Bus: Scaling value LFSMO Droop from EU [Hz] *)
		bLFSMO_Droop_BC_SetErr : BOOL; (* Bus: LFSMO Droop measuring signal failure *)
		bLFSMU_Droop_AI_COn : BOOL; (* AI:LFSMU Droop set command on *)
		bLFSMU_Droop_AI_COf : BOOL; (* AI:LFSMU Droop set command off *)
		bLFSMU_Droop_BC_COn : BOOL; (* Bus:LFSMU Droop set command on *)
		bLFSMU_Droop_BC_COf : BOOL; (* Bus:LFSMU Droop set command off *)
		rP_LFSMU_Droop_BC : REAL; (* Bus: Scaling value LFSMU Droop from EU [Hz] *)
		bLFSMU_Droop_BC_SetErr : BOOL; (* Bus: LFSMU Droop measuring signal failure *)
		bFSMU_Droop_AI_COn : BOOL; (* AI:FSMU Droop set command on *)
		bFSMU_Droop_AI_COf : BOOL; (* AI:FSMU Droop set command off *)
		bFSMU_Droop_BC_COn : BOOL; (* Bus:FSMU Droop set command on *)
		bFSMU_Droop_BC_COf : BOOL; (* Bus:FSMU Droop set command off *)
		rP_FSMU_Droop_BC : REAL; (* Bus: Scaling value FSMU Droop from EU [Hz] *)
		bFSMU_Droop_BC_SetErr : BOOL; (* Bus: FSMU Droop measuring signal failure *)
		bFSMO_Droop_AI_COn : BOOL; (* AI:FSMO Droop set command on *)
		bFSMO_Droop_AI_COf : BOOL; (* AI:FSMO Droop set command off *)
		bFSMO_Droop_BC_COn : BOOL; (* Bus:FSMO Droop set command on *)
		bFSMO_Droop_BC_COf : BOOL; (* Bus:FSMO Droop set command off *)
		rP_FSMO_Droop_BC : REAL; (* Bus: Scaling value FSMO Droop from EU [Hz] *)
		bFSMO_Droop_BC_SetErr : BOOL; (* Bus: FSMO Droop measuring signal failure *)
		bFSMU_DB_AI_COn : BOOL; (* AI:FSMU Deadband set command on *)
		bFSMU_DB_AI_COf : BOOL; (* AI:FSMU Deadband set command off *)
		bFSMU_DB_BC_COn : BOOL; (* Bus:FSMU Deadband set command on *)
		bFSMU_DB_BC_COf : BOOL; (* Bus:FSMU Deadband set command off *)
		rF_FSMU_DB_BC : REAL; (* Bus: Scaling value FSMU Deadband from EU [Hz] *)
		bFSMU_DB_BC_SetErr : BOOL; (* Bus: FSMU Deadband measuring signal failure *)
		bFSMO_DB_AI_COn : BOOL; (* AI:FSMO Deadband set command on *)
		bFSMO_DB_AI_COf : BOOL; (* AI:FSMO Deadband set command off *)
		bFSMO_DB_BC_COn : BOOL; (* Bus:FSMO Deadband set command on *)
		bFSMO_DB_BC_COf : BOOL; (* Bus:FSMO Deadband set command off *)
		rF_FSMO_DB_BC : REAL; (* Bus: Scaling value FSMO Deadband from EU [Hz] *)
		bFSMO_DB_BC_SetErr : BOOL; (* Bus: FSMO Deadband measuring signal failure *)
		bFSM_RMC_Up_AI_COn : BOOL; (* AI: Positive Margin FSM set command on *)
		bFSM_RMC_Up_AI_COf : BOOL; (* AI: Positive Margin FSM set command off *)
		bFSM_RMC_Up_BC_COn : BOOL; (* Bus: Positive Margin FSM set command on*)
		bFSM_RMC_Up_BC_COf : BOOL; (* Bus: Positive Margin FSM set command off *)
		rP_FSM_RMC_Up_BC : REAL; (* Bus: Scaling value for positive Margin FSM from EU [%Pn]*)
		bFSM_RMC_Up_BC_SetErr : BOOL; (* Bus: Positive Margin FSM setpoint measuring signal failure *)
		bFSM_RMC_Down_AI_COn : BOOL; (* AI: Negative Margin FSM set command on *)
		bFSM_RMC_Down_AI_COf : BOOL; (* AI: Negative Margin FSM set command off *)
		bFSM_RMC_Down_BC_COn : BOOL; (* Bus: Negative Margin FSM set command on*)
		bFSM_RMC_Down_BC_COf : BOOL; (* Bus: Negative Margin FSM set command off *)
		rP_FSM_RMC_Down_BC : REAL; (* Bus: Scaling value for negative Margin FSM from EU [%Pn]*)
		bFSM_RMC_Down_BC_SetErr : BOOL; (* Bus: Negative Margin FSM setpoint measuring signal failure *)
		bU_Droop_AI_COn : BOOL; (* AI: Droop U set command on *)
		bU_Droop_AI_COf : BOOL; (* AI: Droop U set command off *)
		bU_Droop_BC_COn : BOOL; (* Bus: Droop U set command on*)
		bU_Droop_BC_COf : BOOL; (* Bus: Droop U set command off *)
		rU_Droop_BC : REAL; (* Bus: Scaling value for droop U from EU [%]*)
		bU_Droop_BC_SetErr : BOOL; (* Bus: Droop U setpoint measuring signal failure *)
		bFSM_Rmp_AI_COn : BOOL; (* AI: Ramp rate set command on *)
		bFSM_Rmp_AI_COf : BOOL; (* AI: Ramp rate set command off *)
		bFSM_Rmp_BC_COn : BOOL; (* Bus: Ramp rate set command on*)
		bFSM_Rmp_BC_COf : BOOL; (* Bus: Ramp rate set command off *)
		rP_FSM_Rmp_Up_BC : REAL; (* Bus: Scaling value for ramp rate from EU [%Pnom/s]*)
		bFSM_Rmp_BC_SetErr : BOOL; (* Bus: Ramp rate setpoint measuring signal failure *)
		rP_FSM_Rmp_Down_BC : REAL; (* Bus: Scaling value for ramp rate DOWN from EU [%Pnom/s]*)
		bF_Ref_FSM_AI_COn : BOOL; (* AI: Frequency reference for FSM/LFSM set command on *)
		bF_Ref_FSM_AI_COf : BOOL; (* AI: Frequency reference for FSM/LFSM set command off *)
		bF_Ref_FSM_BC_COn : BOOL; (* Bus: Frequency reference for FSM/LFSM set command on*)
		bF_Ref_FSM_BC_COf : BOOL; (* Bus: Frequency reference for FSM/LFSM set command off *)
		rF_Ref_FSM_BC : REAL; (* Bus: Scaling value for Frequency reference for FSM/LFSM from EU [%Pnom/s]*)
		bF_Ref_FSM_BC_SetErr : BOOL; (* Bus: Frequency reference for FSM/LFSM setpoint measuring signal failure *)
		bLFSM_TestStop : BOOL; (* Stop of FC testmode*)
		bCheck_CU2GR : BOOL; (* Controlbit for Custom to Grid structure *)
	END_STRUCT;
	CUSTOM2GASTRAIN_Struct : 	STRUCT
		iGC_Select_Option : DINT; (*V4.07 new*)
		rCust_GT : ARRAY[0..15]OF REAL; (*V4.07 new*)
		tiGT_TestDuration : TIME; (*V4.07 new*)
		tiGCPulse_Duration_min : TIME; (*V4.07 new*)
		tiGV_Feedback_Delay_max : TIME; (*V4.07 new*)
		tIF_Revision : Revision_type; (*Revision number  of  latest interface change *)
	END_STRUCT;
	HALIO2CUSTOM_Struct : 	STRUCT
		tSet_LFSMO_DB_COn : HALioDi_Type; (*DI: Activation of LFSMO Deadband via AI*)
		tSet_LFSMO_DB_COf : HALioDi_Type; (*DI: De-activation of LFSMO Deadband via AI*)
		tSet_LFSMU_DB_COn : HALioDi_Type; (*DI: Activation of LFSMU Deadband via AI*)
		tSet_LFSMU_DB_COf : HALioDi_Type; (*DI: De-activation of LFSMU Deadband via AI*)
		tSet_LFSMO_Droop_COn : HALioDi_Type; (*DI: Activation of LFSMO Droop via AI*)
		tSet_LFSMO_Droop_COf : HALioDi_Type; (*DI: De-activation of LFSMO Droop via AI*)
		tSet_LFSMU_Droop_COn : HALioDi_Type; (*DI: Activation of LFSMO Droop via AI*)
		tSet_LFSMU_Droop_COf : HALioDi_Type; (*DI: De-activation of LFSMO Droop via AI*)
		tSet_FSMU_Droop_COn : HALioDi_Type; (*DI: Activation of FSMU Droop via AI*)
		tSet_FSMU_Droop_COf : HALioDi_Type; (*DI: De-activation of FSMU Droop via AI*)
		tSet_FSMO_Droop_COn : HALioDi_Type; (*DI: Activation of FSMO Droop via AI*)
		tSet_FSMO_Droop_COf : HALioDi_Type; (*DI: De-activation of FSMO Droop via AI*)
		tSet_FSMU_DB_COn : HALioDi_Type; (*DI: Activation of FSMU Deadband via AI*)
		tSet_FSMU_DB_COf : HALioDi_Type; (*DI: De-activation of FSMO Deadband via AI*)
		tSet_FSMO_DB_COn : HALioDi_Type; (*DI: Activation of FSMO Deadband via AI*)
		tSet_FSMO_DB_COf : HALioDi_Type; (*DI: De-activation of FSMO Deadband via AI*)
		tSet_FSM_RMC_Up_COn : HALioDi_Type; (*DI: Activation of positive Margin FSM via AI*)
		tSet_FSM_RMC_Up_COf : HALioDi_Type; (*DI: De-activation of positive Margin FSM via AI*)
		tSet_FSM_RMC_Down_COn : HALioDi_Type; (*DI: Activation of negative Margin FSM via AI*)
		tSet_FSM_RMC_Down_COf : HALioDi_Type; (*DI: De-activation of negative Margin FSM via AI*)
		tSet_U_Droop_COn : HALioDi_Type; (*DI: Activation of droop U via AI*)
		tSet_U_Droop_COf : HALioDi_Type; (*DI: De-activation of droop U via AI*)
		tSet_FSM_Rmp_COn : HALioDi_Type; (*DI: Activation of Ramp rate via AI*)
		tSet_FSM_Rmp_COf : HALioDi_Type; (*DI: De-activation of Ramp rate via AI*)
		tSet_F_Ref_FSM_COn : HALioDi_Type; (*DI: Activation of Reference frequency for FSM/LFSM via AI*)
		tSet_F_Ref_FSM_COf : HALioDi_Type; (*DI:De-activation of Reference frequency for FSM/LFSM via AI*)
		bCheck_HA2CU : BOOL; (* Controlbit for HALio to Custom structure *)
	END_STRUCT;
	Values_Struct : 	STRUCT
		iCnt_OpHours : DINT; (*IF541 oper.hours count.high word	*) (* OldName:  	BTRB_high	; Cycle: 5;*)
		iCnt_Starts : DINT; (*IF543 start counter    high word	*) (* OldName:  	STRT_high	; Cycle: 5;*)
		rEO_Level : REAL; (*IF630 oil level	*) (* OldName:  	ANA.OELST	; Cycle: 5;*)
		rF_MMD : ARRAY[0..2]OF REAL; (* frequency multi measure device *) (* OldName:ssFreq; Cycle: *)
		rGT_CH4 : REAL; (*CH4 content, 1.0 = 100% *) (* OldName: 	ANA_CH4	; Cyclic: ; *)
		rGT_O2 : REAL; (*O2 content *) (* OldName: 	ANA_O2	; Cyclic: ; *)
		rI_Avg : ARRAY[0..2]OF REAL; (* current average *) (* OldName:ssIAvg; Cycle: *)
		rI_L1 : ARRAY[0..2]OF REAL; (* current 1 *) (* OldName:ssIL1; Cycle: *)
		rI_L2 : ARRAY[0..2]OF REAL; (* current 2 *) (* OldName:ssIL2; Cycle: *)
		rI_L3 : ARRAY[0..2]OF REAL; (* current 3 *) (* OldName:ssIL3; Cycle: *)
		rI_N : ARRAY[0..2]OF REAL; (* current neutral *) (* OldName:ssIN; Cycle: *)
		rLam_Eng_LL_Set : REAL; (* Leanox Lambda set point *) (* OldName: ssPosGasmixerNominal; Cycle:2; *)
		rN_EngAct : REAL; (*IF611 speed	*) (* OldName:  	ANA.DREHZ	; Cycle: 5;*)
		rPF_Act : ARRAY[0..2]OF REAL; (* power factor *) (* OldName:ssCosPhi; Cycle: *)
		rPos_CBV : REAL; (* compressor bypass valve position *) (*OldName: rPos_CBV; Cycle: 2 *)
		rPos_GM_Set_Norm : REAL; (* set point for the gasmixer *) (*OldName: ssPosGasmixerNominal; Cycle:2; *)
		rPos_TV : REAL; (* throttle valve position *) (*OldName: drkl_y; Cycle:2; *)
		rPr_Ch_P2s_Avg : REAL; (*average charge pressure p2' (after throttle valve) [bar]*)
		rPr_ECW : REAL; (*IF502 jacket water pressure *) (* OldName:  	ANA.KWD		; Cycle: 5;*)
		rPr_EngLubOil : REAL; (*IF504 oil pressure *) (* OldName:  	ANA.ODR		; Cycle: 5;*)
		rPr_GT_Gas : REAL; (*Gas pressure *) (* OldName: 	ANA_GD	; Cyclic: ; *)
		rPr_GT_Suct : REAL; (*Gas suction pressure *) (* OldName: 	ANA_SD	; Cyclic: ; *)
		rPr_PCG : REAL; (*Pressure pre chamber gas compressor  *) (* OldName: 	ANA_VKGD	; Cyclic: ; *)
		rPr_PC_Diff : REAL; (*Prechamber differential pressure*) (* OldName: 	ANA_PDIFF	; Cyclic: ; *)
		rP_Act : ARRAY[0..2]OF REAL; (* IF500 active power (IF LIST FROM TASK snd_cst) ??normiert 0-1?? 	*) (*OldName: ANA.P_IST	; Cycle: 5;*)
		rP_Set : REAL; (*IF540 setpoint power control	*) (* OldName:  	ANA.SOLL_PREG ; Cycle: 5;*)
		rP_WorkAct : ARRAY[0..2]OF REAL; (*IF536 total act.  outp.high word OldName > iP_WorkAct?	*) (* OldName:  	ANA.WARBH	; Cycle: 5;*)
		rQ_Act : ARRAY[0..2]OF REAL; (* power reactive *) (* OldName:ssPReac; Cycle: *)
		rQ_WorkReac : ARRAY[0..2]OF REAL; (*IF538 total react.outp.high word  OldName > iQ_WorkReac?*) (* OldName:  	ANA.BARBH	; Cycle: 5;*)
		rS_Act : ARRAY[0..2]OF REAL; (* power apperent *) (* OldName:ssPApper; Cycle: *)
		rT_AirER : REAL; (*vis air engine room temperature [degC]*) (*OldName:ANA_RTM; Cycle:5;*)
		rT_AirOutdoor : REAL; (*temperature air outdoor *) (*OldName:ANA_ULT; Cycle:5;*)
		rT_Cat : REAL; (*AI exhaust gas temperature catalyst general (before)*) (*OldName:ANA.KATP;Cycle:;*)
		rT_Ch_T1LP_Avg : REAL; (*average charge temperature before low-pressure turbocharger (= engine intake air) [degC]*) (*OldName:ssIATemp,ANA_ZLTP,rT_InAirER; Cycle:5;*) (* V04.04.00.00 *)
		rT_Ch_T2s_Avg : REAL; (*average charge temperature t2' (after throttle valve) [degC]*)
		rT_ECW : REAL; (*IF501 jacket water temperature	*) (* OldName:  	ANA.KWT		; Cycle: 5;*)
		rT_EGaCat : REAL; (*exhaust gas temperature after catalyst*) (*OldName:ANA.NKAT;Cycle:;*)
		rT_EGaHE : REAL; (*AI exhaust gas temperature after heat exchanger [degC]*) (*OldName:ANA.NABK;Cycle:5*)
		rT_EGaHE1 : REAL; (*exhaust gas temperature after heat exchanger 1*) (*OldName:NWTT1_WE;Cycle:5*)
		rT_EGaHE2 : REAL; (*exhaust gas temperature after heat exchanger 2*) (*OldName:NWTT2_WE;Cycle:5*)
		rT_EGaTC : REAL; (*AI exhaust gas temperature after turbo charger [degC]*) (*OldName:ANA.VABK;Cycle:5*)
		rT_EGbCat : REAL; (*exhaust gas temperature before catalyst*) (*OldName:ANA.VKAT;Cycle:;*)
		rT_EGbTC : REAL; (*AI exhaust gas temperature before turbo charger*) (*OldName:ANA.T3;Cycle:5*)
		rT_EG_Avg : REAL; (* cylinder temperature average [degC] *) (* OldName: t_zyl_mw; Cycle:5; *)
		rT_EO : REAL; (*IF503 oil temperature	*) (* OldName:  	ANA.OTP		; Cycle: 5;*)
		rT_EPU_EG : ARRAY[0..24]OF REAL; (*EngineController::  engine power unit exhaust gas temperatures *) (* OldName:  T_ZYL ; Cycle: 5;*)
		rT_Gen_Bear_A_Act : REAL; (*IF609 gen.bearing temp.(A)	*) (* OldName:  	ANA.LAG1	; Cycle: 5;*)
		rT_Gen_Bear_B_Act : REAL; (*IF610 gen.bearing temp.(B)	*) (* OldName:  	ANA.LAG2	; Cycle: 5;*)
		rT_Gen_Wind_Act : REAL; (* generator winding temperature signal *) (*OldName:ANA.WICK;Cycle:;*)
		rT_Gen_Wind_Act_L1 : REAL; (*IF606 gen.winding temp.L1	*) (* OldName:  	ANA.WICK1	; Cycle: 5;*)
		rT_Gen_Wind_Act_L2 : REAL; (*IF607 gen.winding temp.L2	*) (* OldName:  	ANA.WICK2	; Cycle: 5;*)
		rT_Gen_Wind_Act_L3 : REAL; (*IF608 gen.winding temp.L3	*) (* OldName:  	ANA.WICK3	; Cycle: 5;*)
		rT_GT : REAL; (*Gas temperature *) (* OldName: 	ANA_GT	; Cyclic: ; *)
		rT_HW_Re : REAL; (*IF509 return water temperature	*) (* OldName:  	ANA.RLTP	; Cycle: 5;*)
		rT_HW_ReAfEC : REAL; (*temperature heat water return after emergency cooler [degC]*) (*OldName:ANA.RLT_NK; Cycle:5;*)
		rT_HW_Su : REAL; (*IF510 supply water temperature	*) (* OldName:  	ANA.VLTP	; Cycle: 5;*)
		rT_PlateHE : REAL; (*AI exhaust gas temperature before heat exchanger*) (*OldName:ANA.ROHR;Cycle:5*)
		rU_Avg : ARRAY[0..2]OF REAL; (* voltage average *) (* OldName:ssUAvg; Cycle: *)
		rU_Gen_Exc : REAL; (*IF605 gen.excitation voltage*) (*OldName: ANA.ERREG; Cycle:;*)
		rU_L1L2 : ARRAY[0..2]OF REAL; (* voltage 12 *) (* OldName:ssUL1L2; Cycle: *)
		rU_L1N : ARRAY[0..2]OF REAL; (* voltage 1 *) (* OldName:ssUL1N; Cycle: *)
		rU_L2L3 : ARRAY[0..2]OF REAL; (* voltage 23 *) (* OldName:ssUL2L3; Cycle: *)
		rU_L2N : ARRAY[0..2]OF REAL; (* voltage 2 *) (* OldName:ssUL2N; Cycle: *)
		rU_L3L1 : ARRAY[0..2]OF REAL; (* voltage 31 *) (* OldName:ssUL3L1; Cycle: *)
		rU_L3N : ARRAY[0..2]OF REAL; (* voltage 3 *) (* OldName:ssUL3N; Cycle: *)
		rVol_GT : REAL; (*Gas volume *) (* OldName: 	ANA_GM	; Cyclic: ; *)
		tCustAnaIn : ARRAY[0..120]OF HALioAi_Type; (*Replacement for RAN_KANAL...*) (*OldName: ANA_RAN	; Cycle: 5;*)
		bImpClock : BOOL; (*Keep Alive signal*)
		iMaintenanceCount : ARRAY[0..20]OF DINT;
		iCount : ARRAY[0..20]OF DINT;
	END_STRUCT;
	Messages_Struct : 	STRUCT
		bMsg : ARRAY[0..9999]OF BOOL;
		bEng_Rdy_Rem : BOOL;
		bEng_Aux_Dem_CDR : BOOL;
		bGCB_DemSy : BOOL;
		bMCB_DemSy : BOOL;
		bImp_OpHour : BOOL;
		bImp_Start : BOOL;
	END_STRUCT;
	Spare_Struct : 	STRUCT
		bCustDigOpcUa : ARRAY[0..20]OF BOOL;
		rCustAnaOpcUa : ARRAY[0..60]OF REAL;
	END_STRUCT;
	Control_Struct : 	STRUCT
		bBus_Dem_OpcUa : BOOL;
		bBusPulse_OpcUa : BOOL;
		rP_Set_OpcUa : REAL;
	END_STRUCT;
	Eng2Cust_Struct : 	STRUCT
		tMessages : Messages_Struct;
		tValues : Values_Struct;
		tSpare : Spare_Struct;
	END_STRUCT;
	Cust2Eng_Struct : 	STRUCT
		tControl : Control_Struct;
		tSpare : Spare_Struct;
	END_STRUCT;
	tPlantComData_Cust100ms : 	STRUCT
		digitalSignals : ARRAY[0..31]OF tDigitalSignal_Struct;
		analogSignals : ARRAY[0..15]OF tAnalogSignal_Struct;
	END_STRUCT;
	tPlantComData_Cust10ms : 	STRUCT
		digitalSignals : ARRAY[0..15]OF tDigitalSignal_Struct;
		analogSignals : ARRAY[0..7]OF tAnalogSignal_Struct;
	END_STRUCT;
	tAnalogSignal_Struct : 	STRUCT
		Value : REAL;
		GoodQual : BOOL;
	END_STRUCT;
	tDigitalSignal_Struct : 	STRUCT
		Value : BOOL;
		GoodQual : BOOL;
	END_STRUCT;
	tPlantComm_Para : 	STRUCT
		iMas_Num_Min : USINT; (*[Para 15022] First Master in the Communication*)
		iMas_Num_Max : USINT; (*[Para 15023] Last Master in the Communication*)
		iEng_Num_Min : USINT; (*[Para 15024] First Engine in the Communication*)
		iEng_Num_Max : USINT; (*[Para 15025] Last Engine in the Communication*)
	END_STRUCT;
END_TYPE
```
